(* IEC 61131-3 sources: Explicit_MPC_on_PLC/Quad-Tank/MATLAB_Files/plcsrc, 1 file *)

(* ---- sim_mixed.st ---- *)
(*
 *
 * File: sim_mixed.st
 *
 * IEC 61131-3 Structured Text (ST) code generated for subsystem "sim_mixed/Explicit Controller"
 *
 * Model name                      : sim_mixed
 * Model version                   : 1.162
 * Model creator                   : andrewralea
 * Model last modified by          : andrewralea
 * Model last modified on          : Fri May 21 18:47:45 2021
 * Model sample time               : 0s
 * Subsystem name                  : sim_mixed/Explicit Controller
 * Subsystem sample time           : 0.5s
 * Simulink PLC Coder version      : 3.3 (R2020b) 29-Jul-2020
 * ST code generated on            : Fri May 21 23:25:07 2021
 *
 * Target IDE selection            : Beckhoff TwinCAT 3
 * Test Bench included             : No
 *
 *)
FUNCTION_BLOCK Explicit
VAR_INPUT
    ssMethodType: SINT;
    MeasuredTankOutputs: ARRAY [0..1] OF LREAL;
    ref: ARRAY [0..1] OF LREAL;
END_VAR
VAR_OUTPUT
    mv: ARRAY [0..1] OF LREAL;
END_VAR
VAR
    last_x_PreviousInput: ARRAY [0..5] OF LREAL;
    last_mv_DSTATE: ARRAY [0..1] OF LREAL;
    Explicit_b_M: ARRAY [0..11] OF LREAL := 1.23046367255072E-5,1.0600898470460902E-6,2.3336033090402565E-6,
        8.7638681898692419E-6,0.39038774660580289,5.7642544662640772E-8,2.7337306073553671E-6,1.2817201955703276E-5,
        8.74919612830075E-6,2.5558076546081948E-6,-1.9842244313224275E-7,0.39038772758565754;
    Explicit_b_Cm: ARRAY [0..11] OF LREAL := 0.15299877600979192,0.0,0.0,0.15299877600979192,0.0,0.0,0.0,0.0,1.0,
        0.0,0.0,1.0;
    Explicit_b_thmin: ARRAY [0..9] OF LREAL := -12.5,-17.5,-3.260954352640991,-0.9466686383552787,-1.25,-1.25,-12.5,
        -17.5,-44.314868949193837,-76.652836957418671;
    Explicit_b_thmax: ARRAY [0..9] OF LREAL := 30.0,25.0,39.239045647359006,41.553331361644723,1.25,1.25,25.0,20.0,
        150.328,150.328;
    b_i1: ARRAY [0..124] OF INT := 1,31,57,83,108,132,157,182,208,234,258,283,308,333,355,381,402,422,442,463,481,
        502,521,544,564,587,608,627,648,668,687,708,723,742,763,779,799,817,837,852,872,892,907,926,948,968,985,
        1011,1032,1049,1072,1093,1112,1126,1146,1165,1185,1205,1222,1243,1265,1287,1306,1326,1346,1365,1390,1411,
        1427,1446,1466,1485,1504,1524,1544,1560,1579,1597,1616,1632,1653,1672,1691,1709,1731,1751,1771,1787,1807,
        1825,1845,1861,1886,1904,1922,1941,1961,1982,1998,2015,2036,2057,2075,2096,2114,2134,2153,2174,2194,2216,
        2235,2254,2272,2293,2313,2330,2350,2370,2390,2410,2429,2450,2469,2487,2507;
    b_i2: ARRAY [0..124] OF INT := 30,56,82,107,131,156,181,207,233,257,282,307,332,354,380,401,421,441,462,480,501,
        520,543,563,586,607,626,647,667,686,707,722,741,762,778,798,816,836,851,871,891,906,925,947,967,984,1010,
        1031,1048,1071,1092,1111,1125,1145,1164,1184,1204,1221,1242,1264,1286,1305,1325,1345,1364,1389,1410,1426,
        1445,1465,1484,1503,1523,1543,1559,1578,1596,1615,1631,1652,1671,1690,1708,1730,1750,1770,1786,1806,1824,
        1844,1860,1885,1903,1921,1940,1960,1981,1997,2014,2035,2056,2074,2095,2113,2133,2152,2173,2193,2215,2234,
        2253,2271,2292,2312,2329,2349,2369,2389,2409,2428,2449,2468,2486,2506,2526;
    Explicit_b_L: ARRAY [0..11] OF LREAL := 1.19928863023028E-5,2.1952511223334454E-6,2.1569802942442451E-6,
        7.5728062260383986E-6,0.39038774660580267,5.7642544623488507E-8,3.2749111187589827E-6,1.2730433289085341E-5,
        8.0869972913321024E-6,2.2084581488572959E-6,-1.9842244312551109E-7,0.39038772758565737;
    Explicit_b_Bu: ARRAY [0..11] OF LREAL := 0.010205131094390857,0.00040302205517911383,0.0,0.0054488837150258882,
        0.0,0.0,0.00022154024327610144,0.010236745349900997,0.0056320000157246437,0.0,0.0,0.0;
    Explicit_b_A: ARRAY [0..35] OF LREAL := 0.96059819818356329,0.0,0.0,0.0,0.0,0.0,0.0,0.96659623833897423,0.0,0.0,
        0.0,0.0,0.074166176359097585,0.0,0.92431317949013092,0.0,0.0,0.0,0.0,0.1335679905776915,0.0,
        0.86409403496045134,0.0,0.0,0.0,0.0,0.0,0.0,1.0,0.0,0.0,0.0,0.0,0.0,0.0,1.0;
    Explicit_c_K: ARRAY [0..2525] OF LREAL := 85.828012190346456,83.122636404418486,64.080512591089587,
        62.020995879684413,58.758889676769776,56.867312090766596,6.1162428161412166,8.53615478597103,
        4.5664808584950682,6.3691533823982,4.1872534117759654,5.8399035361094738,30.0,25.0,39.239045647359006,
        41.553331361644723,1.25,1.25,25.0,20.0,150.328,150.328,12.5,17.5,3.260954352640991,0.9466686383552787,1.25,
        1.25,12.5,17.5,-85.828012190346442,83.160013557517672,0.39842731610608123,62.06462880871775,
        0.41050111399720146,56.91260957310422,8.4951416229813166,6.3221365550079094,5.7913950841796,30.0,25.0,
        39.239045647359006,41.553331361644723,1.25,1.25,20.0,150.328,150.328,12.5,17.5,3.260954352640991,
        0.9466686383552787,1.25,1.25,12.5,17.5,-83.122636404418486,85.864225454146336,64.121415141998071,
        0.38892275664372283,58.800482042349721,0.400834317759825,6.0763592904683081,4.52235846378462,
        4.1427133961342912,30.0,25.0,39.239045647359006,41.553331361644723,1.25,1.25,25.0,150.328,150.328,12.5,17.5,
        3.260954352640991,0.9466686383552787,1.25,1.25,12.5,17.5,-64.080512591089587,8.505599391495803,
        5.8036863919186326,-77.527008024685543,118.15715787051693,83.1493054364041,62.0524437250436,
        56.9000995036549,6.33408222099711,30.0,25.0,39.239045647359006,41.553331361644723,1.25,1.25,25.0,20.0,
        150.328,12.5,17.5,3.260954352640991,0.9466686383552787,1.25,1.25,17.5,-62.020995879684421,6.085443991111319,
        4.1528211444790628,-75.0536194743548,85.854610754335354,114.60675801046474,64.110937969245654,
        58.789954915559505,30.0,25.0,39.239045647359006,41.553331361644723,1.25,1.25,25.0,20.0,150.328,12.5,17.5,
        3.260954352640991,0.9466686383552787,1.25,1.25,12.5,-58.758889676769776,106.51779109033414,
        83.142049521683674,77.527008024685614,62.043935540441744,56.891257027927281,8.5137096448380447,
        6.3433957805279579,5.813284165486909,30.0,25.0,39.239045647359006,41.553331361644723,1.25,1.25,25.0,20.0,
        150.328,12.5,17.5,3.260954352640991,0.9466686383552787,1.25,1.25,17.5,-56.8673120907666,85.84776398721317,
        103.24892161906958,64.103194722139946,75.053619474354818,58.78208141394331,6.0931186576995735,
        4.5408406057656192,4.161356421857743,30.0,25.0,39.239045647359006,41.553331361644723,1.25,1.25,25.0,20.0,
        150.328,12.5,17.5,3.260954352640991,0.9466686383552787,1.25,1.25,12.5,-6.1162428161412148,
        83.116440481385681,62.014599085134925,56.860964676950751,8.53871469911331,0.028392574262163343,
        6.3721662785907309,0.029252972606836448,5.8430399803330584,30.0,25.0,39.239045647359006,41.553331361644723,
        1.25,1.25,25.0,20.0,150.328,12.5,17.5,3.260954352640991,0.9466686383552787,1.25,1.25,17.5,
        44.314868949193837,-8.53615478597103,85.820515372368362,64.072997847575692,58.751584273947309,
        6.1200693722462738,4.5707757582069863,0.039939840627104373,4.1916111645367051,0.041163080575065084,30.0,
        25.0,39.239045647359006,41.553331361644723,1.25,1.25,25.0,20.0,150.328,12.5,17.5,3.260954352640991,
        0.9466686383552787,1.25,1.25,12.5,76.652836957418671,-4.5664808584950682,-5.524699847834043,
        83.11695127091906,62.015234820715769,56.861634602583806,8.420069969679389,8.5379442187057482,
        5.8421419917176536,30.0,25.0,39.239045647359006,41.553331361644723,1.25,1.25,20.0,150.328,12.5,17.5,
        3.260954352640991,0.9466686383552787,1.25,1.25,12.5,17.5,-6.3691533823982,85.821037326316272,
        58.752296293187449,-7.7075191643753813,64.073586813938277,6.1190978799236042,11.769369550983704,
        4.5697137015683689,4.1905427066538907,30.0,25.0,39.239045647359006,41.553331361644723,1.25,1.25,25.0,
        150.328,12.5,17.5,3.260954352640991,0.9466686383552787,1.25,1.25,12.5,17.5,-4.1872534117759654,
        83.118307397217492,62.016623545698224,56.863007536175935,7.5906298878580278,8.5374517693042264,
        5.5246998478340474,6.3707077752714794,5.8415336572382541,30.0,25.0,39.239045647359006,41.553331361644723,
        1.25,1.25,20.0,150.328,12.5,17.5,3.260954352640991,0.9466686383552787,1.25,1.25,12.5,17.5,
        -5.8399035361094747,85.822512499078186,64.075138367645479,58.75372340844936,6.1183701458345565,
        10.602993535201676,4.5688969602600853,7.7075191643753822,4.1897144273516966,30.0,25.0,39.239045647359006,
        41.553331361644723,1.25,1.25,25.0,150.328,12.5,17.5,3.260954352640991,0.9466686383552787,1.25,1.25,12.5,
        17.5,-85.864225454146322,-83.160013557517686,0.44629698661502609,0.44356800965144572,0.45744577207009696,
        0.45640388165452567,30.0,25.0,39.239045647359006,41.553331361644723,1.25,1.25,150.328,150.328,12.5,17.5,
        3.260954352640991,0.9466686383552787,1.25,1.25,12.5,17.5,-0.398427316106117,-118.15715787051693,
        -0.37406353461084024,83.159322276278772,62.063996287931914,56.912013263967516,8.4950256940452444,
        6.3220198554896259,5.7912802018971812,30.0,25.0,39.239045647359006,41.553331361644723,1.25,1.25,25.0,20.0,
        150.328,150.328,12.5,17.5,3.260954352640991,0.9466686383552787,1.25,1.25,17.5,-85.8546972344799,
        114.6331530507331,0.42416405806333568,12.5,-118.17578392102031,-62.063996287931936,0.4242260045196693,30.0,
        25.0,39.239045647359006,41.553331361644723,1.25,1.25,25.0,150.328,12.5,17.5,3.260954352640991,
        0.9466686383552787,1.25,1.25,-106.51779109033414,-0.41050111399722317,83.159485968072531,
        0.37406353461083286,5.7913051165041507,30.0,25.0,39.239045647359006,41.553331361644723,1.25,1.25,150.328,
        150.328,12.5,17.5,3.260954352640991,0.9466686383552787,1.25,1.25,17.5,-85.847763987213185,75.09263865743236,
        12.5,-118.17085773789718,-56.91201326396753,30.0,25.0,39.239045647359006,41.553331361644723,1.25,1.25,25.0,
        20.0,150.328,12.5,17.5,3.260954352640991,0.9466686383552787,1.25,1.25,-85.820515372368362,
        -8.4951416229813166,12.5,-118.15424814904154,0.4416142007094101,-0.014455303353979251,30.0,25.0,
        39.239045647359006,41.553331361644723,1.25,1.25,20.0,150.328,12.5,17.5,3.260954352640991,0.9466686383552787,
        1.25,1.25,76.652836957418671,-85.821037326316258,-6.3221365550079085,0.39462833151258975,11.743492163705721,
        -0.020734861096918376,30.0,25.0,39.239045647359006,1.25,1.25,150.328,12.5,17.5,3.260954352640991,
        0.9466686383552787,1.25,1.25,12.5,-85.8225124990782,-5.7913950841796,0.395566095525043,0.40769403601124449,
        10.57062075206243,7.6648400160986254,30.0,25.0,39.239045647359006,41.553331361644723,1.25,1.25,150.328,12.5,
        17.5,3.260954352640991,0.9466686383552787,1.25,1.25,12.5,17.5,-83.1493575575283,-64.120717438993182,
        -114.62360062013384,118.1846753798998,0.41885284236598441,30.0,25.0,39.239045647359006,41.553331361644723,
        1.25,1.25,20.0,150.328,12.5,17.5,3.260954352640991,0.9466686383552787,1.25,1.25,-114.60941055213036,
        -0.38892275664366538,85.863418000357726,64.120717438993168,58.799849575245759,0.43609812832468658,
        6.0762590176834195,4.5222612688740718,4.1426203395211836,30.0,25.0,39.239045647359006,41.553331361644723,
        1.25,1.25,25.0,150.328,12.5,17.5,3.260954352640991,0.9466686383552787,1.25,1.25,-83.142049521683688,
        -58.800482042349707,106.54814350107794,77.565803690576558,0.4188608700639273,30.0,25.0,39.239045647359006,
        41.553331361644723,1.25,1.25,25.0,150.328,12.5,17.5,3.260954352640991,0.9466686383552787,1.25,1.25,17.5,
        -103.24892161906961,-0.40083431775979822,58.799926098422773,6.0762686203119909,4.5222701309312336,
        4.1426286413254676,30.0,25.0,39.239045647359006,41.553331361644723,1.25,1.25,25.0,20.0,150.328,150.328,12.5,
        17.5,3.260954352640991,0.9466686383552787,1.25,1.25,12.5,-83.116440481385666,-6.076359290468309,
        0.38503032707136814,-0.01947372407836211,-0.017687831808316137,30.0,25.0,39.239045647359006,
        41.553331361644723,1.25,1.25,25.0,150.328,12.5,17.5,3.260954352640991,0.9466686383552787,1.25,1.25,17.5,
        44.314868949193837,-83.117007264204418,-4.52235846378462,0.38602131564609687,8.3918353890059159,
        -0.017493533221530456,30.0,25.0,39.239045647359006,41.553331361644723,1.25,1.25,150.328,12.5,17.5,
        3.260954352640991,0.9466686383552787,1.25,1.25,17.5,-83.1183073972175,-4.1427133961342912,
        0.38679247515387888,0.39865998103592931,7.55674387574281,5.4820594007599839,30.0,25.0,39.239045647359006,
        41.553331361644723,1.25,1.25,150.328,12.5,17.5,3.260954352640991,0.9466686383552787,1.25,1.25,12.5,17.5,
        -64.111012657460421,-62.05249072734096,-77.555645848818614,-75.081475575886287,118.17571595289762,
        114.62356476522335,30.0,25.0,39.239045647359006,41.553331361644723,1.25,1.25,25.0,20.0,12.5,17.5,
        3.260954352640991,0.9466686383552787,1.25,1.25,-64.103194722139961,-56.900143592917374,-77.548207597133882,
        118.17085773789714,75.081423676406,30.0,25.0,39.239045647359006,41.553331361644723,1.25,1.25,25.0,20.0,12.5,
        17.5,3.260954352640991,0.9466686383552787,1.25,1.25,-64.072997847575721,-0.00038946835147730041,
        -77.519066370906955,-8.5055900532206987,118.1515689116242,-0.00082231448690014367,30.0,25.0,
        39.239045647359006,41.553331361644723,1.25,1.25,25.0,20.0,12.5,17.5,3.260954352640991,0.9466686383552787,
        1.25,1.25,76.652836957418671,-77.51962271516804,-6.3340822209971117,118.15191973090961,11.750255328683597,
        -0.0063432264244943359,30.0,25.0,39.239045647359006,1.25,1.25,12.5,3.260954352640991,0.9466686383552787,
        1.25,1.25,-62.043935540441744,-58.790022508827825,-75.073834709949978,114.61897100925754,77.555554626286366,
        30.0,25.0,39.239045647359006,41.553331361644723,1.25,1.25,25.0,20.0,12.5,17.5,3.260954352640991,
        0.9466686383552787,1.25,1.25,-62.014599085134925,-0.0070706326789994178,-75.047283265141758,
        -6.0854329422821021,114.60272685911939,-0.0086568972280961238,30.0,25.0,39.239045647359006,
        41.553331361644723,1.25,1.25,25.0,20.0,12.5,17.5,3.260954352640991,0.9466686383552787,1.25,1.25,
        44.314868949193837,-62.015286283395191,-75.047891103343,-4.5323625462609973,114.603090854087,
        8.3983970252048046,-0.0074926324264197172,30.0,25.0,41.553331361644723,1.25,1.25,17.5,3.260954352640991,
        0.9466686383552787,1.25,1.25,-62.016623545698216,7.5645109612818882,5.4917443184814969,-75.049221181750653,
        -4.1528107607208362,114.60393228403262,30.0,25.0,39.239045647359006,41.553331361644723,1.25,1.25,20.0,12.5,
        17.5,3.260954352640991,0.9466686383552787,1.25,1.25,12.5,-58.782081413943317,-56.891257027927274,
        77.548207597133867,75.073834709949978,30.0,25.0,39.239045647359006,41.553331361644723,1.25,1.25,25.0,20.0,
        12.5,17.5,3.260954352640991,0.9466686383552787,1.25,1.25,-58.7515842739473,-8.5137096448380465,
        77.519066370907012,0.010004976673610552,0.01060860807900669,30.0,25.0,39.239045647359006,41.553331361644723,
        1.25,1.25,25.0,20.0,12.5,17.5,3.260954352640991,0.9466686383552787,1.25,1.25,76.652836957418671,
        -58.752296293187442,-6.3433957805279588,77.519622715168069,11.755417270134494,0.0051808031401439766,30.0,
        25.0,39.239045647359006,1.25,1.25,12.5,3.260954352640991,0.9466686383552787,1.25,1.25,-58.753723408449368,
        -5.8132841654869081,106.51277089775623,77.5211858423469,10.585362190891489,7.6842594239932183,30.0,25.0,
        39.239045647359006,41.553331361644723,1.25,1.25,25.0,12.5,17.5,3.260954352640991,0.9466686383552787,1.25,
        1.25,17.5,-56.860964676950758,-6.0931186576995744,75.047283265141758,0.0004819952794122263,
        0.0018653631060791922,30.0,25.0,39.239045647359006,41.553331361644723,1.25,1.25,25.0,20.0,12.5,17.5,
        3.260954352640991,0.9466686383552787,1.25,1.25,44.314868949193837,-56.861683329367956,-4.5408406057656192,
        75.047891103343034,8.4039168003417171,0.00086263338459051614,30.0,25.0,41.553331361644723,1.25,1.25,17.5,
        3.260954352640991,0.9466686383552787,1.25,1.25,-56.863007536175942,-4.1613564218577421,75.049221181750667,
        7.5710632281136787,5.4999590543921695,30.0,25.0,39.239045647359006,41.553331361644723,1.25,1.25,20.0,12.5,
        17.5,3.260954352640991,0.9466686383552787,1.25,1.25,12.5,-6.1200693722462729,-8.53871469911331,
        0.033308379514583306,0.043833998920251686,0.034073770963663527,0.045123106671733478,30.0,25.0,
        39.239045647359006,41.553331361644723,1.25,1.25,25.0,20.0,12.5,17.5,3.260954352640991,0.9466686383552787,
        1.25,1.25,44.314868949193837,76.652836957418671,-8.4202608646752974,-0.028392574262167184,
        83.115761676948409,0.03179317101742711,5.8429818276867413,30.0,25.0,39.239045647359006,41.553331361644723,
        1.25,1.25,150.328,12.5,17.5,3.260954352640991,0.9466686383552787,1.25,1.25,17.5,44.314868949193837,
        -6.1191038992749363,-6.3721662785907309,11.771265259713571,0.032197136802679695,0.0329836210389647,
        0.041726222624840562,30.0,25.0,39.239045647359006,1.25,1.25,12.5,3.260954352640991,0.9466686383552787,1.25,
        1.25,44.314868949193837,-7.5906298878580269,-0.029252972606838269,-8.4200699696793873,-0.031793171017425036,
        83.115705542269154,62.013916295543666,56.860316251743967,8.5386424280548709,5.8429772141207312,30.0,25.0,
        39.239045647359006,41.553331361644723,1.25,1.25,20.0,150.328,12.5,17.5,3.260954352640991,0.9466686383552787,
        1.25,1.25,12.5,17.5,44.314868949193837,-6.1183701458345565,-5.8430399803330584,10.604988621801292,
        0.031259206362317861,7.7101954083892581,0.0320659337330362,30.0,25.0,39.239045647359006,41.553331361644723,
        1.25,1.25,25.0,12.5,17.5,3.260954352640991,0.9466686383552787,1.25,1.25,17.5,44.314868949193837,
        -8.5379496848197061,-4.5707757582069872,8.4229686692129437,0.042844600630423051,0.031233264023239459,
        0.0441245220372481,30.0,25.0,41.553331361644723,1.25,1.25,17.5,3.260954352640991,0.9466686383552787,1.25,
        1.25,76.652836957418671,-11.76964194978159,-0.039939840627101146,85.81966393244727,64.0722512761259,
        58.750902412901056,6.1200130855938886,4.5707274317413553,4.1915675018658884,0.044784444842926388,30.0,25.0,
        39.239045647359006,1.25,1.25,150.328,12.5,17.5,3.260954352640991,0.9466686383552787,1.25,1.25,12.5,
        76.652836957418671,-8.5374517693042282,-4.1916111645367051,7.5938505626709718,5.5287967204295976,
        0.042073371583645526,0.043340776816804351,30.0,25.0,39.239045647359006,41.553331361644723,1.25,1.25,20.0,
        12.5,17.5,3.260954352640991,0.9466686383552787,1.25,1.25,12.5,76.652836957418671,-10.602993535201678,
        -0.041163080575063606,58.750981868299043,6.1200199184728907,0.03747611419719786,30.0,25.0,
        39.239045647359006,41.553331361644723,1.25,1.25,25.0,12.5,17.5,3.260954352640991,0.9466686383552787,1.25,
        1.25,76.652836957418671,-4.5697188630749395,-6.3712960830276284,8.4222683561715836,11.770769743636622,
        0.030205806756567293,0.040700404868083094,30.0,25.0,1.25,1.25,3.260954352640991,0.9466686383552787,1.25,
        1.25,-4.5688969602600862,-5.5269808091791131,-5.8421419917176527,8.4215544623245489,10.604372229290151,
        7.7093889571683532,30.0,25.0,39.239045647359006,41.553331361644723,1.25,1.25,12.5,17.5,3.260954352640991,
        0.9466686383552787,1.25,1.25,12.5,17.5,-6.3707077752714785,-4.1905473601194307,7.593021267767619,
        11.77045485602477,5.52776745213207,0.039879617824932635,30.0,25.0,39.239045647359006,41.553331361644723,
        1.25,1.25,12.5,17.5,3.260954352640991,0.9466686383552787,1.25,1.25,12.5,-4.1897144273516975,
        -5.8415336572382524,7.5924009228672258,10.603989796750705,5.5269808091791148,7.7088729521925243,30.0,25.0,
        39.239045647359006,41.553331361644723,1.25,1.25,12.5,17.5,3.260954352640991,0.9466686383552787,1.25,1.25,
        12.5,17.5,-0.44634767231186967,-118.18206484525585,-114.63269219140271,-0.002932140532956061,
        0.49446522872235754,30.0,25.0,39.239045647359006,41.553331361644723,1.25,1.25,25.0,150.328,150.328,12.5,
        17.5,3.260954352640991,0.9466686383552787,1.25,1.25,-85.863418000357726,-114.63315305073311,
        -0.44356800965144572,0.44634767231188421,0.49440252833552661,30.0,25.0,39.239045647359006,
        41.553331361644723,1.25,1.25,17.5,3.260954352640991,0.9466686383552787,1.25,1.25,12.5,-106.54814350107794,
        -0.45744577207011383,-118.18270354170637,-83.159322276278786,0.44362468763113161,30.0,25.0,
        39.239045647359006,41.553331361644723,1.25,1.25,25.0,150.328,150.328,12.5,17.5,3.260954352640991,
        0.9466686383552787,1.25,1.25,17.5,-85.854610754335368,114.63050198966798,12.5,-0.4242192328574797,
        -118.17571595289762,-0.68401755435542955,-0.0009446396613658611,30.0,25.0,39.239045647359006,
        41.553331361644723,1.25,1.25,25.0,20.0,150.328,12.5,17.5,3.260954352640991,0.9466686383552787,1.25,1.25,
        -106.51277089775624,-0.40769403601121151,-118.15302843537035,-0.44350123965052496,-5.7912802018971812,
        10.570524291867653,7.6647227436564362,30.0,25.0,39.239045647359006,41.553331361644723,1.25,1.25,25.0,
        150.328,12.5,17.5,3.260954352640991,0.9466686383552787,1.25,1.25,17.5,-85.81966393244727,
        -11.743492163705717,0.01470368365977508,0.39351182868930534,-0.01351795809839609,30.0,25.0,
        39.239045647359006,1.25,1.25,150.328,12.5,17.5,3.260954352640991,0.9466686383552787,1.25,1.25,12.5,
        76.652836957418671,-85.820945816693865,-7.6648400160986263,0.394628129370387,0.4067764251094641,
        11.743217822719652,30.0,25.0,39.239045647359006,41.553331361644723,1.25,1.25,150.328,12.5,17.5,
        3.260954352640991,0.9466686383552787,1.25,1.25,12.5,17.5,-83.1493054364041,-77.5658036905766,
        -0.41879942848729695,118.18270354170636,0.429688452146867,30.0,25.0,39.239045647359006,41.553331361644723,
        1.25,1.25,25.0,150.328,12.5,17.5,3.260954352640991,0.9466686383552787,1.25,1.25,17.5,-0.41886087006396983,
        -58.799849575245752,-114.61897100925758,77.564863200154221,30.0,25.0,39.239045647359006,41.553331361644723,
        1.25,1.25,25.0,20.0,150.328,12.5,17.5,3.260954352640991,0.9466686383552787,1.25,1.25,-114.60675801046473,
        -0.00097133111195961744,85.863332283572987,64.120643632089468,58.799782885627366,6.0762470854561723,
        4.5222494737506054,4.1426089522719654,30.0,25.0,39.239045647359006,41.553331361644723,1.25,1.25,25.0,20.0,
        150.328,150.328,12.5,17.5,3.260954352640991,0.9466686383552787,1.25,1.25,12.5,-0.38503032707140167,
        -0.017735509254940576,-114.60272685911937,-6.0762470854561732,-0.019529134072728146,30.0,25.0,
        39.239045647359006,41.553331361644723,1.25,1.25,25.0,20.0,150.328,12.5,17.5,3.260954352640991,
        0.9466686383552787,1.25,1.25,44.314868949193837,-0.38602131564614095,-114.60309085408703,
        -4.5222494737506045,8.391750925351861,-0.017545002408333659,30.0,25.0,41.553331361644723,1.25,1.25,150.328,
        17.5,3.260954352640991,0.9466686383552787,1.25,1.25,-114.60658526808871,-0.38679247515393256,
        -4.1426203395211836,0.43379366916949563,7.5566517708082808,5.4819530873798339,30.0,25.0,39.239045647359006,
        41.553331361644723,1.25,1.25,150.328,12.5,17.5,3.260954352640991,0.9466686383552787,1.25,1.25,
        -114.60393228403267,-0.00096624459998579521,-0.033098274961671253,7.55664099352456,5.4819404256920183,30.0,
        25.0,39.239045647359006,41.553331361644723,1.25,1.25,20.0,150.328,12.5,17.5,3.260954352640991,
        0.9466686383552787,1.25,1.25,12.5,-83.115761676948424,-8.3918353890059141,0.0194737240783594,
        -0.012398005368195967,30.0,25.0,39.239045647359006,41.553331361644723,1.25,1.25,150.328,12.5,17.5,
        3.260954352640991,0.9466686383552787,1.25,1.25,17.5,44.314868949193837,-83.1158775962047,
        -114.60500434458611,-7.5566517708082817,0.017735509254940669,0.43194320846841294,-0.023118977973232171,25.0,
        39.239045647359006,41.553331361644723,1.25,1.25,150.328,12.5,17.5,3.260954352640991,0.9466686383552787,1.25,
        1.25,44.314868949193837,-83.11695127091906,-5.4820594007599839,0.38602116679095089,0.39787613417225604,
        8.3916432470157343,30.0,25.0,39.239045647359006,41.553331361644723,1.25,1.25,150.328,12.5,17.5,
        3.260954352640991,0.9466686383552787,1.25,1.25,12.5,17.5,-77.521185842346924,-0.37195926026359716,
        -5.803677090646552,118.15302843537032,10.578959214695042,7.6758005279589154,30.0,25.0,39.239045647359006,
        41.553331361644723,1.25,1.25,25.0,12.5,17.5,3.260954352640991,0.9466686383552787,1.25,1.25,17.5,
        -77.518169208191026,-11.750255328683602,0.00082231448689868152,118.1508991703279,0.0008731014305541501,30.0,
        25.0,39.239045647359006,1.25,1.25,3.260954352640991,0.9466686383552787,1.25,1.25,12.5,76.652836957418671,
        -64.073586813938277,-77.519526121135655,-7.6758005279589119,118.15184831703415,11.749981442806606,30.0,25.0,
        39.239045647359006,41.553331361644723,1.25,1.25,25.0,12.5,17.5,3.260954352640991,0.9466686383552787,1.25,
        1.25,17.5,-62.01407694508385,-7.56451096128189,0.0070706326789994178,114.60500434458612,0.36170035909111187,
        -0.01183364944556279,25.0,39.239045647359006,41.553331361644723,1.25,1.25,12.5,17.5,3.260954352640991,
        0.9466686383552787,1.25,1.25,44.314868949193837,-62.015234820715762,-75.0478352471966,-5.4917325994290085,
        114.6030525611145,8.39820515126693,30.0,25.0,39.239045647359006,41.553331361644723,1.25,1.25,20.0,12.5,17.5,
        3.260954352640991,0.9466686383552787,1.25,1.25,12.5,-58.750902412901056,-11.755417270134494,
        -0.010004976673607866,77.518169208190983,0.012396379096950183,30.0,25.0,39.239045647359006,1.25,1.25,
        3.260954352640991,0.9466686383552787,1.25,1.25,12.5,76.652836957418671,-10.585362190891495,
        -0.01060860807900669,77.518274070116234,-0.46940252178175107,-11.755143770144398,106.51012568504407,30.0,
        25.0,39.239045647359006,41.553331361644723,1.25,1.25,25.0,12.5,17.5,3.260954352640991,0.9466686383552787,
        1.25,1.25,17.5,76.652836957418671,-58.752222969626445,-7.6842594239932129,106.51134625768024,
        77.519526121135613,11.755143770144398,30.0,25.0,39.239045647359006,41.553331361644723,1.25,1.25,25.0,12.5,
        17.5,3.260954352640991,0.9466686383552787,1.25,1.25,17.5,-56.860468976817742,-7.5710632281136787,
        -0.0018653631060791924,75.0467199903292,-0.002304359115311651,30.0,25.0,39.239045647359006,
        41.553331361644723,1.25,1.25,20.0,12.5,17.5,3.260954352640991,0.9466686383552787,1.25,1.25,
        44.314868949193837,-56.861634602583806,-5.4999590543921677,75.0478352471966,8.4037251597977,30.0,25.0,
        39.239045647359006,41.553331361644723,1.25,1.25,20.0,12.5,17.5,3.260954352640991,0.9466686383552787,1.25,
        1.25,12.5,-7.5938505626709727,-8.5386594834923439,-0.034073770963664769,-8.4227778770978858,
        0.043838081888991604,0.045127298509467346,30.0,25.0,39.239045647359006,41.553331361644723,1.25,1.25,20.0,
        12.5,17.5,3.260954352640991,0.9466686383552787,1.25,1.25,12.5,44.314868949193837,76.652836957418671,
        -6.1200199184728907,-10.604988621801295,-0.045123106671733464,0.033313252740456621,0.041237554015286768,
        0.034078572021591425,30.0,39.239045647359006,41.553331361644723,1.25,1.25,25.0,12.5,17.5,3.260954352640991,
        0.9466686383552787,1.25,1.25,44.314868949193837,76.652836957418671,-0.031259206362318236,
        -8.4215544623245453,-0.029630789771451348,-5.8429772141207321,7.7101231200214224,30.0,25.0,
        39.239045647359006,41.553331361644723,1.25,1.25,12.5,17.5,3.260954352640991,0.9466686383552787,1.25,1.25,
        12.5,17.5,44.314868949193837,-7.5930212677676163,-6.3721156394759433,-0.032983621038964073,
        11.771228317467887,0.030609387563068639,0.041729840131366033,25.0,39.239045647359006,1.25,1.25,12.5,
        3.260954352640991,0.9466686383552787,1.25,1.25,44.314868949193837,-6.1190978799236042,-7.71019540838926,
        11.770992953268273,0.032197753901730748,0.032984231966322344,30.0,25.0,39.239045647359006,
        41.553331361644723,1.25,1.25,25.0,12.5,17.5,3.260954352640991,0.9466686383552787,1.25,1.25,17.5,
        44.314868949193837,-7.5924009228672258,-0.032065933733037143,-5.8429921672978837,10.604940845072546,
        0.02963078977144552,7.7101402281230822,25.0,39.239045647359006,41.553331361644723,1.25,1.25,12.5,17.5,
        3.260954352640991,0.9466686383552787,1.25,1.25,44.314868949193837,-8.5379442187057482,-5.5287967204295967,
        8.4227778770978876,0.042844970869026749,0.044124904981453182,30.0,25.0,39.239045647359006,
        41.553331361644723,1.25,1.25,20.0,12.5,17.5,3.260954352640991,0.9466686383552787,1.25,1.25,12.5,
        76.652836957418671,-10.604377024927771,-4.5707333389510429,-0.044124522037249814,8.42292953358605,
        0.040266686663842088,0.031237784200925479,30.0,41.553331361644723,1.25,1.25,17.5,3.260954352640991,
        0.9466686383552787,1.25,1.25,76.652836957418671,-11.769369550983704,-0.00016426179431715824,
        85.819572220872473,64.07217074193909,58.750828893770574,6.1200071481566889,4.570722363900976,
        4.1915629441287612,30.0,25.0,39.239045647359006,41.553331361644723,1.25,1.25,25.0,150.328,12.5,17.5,
        3.260954352640991,0.9466686383552787,1.25,1.25,12.5,17.5,76.652836957418671,-5.5277674521320668,
        -6.3712911253249436,8.4220775324286361,11.770765990925339,0.040700817731536956,30.0,25.0,39.239045647359006,
        41.553331361644723,1.25,1.25,12.5,17.5,3.260954352640991,0.9466686383552787,1.25,1.25,12.5,
        -4.569713701568368,-7.7093944030003776,8.4222636116464233,11.770497400517035,0.030206389050708594,30.0,25.0,
        39.239045647359006,41.553331361644723,1.25,1.25,12.5,17.5,3.260954352640991,0.9466686383552787,1.25,1.25,
        17.5,-7.70887295219252,-4.1905427066538907,7.59301540205904,11.770182495369303,5.5277611045797483,30.0,25.0,
        39.239045647359006,41.553331361644723,1.25,1.25,12.5,17.5,3.260954352640991,0.9466686383552787,1.25,1.25,
        12.5,17.5,-85.863332283572987,-114.63050198966802,-0.49440252833559767,0.44635490076680528,30.0,25.0,
        39.239045647359006,41.553331361644723,1.25,1.25,20.0,150.328,150.328,12.5,17.5,3.260954352640991,
        0.9466686383552787,1.25,1.25,12.5,-118.15156891162422,-0.00098058513524279045,-8.4950256940452444,
        -0.014758817879689093,-0.014461312360842374,30.0,25.0,39.239045647359006,41.553331361644723,1.25,1.25,25.0,
        20.0,150.328,12.5,17.5,3.260954352640991,0.9466686383552787,1.25,1.25,76.652836957418671,
        -118.15191973090963,-0.44264422484231769,-6.3220198554896267,11.743416534177809,-0.020795705173902376,30.0,
        25.0,39.239045647359006,1.25,1.25,150.328,12.5,3.260954352640991,0.9466686383552787,1.25,1.25,
        -0.39351182868926454,0.014752997394703711,-118.15089917032793,-11.743416534177813,9.7548511906835519E-5,
        -0.013578719429673154,30.0,25.0,39.239045647359006,1.25,1.25,3.260954352640991,0.9466686383552787,1.25,1.25,
        12.5,76.652836957418671,-106.51134625768027,-0.40677642510946205,-7.6647485126274715,-118.15184831703417,
        -0.069818470214603592,11.74314218041998,30.0,25.0,39.239045647359006,41.553331361644723,1.25,1.25,25.0,
        150.328,12.5,17.5,3.260954352640991,0.9466686383552787,1.25,1.25,17.5,-85.819572220872473,
        -11.743217822719652,0.015304801598363425,0.39351151324681566,0.40568104262717841,30.0,25.0,
        39.239045647359006,41.553331361644723,1.25,1.25,150.328,12.5,17.5,3.260954352640991,0.9466686383552787,1.25,
        1.25,12.5,17.5,76.652836957418671,-118.15452758849368,-0.39462812937039843,-7.6647328602357874,
        0.44264413175858619,11.743148813560541,30.0,25.0,39.239045647359006,41.553331361644723,1.25,1.25,150.328,
        12.5,17.5,3.260954352640991,0.9466686383552787,1.25,1.25,-77.564953604651592,-0.42968845214694085,
        -0.41884602854483993,-114.62356476522336,-0.000929749021845083,118.18199739509683,30.0,25.0,
        39.239045647359006,41.553331361644723,1.25,1.25,25.0,20.0,150.328,12.5,17.5,3.260954352640991,
        0.9466686383552787,1.25,1.25,-114.60570567060375,-0.386021166790991,-5.4819530873798357,0.43297278618731544,
        8.39156757255133,30.0,25.0,39.239045647359006,41.553331361644723,1.25,1.25,150.328,12.5,17.5,
        3.260954352640991,0.9466686383552787,1.25,1.25,-0.00096214311185142476,20.0,12.5,-114.60489159987256,
        -8.3915675725513328,0.00010087232721741922,30.0,25.0,39.239045647359006,41.553331361644723,1.25,1.25,
        150.328,12.5,17.5,3.260954352640991,0.9466686383552787,1.25,1.25,44.314868949193837,-114.60305256111451,
        -0.00096442945721852611,-0.049759590977661979,8.39155877484419,30.0,25.0,39.239045647359006,
        41.553331361644723,1.25,1.25,20.0,150.328,12.5,17.5,3.260954352640991,0.9466686383552787,1.25,1.25,12.5,
        -83.115705542269168,-8.3916432470157325,0.0001006508275222847,0.38502778786240521,0.39687344589249135,30.0,
        25.0,39.239045647359006,41.553331361644723,1.25,1.25,150.328,12.5,17.5,3.260954352640991,0.9466686383552787,
        1.25,1.25,12.5,17.5,44.314868949193837,-10.578959214695042,0.00039451180860772874,118.15097923815829,
        -0.70363179395700481,-11.749981442806607,30.0,25.0,39.239045647359006,41.553331361644723,1.25,1.25,25.0,
        12.5,17.5,3.260954352640991,0.9466686383552787,1.25,1.25,17.5,76.652836957418671,-0.36170035909112136,
        -7.5645009189634447,0.00707627176763845,114.60235116779576,-0.6836039993018449,-0.0008054098834180505,
        -8.3982051512669322,30.0,25.0,39.239045647359006,41.553331361644723,1.25,1.25,20.0,12.5,17.5,
        3.260954352640991,0.9466686383552787,1.25,1.25,12.5,44.314868949193837,-62.013916295543666,
        -8.3982133423179413,0.011833649445564786,114.60489159987254,0.36169963089352436,30.0,25.0,
        39.239045647359006,41.553331361644723,1.25,1.25,12.5,17.5,3.260954352640991,0.9466686383552787,1.25,1.25,
        12.5,44.314868949193837,-56.860316251743967,-8.4037251597977018,0.0023043591153104723,75.046547210187924,
        30.0,25.0,39.239045647359006,41.553331361644723,1.25,1.25,20.0,12.5,17.5,3.260954352640991,
        0.9466686383552787,1.25,1.25,12.5,44.314868949193837,-7.5938023247904125,-10.604940845072548,
        -0.034078572021590869,-0.045126507890494459,0.03176800656216968,0.041240681639767594,39.239045647359006,
        41.553331361644723,1.25,1.25,12.5,17.5,3.260954352640991,0.9466686383552787,1.25,1.25,44.314868949193837,
        76.652836957418671,-6.1200071481566889,-11.770992953268275,-0.041237554015278816,0.033314253447269578,
        0.034079552664745452,30.0,25.0,39.239045647359006,41.553331361644723,1.25,1.25,25.0,12.5,17.5,
        3.260954352640991,0.9466686383552787,1.25,1.25,17.5,44.314868949193837,76.652836957418671,
        -6.3720998478778679,12.5,-8.4222636116464233,-0.032197753901727778,-7.7101285249689635,11.770948537206152,
        30.0,25.0,39.239045647359006,41.553331361644723,1.25,1.25,12.5,17.5,3.260954352640991,0.9466686383552787,
        1.25,1.25,17.5,44.314868949193837,-7.5930154020590379,-7.7101402281230875,-0.032984231966323295,
        11.770956002817599,0.030610017337793428,25.0,39.239045647359006,41.553331361644723,1.25,1.25,12.5,17.5,
        3.260954352640991,0.9466686383552787,1.25,1.25,44.314868949193837,-4.570722363900976,-11.770493646915464,
        -0.050184311204822224,-0.00010672665139996041,8.422728557974823,30.0,25.0,39.239045647359006,
        41.553331361644723,1.25,1.25,12.5,17.5,3.260954352640991,0.9466686383552787,1.25,1.25,12.5,17.5,
        76.652836957418671,-11.770182495369301,-0.00017323226355056993,-0.0334894035237961,7.593789840265794,
        5.528731223950869,30.0,25.0,39.239045647359006,41.553331361644723,1.25,1.25,12.5,17.5,3.260954352640991,
        0.9466686383552787,1.25,1.25,12.5,17.5,76.652836957418671,-5.5277611045797475,-7.7093889571683558,
        -0.030206389050703015,-0.040700817731524709,8.4220727871303609,11.770493646915462,30.0,25.0,
        39.239045647359006,41.553331361644723,1.25,1.25,12.5,17.5,3.260954352640991,0.9466686383552787,1.25,1.25,
        12.5,17.5,-118.18467537989979,-114.63007650534455,-0.0029377381217029126,-0.0011013946382212041,
        0.49039849886577358,30.0,25.0,39.239045647359006,41.553331361644723,1.25,1.25,20.0,150.328,150.328,12.5,
        17.5,3.260954352640991,0.9466686383552787,1.25,1.25,-118.15097923815836,6.3888721868823271E-5,
        -0.0153570751143045,30.0,25.0,39.239045647359006,1.25,1.25,25.0,20.0,150.328,150.328,12.5,17.5,
        3.260954352640991,0.9466686383552787,1.25,1.25,76.652836957418671,-118.15350694827737,6.7292882587897872E-5,
        -0.0016098236165544761,-11.74314218041998,6.7316800382371969E-5,30.0,25.0,39.239045647359006,
        41.553331361644723,1.25,1.25,25.0,150.328,12.5,17.5,3.260954352640991,0.9466686383552787,1.25,1.25,17.5,
        76.652836957418671,-106.5101256850441,-0.0017851219951556655,-11.743158642519889,0.368955677450731,30.0,
        25.0,39.239045647359006,41.553331361644723,1.25,1.25,150.328,12.5,17.5,3.260954352640991,0.9466686383552787,
        1.25,1.25,17.5,76.652836957418671,-7.5937898402657913,-11.7709560028176,-0.00018077542171376562,
        -0.00014996056668787019,0.031769047906501834,25.0,39.239045647359006,41.553331361644723,1.25,1.25,12.5,17.5,
        3.260954352640991,0.9466686383552787,1.25,1.25,44.314868949193837,76.652836957418671,-8.4229193569742868,
        -0.00021926174033258425,-11.770944808710672,-0.00010902148921661218,30.0,25.0,39.239045647359006,
        41.553331361644723,1.25,1.25,12.5,17.5,3.260954352640991,0.9466686383552787,1.25,1.25,12.5,17.5,
        44.314868949193837,76.652836957418671,-118.1819973950968,-114.63004102821941,-0.0010889190560573953,
        -0.0011014109134511317,30.0,25.0,39.239045647359006,41.553331361644723,1.25,1.25,25.0,20.0,150.328,150.328,
        12.5,17.5,3.260954352640991,0.9466686383552787,1.25,1.25;
    Explicit_g_H: ARRAY [0..25259] OF LREAL := -0.077476528795167823,-0.0036970316053708055,-0.086721354914861964,
        -0.0037551531516151274,-0.088333425061435933,-0.0036263143516392839,0.077476528795167823,
        0.0036970316053708055,0.086721354914861964,0.0037551531516151274,0.088333425061435933,0.0036263143516392839,
        1.0,0.0,0.0,0.0,0.0,0.0,0.0,0.0,0.0,0.0,-1.0,-0.0,-0.0,-0.0,-0.0,-0.0,-0.0,-0.0,0.077476528795167809,
        -0.0037336016594598032,-0.096558209785564425,-0.0037971247337723361,-0.096261840305030433,
        -0.0036696470680512121,0.0037336016594598032,0.0037971247337723361,0.0036696470680512121,1.0,0.0,0.0,0.0,
        0.0,0.0,0.0,0.0,0.0,-1.0,-0.0,-0.0,-0.0,-0.0,-0.0,-0.0,-0.0,0.0036970316053708055,-0.0774751990947586,
        -0.086719240202544429,-0.0033360406615825823,-0.08833126085023621,-0.0029980663592998539,0.0774751990947586,
        0.086719240202544429,0.0883312608502362,1.0,0.0,0.0,0.0,0.0,0.0,0.0,0.0,0.0,-1.0,-0.0,-0.0,-0.0,-0.0,-0.0,
        -0.0,-0.0,0.086721354914861964,0.0037377448931881934,0.0036747051937017308,0.081735628272827751,
        -0.05352855586820774,-0.003738667688927728,-0.0038030215471528527,-0.0036758118677038785,
        0.0038030215471528527,1.0,0.0,0.0,0.0,0.0,0.0,0.0,0.0,0.0,-1.0,-0.0,-0.0,-0.0,-0.0,-0.0,-0.0,
        0.0037551531516151274,0.077474910522772944,0.088330866369964178,0.0040622390547605577,-0.077474853387268755,
        -0.0032595505975352855,-0.086718768354052969,-0.088330785510104329,1.0,0.0,0.0,0.0,0.0,0.0,0.0,0.0,0.0,-1.0,
        -0.0,-0.0,-0.0,-0.0,-0.0,-0.0,0.088333425061435933,-0.064270763159980787,-0.003730227048632441,
        -0.081735628272827862,-0.0037933258252242827,-0.0036658026975738616,0.003730227048632441,
        0.0037933258252242827,0.0036658026975738616,1.0,0.0,0.0,0.0,0.0,0.0,0.0,0.0,0.0,-1.0,-0.0,-0.0,-0.0,-0.0,
        -0.0,-0.0,0.0036263143516392839,-0.07747514736147483,-0.0035996316889970238,-0.086719240415959062,
        -0.0040622390547605594,-0.088331268656470549,0.07747514736147483,0.086719240415959062,0.088331268656470549,
        1.0,0.0,0.0,0.0,0.0,0.0,0.0,0.0,0.0,-1.0,-0.0,-0.0,-0.0,-0.0,-0.0,-0.0,-0.077476528795167809,
        -0.0037336016594598032,-0.0037971247337723361,-0.0036696470680512121,0.0037336016594598032,
        0.096558209785564425,0.0037971247337723361,0.096261840305030419,0.0036696470680512121,1.0,0.0,0.0,0.0,0.0,
        0.0,0.0,0.0,0.0,-1.0,-0.0,-0.0,-0.0,-0.0,-0.0,-0.0,-0.0,-0.0036970316053708055,-0.0774751990947586,
        -0.086719240202544429,-0.08833126085023621,0.0774751990947586,0.086719240202544429,0.0033360406615825823,
        0.0883312608502362,0.0029980663592998539,1.0,0.0,0.0,0.0,0.0,0.0,0.0,0.0,0.0,-1.0,-0.0,-0.0,-0.0,-0.0,-0.0,
        -0.0,-0.0,-0.086721354914861964,-0.081735628272827779,-0.003738667688927728,-0.0038030215471528527,
        -0.0036758118677038785,0.05352855586820774,0.003738667688927728,0.0036758118677038785,1.0,0.0,0.0,0.0,0.0,
        0.0,0.0,0.0,-1.0,-0.0,-0.0,-0.0,-0.0,-0.0,-0.0,-0.0,-0.0037551531516151274,-0.077474910522772944,
        -0.088330866369964192,-0.0040622390547605577,-0.086718768354052969,0.077474853387268755,
        0.0032595505975352855,0.086718768354052969,0.088330785510104315,1.0,0.0,0.0,0.0,0.0,0.0,0.0,0.0,-1.0,-0.0,
        -0.0,-0.0,-0.0,-0.0,-0.0,-0.0,-0.088333425061435933,-0.003730227048632441,-0.0037933258252242827,
        -0.0036658026975738616,0.064270763159980787,0.003730227048632441,0.081735628272827862,0.0037933258252242827,
        0.0036658026975738616,1.0,0.0,0.0,0.0,0.0,0.0,0.0,0.0,-1.0,-0.0,-0.0,-0.0,-0.0,-0.0,-0.0,-0.0,
        -0.0036263143516392839,-0.07747514736147483,-0.086719240415959062,-0.088331268656470549,0.07747514736147483,
        0.0035996316889970238,0.086719240415959062,0.0040622390547605594,0.088331268656470549,1.0,0.0,0.0,0.0,0.0,
        0.0,0.0,0.0,-1.0,-0.0,-0.0,-0.0,-0.0,-0.0,-0.0,-0.0,0.077475199094758584,0.0037336016594598036,
        -0.096555446100995979,-0.0033851653375543203,-0.096259405810541626,-0.003048048206429072,1.0,0.0,0.0,0.0,
        0.0,0.0,0.0,0.0,-1.0,-0.0,-0.0,-0.0,-0.0,-0.0,-0.0,-0.0,0.0965582097855644,0.053528555868207726,
        0.097144200416782928,-0.0037434082923276293,-0.0038084364001372724,-0.003681379431249545,
        0.0037434082923276293,0.0038084364001372724,0.003681379431249545,1.0,0.0,0.0,0.0,0.0,0.0,0.0,0.0,0.0,0.0,
        -1.0,-0.0,-0.0,-0.0,-0.0,-0.0,-0.0,0.07747491052277293,-0.0032828819692694222,-0.0020476052876290248,-0.0,
        0.053528511294535119,0.0038084364001372728,-0.00206233763359849,1.0,0.0,0.0,0.0,0.0,0.0,0.0,0.0,-1.0,-0.0,
        -0.0,-0.0,-0.0,-0.0,0.064270763159980773,0.096261840305030391,-0.003741367013872285,-0.097144200416783025,
        0.0036789408701099892,1.0,0.0,0.0,0.0,0.0,0.0,0.0,0.0,-1.0,-0.0,-0.0,-0.0,-0.0,-0.0,-0.0,
        0.077475147361474844,-0.0041002780928197317,-0.0,0.053528477903539248,0.0036813794312495437,1.0,0.0,0.0,0.0,
        0.0,0.0,0.0,0.0,0.0,-1.0,-0.0,-0.0,-0.0,-0.0,-0.0,0.077475199094758584,-0.0037336016594598036,-0.0,
        0.053525792212392634,-0.095362049810915089,0.0030604564304645169,1.0,0.0,0.0,0.0,0.0,0.0,0.0,0.0,-1.0,-0.0,
        -0.0,-0.0,-0.0,-0.0,-0.0,0.07747491052277293,-0.0037971247337723361,-0.096554979303422925,
        0.0032828819692694222,0.0020476052876290253,1.0,0.0,0.0,0.0,0.0,0.0,-1.0,-0.0,-0.0,-0.0,-0.0,-0.0,-0.0,
        0.077475147361474844,-0.0036696470680512121,-0.0965555005652539,-0.0962594506372809,0.0036284930825631052,
        0.0041002780928197317,1.0,0.0,0.0,0.0,0.0,0.0,0.0,-1.0,-0.0,-0.0,-0.0,-0.0,-0.0,-0.0,-0.0,
        0.0037377448931881943,0.0867186204896591,0.0032853953061778079,-0.053525720906035079,-0.095360309634866941,
        1.0,0.0,0.0,0.0,0.0,0.0,0.0,0.0,-1.0,-0.0,-0.0,-0.0,-0.0,-0.0,0.0032595408520208523,0.0033360406615825819,
        -0.077474779701193708,-0.086718620489659087,-0.088330631297803677,-0.0019964228655007152,
        0.077474779701193708,0.086718620489659087,0.088330631297803677,1.0,0.0,0.0,0.0,0.0,0.0,0.0,0.0,-1.0,-0.0,
        -0.0,-0.0,-0.0,-0.0,0.0037302270486324414,0.088331260850236182,-0.064270277646497315,-0.081733734629335822,
        -0.0033808752939656975,1.0,0.0,0.0,0.0,0.0,0.0,0.0,0.0,-1.0,-0.0,-0.0,-0.0,-0.0,-0.0,-0.0,
        0.0035996316889970238,0.0029980663592998548,-0.0883306802521518,0.077474806162417684,0.086718668191616846,
        0.088330680252151766,1.0,0.0,0.0,0.0,0.0,0.0,0.0,0.0,0.0,0.0,-1.0,-0.0,-0.0,-0.0,-0.0,-0.0,-0.0,
        0.0037336016594598028,-0.077475199094758612,-0.0033851653375543203,0.09655544610099602,0.096259405810541571,
        1.0,0.0,0.0,0.0,0.0,0.0,0.0,0.0,-1.0,-0.0,-0.0,-0.0,-0.0,-0.0,-0.0,-0.0,0.0037377448931881943,
        -0.086719240202544429,-0.0033909861531741582,0.053525792212392627,0.0953608011034519,1.0,0.0,0.0,0.0,0.0,
        0.0,0.0,-1.0,-0.0,-0.0,-0.0,-0.0,-0.0,-0.0,0.0037302270486324414,-0.088331260850236182,
        -0.0033808752939656975,-0.0030438513190736054,0.064270277646497315,0.08173373462933585,1.0,0.0,0.0,0.0,0.0,
        0.0,0.0,-1.0,-0.0,-0.0,-0.0,-0.0,-0.0,-0.0,-0.0,0.086718848216881667,0.0038019574628289773,
        0.081733362969809764,0.0041044771204881876,-0.053528496548426494,-0.0032859751799926063,1.0,0.0,0.0,0.0,0.0,
        0.0,0.0,0.0,-1.0,-0.0,-0.0,-0.0,-0.0,-0.0,0.086719240415959048,0.0036747051937017308,0.081733710919780447,
        -0.053528477903539262,-0.004105420208706986,1.0,0.0,0.0,0.0,0.0,0.0,0.0,0.0,-1.0,-0.0,-0.0,-0.0,-0.0,-0.0,
        0.086719240202544443,0.0030541120213779097,0.081733734629335753,-0.0037386676889277271,
        -0.053528602848912449,0.0033922419380553385,1.0,0.0,0.0,0.0,0.0,0.0,0.0,0.0,-1.0,-0.0,-0.0,-0.0,-0.0,-0.0,
        -0.0,0.081733362969809764,-0.0038030215471528536,-0.053528511294535126,0.0032859634458799053,
        0.0020558076887912374,1.0,0.0,0.0,0.0,0.0,-1.0,-0.0,-0.0,-0.0,-0.0,0.0037933258252242823,
        0.088330866369964178,0.0040966303107997674,-0.0032806030586776964,-0.081733288636505308,1.0,0.0,0.0,0.0,0.0,
        0.0,0.0,0.0,-1.0,-0.0,-0.0,-0.0,-0.0,-0.0,0.0037971247337723357,0.096258993277645352,0.0041002780928197291,
        -0.077474853387268755,-0.0032828934231975719,0.096554881960142766,1.0,0.0,0.0,0.0,0.0,0.0,0.0,0.0,-1.0,-0.0,
        -0.0,-0.0,-0.0,-0.0,-0.0,0.0038019574628289751,0.0041044771204881867,-0.086718768354052969,
        -0.0032853953061778097,0.05352568587932538,0.095360481095178293,1.0,0.0,0.0,0.0,0.0,-0.0,-0.0,-0.0,-0.0,
        -0.0,0.0037933258252242823,0.0642701047402686,0.081733362969809792,0.0040966303107997674,
        -0.088330785510104287,-0.0032806030586776951,1.0,0.0,0.0,0.0,0.0,0.0,0.0,-1.0,-0.0,-0.0,-0.0,-0.0,-0.0,-0.0,
        0.088331268656470577,0.0036658026975738608,-0.0817337109197805,-0.00409663031079977,1.0,0.0,0.0,0.0,0.0,0.0,
        0.0,0.0,-1.0,-0.0,-0.0,-0.0,-0.0,-0.0,0.08833126085023621,-0.003730227048632441,-0.081733734629335864,
        0.0033808752939656983,0.003043851319073605,1.0,0.0,0.0,0.0,0.0,0.0,0.0,0.0,-1.0,-0.0,-0.0,-0.0,-0.0,-0.0,
        -0.0,0.088330866369964192,-0.0037933258252242827,-0.081733362969809792,0.0032805917192938643,
        0.0020436855192036149,1.0,0.0,0.0,0.0,0.0,-1.0,-0.0,-0.0,-0.0,-0.0,0.088331268656470577,
        -0.0036658026975738608,-0.0642701751144813,-0.0817337109197805,0.0036256899023540735,0.00409663031079977,
        1.0,0.0,0.0,0.0,0.0,0.0,0.0,-1.0,-0.0,-0.0,-0.0,-0.0,-0.0,-0.0,0.0036696470680512121,-0.077475147361474844,
        -0.0041002780928197325,0.096555500565253888,0.096259450637280822,1.0,0.0,0.0,0.0,0.0,0.0,0.0,0.0,-1.0,-0.0,
        -0.0,-0.0,-0.0,-0.0,-0.0,0.00367470519370173,-0.086719240415959062,-0.00410447712048819,
        0.053525667262608191,0.095360820958319881,1.0,0.0,0.0,0.0,0.0,-0.0,-0.0,-0.0,-0.0,-0.0,
        0.0036658026975738612,-0.088331268656470549,-0.0040966303107997691,0.0642701751144813,0.081733710919780544,
        1.0,0.0,0.0,0.0,0.0,0.0,0.0,-1.0,-0.0,-0.0,-0.0,-0.0,-0.0,-0.0,-0.077475199094758584,-0.0037336016594598036,
        0.096555446100995979,0.0033851653375543203,0.096259405810541585,0.0030480482064290729,1.0,0.0,0.0,0.0,0.0,
        0.0,0.0,0.0,-1.0,-0.0,-0.0,-0.0,-0.0,-0.0,-0.0,-0.0,-0.053525745363213646,-0.0965582097855644,
        -0.0037424848355660516,0.0953635804275615,0.0036802719765434704,1.0,0.0,0.0,0.0,0.0,0.0,0.0,-1.0,-0.0,-0.0,
        -0.0,-0.0,-0.0,-0.0,-0.0,-0.07747491052277293,-0.0037971247337723361,0.0032828819692694222,
        0.096554979303422925,0.09625899327764538,0.0020476052876290253,1.0,0.0,0.0,0.0,0.0,-1.0,-0.0,-0.0,-0.0,-0.0,
        -0.0,-0.064270763159980773,-0.096261840305030377,-0.053528555868207733,-0.0953635804275615,
        -0.0037434082923276293,-0.0038084364001372724,-0.003681379431249545,0.0037434082923276293,
        0.003681379431249545,1.0,0.0,0.0,0.0,0.0,0.0,0.0,0.0,-1.0,-0.0,-0.0,-0.0,-0.0,-0.0,-0.0,-0.0,-0.0,
        -0.077475147361474844,-0.0036696470680512121,0.0036284930825631052,0.0965555005652539,0.0041002780928197317,
        0.096259450637280863,1.0,0.0,0.0,0.0,0.0,0.0,0.0,-1.0,-0.0,-0.0,-0.0,-0.0,-0.0,-0.0,-0.0,
        -0.0037377448931881943,-0.086719240202544429,0.053525792212392627,0.0033909861531741582,0.0953608011034519,
        0.0030541120213779067,1.0,0.0,0.0,0.0,0.0,-0.0,-0.0,-0.0,-0.0,-0.0,-0.0,-0.0032595408520208523,
        -0.0033360406615825823,-0.077474779701193708,-0.086718620489659087,-0.088330631297803677,
        0.077474779701193708,0.086718620489659087,0.088330631297803677,0.0019964228655007152,1.0,0.0,0.0,0.0,0.0,
        0.0,-1.0,-0.0,-0.0,-0.0,-0.0,-0.0,-0.0,-0.0,-0.0037302270486324414,-0.088331260850236182,
        0.064270277646497315,0.08173373462933585,0.0033808752939656975,0.0030438513190736054,1.0,0.0,0.0,0.0,0.0,
        0.0,0.0,-1.0,-0.0,-0.0,-0.0,-0.0,-0.0,-0.0,-0.0,-0.0035996316889970238,-0.0029980663592998548,
        -0.0883306802521518,0.077474806162417684,0.0040161961339407514,1.0,0.0,0.0,0.0,0.0,0.0,0.0,-1.0,-0.0,-0.0,
        -0.0,-0.0,-0.0,-0.0,-0.086718848216881667,-0.0038019574628289773,0.053525700631027615,0.00328538361939746,
        0.095360537347830912,0.0020543895893986456,1.0,0.0,0.0,0.0,-0.0,-0.0,-0.0,-0.0,-0.086719240415959048,
        -0.081733710919780475,-0.0036758118677038781,0.053528477903539269,0.0036323443884875278,
        0.004105420208706986,1.0,0.0,0.0,0.0,0.0,0.0,-1.0,-0.0,-0.0,-0.0,-0.0,-0.0,-0.0,-0.0,-0.0037933258252242823,
        -0.088330866369964178,0.0642701047402686,0.0032805917192938643,0.081733362969809834,0.002043685519203618,
        1.0,0.0,0.0,0.0,0.0,0.0,-1.0,-0.0,-0.0,-0.0,-0.0,-0.0,-0.0,-0.088331268656470577,-0.0036658026975738608,
        0.0642701751144813,0.0036256899023540735,0.081733710919780531,0.00409663031079977,1.0,0.0,0.0,0.0,0.0,0.0,
        -1.0,-0.0,-0.0,-0.0,-0.0,-0.0,-0.0,-0.0,0.096554668429779264,0.053528546349668679,0.0032890369305916766,
        2.246257328490169E-5,-0.0020636698815925556,1.0,0.0,0.0,0.0,0.0,0.0,0.0,0.0,0.0,-1.0,-0.0,-0.0,-0.0,-0.0,
        -0.0,0.077474779701193708,0.0032828819692694209,0.00338516533755432,-0.096554668429779222,
        -0.00204893865289483,1.0,0.0,0.0,0.0,0.0,0.0,-0.0,-0.0,-0.0,-0.0,-0.0,-0.0,0.0642702776464973,
        0.09625940581054164,0.053528602848912407,0.0037434082923276288,-0.0033985247108398306,1.0,0.0,0.0,0.0,0.0,
        0.0,0.0,0.0,0.0,-1.0,-0.0,-0.0,-0.0,-0.0,-0.0,-0.0,0.077474853387268741,-0.0032828934231975719,-0.0,
        0.0020609185794669728,0.053528496548426514,3.744179842189145E-5,4.5922831299071462E-6,1.0,0.0,0.0,0.0,0.0,
        0.0,0.0,0.0,0.0,-1.0,-0.0,-0.0,-0.0,-0.0,-0.0,0.064270175114481284,0.0962594506372809,0.053528477903539248,
        0.095362069702500829,-0.0036813794312495437,0.0036361307619490525,0.0041103880254833337,1.0,0.0,0.0,0.0,0.0,
        0.0,0.0,0.0,-1.0,-0.0,-0.0,-0.0,-0.0,-0.0,-0.0,0.077474779701193708,-0.0032828819692694209,
        -0.00338516533755432,-0.096554668429779222,0.00204893865289483,1.0,0.0,0.0,0.0,0.0,0.0,-1.0,-0.0,-0.0,-0.0,
        -0.0,-0.0,-0.0,-0.0,0.077474853387268741,-0.0041002780928197308,-0.096554881960142849,-0.096258906749754139,
        0.0032828934231975719,1.0,0.0,0.0,0.0,0.0,0.0,0.0,-1.0,-0.0,-0.0,-0.0,-0.0,-0.0,-0.0,-0.0,
        0.0037386676889277271,0.081733734629335822,0.095360801103452145,-0.053528602848912435,
        -0.0033922419380553364,1.0,0.0,0.0,0.0,0.0,0.0,0.0,0.0,-1.0,-0.0,-0.0,-0.0,-0.0,-0.0,-0.0,
        0.0033808752939656983,0.088330631297803663,0.0032806030586776951,-0.081733090816521414,1.0,0.0,0.0,0.0,0.0,
        0.0,0.0,0.0,0.0,-1.0,-0.0,-0.0,-0.0,-0.0,-0.0,0.0032595505975352851,4.4466772864598856E-6,
        -0.077474722496114493,-0.086718540525974191,-0.088330550333579838,0.077474722496114493,0.086718540525974191,
        0.088330550333579824,1.0,0.0,0.0,0.0,0.0,0.0,0.0,0.0,0.0,0.0,-1.0,-0.0,-0.0,-0.0,-0.0,-0.0,-0.0,
        0.0033851653375543207,0.09625871958337659,0.0032828934231975706,-0.077474722496114493,0.096554570952769647,
        1.0,0.0,0.0,0.0,0.0,0.0,0.0,0.0,0.0,-1.0,-0.0,-0.0,-0.0,-0.0,-0.0,-0.0,0.0033909861531741603,
        0.0032853953061778083,-0.086718540525974178,0.053525720906035079,0.095360309634866927,1.0,0.0,0.0,0.0,0.0,
        0.0,-0.0,-0.0,-0.0,-0.0,-0.0,0.0032805917192938643,0.0033808752939656983,-0.088330631297803663,
        -0.0020450187866071388,0.064270077055509661,0.0817331652386774,1.0,0.0,0.0,0.0,0.0,0.0,0.0,-1.0,-0.0,-0.0,
        -0.0,-0.0,-0.0,0.0032806030586776946,4.5551341567806142E-6,-0.00070573613781555692,0.064270045132796841,
        0.081733090816521484,1.0,0.0,0.0,0.0,0.0,0.0,0.0,0.0,-1.0,-0.0,-0.0,-0.0,-0.0,-0.0,-0.0,
        0.0037424848355660512,-0.053525792212392669,-0.096555446100995992,0.09536204981091484,1.0,0.0,0.0,0.0,0.0,
        0.0,0.0,-1.0,-0.0,-0.0,-0.0,-0.0,-0.0,-0.0,-0.0,0.0037413670138722855,0.0032877566122254086,
        -0.064270077055509675,-0.09625871958337652,-0.0020606458502567715,0.097139764931133091,0.0,0.0,0.0,0.0,0.0,
        0.0,-1.0,-0.0,-0.0,-0.0,-0.0,-0.0,-0.0,0.0037386676889277271,-0.081733734629335836,-0.0033922419380553364,
        -0.0030554087647135957,0.053528602848912435,1.0,0.0,0.0,0.0,0.0,0.0,0.0,-1.0,-0.0,-0.0,-0.0,-0.0,-0.0,-0.0,
        -0.0,0.081733710919780447,0.095360820958320186,-0.0036758118677038781,-0.053528477903539262,
        0.0036323443884875278,0.004105420208706986,1.0,0.0,0.0,0.0,0.0,0.0,0.0,-1.0,-0.0,-0.0,-0.0,-0.0,-0.0,-0.0,
        0.081733165238677352,-0.003285963445879904,-0.00339224193805534,-0.053528546349668707,0.0020571402226554035,
        1.0,0.0,0.0,0.0,0.0,-0.0,-0.0,-0.0,-0.0,-0.0,-0.0,0.086718768354052955,0.081733288636505308,
        -0.0041054202087069886,-0.05352849654842648,0.0032859751799926037,1.0,0.0,0.0,0.0,0.0,0.0,0.0,-1.0,-0.0,
        -0.0,-0.0,-0.0,-0.0,-0.0,0.0038060814101328554,-0.0642701047402686,-0.096258993277645352,
        -0.00328775661222541,-0.0020593133828706875,0.097140154750072039,0.0,0.0,0.0,0.0,0.0,-1.0,-0.0,-0.0,-0.0,
        -0.0,-0.0,-0.0,0.0038030215471528527,0.004105420208706986,-0.081733288636505336,-0.0032859751799926059,
        0.0535284965484265,1.0,0.0,0.0,0.0,0.0,0.0,0.0,-1.0,-0.0,-0.0,-0.0,-0.0,-0.0,-0.0,0.088330631297803663,
        -0.0032805917192938639,-0.0033808752939656979,-0.081733165238677324,0.0020450187866071436,1.0,0.0,0.0,0.0,
        0.0,-0.0,-0.0,-0.0,-0.0,-0.0,-0.0,-0.0036256899023540726,-0.003043851319073605,-0.081733207269128971,
        0.00070573613781555681,-0.0032806030586776946,-0.064270045132796827,1.0,0.0,0.0,0.0,0.0,0.0,0.0,-1.0,-0.0,
        -0.0,-0.0,-0.0,-0.0,-0.0,-0.0,0.088330785510104329,-0.0040966303107997639,-0.064270072853593943,
        -0.081733288636505252,0.0032806030586776968,1.0,0.0,0.0,0.0,0.0,0.0,0.0,-1.0,-0.0,-0.0,-0.0,-0.0,-0.0,-0.0,
        0.0036789408701099883,-0.064270175114481312,-0.096259450637280849,-0.00410827263902433,0.09714081282206144,
        1.0,0.0,0.0,0.0,0.0,0.0,0.0,-1.0,-0.0,-0.0,-0.0,-0.0,-0.0,-0.0,0.0036758118677038777,-0.081733710919780544,
        -0.0041054202087069868,0.053528477903539234,1.0,0.0,0.0,0.0,0.0,0.0,0.0,-1.0,-0.0,-0.0,-0.0,-0.0,-0.0,-0.0,
        -0.0642702776464973,-0.0037413670138722855,-0.096259405810541585,-0.053528602848912407,
        0.0033985247108398306,0.0030617540729862567,1.0,0.0,0.0,0.0,0.0,0.0,0.0,-1.0,-0.0,-0.0,-0.0,-0.0,-0.0,-0.0,
        -0.0,-0.0,-0.07747480616241767,-0.0036284930825631048,-0.003048048206429072,0.096554733505586993,
        0.0040635927394609929,0.0962587757779151,1.0,0.0,0.0,0.0,0.0,0.0,-1.0,-0.0,-0.0,-0.0,-0.0,-0.0,-0.0,-0.0,
        -0.0965555005652539,-0.053528477903539248,-0.097140812822061412,-0.0036813794312495437,
        0.0041103880254833337,1.0,0.0,0.0,0.0,0.0,0.0,-1.0,-0.0,-0.0,-0.0,-0.0,-0.0,-0.0,-0.0,-0.0,
        -0.064270104740268577,-0.0038060814101328558,-0.09625899327764538,0.0032877566122254103,
        0.097140154750072039,0.00205931338287069,0.0,0.0,0.0,0.0,-1.0,-0.0,-0.0,-0.0,-0.0,-0.0,
        -0.077474853387268741,-0.0041002780928197308,0.0032828934231975719,0.096554881960142849,
        0.096258906749754111,1.0,0.0,0.0,0.0,0.0,0.0,0.0,-1.0,-0.0,-0.0,-0.0,-0.0,-0.0,-0.0,-0.0,
        -0.064270175114481284,-0.096259450637280863,-0.0036789408701099887,0.0036345377179377619,
        0.097140812822061551,0.0041082726390243261,0.0,0.0,0.0,0.0,0.0,-1.0,-0.0,-0.0,-0.0,-0.0,-0.0,-0.0,
        -0.0037386676889277271,-0.081733734629335836,0.053528602848912435,0.0033922419380553364,
        0.0030554087647135957,1.0,0.0,0.0,0.0,0.0,0.0,0.0,-1.0,-0.0,-0.0,-0.0,-0.0,-0.0,-0.0,-0.0,
        -0.0036316281145198134,-0.08671866819161686,-0.0030541120213779089,0.053525725625599235,
        0.0040689244198050265,0.09536039894190243,1.0,0.0,0.0,0.0,-0.0,-0.0,-0.0,-0.0,-0.0,-0.0,
        -0.0032595505975352851,-1.760341479960766E-5,-0.077474722496114493,-0.086718540525974191,
        -0.088330550333579838,0.077474722496114493,0.086718540525974191,0.088330550333579824,1.0,0.0,0.0,0.0,0.0,
        0.0,0.0,0.0,-1.0,-0.0,-0.0,-0.0,-0.0,-0.0,-0.0,-0.0,-0.0,-0.081733362969809778,-0.0038030215471528519,
        0.053528511294535126,0.0032859634458799083,0.0020558076887912538,1.0,0.0,0.0,0.0,0.0,0.0,-1.0,-0.0,-0.0,
        -0.0,-0.0,-0.0,-0.0,-0.086718768354052955,-0.0041044771204881876,0.053525685879325394,0.0032853953061778105,
        0.095360481095178265,1.0,0.0,0.0,0.0,0.0,0.0,-1.0,-0.0,-0.0,-0.0,-0.0,-0.0,-0.0,-0.0040966303107997674,
        -0.0883307855101043,0.064270072853593943,0.0032806030586776964,0.0817332886365053,1.0,0.0,0.0,0.0,0.0,0.0,
        -1.0,-0.0,-0.0,-0.0,-0.0,-0.0,-0.0,-0.0,0.077474722496114479,0.0032828934231975714,0.0020489386528948252,
        -0.096554570952769689,1.0,0.0,0.0,0.0,0.0,0.0,0.0,0.0,0.0,-1.0,-0.0,-0.0,-0.0,-0.0,-0.0,-0.0,
        0.053528602848912407,0.00021174728611677174,-0.0037434082923276288,0.0033985247108398306,
        0.0030617540729862567,1.0,0.0,0.0,0.0,0.0,0.0,0.0,0.0,0.0,-1.0,-0.0,-0.0,-0.0,-0.0,-0.0,-0.0,
        0.053528511294535105,0.095361785907785684,-0.0038084364001372728,0.0032890369305916753,0.00206233763359849,
        1.0,0.0,0.0,0.0,0.0,0.0,-1.0,-0.0,-0.0,-0.0,-0.0,0.096554668429779236,-0.0033972680454078283,
        0.053528546349668686,-0.0032890369305916753,-2.24625732849017E-5,0.0020636698815925587,1.0,0.0,0.0,0.0,0.0,
        -0.0,-0.0,-0.0,-0.0,-0.0,-0.0,0.064270072853593929,0.096258906749754153,-0.0041082726390243279,
        0.053528496548426514,-3.744179842189147E-5,0.0032890488730985008,1.0,0.0,0.0,0.0,0.0,0.0,0.0,0.0,-1.0,-0.0,
        -0.0,-0.0,-0.0,-0.0,-0.0,0.077474722496114479,-0.0032828934231975714,-0.0040635927394609929,
        -0.096554570952769689,-0.096258632930764434,1.0,0.0,0.0,0.0,0.0,0.0,0.0,-1.0,-0.0,-0.0,-0.0,-0.0,-0.0,-0.0,
        -0.0,-0.0,0.05352568587932538,0.096554881960142822,-0.0041094442537653805,-0.095361729623989588,
        0.00328846857351035,1.0,0.0,0.0,0.0,0.0,0.0,0.0,-1.0,-0.0,-0.0,-0.0,-0.0,-0.0,0.081733165238677366,
        0.0033922419380553381,0.095360365986835671,0.0032859751799926059,0.00021167614407259223,
        -0.053528531588205183,1.0,0.0,0.0,0.0,0.0,0.0,0.0,0.0,0.0,-1.0,-0.0,-0.0,-0.0,-0.0,-0.0,
        0.0032859634458799053,0.0033922419380553377,-0.08173316523867738,-0.0020571402226554139,
        0.053528546349668693,1.0,0.0,0.0,0.0,0.0,0.0,0.0,-1.0,-0.0,-0.0,-0.0,-0.0,-0.0,4.5967813251915519E-6,0.0,
        -0.0,0.0032890369305916766,-0.053528546349668714,-0.00042383855226207613,1.0,0.0,0.0,0.0,0.0,0.0,0.0,-1.0,
        -0.0,-0.0,-0.0,-0.0,-0.0,-0.0,0.0032859751799926059,4.5821970609936686E-6,-0.00074189152974182631,
        0.053528531588205169,1.0,0.0,0.0,0.0,0.0,0.0,0.0,0.0,-1.0,-0.0,-0.0,-0.0,-0.0,-0.0,-0.0,
        0.0037434082923276288,-0.053528602848912442,-0.00042383659715075443,-0.003398524710839831,
        -0.0030617540729862567,1.0,0.0,0.0,0.0,0.0,0.0,0.0,-1.0,-0.0,-0.0,-0.0,-0.0,-0.0,-0.0,-0.0,-0.0,
        -0.0036323443884875265,-0.0030554087647135957,-0.053528536300004093,0.000741891529741826,
        -0.0032859751799926042,1.0,0.0,0.0,0.0,0.0,0.0,0.0,-1.0,-0.0,-0.0,-0.0,-0.0,-0.0,-0.0,-0.0,
        0.00205931338287068,-0.064270072853593971,-0.096258906749754083,-0.0032877684548394651,3.74417984218915E-5,
        4.5922831299071115E-6,-0.053528496548426528,1.0,0.0,0.0,0.0,0.0,0.0,0.0,-1.0,-0.0,-0.0,-0.0,-0.0,-0.0,-0.0,
        -0.0,0.0038084364001372728,-0.053528511294535154,-0.097140154750072011,-0.0032890369305916744,
        -0.0020623376335984836,1.0,0.0,0.0,0.0,0.0,0.0,-1.0,-0.0,-0.0,-0.0,-0.0,-0.0,-0.0,-0.0,
        0.0036813794312495446,-0.053528477903539283,-0.097140812822061384,-0.0041103880254833337,1.0,0.0,0.0,0.0,
        0.0,0.0,0.0,-1.0,-0.0,-0.0,-0.0,-0.0,-0.0,-0.0,-0.0,-0.064270080950603922,-0.0036345377179377619,
        -0.096258775777915084,-0.0030589105208496891,0.09713984949811369,0.0040735945200531861,0.0,0.0,0.0,0.0,-1.0,
        -0.0,-0.0,-0.0,-0.0,-0.0,-0.0,-0.0,-0.077474722496114479,-0.0032828934231975714,-0.0040635927394609929,
        0.096554570952769689,0.096258632930764421,1.0,0.0,0.0,0.0,0.0,0.0,0.0,-1.0,-0.0,-0.0,-0.0,-0.0,-0.0,-0.0,
        -0.0,-0.0,-0.0038084364001372728,-0.0,-0.05352568587932538,-0.096554881960142822,-0.0041094442537653805,
        0.00328846857351035,1.0,0.0,0.0,0.0,0.0,0.0,-1.0,-0.0,-0.0,-0.0,-0.0,-0.0,-0.0,-0.0,-0.064270072853593929,
        -0.0041082726390243279,-0.096258906749754125,0.0032877684548394646,0.0971400347070677,0.0,0.0,0.0,0.0,0.0,
        -1.0,-0.0,-0.0,-0.0,-0.0,-0.0,-0.0,-0.0867185405259742,-0.0032859751799926059,-0.00074189152974182642,
        -4.5821970609936661E-6,0.053528531588205183,1.0,0.0,0.0,0.0,0.0,0.0,-1.0,-0.0,-0.0,-0.0,-0.0,-0.0,-0.0,-0.0,
        -0.0,-0.0032806030586776951,-1.7792453231023226E-5,-0.00070573613781555692,0.064270045132796827,
        0.081733090816521414,1.0,0.0,0.0,0.0,0.0,0.0,-1.0,-0.0,-0.0,-0.0,-0.0,-0.0,-0.0,-0.0,-0.0,
        -0.081733288636505322,-0.0041054202087069877,-0.095360481095178154,-0.0020558076887912404,
        0.05352849654842648,0.0032859751799926063,1.0,0.0,0.0,0.0,0.0,0.0,-1.0,-0.0,-0.0,-0.0,-0.0,-0.0,-0.0,-0.0,
        0.053525720906035051,0.0032884685735103504,0.00063548544762325539,4.5936164882535738E-6,
        -0.095361558052087569,1.0,0.0,0.0,0.0,0.0,0.0,0.0,0.0,0.0,-1.0,-0.0,-0.0,-0.0,-0.0,-0.0,
        0.053528536300004093,-1.3526542371728022E-5,0.0040762541459071506,1.0,0.0,0.0,0.0,0.0,0.0,0.0,0.0,0.0,-1.0,
        -0.0,-0.0,-0.0,-0.0,-0.0,-0.0,0.053525720906035038,-1.786284616987506E-5,0.0004238386986740823,
        -0.0032890488730985008,-1.786801097252406E-5,1.0,0.0,0.0,0.0,0.0,0.0,0.0,0.0,-1.0,-0.0,-0.0,-0.0,-0.0,-0.0,
        -0.0,-0.0,0.064270045132796813,0.00042356774118783937,-0.0032877684548394642,-0.097139644735603992,1.0,0.0,
        0.0,0.0,0.0,0.0,0.0,-1.0,-0.0,-0.0,-0.0,-0.0,-0.0,-0.0,-0.0,-0.064270045132796827,-0.0032877684548394655,
        -1.7856294754925308E-5,-0.0004235677411878392,0.097139644735603867,0.0,0.0,0.0,0.0,0.0,-1.0,-0.0,-0.0,-0.0,
        -0.0,-0.0,-0.0,-0.0,-0.053525720906035051,-0.00063548544762325539,-0.0032890488730985016,
        -4.5967813251915774E-6,1.0,0.0,0.0,0.0,0.0,0.0,-1.0,-0.0,-0.0,-0.0,-0.0,-0.0,-0.0,-0.0,-0.0,-0.0,
        0.053528531588205142,0.0032890488730985016,0.00021174823744038085,4.5967813251915774E-6,1.0,0.0,0.0,0.0,0.0,
        0.0,0.0,0.0,0.0,0.0,-1.0,-0.0,-0.0,-0.0,-0.0,-0.0,-0.0066911055783920089,-0.07890051805766235,
        -0.0068363474510417148,-0.088265396281155942,-0.0066161395077661729,-0.089903879918856469,
        0.0066911055783920089,0.07890051805766235,0.0068363474510417148,0.088265396281155942,0.0066161395077661712,
        0.089903879918856455,0.0,1.0,0.0,0.0,0.0,0.0,0.0,0.0,0.0,0.0,-0.0,-1.0,-0.0,-0.0,-0.0,-0.0,-0.0,-0.0,
        0.006691105578392008,-0.078900559120748739,-0.006163079957235881,-0.088264669807283563,
        -0.0055621477032858748,-0.089903034703890675,0.078900559120748739,0.088264669807283563,0.089903034703890661,
        0.0,1.0,0.0,0.0,0.0,0.0,0.0,0.0,0.0,-0.0,-1.0,-0.0,-0.0,-0.0,-0.0,-0.0,-0.0,0.07890051805766235,
        -0.0067284644196904985,-0.006877704736632846,-0.098249906447994834,-0.0066579212217880539,
        -0.097975501728056191,0.0067284644196904985,0.006877704736632846,0.0066579212217880513,0.0,1.0,0.0,0.0,0.0,
        0.0,0.0,0.0,0.0,-0.0,-1.0,-0.0,-0.0,-0.0,-0.0,-0.0,-0.0,0.0068363474510417157,0.078900439184654059,
        0.0899028560363271,0.0073567864102199376,-0.0058246010853626861,-0.078900422955217944,-0.088264467351155715,
        -0.0899028234772885,0.088264467351155715,0.0,1.0,0.0,0.0,0.0,0.0,0.0,0.0,0.0,-0.0,-1.0,-0.0,-0.0,-0.0,-0.0,
        -0.0,0.088265396281155942,0.0067342482080704246,0.0066644827548763986,0.0832050411250591,
        -0.0067354608622506237,-0.054584413035237804,-0.0068855488483819168,-0.0066658657231402118,0.0,1.0,0.0,0.0,
        0.0,0.0,0.0,0.0,0.0,-0.0,-1.0,-0.0,-0.0,-0.0,-0.0,-0.0,0.006616139507766172,-0.0064653841410221794,
        -0.078900403556479828,-0.0073567864102199419,-0.088264630109820233,-0.089903014806282017,
        0.078900403556479828,0.088264630109820233,0.089903014806282,0.0,1.0,0.0,0.0,0.0,0.0,0.0,0.0,0.0,-0.0,-1.0,
        -0.0,-0.0,-0.0,-0.0,-0.0,0.089903879918856469,-0.0067270634377785653,-0.065500982446408618,
        -0.0068762774998331775,-0.083205041125059123,-0.006656512283104341,0.0067270634377785653,
        0.0068762774998331775,0.0066565122831043393,0.0,1.0,0.0,0.0,0.0,0.0,0.0,0.0,0.0,-0.0,-1.0,-0.0,-0.0,-0.0,
        -0.0,-0.0,-0.006691105578392008,-0.078900559120748739,-0.088264669807283563,-0.089903034703890675,
        0.078900559120748739,0.006163079957235881,0.088264669807283563,0.0055621477032858687,0.089903034703890661,
        0.0,1.0,0.0,0.0,0.0,0.0,0.0,0.0,0.0,-0.0,-1.0,-0.0,-0.0,-0.0,-0.0,-0.0,-0.0,-0.07890051805766235,
        -0.0067284644196904985,-0.006877704736632846,-0.0066579212217880539,0.0067284644196904985,
        0.006877704736632846,0.098249906447994834,0.0066579212217880513,0.097975501728056164,0.0,1.0,0.0,0.0,0.0,
        0.0,0.0,0.0,0.0,-0.0,-1.0,-0.0,-0.0,-0.0,-0.0,-0.0,-0.0,-0.0068363474510417157,-0.0073567864102199428,
        -0.078900422955217944,-0.088264467351155715,-0.0899028234772885,0.0058246010853626852,0.078900422955217944,
        0.089902823477288479,0.0,1.0,0.0,0.0,0.0,0.0,0.0,0.0,-0.0,-1.0,-0.0,-0.0,-0.0,-0.0,-0.0,-0.0,
        -0.088265396281155942,-0.0067342482080704246,-0.0066644827548764012,-0.083205041125059123,
        -0.0068855488483819168,0.0067354608622506237,0.054584413035237783,0.0068855488483819168,0.00666586572314021,
        0.0,1.0,0.0,0.0,0.0,0.0,0.0,0.0,-0.0,-1.0,-0.0,-0.0,-0.0,-0.0,-0.0,-0.0,-0.0066161395077661712,
        -0.078900403556479828,-0.088264630109820233,-0.089903014806282017,0.0064653841410221794,
        0.078900403556479828,0.0073567864102199454,0.088264630109820233,0.089903014806282,0.0,1.0,0.0,0.0,0.0,0.0,
        0.0,0.0,-0.0,-1.0,-0.0,-0.0,-0.0,-0.0,-0.0,-0.0,-0.089903879918856455,-0.0067270634377785653,
        -0.0068762774998331775,-0.006656512283104341,0.0067270634377785653,0.065500982446408618,
        0.0068762774998331775,0.083205041125059165,0.0066565122831043393,0.0,1.0,0.0,0.0,0.0,0.0,0.0,0.0,-0.0,-1.0,
        -0.0,-0.0,-0.0,-0.0,-0.0,-0.0,0.0067284644196904976,0.078900559120748739,-0.0062082033463722475,
        -0.098248210795103,-0.0056064437356273134,-0.097973967439853871,0.0,1.0,0.0,0.0,0.0,0.0,0.0,0.0,-0.0,-1.0,
        -0.0,-0.0,-0.0,-0.0,-0.0,-0.0,0.0061630799572358827,0.0058246010853626835,0.0073727576513090464,
        -0.078900469896698883,-0.08826440165511483,-0.089902739686908359,0.078900469896698883,0.08826440165511483,
        0.089902739686908345,0.0,1.0,0.0,0.0,0.0,0.0,0.0,0.0,0.0,0.0,-0.0,-1.0,-0.0,-0.0,-0.0,-0.0,-0.0,
        0.0067342482080704228,-0.054582503993362751,-0.0971529032726468,-0.0,0.0058552526337344261,
        0.08826440165511483,-0.09715259031372557,0.0,1.0,0.0,0.0,0.0,0.0,0.0,0.0,-0.0,-1.0,-0.0,-0.0,-0.0,-0.0,
        0.0064653841410221785,0.005562147703285873,-0.078900477182149778,-0.0073727576513090464,
        0.089902794278946513,0.0,1.0,0.0,0.0,0.0,0.0,0.0,0.0,-0.0,-1.0,-0.0,-0.0,-0.0,-0.0,-0.0,
        0.0067270634377785653,-0.083204667535680926,-0.0,0.005850041999444641,0.089902739686908359,0.0,1.0,0.0,0.0,
        0.0,0.0,0.0,0.0,0.0,-0.0,-1.0,-0.0,-0.0,-0.0,-0.0,0.0067284644196904976,-0.078900559120748739,-0.0,
        0.00585124190111772,-0.00382410479030098,0.097973566528557168,0.0,1.0,0.0,0.0,0.0,0.0,0.0,0.0,-0.0,-1.0,
        -0.0,-0.0,-0.0,-0.0,-0.0,0.0067342482080704228,-0.088264669807283549,-0.0062154506546600041,
        0.054582503993362751,0.09715290327264671,0.0,1.0,0.0,0.0,0.0,0.0,-0.0,-1.0,-0.0,-0.0,-0.0,-0.0,-0.0,
        0.0067270634377785653,-0.089903034703890661,-0.00620691946854217,-0.0056052081304373879,0.0655016932872773,
        0.083204667535680968,0.0,1.0,0.0,0.0,0.0,0.0,0.0,-0.0,-1.0,-0.0,-0.0,-0.0,-0.0,-0.0,-0.0,
        0.078900439184654059,0.0068889490139224735,0.054585368753362618,-0.00585919104027798,-0.00383471710458173,
        0.0,1.0,0.0,0.0,0.0,0.0,0.0,0.0,-0.0,-1.0,-0.0,-0.0,-0.0,-0.0,0.054581513793381407,0.098249906447994875,
        -0.0067385738200007195,-0.0068889490139224727,-0.0066692894645364867,-0.09715507100044829,
        0.0067385738200007195,0.0068889490139224727,0.0066692894645364849,0.0,1.0,0.0,0.0,0.0,0.0,0.0,0.0,-0.0,-1.0,
        -0.0,-0.0,-0.0,-0.0,0.078900403556479842,0.006657921221788053,-0.0064971260842139906,-0.0073966778428481593,
        -0.0982483356597771,0.0,1.0,0.0,0.0,0.0,0.0,0.0,0.0,-0.0,-1.0,-0.0,-0.0,-0.0,-0.0,-0.0,0.065500982446408632,
        0.097975501728056191,-0.0066682627334341913,0.0067376264600041268,0.0068879216085573286,
        0.0066682627334341887,0.0,1.0,0.0,0.0,0.0,0.0,0.0,0.0,0.0,0.0,-0.0,-1.0,-0.0,-0.0,-0.0,-0.0,-0.0,
        0.078900559120748726,-0.0067284644196904993,-0.098248210795103041,0.0062082033463722467,
        0.0056064437356273065,0.0,1.0,0.0,0.0,0.0,0.0,0.0,0.0,-0.0,-1.0,-0.0,-0.0,-0.0,-0.0,-0.0,-0.0,
        0.078900439184654059,-0.0068777047366328451,-0.098247986163974121,0.0058512419011177222,
        0.0038218069458475176,0.0,1.0,0.0,0.0,0.0,0.0,0.0,-0.0,-1.0,-0.0,-0.0,-0.0,-0.0,-0.0,0.078900403556479842,
        -0.0066579212217880513,-0.0982483356597771,-0.0979740721734243,0.0064971260842139915,0.0073966778428481645,
        0.0,1.0,0.0,0.0,0.0,0.0,0.0,-0.0,-1.0,-0.0,-0.0,-0.0,-0.0,-0.0,-0.0,0.0068841868972328336,
        0.0882644978684177,0.0074028962019264018,0.083204517782092591,-0.0058560823614811283,-0.054585373826226039,
        0.0,1.0,0.0,0.0,0.0,0.0,0.0,0.0,-0.0,-1.0,-0.0,-0.0,-0.0,-0.0,0.0068762774998331784,0.0899028560363271,
        0.0073952142518775446,-0.0058500419994446436,-0.083204493772720892,0.0,1.0,0.0,0.0,0.0,0.0,0.0,0.0,-0.0,
        -1.0,-0.0,-0.0,-0.0,-0.0,0.0068777047366328468,0.097973756761605024,0.007396677842848161,
        -0.078900422955217944,-0.0058512700152415888,0.0982479399525699,0.0,1.0,0.0,0.0,0.0,0.0,0.0,0.0,-0.0,-1.0,
        -0.0,-0.0,-0.0,-0.0,-0.0,0.0074028962019264,-0.088264467351155729,-0.0058552526337344243,
        0.054582474317580759,0.0971527128705612,0.0,1.0,0.0,0.0,0.0,-0.0,-0.0,-0.0,-0.0,-0.0,0.0882646301098202,
        0.0066644827548764012,0.083204572117854689,-0.054585132435202473,-0.0074041913329832305,0.0,1.0,0.0,0.0,0.0,
        0.0,0.0,0.0,-0.0,-1.0,-0.0,-0.0,-0.0,-0.0,0.088264669807283549,0.0056135514717663929,0.083204667535680885,
        -0.0067354608622506246,-0.054585403472766414,0.0062169798578465005,0.0,1.0,0.0,0.0,0.0,0.0,0.0,0.0,-0.0,
        -1.0,-0.0,-0.0,-0.0,-0.0,-0.0,0.088264497868417668,0.083204517782092577,-0.0068855488483819159,
        -0.054585368753362618,0.0058560540134461594,0.0038299476112679106,0.0,1.0,0.0,0.0,0.0,-1.0,-0.0,-0.0,-0.0,
        -0.0,0.0882646301098202,0.0065019558665754219,0.0074028962019264052,0.083204572117854689,
        -0.0066658657231402083,-0.054585132435202473,0.0,1.0,0.0,0.0,0.0,0.0,0.0,-0.0,-1.0,-0.0,-0.0,-0.0,-0.0,-0.0,
        0.006656512283104341,0.089903014806281989,-0.0073952142518775464,-0.083204572117854772,0.0,1.0,0.0,0.0,0.0,
        0.0,0.0,0.0,-0.0,-1.0,-0.0,-0.0,-0.0,-0.0,0.006657921221788053,-0.078900403556479842,-0.0073966778428481671,
        0.098248335659777,0.097974072173424229,0.0,1.0,0.0,0.0,0.0,0.0,0.0,0.0,-0.0,-1.0,-0.0,-0.0,-0.0,-0.0,-0.0,
        0.0066644827548763995,-0.088264630109820233,-0.0074028962019264044,0.054582232982383738,
        0.097152952807911461,0.0,1.0,0.0,0.0,0.0,-0.0,-0.0,-0.0,-0.0,-0.0,0.006656512283104341,
        -0.089903014806281975,-0.0064957925478311522,-0.0073952142518775464,0.065501447211985434,
        0.083204572117854814,0.0,1.0,0.0,0.0,0.0,0.0,0.0,-0.0,-1.0,-0.0,-0.0,-0.0,-0.0,-0.0,0.089903034703890661,
        -0.0067270634377785661,-0.083204667535680926,0.0062069194685421677,0.0056052081304373783,0.0,1.0,0.0,0.0,
        0.0,0.0,0.0,0.0,-0.0,-1.0,-0.0,-0.0,-0.0,-0.0,-0.0,0.0899028560363271,-0.0068762774998331775,
        -0.083204517782092619,0.0058500139029652532,0.00382071618166485,0.0,1.0,0.0,0.0,0.0,-1.0,-0.0,-0.0,-0.0,
        -0.0,0.089903014806282,-0.0066565122831043393,-0.08320457211785473,0.0064957925478311539,
        0.0073952142518775542,0.0,1.0,0.0,0.0,0.0,0.0,0.0,-0.0,-1.0,-0.0,-0.0,-0.0,-0.0,-0.0,-0.0067284644196904976,
        -0.078900559120748739,0.0062082033463722475,0.098248210795103,0.0056064437356273073,0.0979739674398539,0.0,
        1.0,0.0,0.0,0.0,0.0,0.0,0.0,-0.0,-1.0,-0.0,-0.0,-0.0,-0.0,-0.0,-0.0,-0.00582457412621729,
        -0.0061630799572358827,-0.078900486165718819,0.0037822955399082294,0.089902772322115618,0.0,1.0,0.0,0.0,0.0,
        0.0,0.0,-0.0,-1.0,-0.0,-0.0,-0.0,-0.0,-0.0,-0.0,-0.0067342482080704228,-0.088264669807283549,
        0.054582503993362751,0.0062154506546600041,0.0056135514717663947,0.09715290327264671,0.0,1.0,0.0,0.0,0.0,
        -0.0,-0.0,-0.0,-0.0,-0.0,-0.0,-0.0064653841410221794,-0.00556214770328587,-0.0058246010853626852,
        -0.003782295539908232,-0.078900469896698883,-0.08826440165511483,-0.089902739686908359,0.078900469896698883,
        0.089902739686908345,0.0,1.0,0.0,0.0,0.0,0.0,0.0,0.0,-0.0,-1.0,-0.0,-0.0,-0.0,-0.0,-0.0,-0.0,-0.0,
        -0.0067270634377785653,-0.089903034703890661,0.0655016932872773,0.00620691946854217,0.083204667535680968,
        0.0056052081304373818,0.0,1.0,0.0,0.0,0.0,0.0,0.0,-0.0,-1.0,-0.0,-0.0,-0.0,-0.0,-0.0,-0.0,
        -0.078900439184654059,-0.0068777047366328451,0.0058512419011177222,0.098247986163974121,
        0.0038218069458475176,0.097973756761605024,0.0,1.0,0.0,0.0,0.0,-1.0,-0.0,-0.0,-0.0,-0.0,-0.0,
        -0.054581513793381407,-0.098249906447994889,-0.0067385738200007195,-0.0068889490139224727,
        -0.0066692894645364867,0.0067385738200007195,0.0068889490139224727,0.0066692894645364849,
        0.097155071000448165,0.0,1.0,0.0,0.0,0.0,0.0,-0.0,-1.0,-0.0,-0.0,-0.0,-0.0,-0.0,-0.0,-0.078900403556479842,
        -0.0066579212217880513,0.0064971260842139915,0.0073966778428481645,0.0982483356597771,0.09797407217342427,
        0.0,1.0,0.0,0.0,0.0,0.0,0.0,-0.0,-1.0,-0.0,-0.0,-0.0,-0.0,-0.0,-0.0,-0.065500982446408645,
        -0.097975501728056164,-0.0066682627334341913,0.0067376264600041268,0.09879842016046593,0.0,1.0,0.0,0.0,0.0,
        0.0,0.0,-0.0,-1.0,-0.0,-0.0,-0.0,-0.0,-0.0,-0.0068841868972328336,-0.0882644978684177,0.0058552243280781671,
        0.05458246924988279,0.0038284953491074382,0.097152743979504255,0.0,1.0,0.0,0.0,-0.0,-0.0,-0.0,-0.0,
        -0.0068762774998331784,-0.0073952142518775524,-0.089902823477288479,0.0058500419994446436,
        0.065501624272337883,0.083204493772720947,0.0,1.0,0.0,0.0,0.0,0.0,-0.0,-1.0,-0.0,-0.0,-0.0,-0.0,-0.0,-0.0,
        -0.0882646301098202,-0.0066644827548763995,0.0065019558665754219,0.054582232982383766,0.00740289620192641,
        0.097152952807911613,0.0,1.0,0.0,0.0,0.0,0.0,-0.0,-1.0,-0.0,-0.0,-0.0,-0.0,-0.0,-0.00665651228310434,
        -0.089903014806281975,0.0064957925478311539,0.065501447211985434,0.0073952142518775516,0.083204572117854814,
        0.0,1.0,0.0,0.0,0.0,0.0,-0.0,-1.0,-0.0,-0.0,-0.0,-0.0,-0.0,-0.0,0.0062205881626396691,0.0058583892699475767,
        0.0545826542019275,0.00064936905438700327,-0.097153733897863068,0.0,1.0,0.0,0.0,0.0,0.0,0.0,0.0,0.0,-0.0,
        -1.0,-0.0,-0.0,-0.0,-0.0,0.0067385738200007187,0.054582503993362758,0.098248210795102958,
        -0.0062205881626396682,-0.097154047019902,0.0,1.0,0.0,0.0,0.0,0.0,-1.0,-0.0,-0.0,-0.0,-0.0,-0.0,
        0.00649712608421399,0.0056064437356273152,0.0058512700152415879,0.078900469896698869,-0.098247727444134764,
        0.0,1.0,0.0,0.0,0.0,0.0,0.0,0.0,0.0,-0.0,-1.0,-0.0,-0.0,-0.0,-0.0,-0.0,0.0067354608622506229,
        -0.054585403472766435,-0.0,0.0971526215369334,0.0058560823614811248,0.00075791516333985364,
        0.00021633324934580575,0.0,1.0,0.0,0.0,0.0,0.0,0.0,0.0,0.0,-0.0,-1.0,-0.0,-0.0,-0.0,-0.0,
        0.0064957925478311513,0.00560520813043739,0.005850041999444641,0.0038230136475926814,-0.089902739686908345,
        0.06550176750368647,0.083204481168909758,0.0,1.0,0.0,0.0,0.0,0.0,0.0,0.0,-0.0,-1.0,-0.0,-0.0,-0.0,-0.0,-0.0,
        0.0067385738200007187,-0.054582503993362758,-0.098248210795102958,-0.0062205881626396682,
        0.097154047019901879,0.0,1.0,0.0,0.0,0.0,0.0,-0.0,-1.0,-0.0,-0.0,-0.0,-0.0,-0.0,-0.0,0.0067354608622506229,
        -0.0832046675356809,-0.0062169798578465057,-0.0056150615503170534,0.054585403472766435,0.0,1.0,0.0,0.0,0.0,
        0.0,0.0,-0.0,-1.0,-0.0,-0.0,-0.0,-0.0,-0.0,-0.0,0.078900422955217944,0.0073966778428481593,
        0.0038218069458475436,-0.00585127001524159,-0.098247939952569877,0.0,1.0,0.0,0.0,0.0,0.0,0.0,0.0,-0.0,-1.0,
        -0.0,-0.0,-0.0,-0.0,-0.0,0.098248335659777086,0.0066692894645364875,0.054585132435202452,
        -0.0074087967816751574,0.0,1.0,0.0,0.0,0.0,0.0,0.0,0.0,0.0,-0.0,-1.0,-0.0,-0.0,-0.0,-0.0,
        0.05458441303523779,0.00021639566193494715,-0.0067397872086759729,-0.0068903117801117717,
        -0.0066706732583767542,0.0067397872086759729,0.0068903117801117717,0.0066706732583767516,0.0,1.0,0.0,0.0,
        0.0,0.0,0.0,0.0,0.0,0.0,-0.0,-1.0,-0.0,-0.0,-0.0,-0.0,-0.0,0.098248210795102986,0.0056185970201033395,
        0.054585403472766407,-0.0067397872086759738,0.0062221182641002178,0.0,1.0,0.0,0.0,0.0,0.0,0.0,0.0,0.0,-0.0,
        -1.0,-0.0,-0.0,-0.0,-0.0,-0.0,0.098247986163974135,0.05458536875336259,-0.0068903117801117708,
        0.0058591910402779777,0.0038347171045817014,0.0,1.0,0.0,0.0,0.0,0.0,-1.0,-0.0,-0.0,-0.0,-0.0,
        0.054582232982383745,0.098248335659777086,-0.0066692894645364858,-0.097154096608237525,
        0.0065056592751906736,0.0074075008698108805,0.0,1.0,0.0,0.0,0.0,0.0,0.0,-0.0,-1.0,-0.0,-0.0,-0.0,-0.0,
        0.054585132435202445,0.00021640385253652057,-5.329679441843836E-5,0.0065066659943081714,
        0.0074087967816751626,0.0,1.0,0.0,0.0,0.0,0.0,0.0,0.0,-0.0,-1.0,-0.0,-0.0,-0.0,-0.0,-0.0,
        0.078900486165718833,-0.0058512419011177213,-0.0062082033463722484,0.0038241047903009593,0.0,1.0,0.0,0.0,
        0.0,0.0,0.0,-0.0,-1.0,-0.0,-0.0,-0.0,-0.0,-0.0,-0.0,0.0789004771821498,0.054582609835987422,
        -0.0065056592751906745,-0.0056185970201033386,-0.0971537969830813,0.0074323718720727475,1.0,0.0,0.0,0.0,0.0,
        0.0,-0.0,-1.0,-0.0,-0.0,-0.0,-0.0,-0.0,0.078900422955217944,-0.0073966778428481653,-0.098247939952569877,
        -0.097973713942593882,0.00585127001524159,0.0,1.0,0.0,0.0,0.0,0.0,0.0,-0.0,-1.0,-0.0,-0.0,-0.0,-0.0,-0.0,
        -0.0,0.0073952142518775446,0.0038207161816648759,-0.089902823477288479,-0.0058500419994446436,
        0.065501624272337883,0.083204493772720947,0.0,1.0,0.0,0.0,0.0,0.0,0.0,-0.0,-1.0,-0.0,-0.0,-0.0,-0.0,-0.0,
        0.0074075008698108787,-0.054582474317580752,-0.098247939952569918,-0.0058583892699475776,
        0.097153856531895927,0.0,1.0,0.0,0.0,0.0,-0.0,-0.0,-0.0,-0.0,-0.0,-0.0,0.0068855488483819186,
        0.0074041913329832331,-0.083204493772720961,-0.0058560823614811292,0.054585373826226,0.0,1.0,0.0,0.0,0.0,
        0.0,0.0,-0.0,-1.0,-0.0,-0.0,-0.0,-0.0,-0.0,0.088264449906324149,-0.0065019558665754228,
        -0.0056135514717663938,-0.054582609835987457,-0.097152653365209174,0.007427051555939564,1.0,0.0,0.0,0.0,0.0,
        -0.0,-1.0,-0.0,-0.0,-0.0,-0.0,-0.0,0.088264467351155715,0.083204493772720933,-0.0074041913329832339,
        -0.054585373826225983,0.0058560823614811275,0.0,1.0,0.0,0.0,0.0,0.0,0.0,-0.0,-1.0,-0.0,-0.0,-0.0,-0.0,-0.0,
        0.0066692894645364867,-0.05458223298238378,-0.098248335659777045,-0.0074075008698108779,0.0971540966082374,
        0.0,1.0,0.0,0.0,0.0,-0.0,-0.0,-0.0,-0.0,-0.0,-0.0,-0.065501447211985447,-0.097974072173424229,
        -0.0074064803715496981,5.3296794418438353E-5,-0.054585132435202473,-0.00650666599430817,0.0,1.0,0.0,0.0,0.0,
        0.0,0.0,-0.0,-1.0,-0.0,-0.0,-0.0,-0.0,-0.0,-0.0,0.0066658657231402109,-0.08320457211785473,
        -0.006502961965049194,-0.0074041913329832313,0.054585132435202459,0.0,1.0,0.0,0.0,0.0,0.0,0.0,-0.0,-1.0,
        -0.0,-0.0,-0.0,-0.0,-0.0,0.089902794278946527,-0.0064957925478311565,-0.0056052081304373792,
        -0.083204510522891642,0.0074181462343939717,0.0,1.0,0.0,0.0,0.0,0.0,0.0,-0.0,-1.0,-0.0,-0.0,-0.0,-0.0,-0.0,
        0.0899028234772885,-0.0073952142518775542,-0.083204493772720933,0.005850041999444641,0.0,1.0,0.0,0.0,0.0,
        0.0,0.0,-0.0,-1.0,-0.0,-0.0,-0.0,-0.0,-0.0,-0.0064971260842139923,-0.0789004771821498,
        -0.0056064437356273065,-0.0058512700152415879,0.098247727444134764,0.097973523596097969,0.0,1.0,0.0,0.0,0.0,
        0.0,0.0,-0.0,-1.0,-0.0,-0.0,-0.0,-0.0,-0.0,-0.0,-0.0,-0.0067376264600041268,-0.065501693287277313,
        -0.097973967439853843,0.00621951472423367,0.0987964165818141,0.00561756258799417,0.0,0.0,0.0,0.0,0.0,0.0,
        -0.0,-1.0,-0.0,-0.0,-0.0,-0.0,-0.0,-0.0,-0.0062069194685421721,-0.00585004199944464,-0.0074181462343939717,
        -0.089902739686908345,0.083204481168909758,0.0,1.0,0.0,0.0,0.0,0.0,-0.0,-1.0,-0.0,-0.0,-0.0,-0.0,-0.0,-0.0,
        -0.0,-0.0065019558665754219,-0.088264449906324149,-0.0056135514717663947,0.054582609835987464,
        0.007427051555939564,0.0971526533652088,1.0,0.0,0.0,0.0,-0.0,-0.0,-0.0,-0.0,-0.0,-0.0,
        -0.0067354608622506229,-0.0832046675356809,0.054585403472766435,0.0062169798578465057,0.0056150615503170473,
        0.0,1.0,0.0,0.0,0.0,0.0,0.0,-0.0,-1.0,-0.0,-0.0,-0.0,-0.0,-0.0,-0.0,-0.0064957925478311531,
        -0.0056052081304373844,-0.089902794278946527,0.065501738694921013,0.0074181462343939769,
        0.083204510522891614,1.0,0.0,0.0,0.0,0.0,-0.0,-1.0,-0.0,-0.0,-0.0,-0.0,-0.0,-0.078900422955217944,
        -0.0073966778428481653,0.00585127001524159,0.098247939952569877,0.097973713942593854,0.0,1.0,0.0,0.0,0.0,
        0.0,0.0,-0.0,-1.0,-0.0,-0.0,-0.0,-0.0,-0.0,-0.0,-0.0655016264921725,-0.0068879216085573295,
        -0.097973756761605,0.0058576452378786862,0.098796169093499323,0.0038323462521122906,0.0,0.0,0.0,0.0,-1.0,
        -0.0,-0.0,-0.0,-0.0,-0.0,-0.054584413035237804,-0.00043304398331863418,-0.0067397872086759729,
        -0.0068903117801117717,-0.0066706732583767542,0.0067397872086759729,0.0068903117801117717,
        0.0066706732583767516,0.0,1.0,0.0,0.0,0.0,0.0,0.0,0.0,-0.0,-1.0,-0.0,-0.0,-0.0,-0.0,-0.0,-0.0,-0.0,
        -0.0074028962019264061,-0.0882644673511557,0.0058552526337344226,0.054582474317580787,0.0971527128705616,
        0.0,1.0,0.0,0.0,0.0,0.0,-0.0,-1.0,-0.0,-0.0,-0.0,-0.0,-0.0,-0.0068855488483819186,-0.0832045177820926,
        0.0058560540134461551,0.054585368753362624,0.0038299476112678842,0.0,1.0,0.0,0.0,0.0,0.0,-0.0,-1.0,-0.0,
        -0.0,-0.0,-0.0,-0.0,-0.083204572117854717,-0.0066658657231402092,0.0065029619650491949,0.054585132435202473,
        0.0074041913329832339,0.0,1.0,0.0,0.0,0.0,0.0,-0.0,-1.0,-0.0,-0.0,-0.0,-0.0,-0.0,-0.0,0.0067397872086759738,
        0.054585403472766428,0.097154047019901976,-0.00622211826410022,0.0,1.0,0.0,0.0,0.0,0.0,0.0,0.0,0.0,-0.0,
        -1.0,-0.0,-0.0,-0.0,-0.0,-0.0,0.0058512700152415871,8.4912584490156191E-6,-0.078900469896698883,
        0.098247727444134722,0.097973523596097942,0.0,1.0,0.0,0.0,0.0,0.0,0.0,0.0,0.0,-0.0,-1.0,-0.0,-0.0,-0.0,-0.0,
        -0.0,0.0058552526337344261,0.0038307934422769628,-0.088264401655114816,0.054582654201927511,
        0.097152590313725321,0.0,1.0,0.0,0.0,0.0,0.0,-0.0,-0.0,-0.0,-0.0,-0.0,0.0062205881626396691,
        -0.098247773768529445,0.0058583892699475767,-0.054582654201927455,-0.0006493690543870037,
        0.097153733897862971,0.0,1.0,0.0,0.0,0.0,-0.0,-0.0,-0.0,-0.0,-0.0,-0.0,0.0065029619650491931,
        0.0056150615503170508,-0.083204510522891614,0.0058560823614811248,-0.0007579151633398544,
        0.054585553741930588,0.0,1.0,0.0,0.0,0.0,0.0,0.0,0.0,-0.0,-1.0,-0.0,-0.0,-0.0,-0.0,-0.0,
        0.0067397872086759738,-0.054585403472766421,-0.098796416581814067,-0.00622211826410022,
        -0.0056201079854152026,0.0,1.0,0.0,0.0,0.0,0.0,0.0,-0.0,-1.0,-0.0,-0.0,-0.0,-0.0,-0.0,-0.0,-0.0,
        0.0058560540134461559,0.0062169798578465049,-0.083204505229654863,-0.0038322457367332527,
        0.054585548665854335,0.0,1.0,0.0,0.0,0.0,0.0,0.0,-0.0,-1.0,-0.0,-0.0,-0.0,-0.0,0.0074075008698108735,
        0.098247939952569946,0.0038332639910602486,0.054585373826226004,8.5121171839220313E-6,
        -0.0058592195178481313,0.0,1.0,0.0,0.0,0.0,0.0,0.0,0.0,0.0,-0.0,-1.0,-0.0,-0.0,-0.0,-0.0,
        0.054582474317580738,0.098247939952569946,-0.0074075008698108787,-0.097153856531896066,
        0.0058583892699475785,0.0,1.0,0.0,0.0,0.0,0.0,0.0,-0.0,-1.0,-0.0,-0.0,-0.0,-0.0,0.00021640790207670476,0.0,
        -0.0,0.0545826542019275,-0.0058583892699475776,-3.2428797170406639E-5,0.0,1.0,0.0,0.0,0.0,0.0,0.0,-0.0,-1.0,
        -0.0,-0.0,-0.0,-0.0,-0.0,0.054585373826226,0.00021640630568683743,-6.72496723541531E-5,
        0.0058592195178481278,0.0,1.0,0.0,0.0,0.0,0.0,0.0,0.0,-0.0,-1.0,-0.0,-0.0,-0.0,-0.0,-0.0,
        0.078900469896698883,-0.0058512700152415888,-3.2372276985735869E-5,-0.098247727444134778,
        -0.097973523596097969,0.0,1.0,0.0,0.0,0.0,0.0,0.0,-0.0,-1.0,-0.0,-0.0,-0.0,-0.0,-0.0,-0.0,-0.0,
        -0.065501624272337855,-0.097973713942593868,-0.0058576736506951114,6.7249672354153031E-5,
        -0.054585373826226018,0.0,1.0,0.0,0.0,0.0,0.0,0.0,-0.0,-1.0,-0.0,-0.0,-0.0,-0.0,-0.0,-0.0,
        0.097152653365208869,-0.0065029619650491975,-0.0056150615503170413,-0.054585509362638229,
        0.00075791516333985494,0.00021633324934580478,-0.0058560823614811292,0.0,1.0,0.0,0.0,0.0,0.0,0.0,-0.0,-1.0,
        -0.0,-0.0,-0.0,-0.0,-0.0,-0.0,0.08826440165511483,-0.0058552526337344321,-0.0074270515559395579,
        -0.054582654201927469,-0.097152590313725487,0.0,1.0,0.0,0.0,0.0,0.0,-0.0,-1.0,-0.0,-0.0,-0.0,-0.0,-0.0,-0.0,
        0.089902739686908345,-0.0058500419994446445,-0.0074181462343939674,-0.083204481168909716,0.0,1.0,0.0,0.0,
        0.0,0.0,0.0,-0.0,-1.0,-0.0,-0.0,-0.0,-0.0,-0.0,-0.0,-0.0065048246753232923,-0.065501738694921,
        -0.00561756258799417,-0.097973614654771057,0.0074312205013612881,0.09879597673186849,0.0,0.0,0.0,0.0,-0.0,
        -1.0,-0.0,-0.0,-0.0,-0.0,-0.0,-0.0,-0.0067397872086759738,-0.054585403472766421,-0.098796416581814067,
        0.00622211826410022,0.0056201079854151974,0.0,1.0,0.0,0.0,0.0,0.0,0.0,-0.0,-1.0,-0.0,-0.0,-0.0,-0.0,-0.0,
        -0.0,-0.0,-0.08826440165511483,-0.0,-0.0058560540134461559,-0.0062169798578465049,-0.083204505229654863,
        0.054585548665854335,0.0,1.0,0.0,0.0,0.0,0.0,-0.0,-1.0,-0.0,-0.0,-0.0,-0.0,-0.0,-0.0,-0.006502961965049194,
        -0.0832045105228916,-0.0056150615503170447,0.054585509362638292,0.0074286186340326637,1.0,0.0,0.0,0.0,0.0,
        -0.0,-1.0,-0.0,-0.0,-0.0,-0.0,-0.0,-0.0068903117801117708,-0.054585373826226004,-6.7249672354153072E-5,
        -0.00021640630568683708,0.0058592195178481295,0.0,1.0,0.0,0.0,0.0,0.0,-0.0,-1.0,-0.0,-0.0,-0.0,-0.0,-0.0,
        -0.0,-0.0,-0.054585132435202459,-0.00043305825939417666,-5.3296794418438367E-5,0.00650666599430817,
        0.0074087967816751574,0.0,1.0,0.0,0.0,0.0,0.0,-0.0,-1.0,-0.0,-0.0,-0.0,-0.0,-0.0,-0.0,-0.0,
        -0.0074041913329832383,-0.083204493772720947,-0.0038299476112678916,-0.097152712870561236,
        0.0058560823614811275,0.054585373826226039,0.0,1.0,0.0,0.0,0.0,0.0,-0.0,-1.0,-0.0,-0.0,-0.0,-0.0,-0.0,-0.0,
        0.0058591910402779777,0.054585548665854307,4.0951614938672555E-5,0.00021640777473473565,
        -0.0038370155782307246,0.0,1.0,0.0,0.0,0.0,0.0,0.0,0.0,0.0,-0.0,-1.0,-0.0,-0.0,-0.0,-0.0,
        0.0058576736506951105,-0.00043283783956480509,0.098795860873172964,0.0,1.0,0.0,0.0,0.0,0.0,0.0,0.0,0.0,-0.0,
        -1.0,-0.0,-0.0,-0.0,-0.0,-0.0,0.0058591910402779768,-0.00043306541148648795,3.2435689974901612E-5,
        -0.054585553741930574,-0.00043306561930008404,0.0,1.0,0.0,0.0,0.0,0.0,0.0,0.0,-0.0,-1.0,-0.0,-0.0,-0.0,-0.0,
        -0.0,-0.0,0.00650666599430817,2.4730212471709076E-5,-0.054585509362638229,-0.0074339398709295035,0.0,1.0,
        0.0,0.0,0.0,0.0,0.0,-0.0,-1.0,-0.0,-0.0,-0.0,-0.0,-0.0,-0.0,-0.0065066659943081705,-0.054585509362638236,
        -0.00043306472267690317,-2.4730212471709049E-5,0.0074339398709295087,1.0,0.0,0.0,0.0,0.0,-0.0,-1.0,-0.0,
        -0.0,-0.0,-0.0,-0.0,-0.0,-0.0058591910402779777,-4.0951614938672562E-5,-0.054585553741930623,
        -0.00021640790207670509,0.0,1.0,0.0,0.0,0.0,0.0,-0.0,-1.0,-0.0,-0.0,-0.0,-0.0,-0.0,-0.0,-0.0,-0.0,
        0.0058592195178481252,0.054585553741930623,8.520008505711021E-6,0.00021640790207670536,0.0,1.0,0.0,0.0,0.0,
        0.0,0.0,0.0,0.0,0.0,-0.0,-1.0,-0.0,-0.0,-0.0,-0.0,-0.013355084776427602,-0.00070241106942519444,
        -0.015696854540883667,-0.00073180354810950109,-0.016360890164250554,-0.0007121884817449227,
        0.013355084776427602,0.00070241106942519444,0.015696854540883667,0.00073180354810950109,
        0.016360890164250557,0.0007121884817449227,0.0,0.0,1.0,0.0,0.0,0.0,0.0,0.0,0.0,0.0,-0.0,-0.0,-1.0,-0.0,-0.0,
        -0.0,-0.0,-0.0,0.0133550847764276,-0.000708712280935733,-0.01913681977138957,-0.00073903425520361,
        -0.01967530511425436,-0.00071965353685171413,0.000708712280935733,0.00073903425520361,
        0.00071965353685171413,0.0,0.0,1.0,0.0,0.0,0.0,0.0,0.0,0.0,-0.0,-0.0,-1.0,-0.0,-0.0,-0.0,-0.0,-0.0,
        0.00070241106942519433,-0.013354886628180915,-0.015696489327294644,-0.0006949277575493321,
        -0.016360498733859103,-0.00063267402481259887,0.013354886628180915,0.015696489327294644,
        0.016360498733859103,0.0,0.0,1.0,0.0,0.0,0.0,0.0,0.0,0.0,-0.0,-0.0,-1.0,-0.0,-0.0,-0.0,-0.0,-0.0,
        0.015696854540883667,0.00070977892002071043,0.00072094437214855291,0.013815309769759592,
        -0.0078504940691150014,-0.00070998479812853861,-0.00074050995988770771,-0.00072119125834864851,
        0.00074050995988770771,0.0,0.0,1.0,0.0,0.0,0.0,0.0,0.0,0.0,-0.0,-0.0,-1.0,-0.0,-0.0,-0.0,-0.0,
        0.00073180354810950109,0.01335484741688741,0.016360436265260729,0.00077719632837294642,-0.01335483887448634,
        -0.00058545773453366626,-0.015696416044310806,-0.01636042241173408,0.0,0.0,1.0,0.0,0.0,0.0,0.0,0.0,0.0,-0.0,
        -0.0,-1.0,-0.0,-0.0,-0.0,-0.0,0.016360890164250554,-0.010053984761327208,-0.00070855886012245229,
        -0.013815309769759605,-0.00073887229766321256,-0.00071950068311493829,0.00070855886012245229,
        0.00073887229766321256,0.00071950068311493829,0.0,0.0,1.0,0.0,0.0,0.0,0.0,0.0,0.0,-0.0,-0.0,-1.0,-0.0,-0.0,
        -0.0,-0.0,0.00071218848174492281,-0.013354881724508197,-0.00066290338327761684,-0.015696496781502488,
        -0.00077719632837294685,-0.016360509090127547,0.013354881724508197,0.015696496781502488,0.01636050909012755,
        0.0,0.0,1.0,0.0,0.0,0.0,0.0,0.0,0.0,-0.0,-0.0,-1.0,-0.0,-0.0,-0.0,-0.0,-0.0133550847764276,
        -0.000708712280935733,-0.00073903425520361,-0.00071965353685171413,0.000708712280935733,0.01913681977138957,
        0.00073903425520361,0.01967530511425436,0.00071965353685171413,0.0,0.0,1.0,0.0,0.0,0.0,0.0,0.0,0.0,-0.0,
        -0.0,-1.0,-0.0,-0.0,-0.0,-0.0,-0.0,-0.00070241106942519433,-0.013354886628180915,-0.015696489327294644,
        -0.016360498733859103,0.013354886628180915,0.015696489327294644,0.0006949277575493321,0.016360498733859103,
        0.00063267402481259887,0.0,0.0,1.0,0.0,0.0,0.0,0.0,0.0,0.0,-0.0,-0.0,-1.0,-0.0,-0.0,-0.0,-0.0,-0.0,
        -0.015696854540883667,-0.013815309769759589,-0.00070998479812853861,-0.00074050995988770771,
        -0.00072119125834864851,0.0078504940691150014,0.00070998479812853861,0.00072119125834864851,0.0,0.0,1.0,0.0,
        0.0,0.0,0.0,0.0,-0.0,-0.0,-1.0,-0.0,-0.0,-0.0,-0.0,-0.0,-0.00073180354810950109,-0.01335484741688741,
        -0.016360436265260729,-0.00077719632837294642,-0.015696416044310806,0.01335483887448634,
        0.00058545773453366626,0.015696416044310806,0.01636042241173408,0.0,0.0,1.0,0.0,0.0,0.0,0.0,0.0,-0.0,-0.0,
        -1.0,-0.0,-0.0,-0.0,-0.0,-0.0,-0.016360890164250557,-0.00070855886012245229,-0.00073887229766321256,
        -0.00071950068311493829,0.010053984761327205,0.00070855886012245229,0.0138153097697596,
        0.00073887229766321256,0.00071950068311493829,0.0,0.0,1.0,0.0,0.0,0.0,0.0,0.0,-0.0,-0.0,-1.0,-0.0,-0.0,-0.0,
        -0.0,-0.0,-0.00071218848174492281,-0.013354881724508197,-0.015696496781502488,-0.016360509090127547,
        0.013354881724508197,0.00066290338327761684,0.015696496781502488,0.00077719632837294685,0.01636050909012755,
        0.0,0.0,1.0,0.0,0.0,0.0,0.0,0.0,-0.0,-0.0,-1.0,-0.0,-0.0,-0.0,-0.0,-0.0,0.013354886628180915,
        0.00070871228093573313,-0.019136254043089853,-0.00070338839082327153,-0.019674776790317681,
        -0.00064128274259411312,0.0,0.0,1.0,0.0,0.0,0.0,0.0,0.0,-0.0,-0.0,-1.0,-0.0,-0.0,-0.0,-0.0,-0.0,
        0.01913681977138957,0.0078504940691149928,0.01805005232413056,-0.00071067908889347979,
        -0.00074130273940990277,-0.00072200639376403209,0.00071067908889347979,0.00074130273940990277,
        0.00072200639376403209,0.0,0.0,1.0,0.0,0.0,0.0,0.0,0.0,0.0,0.0,-0.0,-0.0,-1.0,-0.0,-0.0,-0.0,-0.0,
        0.013354847416887408,-0.00058947514464916862,-0.00045700543323026527,-0.0,0.0078505513076336155,
        0.00074130273940990277,-0.00045995981458201189,0.0,0.0,1.0,0.0,0.0,0.0,0.0,0.0,-0.0,-0.0,-1.0,-0.0,-0.0,
        -0.0,0.010053984761327205,0.019675305114254353,-0.00071029983670461842,-0.018050052324130553,
        0.00072155339410677672,0.0,0.0,1.0,0.0,0.0,0.0,0.0,0.0,-0.0,-0.0,-1.0,-0.0,-0.0,-0.0,-0.0,
        0.013354881724508197,-0.00078374994311405,-0.0,0.007850534412593509,0.00072200639376403209,0.0,0.0,1.0,0.0,
        0.0,0.0,0.0,0.0,0.0,-0.0,-0.0,-1.0,-0.0,-0.0,-0.0,0.013354886628180915,-0.00070871228093573313,-0.0,
        0.00784983585460256,-0.021264396690767656,0.00064374146358048734,0.0,0.0,1.0,0.0,0.0,0.0,0.0,0.0,-0.0,-0.0,
        -1.0,-0.0,-0.0,-0.0,-0.0,0.013354847416887408,-0.00073903425520361,-0.019136171450666897,
        0.00058947514464916862,0.00045700543323026538,0.0,0.0,1.0,0.0,0.0,0.0,-0.0,-0.0,-1.0,-0.0,-0.0,-0.0,-0.0,
        0.013354881724508197,-0.00071965353685171413,-0.01913627908650652,-0.019674802040209542,
        0.00066787723649602772,0.00078374994311405,0.0,0.0,1.0,0.0,0.0,0.0,0.0,-0.0,-0.0,-1.0,-0.0,-0.0,-0.0,-0.0,
        -0.0,0.00070977892002071054,0.015696387656065527,0.00059013581334217821,-0.0078498418577679328,
        -0.021266481483774708,0.0,0.0,1.0,0.0,0.0,0.0,0.0,0.0,-0.0,-0.0,-1.0,-0.0,-0.0,-0.0,0.00058545213764139327,
        0.00069492775754933231,-0.013354826750081004,-0.015696387656065527,-0.016360391103343891,
        -0.0004481686028084641,0.013354826750081004,0.015696387656065527,0.016360391103343894,0.0,0.0,1.0,0.0,0.0,
        0.0,0.0,0.0,-0.0,-0.0,-1.0,-0.0,-0.0,-0.0,0.00070855886012245251,0.0163604987338591,-0.010053959431077385,
        -0.013815029502340643,-0.00070322802658466608,0.0,0.0,1.0,0.0,0.0,0.0,0.0,0.0,-0.0,-0.0,-1.0,-0.0,-0.0,-0.0,
        -0.0,0.00066290338327761684,0.00063267402481259919,-0.016360399418003064,0.013354829801521528,
        0.0156963952424949,0.016360399418003064,0.0,0.0,1.0,0.0,0.0,0.0,0.0,0.0,0.0,0.0,-0.0,-0.0,-1.0,-0.0,-0.0,
        -0.0,-0.0,0.00070871228093573281,-0.013354886628180915,-0.00070338839082327207,0.019136254043089867,
        0.019674776790317688,0.0,0.0,1.0,0.0,0.0,0.0,0.0,0.0,-0.0,-0.0,-1.0,-0.0,-0.0,-0.0,-0.0,-0.0,
        0.00070977892002071054,-0.015696489327294644,-0.00070486724956031889,0.0078498358546025652,
        0.021266597087506126,0.0,0.0,1.0,0.0,0.0,0.0,0.0,-0.0,-0.0,-1.0,-0.0,-0.0,-0.0,-0.0,0.00070855886012245251,
        -0.016360498733859103,-0.00070322802658466608,-0.00064115033886434007,0.010053959431077382,
        0.013815029502340643,0.0,0.0,1.0,0.0,0.0,0.0,0.0,-0.0,-0.0,-1.0,-0.0,-0.0,-0.0,-0.0,-0.0,
        0.015696429274739486,0.0007402725668637,0.013814978346247547,0.00078483961287594765,-0.0078505504957846264,
        -0.00059026517985183739,0.0,0.0,1.0,0.0,0.0,0.0,0.0,0.0,-0.0,-0.0,-1.0,-0.0,-0.0,-0.0,0.015696496781502492,
        0.00072094437214855291,0.013815028737181446,-0.0078505344125935073,-0.00078505003013483422,0.0,0.0,1.0,0.0,
        0.0,0.0,0.0,0.0,-0.0,-0.0,-1.0,-0.0,-0.0,-0.0,0.015696489327294647,0.00064281278721221359,
        0.013815029502340637,-0.0007099847981285385,-0.00785055587835492,0.00070514735512079252,0.0,0.0,1.0,0.0,0.0,
        0.0,0.0,0.0,-0.0,-0.0,-1.0,-0.0,-0.0,-0.0,-0.0,0.013814978346247547,-0.000740509959887708,
        -0.0078505513076336172,0.0005902592207076454,0.00045900348534280938,0.0,0.0,1.0,0.0,0.0,-0.0,-1.0,-0.0,-0.0,
        -0.0,0.00073887229766321256,0.016360436265260729,0.00078356528008410354,-0.00058935731463155463,
        -0.013814967279330388,0.0,0.0,1.0,0.0,0.0,0.0,0.0,0.0,-0.0,-0.0,-1.0,-0.0,-0.0,-0.0,0.00073903425520360994,
        0.019674701485866784,0.00078374994311404967,-0.01335483887448634,-0.00058948103625439357,
        0.019136152968431349,0.0,0.0,1.0,0.0,0.0,0.0,0.0,0.0,-0.0,-0.0,-1.0,-0.0,-0.0,-0.0,-0.0,
        0.0007402725668636999,0.00078483961287594722,-0.015696416044310803,-0.00059013581334217832,
        0.0078498304624371844,0.021266532224969138,0.0,0.0,0.0,0.0,0.0,-0.0,-1.0,-0.0,-0.0,-0.0,
        0.00073887229766321256,0.01005394241171902,0.01381497834624754,0.00078356528008410354,-0.016360422411734073,
        -0.00058935731463155463,0.0,0.0,1.0,0.0,0.0,0.0,0.0,-0.0,-0.0,-1.0,-0.0,-0.0,-0.0,-0.0,0.016360509090127547,
        0.00071950068311493818,-0.013815028737181451,-0.00078356528008410376,0.0,0.0,1.0,0.0,0.0,0.0,0.0,0.0,-0.0,
        -0.0,-1.0,-0.0,-0.0,-0.0,0.0163604987338591,-0.0007085588601224524,-0.013815029502340658,
        0.00070322802658466575,0.00064115033886434007,0.0,0.0,1.0,0.0,0.0,0.0,0.0,0.0,-0.0,-0.0,-1.0,-0.0,-0.0,-0.0,
        -0.0,0.016360436265260726,-0.00073887229766321266,-0.013814978346247555,0.00058935142225332476,
        0.00045695607481956147,0.0,0.0,1.0,0.0,0.0,-0.0,-1.0,-0.0,-0.0,-0.0,0.016360509090127547,
        -0.00071950068311493818,-0.010053942472644632,-0.013815028737181451,0.00066772991164514863,
        0.00078356528008410376,0.0,0.0,1.0,0.0,0.0,0.0,0.0,-0.0,-0.0,-1.0,-0.0,-0.0,-0.0,-0.0,
        0.00071965353685171413,-0.013354881724508197,-0.00078374994311405011,0.01913627908650653,
        0.019674802040209546,0.0,0.0,1.0,0.0,0.0,0.0,0.0,0.0,-0.0,-0.0,-1.0,-0.0,-0.0,-0.0,-0.0,
        0.00072094437214855281,-0.015696496781502488,-0.00078483961287594754,0.0078498143875897573,
        0.021266622548422189,0.0,0.0,0.0,0.0,0.0,-0.0,-1.0,-0.0,-0.0,-0.0,0.00071950068311493818,
        -0.016360509090127547,-0.00078356528008410376,0.010053942472644628,0.013815028737181455,0.0,0.0,1.0,0.0,0.0,
        0.0,0.0,-0.0,-0.0,-1.0,-0.0,-0.0,-0.0,-0.0,-0.013354886628180915,-0.00070871228093573313,
        0.019136254043089853,0.00070338839082327153,0.019674776790317681,0.00064128274259411333,0.0,0.0,1.0,0.0,0.0,
        0.0,0.0,0.0,-0.0,-0.0,-1.0,-0.0,-0.0,-0.0,-0.0,-0.0,-0.0078497740839998265,-0.01913681977138957,
        -0.00071047308705639756,0.021264803951796803,0.00072175936181417908,0.0,0.0,1.0,0.0,0.0,0.0,0.0,-0.0,-0.0,
        -1.0,-0.0,-0.0,-0.0,-0.0,-0.0,-0.013354847416887408,-0.00073903425520361,0.00058947514464916862,
        0.019136171450666897,0.019674701485866791,0.00045700543323026538,0.0,0.0,1.0,0.0,0.0,-0.0,-1.0,-0.0,-0.0,
        -0.0,-0.0,-0.010053984761327205,-0.019675305114254357,-0.0078504940691149945,-0.021264803951796817,
        -0.00071067908889347979,-0.00074130273940990277,-0.00072200639376403209,0.00071067908889347979,
        0.00072200639376403209,0.0,0.0,1.0,0.0,0.0,0.0,0.0,0.0,-0.0,-0.0,-1.0,-0.0,-0.0,-0.0,-0.0,-0.0,-0.0,
        -0.013354881724508197,-0.00071965353685171413,0.00066787723649602772,0.01913627908650652,
        0.00078374994311405,0.019674802040209542,0.0,0.0,1.0,0.0,0.0,0.0,0.0,-0.0,-0.0,-1.0,-0.0,-0.0,-0.0,-0.0,
        -0.0,-0.00070977892002071054,-0.015696489327294644,0.0078498358546025652,0.00070486724956031889,
        0.021266597087506126,0.00064281278721221337,0.0,0.0,0.0,0.0,0.0,-0.0,-1.0,-0.0,-0.0,-0.0,-0.0,
        -0.00058545213764139327,-0.00069492775754933231,-0.013354826750081004,-0.015696387656065527,
        -0.016360391103343891,0.013354826750081004,0.015696387656065527,0.016360391103343894,0.0004481686028084641,
        0.0,0.0,1.0,0.0,0.0,0.0,-0.0,-0.0,-1.0,-0.0,-0.0,-0.0,-0.0,-0.0,-0.00070855886012245251,
        -0.016360498733859103,0.010053959431077382,0.013815029502340643,0.00070322802658466608,
        0.00064115033886434007,0.0,0.0,1.0,0.0,0.0,0.0,0.0,-0.0,-0.0,-1.0,-0.0,-0.0,-0.0,-0.0,-0.0,
        -0.00066290338327761684,-0.00063267402481259919,-0.016360399418003064,0.013354829801521528,
        0.00082020698923774085,0.0,0.0,1.0,0.0,0.0,0.0,0.0,-0.0,-0.0,-1.0,-0.0,-0.0,-0.0,-0.0,-0.015696429274739486,
        -0.0007402725668637,0.0078498312759191675,0.0005901298647647122,0.021266544761989165,0.00045868723263609631,
        0.0,0.0,0.0,0.0,-1.0,-0.0,-0.0,-0.0,-0.015696496781502492,-0.013815028737181443,-0.00072119125834864851,
        0.0078505344125935142,0.00066885432718430675,0.00078505003013483422,0.0,0.0,1.0,0.0,0.0,0.0,-0.0,-0.0,-1.0,
        -0.0,-0.0,-0.0,-0.0,-0.0,-0.00073887229766321256,-0.016360436265260733,0.01005394241171902,
        0.00058935142225332476,0.013814978346247547,0.00045695607481956217,0.0,0.0,1.0,0.0,0.0,0.0,-0.0,-0.0,-1.0,
        -0.0,-0.0,-0.0,-0.0,-0.01636050909012755,-0.00071950068311493818,0.010053942472644628,
        0.00066772991164514863,0.01381502873718145,0.00078356528008410376,0.0,0.0,1.0,0.0,0.0,0.0,-0.0,-0.0,-1.0,
        -0.0,-0.0,-0.0,-0.0,-0.0,0.019136104037587275,0.0078505627081109745,0.00059070966910656456,
        4.6667541046249082E-6,-0.00046016924547736962,0.0,0.0,1.0,0.0,0.0,0.0,0.0,0.0,0.0,-0.0,-0.0,-1.0,-0.0,-0.0,
        -0.0,0.013354826750081004,0.000589475144649169,0.00070338839082327109,-0.019136104037587275,
        -0.00045721508909140403,0.0,0.0,1.0,0.0,0.0,0.0,-0.0,-1.0,-0.0,-0.0,-0.0,-0.0,0.01005395943107738,
        0.019674776790317691,0.0078505558783549187,0.00071067908889347968,-0.00070606688480528491,0.0,0.0,1.0,0.0,
        0.0,0.0,0.0,0.0,0.0,-0.0,-0.0,-1.0,-0.0,-0.0,-0.0,-0.0,0.01335483887448634,-0.00058948103625439325,-0.0,
        0.00045964338544026849,0.0078505504957846264,7.1576985742576626E-6,1.0242094517058181E-6,0.0,0.0,1.0,0.0,
        0.0,0.0,0.0,0.0,0.0,-0.0,-0.0,-1.0,-0.0,-0.0,-0.0,0.010053942472644626,0.019674802040209546,
        0.007850534412593509,0.021264422151952962,-0.00072200639376403209,0.00066940907433716364,
        0.00078577738649557045,0.0,0.0,1.0,0.0,0.0,0.0,0.0,0.0,-0.0,-0.0,-1.0,-0.0,-0.0,-0.0,-0.0,
        0.013354826750081004,-0.000589475144649169,-0.00070338839082327109,-0.019136104037587275,
        0.00045721508909140403,0.0,0.0,1.0,0.0,0.0,0.0,-0.0,-0.0,-1.0,-0.0,-0.0,-0.0,-0.0,-0.0,0.01335483887448634,
        -0.00078374994311405,-0.019136152968431349,-0.019674684401114268,0.00058948103625439325,0.0,0.0,1.0,0.0,0.0,
        0.0,0.0,-0.0,-0.0,-1.0,-0.0,-0.0,-0.0,-0.0,-0.0,0.00070998479812853861,0.013815029502340646,
        0.021266597087506119,-0.007850555878354917,-0.000705147355120792,0.0,0.0,1.0,0.0,0.0,0.0,0.0,0.0,-0.0,-0.0,
        -1.0,-0.0,-0.0,-0.0,-0.0,0.0007032280265846663,0.016360391103343884,0.000589357314631555,
        -0.013814936811065831,0.0,0.0,1.0,0.0,0.0,0.0,0.0,0.0,0.0,-0.0,-0.0,-1.0,-0.0,-0.0,-0.0,
        0.00058545773453366594,9.9821594966206443E-7,-0.013354818196216901,-0.015696374407663447,
        -0.016360377230620737,0.013354818196216901,0.015696374407663447,0.016360377230620737,0.0,0.0,1.0,0.0,0.0,
        0.0,0.0,0.0,0.0,0.0,-0.0,-0.0,-1.0,-0.0,-0.0,-0.0,-0.0,0.00070338839082327185,0.019674637958108528,
        0.00058948103625439336,-0.013354818196216903,0.019136085528464446,0.0,0.0,1.0,0.0,0.0,0.0,0.0,0.0,0.0,-0.0,
        -0.0,-1.0,-0.0,-0.0,-0.0,-0.0,0.0007048672495603191,0.00059013581334217821,-0.015696374407663444,
        0.00784984185776794,0.021266481483774712,0.0,0.0,0.0,0.0,0.0,0.0,-0.0,-1.0,-0.0,-0.0,-0.0,
        0.00058935142225332465,0.0007032280265846663,-0.016360391103343887,-0.0004571656718651675,
        0.010053943283910695,0.013814947892318402,0.0,0.0,1.0,0.0,0.0,0.0,0.0,-0.0,-0.0,-1.0,-0.0,-0.0,-0.0,
        0.00058935731463155485,1.0183040766464289E-6,-0.00013071479116047661,0.010053939720042822,
        0.013814936811065836,0.0,0.0,1.0,0.0,0.0,0.0,0.0,0.0,-0.0,-0.0,-1.0,-0.0,-0.0,-0.0,-0.0,
        0.00071047308705639756,-0.0078498358546025635,-0.019136254043089867,0.021264396690767625,0.0,0.0,1.0,0.0,
        0.0,0.0,0.0,-0.0,-0.0,-1.0,-0.0,-0.0,-0.0,-0.0,-0.0,0.00071029983670461863,0.00059047175686875969,
        -0.010053943283910698,-0.019674637958108521,-0.00045960759224737192,0.01804924706676608,0.0,1.0,0.0,0.0,0.0,
        0.0,-0.0,-0.0,-1.0,-0.0,-0.0,-0.0,-0.0,0.00070998479812853861,-0.013815029502340641,-0.000705147355120792,
        -0.00064310201354924451,0.007850555878354917,0.0,0.0,1.0,0.0,0.0,0.0,0.0,-0.0,-0.0,-1.0,-0.0,-0.0,-0.0,-0.0,
        -0.0,0.013815028737181446,0.021266622548422178,-0.00072119125834864851,-0.0078505344125935073,
        0.00066885432718430675,0.00078505003013483422,0.0,0.0,1.0,0.0,0.0,0.0,0.0,-0.0,-0.0,-1.0,-0.0,-0.0,-0.0,
        -0.0,0.013814947892318402,-0.0005902592207076454,-0.00070514735512079263,-0.0078505627081109815,
        0.00045921295820314543,0.0,0.0,1.0,0.0,0.0,-1.0,-0.0,-0.0,-0.0,-0.0,-0.0,0.015696416044310803,
        0.01381496727933039,-0.00078505003013483454,-0.0078505504957846247,0.00059026517985183728,0.0,0.0,1.0,0.0,
        0.0,0.0,0.0,-0.0,-0.0,-1.0,-0.0,-0.0,-0.0,-0.0,0.0007408652531395556,-0.010053942411719023,
        -0.019674701485866784,-0.00059047175686875969,-0.00045939812049741193,0.018049321508312247,0.0,1.0,0.0,0.0,
        0.0,-0.0,-0.0,-1.0,-0.0,-0.0,-0.0,-0.0,0.00074050995988770782,0.00078505003013483476,-0.013814967279330386,
        -0.00059026517985183717,0.007850550495784623,0.0,0.0,1.0,0.0,0.0,0.0,0.0,-0.0,-0.0,-1.0,-0.0,-0.0,-0.0,-0.0,
        0.016360391103343887,-0.00058935142225332465,-0.000703228026584666,-0.013814947892318404,
        0.00045716567186516885,0.0,0.0,1.0,0.0,0.0,-1.0,-0.0,-0.0,-0.0,-0.0,-0.0,-0.00066772991164514874,
        -0.00064115033886434018,-0.01381495313599773,0.00013071479116047655,-0.00058935731463155463,
        -0.010053939720042825,0.0,0.0,1.0,0.0,0.0,0.0,0.0,-0.0,-0.0,-1.0,-0.0,-0.0,-0.0,-0.0,-0.0,
        0.016360422411734077,-0.00078356528008410322,-0.010053938852608935,-0.013814967279330383,
        0.00058935731463155474,0.0,0.0,1.0,0.0,0.0,0.0,0.0,-0.0,-0.0,-1.0,-0.0,-0.0,-0.0,-0.0,
        0.00072155339410677672,-0.010053942472644626,-0.019674802040209542,-0.00078538438365502385,
        0.018049442230007151,0.0,0.0,1.0,0.0,0.0,0.0,0.0,-0.0,-0.0,-1.0,-0.0,-0.0,-0.0,-0.0,0.0007211912583486484,
        -0.01381502873718145,-0.00078505003013483443,0.0078505344125935073,0.0,0.0,1.0,0.0,0.0,0.0,0.0,-0.0,-0.0,
        -1.0,-0.0,-0.0,-0.0,-0.0,-0.010053959431077376,-0.00071029983670461863,-0.019674776790317688,
        -0.0078505558783549187,0.00070606688480528491,0.00064403085718071711,0.0,0.0,1.0,0.0,0.0,0.0,0.0,-0.0,-0.0,
        -1.0,-0.0,-0.0,-0.0,-0.0,-0.0,-0.0,-0.013354829801521528,-0.00066787723649602794,-0.00064128274259411312,
        0.019136117134310814,0.00082836908801823649,0.019674650101301497,0.0,1.0,0.0,0.0,0.0,0.0,-0.0,-0.0,-1.0,
        -0.0,-0.0,-0.0,-0.0,-0.0,-0.019136279086506527,-0.0078505344125935073,-0.018049442230007113,
        -0.00072200639376403209,0.00078577738649557045,0.0,0.0,1.0,0.0,0.0,0.0,-0.0,-0.0,-1.0,-0.0,-0.0,-0.0,-0.0,
        -0.0,-0.0,-0.010053942411719021,-0.0007408652531395556,-0.019674701485866787,0.00059047175686876,
        0.018049321508312247,0.00045939812049741166,0.0,1.0,0.0,0.0,-0.0,-1.0,-0.0,-0.0,-0.0,-0.0,
        -0.01335483887448634,-0.00078374994311405,0.00058948103625439325,0.019136152968431349,0.019674684401114268,
        0.0,0.0,1.0,0.0,0.0,0.0,0.0,-0.0,-0.0,-1.0,-0.0,-0.0,-0.0,-0.0,-0.0,-0.010053942472644626,
        -0.019674802040209546,-0.00072155339410677683,0.00066911306678242447,0.018049442230007123,
        0.00078538438365502352,0.0,1.0,0.0,0.0,0.0,-0.0,-0.0,-1.0,-0.0,-0.0,-0.0,-0.0,-0.00070998479812853861,
        -0.013815029502340641,0.007850555878354917,0.000705147355120792,0.00064310201354924451,0.0,0.0,1.0,0.0,0.0,
        0.0,0.0,-0.0,-0.0,-1.0,-0.0,-0.0,-0.0,-0.0,-0.0,-0.00066869452258176915,-0.015696395242494905,
        -0.00064281278721221348,0.0078498388863461367,0.00082974490333613884,0.021266503270189141,0.0,0.0,0.0,0.0,
        -0.0,-1.0,-0.0,-0.0,-0.0,-0.0,-0.00058545773453366594,-3.5950544673529394E-6,-0.013354818196216901,
        -0.015696374407663447,-0.016360377230620737,0.013354818196216901,0.015696374407663447,0.016360377230620737,
        0.0,0.0,1.0,0.0,0.0,0.0,0.0,0.0,-0.0,-0.0,-1.0,-0.0,-0.0,-0.0,-0.0,-0.0,-0.0,-0.013814978346247541,
        -0.00074050995988770782,0.0078505513076336225,0.00059025922070764572,0.00045900348534281133,0.0,0.0,1.0,0.0,
        0.0,0.0,-0.0,-0.0,-1.0,-0.0,-0.0,-0.0,-0.0,-0.015696416044310803,-0.00078483961287594765,
        0.0078498304624371948,0.00059013581334217821,0.021266532224969107,0.0,0.0,1.0,0.0,0.0,0.0,-0.0,-0.0,-1.0,
        -0.0,-0.0,-0.0,-0.0,-0.00078356528008410354,-0.016360422411734073,0.010053938852608933,
        0.00058935731463155463,0.013814967279330381,0.0,0.0,1.0,0.0,0.0,0.0,-0.0,-0.0,-1.0,-0.0,-0.0,-0.0,-0.0,-0.0,
        0.013354818196216903,0.00058948103625439347,0.0004572150890914036,-0.01913608552846445,0.0,0.0,1.0,0.0,0.0,
        0.0,0.0,0.0,0.0,-0.0,-0.0,-1.0,-0.0,-0.0,-0.0,-0.0,0.007850555878354917,4.72166684662135E-5,
        -0.00071067908889347968,0.00070606688480528491,0.00064403085718071711,0.0,0.0,1.0,0.0,0.0,0.0,0.0,0.0,0.0,
        -0.0,-0.0,-1.0,-0.0,-0.0,-0.0,-0.0,0.0078505513076336155,0.021264344306911508,-0.00074130273940990277,
        0.00059070966910656445,0.00045995981458200994,0.0,0.0,1.0,0.0,0.0,0.0,-0.0,-1.0,-0.0,-0.0,-0.0,
        0.019136104037587285,-0.00070578661505656148,0.0078505627081109728,-0.00059070966910656456,
        -4.6667541046249082E-6,0.00046016924547737027,0.0,0.0,1.0,0.0,0.0,-1.0,-0.0,-0.0,-0.0,-0.0,-0.0,
        0.010053938852608935,0.019674684401114268,-0.00078538438365502331,0.0078505504957846282,
        -7.1576985742576693E-6,0.00059071565881779026,0.0,0.0,1.0,0.0,0.0,0.0,0.0,0.0,-0.0,-0.0,-1.0,-0.0,-0.0,-0.0,
        -0.0,0.013354818196216903,-0.00058948103625439347,-0.00082836908801823736,-0.01913608552846445,
        -0.019674620847241392,0.0,0.0,1.0,0.0,0.0,0.0,0.0,-0.0,-0.0,-1.0,-0.0,-0.0,-0.0,-0.0,-0.0,-0.0,
        0.0078498304624371861,0.019136152968431349,-0.00078556684097776574,-0.021264331757721504,
        0.00059058621231803418,0.0,0.0,1.0,0.0,0.0,0.0,0.0,-0.0,-0.0,-1.0,-0.0,-0.0,-0.0,0.013814947892318409,
        0.0007051473551207923,0.0212664940442422,0.0005902651798518375,4.7206293852370952E-5,-0.007850561894963819,
        0.0,0.0,1.0,0.0,0.0,0.0,0.0,0.0,0.0,-0.0,-0.0,-1.0,-0.0,-0.0,-0.0,0.00059025922070764572,
        0.00070514735512079241,-0.013814947892318418,-0.00045921295820314608,0.0078505627081109711,0.0,0.0,1.0,0.0,
        0.0,0.0,0.0,-0.0,-0.0,-1.0,-0.0,-0.0,-0.0,1.0250173309722677E-6,0.0,-0.0,0.00059070966910656467,
        -0.0078505627081109745,-7.8752164488168983E-5,0.0,0.0,1.0,0.0,0.0,0.0,0.0,-0.0,-0.0,-1.0,-0.0,-0.0,-0.0,
        -0.0,0.00059026517985183772,1.0228783844071197E-6,-0.00012539822612430226,0.0078505618949638225,0.0,0.0,1.0,
        0.0,0.0,0.0,0.0,0.0,-0.0,-0.0,-1.0,-0.0,-0.0,-0.0,-0.0,0.00071067908889347979,-0.0078505558783549152,
        -7.8751758300344045E-5,-0.00070606688480528469,-0.00064403085718071711,0.0,0.0,1.0,0.0,0.0,0.0,0.0,-0.0,
        -0.0,-1.0,-0.0,-0.0,-0.0,-0.0,-0.0,-0.0,-0.00066885432718430643,-0.000643102013549245,-0.0078505589212312,
        0.00012539822612430221,-0.00059026517985183706,0.0,0.0,1.0,0.0,0.0,0.0,0.0,-0.0,-0.0,-1.0,-0.0,-0.0,-0.0,
        -0.0,-0.0,0.00045939812049741,-0.010053938852608933,-0.019674684401114268,-0.00059047772800183325,
        7.1576985742576753E-6,1.0242094517058098E-6,-0.00785055049578463,0.0,0.0,1.0,0.0,0.0,0.0,0.0,-0.0,-0.0,-1.0,
        -0.0,-0.0,-0.0,-0.0,-0.0,0.00074130273940990277,-0.00785055130763362,-0.018049321508312233,
        -0.00059070966910656445,-0.00045995981458201091,0.0,0.0,1.0,0.0,0.0,0.0,-0.0,-0.0,-1.0,-0.0,-0.0,-0.0,-0.0,
        -0.0,0.00072200639376403209,-0.007850534412593509,-0.018049442230007113,-0.00078577738649557056,0.0,0.0,1.0,
        0.0,0.0,0.0,0.0,-0.0,-0.0,-1.0,-0.0,-0.0,-0.0,-0.0,-0.0,-0.010053941700689279,-0.00066911306678242458,
        -0.019674650101301497,-0.00064350274257291972,0.018049261985986123,0.00083041340795978814,1.0,0.0,0.0,0.0,
        -0.0,-0.0,-1.0,-0.0,-0.0,-0.0,-0.0,-0.0,-0.013354818196216903,-0.00058948103625439347,
        -0.00082836908801823736,0.01913608552846445,0.019674620847241395,0.0,0.0,1.0,0.0,0.0,0.0,0.0,-0.0,-0.0,-1.0,
        -0.0,-0.0,-0.0,-0.0,-0.0,-0.0,-0.00074130273940990277,-0.0,-0.0078498304624371861,-0.019136152968431349,
        -0.00078556684097776574,0.00059058621231803418,0.0,0.0,1.0,0.0,0.0,0.0,-0.0,-0.0,-1.0,-0.0,-0.0,-0.0,-0.0,
        -0.0,-0.010053938852608928,-0.00078538438365502374,-0.019674684401114275,0.00059047772800183335,
        0.018049300450950378,0.0,1.0,0.0,0.0,0.0,-0.0,-0.0,-1.0,-0.0,-0.0,-0.0,-0.0,-0.015696374407663447,
        -0.0005902651798518375,-0.00012539822612430229,-1.0228783844071214E-6,0.007850561894963819,0.0,0.0,1.0,0.0,
        0.0,0.0,-0.0,-0.0,-1.0,-0.0,-0.0,-0.0,-0.0,-0.0,-0.0,-0.000589357314631555,-3.6300677219671527E-6,
        -0.00013071479116047663,0.01005393972004282,0.013814936811065819,0.0,0.0,1.0,0.0,0.0,0.0,-0.0,-0.0,-1.0,
        -0.0,-0.0,-0.0,-0.0,-0.0,-0.0,-0.013814967279330381,-0.00078505003013483476,-0.021266532224969107,
        -0.00045900348534281117,0.0078505504957846247,0.00059026517985183739,0.0,0.0,1.0,0.0,0.0,0.0,-0.0,-0.0,-1.0,
        -0.0,-0.0,-0.0,-0.0,-0.0,0.0078498418577679363,0.00059058621231803429,0.00012594643379194981,
        1.0243116170212105E-6,-0.021264280982048623,0.0,0.0,1.0,0.0,0.0,0.0,0.0,0.0,0.0,-0.0,-0.0,-1.0,-0.0,-0.0,
        -0.0,0.007850558921231196,-2.8452679316136533E-6,0.0008309073466565292,0.0,0.0,1.0,0.0,0.0,0.0,0.0,0.0,0.0,
        -0.0,-0.0,-1.0,-0.0,-0.0,-0.0,-0.0,0.0078498418577679328,-3.6410799041126835E-6,7.8752197135979057E-5,
        -0.00059071565881779048,-3.6422315821786528E-6,0.0,0.0,1.0,0.0,0.0,0.0,0.0,0.0,-0.0,-0.0,-1.0,-0.0,-0.0,
        -0.0,-0.0,-0.0,0.01005393972004282,8.6574413715050772E-5,-0.00059047772800183325,-0.018049225981178776,0.0,
        0.0,1.0,0.0,0.0,0.0,0.0,-0.0,-0.0,-1.0,-0.0,-0.0,-0.0,-0.0,-0.0,-0.01005393972004282,
        -0.00059047772800183325,-3.6400546269338619E-6,-8.6574413715050745E-5,0.018049225981178765,0.0,1.0,0.0,0.0,
        0.0,-0.0,-0.0,-1.0,-0.0,-0.0,-0.0,-0.0,-0.0,-0.0078498418577679363,-0.00012594643379194981,
        -0.00059071565881779048,-1.0250173309722696E-6,0.0,0.0,1.0,0.0,0.0,0.0,-0.0,-0.0,-1.0,-0.0,-0.0,-0.0,-0.0,
        -0.0,-0.0,-0.0,0.00785056189496382,0.00059071565881779048,4.721686715653703E-5,1.0250173309722696E-6,0.0,
        0.0,1.0,0.0,0.0,0.0,0.0,0.0,0.0,0.0,-0.0,-0.0,-1.0,-0.0,-0.0,-0.0,-0.002139599215214946,
        -0.023117048152407872,-0.0022397649528431126,-0.027072995129471072,-0.0021836277363616002,
        -0.028166145144496873,0.002139599215214946,0.023117048152407872,0.0022397649528431126,0.027072995129471072,
        0.0021836277363616007,0.028166145144496869,0.0,0.0,0.0,1.0,0.0,0.0,0.0,0.0,0.0,0.0,-0.0,-0.0,-0.0,-1.0,-0.0,
        -0.0,-0.0,-0.0,0.0021395992152149455,-0.023117145095115522,-0.0021497242199081533,-0.027072819798329567,
        -0.0019633569630565072,-0.02816590468451018,0.023117145095115522,0.027072819798329567,0.028165904684510173,
        0.0,0.0,0.0,1.0,0.0,0.0,0.0,0.0,0.0,-0.0,-0.0,-0.0,-1.0,-0.0,-0.0,-0.0,-0.0,0.023117048152407872,
        -0.0021505378228925251,-0.0022518711100377505,-0.032822477959688887,-0.00219585787232726,
        -0.0336642766045134,0.0021505378228925251,0.0022518711100377505,0.0021958578723272597,0.0,0.0,0.0,1.0,0.0,
        0.0,0.0,0.0,0.0,-0.0,-0.0,-0.0,-1.0,-0.0,-0.0,-0.0,-0.0,0.0022397649528431126,0.023117136629619534,
        0.028165879272568334,0.002368167038278622,-0.0017636731113387088,-0.023117134816530223,
        -0.027072790466377776,-0.028165871707620763,0.027072790466377776,0.0,0.0,0.0,1.0,0.0,0.0,0.0,0.0,0.0,-0.0,
        -0.0,-0.0,-1.0,-0.0,-0.0,-0.0,0.027072995129471072,0.0021528281310241241,0.0021984476162807444,
        0.023967033731365443,-0.0021532798422932995,-0.013757776970334581,-0.0022549381705200254,
        -0.002198962690806161,0.0,0.0,0.0,1.0,0.0,0.0,0.0,0.0,0.0,-0.0,-0.0,-0.0,-1.0,-0.0,-0.0,-0.0,
        0.0021836277363616002,-0.0020059903769841761,-0.023117107076915992,-0.0023681670382786246,
        -0.027072827080784432,-0.028165923858112191,0.023117107076915992,0.027072827080784432,0.028165923858112184,
        0.0,0.0,0.0,1.0,0.0,0.0,0.0,0.0,0.0,-0.0,-0.0,-0.0,-1.0,-0.0,-0.0,-0.0,0.028166145144496876,
        -0.0021508629271109274,-0.017539733206627071,-0.0022522704855525342,-0.023967033731365443,
        -0.0021962714305260589,0.0021508629271109274,0.0022522704855525342,0.0021962714305260593,0.0,0.0,0.0,1.0,
        0.0,0.0,0.0,0.0,0.0,-0.0,-0.0,-0.0,-1.0,-0.0,-0.0,-0.0,-0.0021395992152149455,-0.023117145095115522,
        -0.027072819798329567,-0.02816590468451018,0.023117145095115522,0.0021497242199081533,0.027072819798329567,
        0.0019633569630565077,0.028165904684510173,0.0,0.0,0.0,1.0,0.0,0.0,0.0,0.0,0.0,-0.0,-0.0,-0.0,-1.0,-0.0,
        -0.0,-0.0,-0.0,-0.023117048152407872,-0.0021505378228925251,-0.0022518711100377505,-0.00219585787232726,
        0.0021505378228925251,0.0022518711100377505,0.032822477959688887,0.0021958578723272597,0.033664276604513384,
        0.0,0.0,0.0,1.0,0.0,0.0,0.0,0.0,0.0,-0.0,-0.0,-0.0,-1.0,-0.0,-0.0,-0.0,-0.0,-0.0022397649528431126,
        -0.0023681670382786225,-0.023117134816530223,-0.027072790466377776,-0.028165871707620763,
        0.0017636731113387079,0.023117134816530223,0.028165871707620756,0.0,0.0,0.0,1.0,0.0,0.0,0.0,0.0,-0.0,-0.0,
        -0.0,-1.0,-0.0,-0.0,-0.0,-0.0,-0.027072995129471072,-0.0021528281310241241,-0.0021984476162807444,
        -0.023967033731365456,-0.0022549381705200254,0.0021532798422932995,0.013757776970334581,
        0.0022549381705200254,0.0021989626908061606,0.0,0.0,0.0,1.0,0.0,0.0,0.0,0.0,-0.0,-0.0,-0.0,-1.0,-0.0,-0.0,
        -0.0,-0.0,-0.0021836277363616007,-0.023117107076915992,-0.027072827080784432,-0.028165923858112191,
        0.0020059903769841761,0.023117107076915992,0.0023681670382786238,0.027072827080784432,0.028165923858112184,
        0.0,0.0,0.0,1.0,0.0,0.0,0.0,0.0,-0.0,-0.0,-0.0,-1.0,-0.0,-0.0,-0.0,-0.0,-0.028166145144496869,
        -0.0021508629271109274,-0.0022522704855525342,-0.0021962714305260589,0.0021508629271109274,
        0.017539733206627078,0.0022522704855525342,0.023967033731365467,0.0021962714305260593,0.0,0.0,0.0,1.0,0.0,
        0.0,0.0,0.0,-0.0,-0.0,-0.0,-1.0,-0.0,-0.0,-0.0,-0.0,0.0021505378228925246,0.023117145095115525,
        -0.0021629274560676956,-0.032821849572960068,-0.0019763195483343526,-0.033663644953626663,0.0,0.0,0.0,1.0,
        0.0,0.0,0.0,0.0,-0.0,-0.0,-0.0,-1.0,-0.0,-0.0,-0.0,-0.0,0.0021497242199081537,0.0017636731113387075,
        0.0025248548165844459,-0.023117153652107741,-0.027072767990336359,-0.028165839066171924,
        0.023117153652107741,0.027072767990336359,0.028165839066171917,0.0,0.0,0.0,1.0,0.0,0.0,0.0,0.0,0.0,0.0,-0.0,
        -0.0,-0.0,-1.0,-0.0,-0.0,-0.0,0.0021528281310241237,-0.013756932403821471,-0.03615897334115932,-0.0,
        0.0017730752489912573,0.027072767990336356,-0.036158836489428262,0.0,0.0,0.0,1.0,0.0,0.0,0.0,0.0,-0.0,-0.0,
        -0.0,-1.0,-0.0,-0.0,0.0020059903769841761,0.0019633569630565068,-0.023117148094275803,
        -0.0025248548165844454,0.028165850749951267,0.0,0.0,0.0,1.0,0.0,0.0,0.0,0.0,-0.0,-0.0,-0.0,-1.0,-0.0,-0.0,
        -0.0,0.0021508629271109274,-0.023967031267238804,-0.0,0.0017716448391260384,0.028165839066171927,0.0,0.0,
        0.0,1.0,0.0,0.0,0.0,0.0,0.0,-0.0,-0.0,-0.0,-1.0,-0.0,-0.0,0.0021505378228925246,-0.023117145095115525,-0.0,
        0.0017714658173675476,-0.0014235573934133095,0.033663511042732373,0.0,0.0,0.0,1.0,0.0,0.0,0.0,0.0,-0.0,-0.0,
        -0.0,-1.0,-0.0,-0.0,-0.0,0.0021528281310241237,-0.027072819798329564,-0.0021657727568646559,
        0.013756932403821471,0.036158973341159265,0.0,0.0,0.0,0.0,0.0,0.0,-0.0,-0.0,-0.0,-1.0,-0.0,-0.0,-0.0,
        0.0021508629271109274,-0.028165904684510176,-0.0021634485653239869,-0.0019768379174131762,
        0.017540054199611115,0.023967031267238814,0.0,0.0,0.0,1.0,0.0,0.0,0.0,-0.0,-0.0,-0.0,-1.0,-0.0,-0.0,-0.0,
        -0.0,0.023117136629619537,0.0022556280308783936,0.013758173064519321,-0.0017741542886565819,
        -0.0014273157197953927,0.0,0.0,0.0,1.0,0.0,0.0,0.0,0.0,-0.0,-0.0,-0.0,-1.0,-0.0,-0.0,0.013756545225322915,
        0.032822477959688887,-0.0021539160439461116,-0.002255628030878394,-0.0021996560033501643,
        -0.036155994182829158,0.0021539160439461116,0.002255628030878394,0.0021996560033501647,0.0,0.0,0.0,1.0,0.0,
        0.0,0.0,0.0,-0.0,-0.0,-0.0,-1.0,-0.0,-0.0,0.023117107076915996,0.0021958578723272597,-0.0020152870120824654,
        -0.0023798449910123255,-0.032821938754042893,0.0,0.0,0.0,1.0,0.0,0.0,0.0,0.0,-0.0,-0.0,-0.0,-1.0,-0.0,-0.0,
        -0.0,0.017539733206627082,0.0336642766045134,-0.00219941213896084,0.00215368729603372,0.0022553827543743792,
        0.00219941213896084,0.0,0.0,0.0,1.0,0.0,0.0,0.0,0.0,0.0,0.0,-0.0,-0.0,-0.0,-1.0,-0.0,-0.0,-0.0,
        0.023117145095115518,-0.0021505378228925251,-0.032821849572960082,0.0021629274560676964,
        0.0019763195483343534,0.0,0.0,0.0,1.0,0.0,0.0,0.0,0.0,-0.0,-0.0,-0.0,-1.0,-0.0,-0.0,-0.0,-0.0,
        0.023117136629619537,-0.00225187111003775,-0.032821807333186945,0.0017714658173675487,0.0014229487589399608,
        0.0,0.0,0.0,1.0,0.0,0.0,0.0,-0.0,-0.0,-0.0,-1.0,-0.0,-0.0,-0.0,0.023117107076915996,-0.0021958578723272597,
        -0.032821938754042893,-0.033663737674327086,0.0020152870120824654,0.0023798449910123263,0.0,0.0,0.0,1.0,0.0,
        0.0,0.0,-0.0,-0.0,-0.0,-1.0,-0.0,-0.0,-0.0,-0.0,0.0022544308843389775,0.027072797014430487,
        0.0023823041653880553,0.023967015852373385,-0.0017733843081747245,-0.013758177150392206,0.0,0.0,0.0,1.0,0.0,
        0.0,0.0,0.0,-0.0,-0.0,-0.0,-1.0,-0.0,-0.0,0.0022522704855525342,0.028165879272568337,0.0023802034757232954,
        -0.0017716448391260397,-0.023967012140249259,0.0,0.0,0.0,1.0,0.0,0.0,0.0,0.0,-0.0,-0.0,-0.0,-1.0,-0.0,-0.0,
        0.0022518711100377505,0.03366360485977575,0.0023798449910123263,-0.023117134816530216,
        -0.0017714855698833817,0.032821793825602318,0.0,0.0,0.0,1.0,0.0,0.0,0.0,0.0,-0.0,-0.0,-0.0,-1.0,-0.0,-0.0,
        -0.0,0.0023823041653880553,-0.027072790466377783,-0.0017730752489912573,0.01375694528625826,
        0.036158931786919049,0.0,0.0,0.0,0.0,0.0,-0.0,-0.0,-1.0,-0.0,-0.0,0.027072827080784432,
        0.0021984476162807444,0.023967007687598831,-0.013758082261467377,-0.0023827866608640042,0.0,0.0,0.0,1.0,0.0,
        0.0,0.0,0.0,-0.0,-0.0,-0.0,-1.0,-0.0,-0.0,0.027072819798329564,0.0019791101348432538,0.0239670312672388,
        -0.0021532798422932995,-0.013758164253474777,0.0021663421034936255,0.0,0.0,0.0,1.0,0.0,0.0,0.0,0.0,-0.0,
        -0.0,-0.0,-1.0,-0.0,-0.0,-0.0,0.02707279701443048,0.023967015852373378,-0.0022549381705200249,
        -0.013758173064519324,0.0017733644650094233,0.001426115796022355,0.0,0.0,1.0,0.0,0.0,-0.0,-0.0,-1.0,-0.0,
        -0.0,0.027072827080784432,0.0020172069825707454,0.0023823041653880544,0.023967007687598831,
        -0.00219896269080616,-0.013758082261467377,0.0,0.0,0.0,1.0,0.0,0.0,0.0,-0.0,-0.0,-0.0,-1.0,-0.0,-0.0,-0.0,
        0.0021962714305260589,0.028165923858112184,-0.0023802034757232967,-0.023967007687598837,0.0,0.0,0.0,1.0,0.0,
        0.0,0.0,0.0,-0.0,-0.0,-0.0,-1.0,-0.0,-0.0,0.0021958578723272597,-0.023117107076915992,
        -0.0023798449910123281,0.032821938754042886,0.033663737674327066,0.0,0.0,0.0,1.0,0.0,0.0,0.0,0.0,-0.0,-0.0,
        -0.0,-1.0,-0.0,-0.0,-0.0,0.002198447616280744,-0.027072827080784435,-0.0023823041653880561,
        0.013756850421972387,0.036159076531973151,0.0,0.0,0.0,0.0,0.0,-0.0,-0.0,-1.0,-0.0,-0.0,
        0.0021962714305260589,-0.028165923858112181,-0.0020155176559669297,-0.0023802034757232967,
        0.017539980122310408,0.023967007687598862,0.0,0.0,0.0,1.0,0.0,0.0,0.0,-0.0,-0.0,-0.0,-1.0,-0.0,-0.0,-0.0,
        0.02816590468451018,-0.0021508629271109274,-0.023967031267238807,0.0021634485653239869,
        0.0019768379174131758,0.0,0.0,0.0,1.0,0.0,0.0,0.0,0.0,-0.0,-0.0,-0.0,-1.0,-0.0,-0.0,-0.0,
        0.028165879272568337,-0.0022522704855525342,-0.023967015852373392,0.0017716250685312594,
        0.0014234593859236441,0.0,0.0,1.0,0.0,0.0,-0.0,-0.0,-1.0,-0.0,-0.0,0.028165923858112191,
        -0.0021962714305260589,-0.023967007687598817,0.0020155176559669297,0.0023802034757232963,0.0,0.0,0.0,1.0,
        0.0,0.0,0.0,-0.0,-0.0,-0.0,-1.0,-0.0,-0.0,-0.0,-0.0021505378228925246,-0.023117145095115525,
        0.0021629274560676956,0.032821849572960068,0.001976319548334353,0.033663644953626656,0.0,0.0,0.0,1.0,0.0,
        0.0,0.0,0.0,-0.0,-0.0,-0.0,-1.0,-0.0,-0.0,-0.0,-0.0,-0.0017636536977724872,-0.0021497242199081537,
        -0.023117155475339022,0.0014113188375514472,0.028165846654428471,0.0,0.0,0.0,1.0,0.0,0.0,0.0,-0.0,-0.0,-0.0,
        -1.0,-0.0,-0.0,-0.0,-0.0,-0.0021528281310241237,-0.027072819798329564,0.013756932403821471,
        0.0021657727568646559,0.0019791101348432556,0.036158973341159265,0.0,0.0,0.0,0.0,0.0,-0.0,-0.0,-1.0,-0.0,
        -0.0,-0.0,-0.0020059903769841757,-0.0019633569630565077,-0.0017636731113387079,-0.0014113188375514463,
        -0.023117153652107741,-0.027072767990336359,-0.028165839066171924,0.023117153652107741,0.028165839066171917,
        0.0,0.0,0.0,1.0,0.0,0.0,0.0,0.0,-0.0,-0.0,-0.0,-1.0,-0.0,-0.0,-0.0,-0.0,-0.0,-0.0021508629271109274,
        -0.028165904684510176,0.017540054199611115,0.0021634485653239869,0.023967031267238814,0.0019768379174131762,
        0.0,0.0,0.0,1.0,0.0,0.0,0.0,-0.0,-0.0,-0.0,-1.0,-0.0,-0.0,-0.0,-0.0,-0.023117136629619537,
        -0.00225187111003775,0.0017714658173675487,0.032821807333186945,0.0014229487589399608,0.033663604859775743,
        0.0,0.0,1.0,0.0,0.0,-0.0,-0.0,-1.0,-0.0,-0.0,-0.0,-0.013756545225322915,-0.032822477959688887,
        -0.0021539160439461116,-0.002255628030878394,-0.0021996560033501643,0.0021539160439461116,
        0.002255628030878394,0.0021996560033501647,0.036155994182829096,0.0,0.0,0.0,0.0,0.0,0.0,-0.0,-0.0,-0.0,-1.0,
        -0.0,-0.0,-0.0,-0.0,-0.023117107076915996,-0.0021958578723272597,0.0020152870120824654,
        0.0023798449910123263,0.032821938754042893,0.033663737674327072,0.0,0.0,0.0,1.0,0.0,0.0,0.0,-0.0,-0.0,-0.0,
        -1.0,-0.0,-0.0,-0.0,-0.0,-0.017539733206627085,-0.033664276604513384,-0.00219941213896084,
        0.00215368729603372,0.03112680478206669,0.0,0.0,0.0,1.0,0.0,0.0,0.0,-0.0,-0.0,-0.0,-1.0,-0.0,-0.0,-0.0,
        -0.0022544308843389775,-0.027072797014430487,0.0017730554216371041,0.013756941202814331,
        0.0014255752842010033,0.0361589433554084,0.0,0.0,0.0,0.0,-0.0,-1.0,-0.0,-0.0,-0.0022522704855525342,
        -0.0023802034757232954,-0.028165871707620752,0.00177164483912604,0.017540060210790732,0.023967012140249284,
        0.0,0.0,0.0,1.0,0.0,0.0,-0.0,-0.0,-0.0,-1.0,-0.0,-0.0,-0.0,-0.0,-0.027072827080784432,
        -0.0021984476162807448,0.0020172069825707454,0.013756850421972387,0.0023823041653880557,
        0.036159076531973207,0.0,0.0,0.0,1.0,0.0,0.0,-0.0,-0.0,-0.0,-1.0,-0.0,-0.0,-0.0,-0.0021962714305260593,
        -0.028165923858112181,0.0020155176559669297,0.017539980122310408,0.0023802034757232963,0.023967007687598862,
        0.0,0.0,0.0,1.0,0.0,0.0,-0.0,-0.0,-0.0,-1.0,-0.0,-0.0,-0.0,-0.0,0.0021670637484648039,0.0017738649457463914,
        0.013757007748269136,0.00021693526799154337,-0.036155235792572543,0.0,0.0,0.0,1.0,0.0,0.0,0.0,0.0,0.0,-0.0,
        -0.0,-0.0,-1.0,-0.0,-0.0,0.002153916043946112,0.013756932403821469,0.032821849572960068,
        -0.002167063748464803,-0.036155372747005976,0.0,0.0,0.0,1.0,0.0,0.0,-0.0,-0.0,-1.0,-0.0,-0.0,-0.0,
        0.002015287012082465,0.0019763195483343526,0.0017714855698833811,0.023117153652107737,-0.032821701216996041,
        0.0,0.0,0.0,1.0,0.0,0.0,0.0,0.0,0.0,-0.0,-0.0,-0.0,-1.0,-0.0,-0.0,-0.0,0.002153279842293299,
        -0.013758164253474777,-0.0,0.036158848104067796,0.0017733843081747236,0.00021831715113692992,
        8.0516212332184942E-5,0.0,0.0,0.0,1.0,0.0,0.0,0.0,0.0,0.0,-0.0,-0.0,-0.0,-1.0,-0.0,-0.0,
        0.0020155176559669297,0.0019768379174131766,0.0017716448391260384,0.0014240679527817289,
        -0.02816583906617192,0.017540113132327881,0.023967016586099663,0.0,0.0,0.0,1.0,0.0,0.0,0.0,0.0,-0.0,-0.0,
        -0.0,-1.0,-0.0,-0.0,-0.0,0.002153916043946112,-0.013756932403821469,-0.032821849572960068,
        -0.002167063748464803,0.036155372747005914,0.0,0.0,0.0,0.0,0.0,0.0,-0.0,-0.0,-0.0,-1.0,-0.0,-0.0,-0.0,-0.0,
        0.002153279842293299,-0.023967031267238814,-0.0021663421034936268,-0.0019796723009276795,
        0.013758164253474772,0.0,0.0,0.0,1.0,0.0,0.0,0.0,-0.0,-0.0,-0.0,-1.0,-0.0,-0.0,-0.0,-0.0,
        0.023117134816530216,0.0023798449910123268,0.0014229487589399567,-0.001771485569883382,
        -0.032821793825602304,0.0,0.0,0.0,1.0,0.0,0.0,0.0,0.0,-0.0,-0.0,-0.0,-1.0,-0.0,-0.0,-0.0,
        0.032821938754042893,0.0021996560033501643,0.013758082261467375,-0.00238394443966586,0.0,0.0,0.0,1.0,0.0,
        0.0,0.0,0.0,0.0,-0.0,-0.0,-0.0,-1.0,-0.0,-0.0,0.013757776970334586,8.0531054257304872E-5,
        -0.0021543679790237634,-0.0022561355647809592,-0.002200171328627197,0.0021543679790237634,
        0.0022561355647809592,0.002200171328627197,0.0,0.0,0.0,1.0,0.0,0.0,0.0,0.0,0.0,0.0,-0.0,-0.0,-0.0,-1.0,-0.0,
        -0.0,-0.0,0.032821849572960062,0.0019803784157214573,0.013758164253474772,-0.0021543679790237639,
        0.0021676333667632283,0.0,0.0,0.0,1.0,0.0,0.0,0.0,0.0,0.0,-0.0,-0.0,-0.0,-1.0,-0.0,-0.0,-0.0,
        0.032821807333186952,0.013758173064519319,-0.0022561355647809588,0.0017741542886565826,
        0.0014273157197953908,0.0,0.0,1.0,0.0,0.0,0.0,-0.0,-0.0,-1.0,-0.0,-0.0,0.013756850421972394,
        0.032821938754042893,-0.0021996560033501647,-0.036155475949002973,0.0020181389031338108,
        0.0023834617064148775,0.0,0.0,0.0,1.0,0.0,0.0,0.0,-0.0,-0.0,-0.0,-1.0,-0.0,-0.0,0.013758082261467373,
        8.05337557427544E-5,-1.7578747218645929E-5,0.0020185138829726234,0.0023839444396658582,0.0,0.0,0.0,1.0,0.0,
        0.0,0.0,0.0,-0.0,-0.0,-0.0,-1.0,-0.0,-0.0,-0.0,0.023117155475339025,-0.0017714658173675481,
        -0.0021629274560676964,0.0014235573934133154,0.0,0.0,0.0,1.0,0.0,0.0,0.0,-0.0,-0.0,-0.0,-1.0,-0.0,-0.0,-0.0,
        -0.0,0.023117148094275806,0.013756987718843332,-0.0020181389031338121,-0.0019803784157214573,
        -0.036155266228744543,0.0025428266645309921,0.0,0.0,1.0,0.0,0.0,0.0,-0.0,-0.0,-0.0,-1.0,-0.0,-0.0,-0.0,
        0.023117134816530216,-0.0023798449910123259,-0.032821793825602304,-0.033663591643505526,
        0.0017714855698833828,0.0,0.0,0.0,1.0,0.0,0.0,0.0,-0.0,-0.0,-0.0,-1.0,-0.0,-0.0,-0.0,-0.0,
        0.0023802034757232954,0.0014234593859236444,-0.028165871707620752,-0.0017716448391260397,
        0.017540060210790732,0.023967012140249284,0.0,0.0,0.0,1.0,0.0,0.0,0.0,-0.0,-0.0,-0.0,-1.0,-0.0,-0.0,-0.0,
        0.0023834617064148788,-0.01375694528625827,-0.032821793825602311,-0.0017738649457463916,0.03615533112817032,
        0.0,0.0,0.0,0.0,0.0,-0.0,-1.0,-0.0,-0.0,-0.0,-0.0,0.0022549381705200249,0.0023827866608640046,
        -0.02396701214024928,-0.0017733843081747234,0.0137581771503922,0.0,0.0,0.0,1.0,0.0,0.0,0.0,-0.0,-0.0,-0.0,
        -1.0,-0.0,-0.0,-0.0,0.027072776376697909,-0.0020172069825707458,-0.0019791101348432543,
        -0.013756987718843334,-0.036158866905630971,0.0025414906519322343,0.0,0.0,1.0,0.0,0.0,-0.0,-0.0,-0.0,-1.0,
        -0.0,-0.0,-0.0,0.027072790466377776,0.023967012140249266,-0.0023827866608640033,-0.013758177150392204,
        0.0017733843081747238,0.0,0.0,0.0,1.0,0.0,0.0,0.0,-0.0,-0.0,-0.0,-1.0,-0.0,-0.0,-0.0,0.0021996560033501638,
        -0.013756850421972376,-0.032821938754042906,-0.0023834617064148788,0.036155475949002897,0.0,0.0,0.0,0.0,0.0,
        -0.0,-1.0,-0.0,-0.0,-0.0,-0.0,-0.0175399801223104,-0.033663737674327059,-0.0023832147743805109,
        1.7578747218645923E-5,-0.013758082261467368,-0.002018513882972623,0.0,0.0,0.0,1.0,0.0,0.0,0.0,-0.0,-0.0,
        -0.0,-1.0,-0.0,-0.0,-0.0,-0.0,0.00219896269080616,-0.023967007687598848,-0.0020175817725937989,
        -0.0023827866608640037,0.013758082261467373,0.0,0.0,0.0,1.0,0.0,0.0,0.0,-0.0,-0.0,-0.0,-1.0,-0.0,-0.0,-0.0,
        0.02816585074995127,-0.0020155176559669297,-0.0019768379174131762,-0.023967016242290962,
        0.0025390630631617036,0.0,0.0,0.0,1.0,0.0,0.0,0.0,-0.0,-0.0,-0.0,-1.0,-0.0,-0.0,-0.0,0.028165871707620759,
        -0.0023802034757232963,-0.023967012140249263,0.0017716448391260375,0.0,0.0,0.0,1.0,0.0,0.0,0.0,-0.0,-0.0,
        -0.0,-1.0,-0.0,-0.0,-0.0,-0.002015287012082465,-0.023117148094275806,-0.0019763195483343526,
        -0.0017714855698833811,0.032821701216996041,0.0336634977860711,0.0,0.0,0.0,1.0,0.0,0.0,0.0,-0.0,-0.0,-0.0,
        -1.0,-0.0,-0.0,-0.0,-0.0,-0.0,-0.0021536872960337197,-0.017540054199611122,-0.033663644953626642,
        0.0021668136920060164,0.03112619259567026,0.0019801394547201774,0.0,0.0,1.0,0.0,0.0,0.0,-0.0,-0.0,-0.0,-1.0,
        -0.0,-0.0,-0.0,-0.0,-0.0021634485653239878,-0.0017716448391260386,-0.0025390630631616988,
        -0.02816583906617192,0.023967016586099663,0.0,0.0,0.0,1.0,0.0,0.0,-0.0,-0.0,-0.0,-1.0,-0.0,-0.0,-0.0,-0.0,
        -0.0,-0.0020172069825707454,-0.027072776376697909,-0.0019791101348432543,0.013756987718843336,
        0.0025414906519322382,0.036158866905630881,0.0,0.0,0.0,0.0,-0.0,-0.0,-1.0,-0.0,-0.0,-0.0,
        -0.002153279842293299,-0.023967031267238814,0.013758164253474772,0.0021663421034936268,0.00197967230092768,
        0.0,0.0,0.0,1.0,0.0,0.0,0.0,-0.0,-0.0,-0.0,-1.0,-0.0,-0.0,-0.0,-0.0,-0.0020155176559669297,
        -0.0019768379174131771,-0.02816585074995127,0.017540096325751132,0.0025390630631616997,0.023967016242290966,
        0.0,0.0,1.0,0.0,0.0,-0.0,-0.0,-0.0,-1.0,-0.0,-0.0,-0.0,-0.023117134816530216,-0.0023798449910123259,
        0.0017714855698833828,0.032821793825602304,0.033663591643505512,0.0,0.0,0.0,1.0,0.0,0.0,0.0,-0.0,-0.0,-0.0,
        -1.0,-0.0,-0.0,-0.0,-0.0,-0.017540057790927686,-0.0022553827543743796,-0.033663604859775743,
        0.0017736671849664688,0.031126147710011594,0.00142656920316686,0.0,1.0,0.0,0.0,-0.0,-0.0,-1.0,-0.0,-0.0,
        -0.0,-0.013757776970334586,-0.00013643209586666446,-0.0021543679790237634,-0.0022561355647809592,
        -0.002200171328627197,0.0021543679790237634,0.0022561355647809592,0.002200171328627197,0.0,0.0,0.0,1.0,0.0,
        0.0,0.0,0.0,-0.0,-0.0,-0.0,-1.0,-0.0,-0.0,-0.0,-0.0,-0.0,-0.0023823041653880544,-0.027072790466377773,
        0.0017730752489912573,0.013756945286258279,0.036158931786919229,0.0,0.0,0.0,1.0,0.0,0.0,-0.0,-0.0,-0.0,-1.0,
        -0.0,-0.0,-0.0,-0.0022549381705200249,-0.0239670158523734,0.0017733644650094235,0.013758173064519321,
        0.0014261157960223586,0.0,0.0,0.0,1.0,0.0,0.0,-0.0,-0.0,-0.0,-1.0,-0.0,-0.0,-0.0,-0.023967007687598844,
        -0.00219896269080616,0.0020175817725937989,0.013758082261467377,0.0023827866608640033,0.0,0.0,0.0,1.0,0.0,
        0.0,-0.0,-0.0,-0.0,-1.0,-0.0,-0.0,-0.0,-0.0,0.0021543679790237634,0.013758164253474772,0.03615537274700599,
        -0.0021676333667632296,0.0,0.0,0.0,1.0,0.0,0.0,0.0,0.0,0.0,-0.0,-0.0,-0.0,-1.0,-0.0,-0.0,-0.0,
        0.001771485569883382,3.1609473085406838E-6,-0.023117153652107744,0.032821701216996027,0.033663497786071091,
        0.0,0.0,0.0,1.0,0.0,0.0,0.0,0.0,0.0,-0.0,-0.0,-0.0,-1.0,-0.0,-0.0,-0.0,0.0017730752489912571,
        0.0014261840281970283,-0.027072767990336359,0.013757007748269138,0.036158836489428171,0.0,0.0,0.0,0.0,0.0,
        0.0,-0.0,-0.0,-1.0,-0.0,-0.0,0.0021670637484648039,-0.032821714763063607,0.0017738649457463914,
        -0.013757007748269151,-0.00021693526799154326,0.036155235792572536,0.0,0.0,0.0,0.0,0.0,-0.0,-1.0,-0.0,-0.0,
        -0.0,-0.0,0.0020175817725937989,0.0019796723009276795,-0.023967016242290948,0.001773384308174724,
        -0.00021831715113693025,0.013758239625790694,0.0,0.0,0.0,1.0,0.0,0.0,0.0,0.0,-0.0,-0.0,-0.0,-1.0,-0.0,-0.0,
        -0.0,0.0021543679790237634,-0.013758164253474772,-0.031126192595670284,-0.0021676333667632296,
        -0.0019809408498811915,0.0,0.0,0.0,1.0,0.0,0.0,0.0,-0.0,-0.0,-0.0,-1.0,-0.0,-0.0,-0.0,-0.0,-0.0,
        0.0017733644650094228,0.0021663421034936259,-0.02396702031125434,-0.0014267245515185119,
        0.013758235536900225,0.0,0.0,0.0,1.0,0.0,0.0,0.0,-0.0,-0.0,-0.0,-1.0,-0.0,-0.0,0.0023834617064148775,
        0.032821793825602311,0.0014267749509501136,0.013758177150392209,3.1682855172904752E-6,
        -0.0017741741644841874,0.0,0.0,0.0,1.0,0.0,0.0,0.0,0.0,0.0,-0.0,-0.0,-0.0,-1.0,-0.0,-0.0,
        0.013756945286258268,0.032821793825602311,-0.002383461706414877,-0.036155331128170466,0.0017738649457463927,
        0.0,0.0,0.0,1.0,0.0,0.0,0.0,-0.0,-0.0,-0.0,-1.0,-0.0,-0.0,8.0535028485727747E-5,0.0,-0.0,
        0.013757007748269136,-0.0017738649457463922,-1.1094817584871507E-5,0.0,0.0,0.0,1.0,0.0,0.0,0.0,-0.0,-0.0,
        -0.0,-1.0,-0.0,-0.0,-0.0,0.013758177150392211,8.05345450981963E-5,-2.1639071390723852E-5,
        0.0017741741644841872,0.0,0.0,0.0,1.0,0.0,0.0,0.0,0.0,-0.0,-0.0,-0.0,-1.0,-0.0,-0.0,-0.0,
        0.023117153652107741,-0.0017714855698833822,-1.107593583908204E-5,-0.032821701216996048,
        -0.033663497786071112,0.0,0.0,0.0,1.0,0.0,0.0,0.0,-0.0,-0.0,-0.0,-1.0,-0.0,-0.0,-0.0,-0.0,-0.0,
        -0.017540060210790728,-0.033663591643505519,-0.001773687040351414,2.1639071390723859E-5,
        -0.013758177150392211,0.0,0.0,0.0,1.0,0.0,0.0,0.0,-0.0,-0.0,-0.0,-1.0,-0.0,-0.0,-0.0,-0.0,
        0.036158866905630936,-0.0020175817725937989,-0.0019796723009276795,-0.013758219590295969,
        0.00021831715113693025,8.0516212332184712E-5,-0.0017733843081747243,0.0,0.0,0.0,1.0,0.0,0.0,0.0,-0.0,-0.0,
        -0.0,-1.0,-0.0,-0.0,-0.0,-0.0,0.027072767990336359,-0.0017730752489912582,-0.0025414906519322356,
        -0.013757007748269127,-0.036158836489428296,0.0,0.0,0.0,1.0,0.0,0.0,-0.0,-0.0,-0.0,-1.0,-0.0,-0.0,-0.0,-0.0,
        0.02816583906617192,-0.0017716448391260386,-0.0025390630631616979,-0.023967016586099656,0.0,0.0,0.0,1.0,0.0,
        0.0,0.0,-0.0,-0.0,-0.0,-1.0,-0.0,-0.0,-0.0,-0.0,-0.002017933713019439,-0.017540096325751129,
        -0.0019801394547201766,-0.033663529390784139,0.0025425544502436937,0.031126075963179154,0.0,1.0,0.0,0.0,
        -0.0,-0.0,-0.0,-1.0,-0.0,-0.0,-0.0,-0.0,-0.0021543679790237634,-0.013758164253474772,-0.031126192595670284,
        0.0021676333667632296,0.0019809408498811919,0.0,0.0,0.0,1.0,0.0,0.0,0.0,-0.0,-0.0,-0.0,-1.0,-0.0,-0.0,-0.0,
        -0.0,-0.0,-0.027072767990336356,-0.0,-0.0017733644650094228,-0.0021663421034936259,-0.02396702031125434,
        0.013758235536900225,0.0,0.0,0.0,1.0,0.0,0.0,-0.0,-0.0,-0.0,-1.0,-0.0,-0.0,-0.0,-0.0,-0.0020175817725937989,
        -0.023967016242290959,-0.00197967230092768,0.013758219590295984,0.0025420742486267352,0.0,0.0,1.0,0.0,0.0,
        -0.0,-0.0,-0.0,-1.0,-0.0,-0.0,-0.0,-0.0022561355647809592,-0.013758177150392209,-2.1639071390723856E-5,
        -8.0534545098196153E-5,0.0017741741644841874,0.0,0.0,0.0,1.0,0.0,0.0,-0.0,-0.0,-0.0,-1.0,-0.0,-0.0,-0.0,
        -0.0,-0.0,-0.013758082261467375,-0.00013643680450863756,-1.7578747218645926E-5,0.0020185138829726234,
        0.0023839444396658587,0.0,0.0,0.0,1.0,0.0,0.0,-0.0,-0.0,-0.0,-1.0,-0.0,-0.0,-0.0,-0.0,-0.0,
        -0.0023827866608640033,-0.023967012140249294,-0.001426115796022355,-0.036158931786919105,
        0.0017733843081747249,0.013758177150392206,0.0,0.0,0.0,1.0,0.0,0.0,-0.0,-0.0,-0.0,-1.0,-0.0,-0.0,-0.0,-0.0,
        0.0017741542886565815,0.013758235536900216,1.4266538049601484E-5,8.0534981096103676E-5,
        -0.0014279245624933968,0.0,0.0,0.0,1.0,0.0,0.0,0.0,0.0,0.0,-0.0,-0.0,-0.0,-1.0,-0.0,-0.0,
        0.0017736870403514127,-0.00014872217635028418,0.031126045000755019,0.0,0.0,0.0,0.0,0.0,0.0,0.0,0.0,0.0,-0.0,
        -0.0,-0.0,-1.0,-0.0,-0.0,-0.0,0.0017741542886565813,-0.00013643903899346717,1.1097382704726312E-5,
        -0.01375823962579072,-0.00013643911633017095,0.0,0.0,0.0,1.0,0.0,0.0,0.0,0.0,-0.0,-0.0,-0.0,-1.0,-0.0,-0.0,
        -0.0,-0.0,0.0020185138829726234,8.7167521048673558E-6,-0.013758219590295984,-0.0025434105399164903,0.0,0.0,
        0.0,1.0,0.0,0.0,0.0,-0.0,-0.0,-0.0,-1.0,-0.0,-0.0,-0.0,-0.0,-0.0020185138829726234,-0.013758219590295977,
        -0.00013643880956405708,-8.7167521048673558E-6,0.0025434105399164829,0.0,0.0,1.0,0.0,0.0,-0.0,-0.0,-0.0,
        -1.0,-0.0,-0.0,-0.0,-0.0,-0.0017741542886565815,-1.4266538049601484E-5,-0.013758239625790697,
        -8.0535028485727734E-5,0.0,0.0,0.0,1.0,0.0,0.0,-0.0,-0.0,-0.0,-1.0,-0.0,-0.0,-0.0,-0.0,-0.0,-0.0,
        0.0017741741644841864,0.013758239625790697,3.1706750128877981E-6,8.0535028485727883E-5,0.0,0.0,0.0,1.0,0.0,
        0.0,0.0,0.0,0.0,0.0,-0.0,-0.0,-0.0,-1.0,-0.0,-0.0,-0.555673663731469,-0.026771909379554294,
        -0.62490021645747618,-0.027265477962947069,-0.63800507768378811,-0.026352061912650541,0.555673663731469,
        0.026771909379554294,0.62490021645747618,0.027265477962947066,0.63800507768378822,0.026352061912650541,0.0,
        0.0,0.0,0.0,1.0,0.0,0.0,0.0,0.0,0.0,-0.0,-0.0,-0.0,-0.0,-1.0,-0.0,-0.0,-0.0,0.555673663731469,
        -0.027034185307057625,-0.70226225634217321,-0.027566488177000262,-0.7025340602672151,-0.026662833272981429,
        0.027034185307057625,0.027566488177000258,0.026662833272981429,0.0,0.0,0.0,0.0,1.0,0.0,0.0,0.0,0.0,-0.0,
        -0.0,-0.0,-0.0,-1.0,-0.0,-0.0,-0.0,0.026771909379554291,-0.55566424910285672,-0.62488504774223075,
        -0.024399835479656965,-0.63798948327222038,-0.021960985394712317,0.55566424910285672,0.62488504774223075,
        0.63798948327222038,0.0,0.0,0.0,0.0,1.0,0.0,0.0,0.0,0.0,-0.0,-0.0,-0.0,-0.0,-1.0,-0.0,-0.0,-0.0,
        0.62490021645747618,0.02706527731251647,0.026700746627905073,0.58505858013174894,-0.37854052611351124,
        -0.027072082181883242,-0.027610578309122807,-0.026708907388227909,0.027610578309122804,0.0,0.0,0.0,0.0,1.0,
        0.0,0.0,0.0,0.0,-0.0,-0.0,-0.0,-0.0,-1.0,-0.0,-0.0,0.027265477962947069,0.55566222109490582,
        0.63798667601923609,0.029437135799321903,-0.55566181651356428,-0.023469887537635181,-0.62488169574462793,
        -0.63798609648432814,0.0,0.0,0.0,0.0,1.0,0.0,0.0,0.0,0.0,-0.0,-0.0,-0.0,-0.0,-1.0,-0.0,-0.0,
        0.63800507768378822,-0.45692709004827581,-0.027011667529779945,-0.58505858013174894,-0.027541181508898387,
        -0.026637267215644224,0.027011667529779945,0.027541181508898383,0.026637267215644224,0.0,0.0,0.0,0.0,1.0,
        0.0,0.0,0.0,0.0,-0.0,-0.0,-0.0,-0.0,-1.0,-0.0,-0.0,0.026352061912650541,-0.55566389422834717,
        -0.02598312883534095,-0.62488507878410182,-0.02943713579932191,-0.637989575133729,0.55566389422834717,
        0.62488507878410182,0.63798957513372911,0.0,0.0,0.0,0.0,1.0,0.0,0.0,0.0,0.0,-0.0,-0.0,-0.0,-0.0,-1.0,-0.0,
        -0.0,-0.555673663731469,-0.027034185307057625,-0.027566488177000262,-0.026662833272981429,
        0.027034185307057625,0.70226225634217321,0.027566488177000258,0.7025340602672151,0.026662833272981429,0.0,
        0.0,0.0,0.0,1.0,0.0,0.0,0.0,0.0,-0.0,-0.0,-0.0,-0.0,-1.0,-0.0,-0.0,-0.0,-0.026771909379554291,
        -0.55566424910285672,-0.62488504774223075,-0.63798948327222038,0.55566424910285672,0.62488504774223075,
        0.024399835479656955,0.63798948327222038,0.021960985394712317,0.0,0.0,0.0,0.0,1.0,0.0,0.0,0.0,0.0,-0.0,-0.0,
        -0.0,-0.0,-1.0,-0.0,-0.0,-0.0,-0.62490021645747618,-0.58505858013174883,-0.027072082181883242,
        -0.027610578309122807,-0.026708907388227909,0.37854052611351124,0.027072082181883242,0.026708907388227909,
        0.0,0.0,0.0,0.0,1.0,0.0,0.0,0.0,-0.0,-0.0,-0.0,-0.0,-1.0,-0.0,-0.0,-0.0,-0.027265477962947069,
        -0.55566222109490582,-0.63798667601923609,-0.029437135799321879,-0.62488169574462793,0.55566181651356428,
        0.023469887537635192,0.62488169574462793,0.63798609648432814,0.0,0.0,0.0,0.0,1.0,0.0,0.0,0.0,-0.0,-0.0,-0.0,
        -0.0,-1.0,-0.0,-0.0,-0.0,-0.63800507768378822,-0.027011667529779945,-0.027541181508898387,
        -0.026637267215644224,0.45692709004827581,0.027011667529779945,0.58505858013174894,0.027541181508898383,
        0.026637267215644224,0.0,0.0,0.0,0.0,1.0,0.0,0.0,0.0,-0.0,-0.0,-0.0,-0.0,-1.0,-0.0,-0.0,-0.0,
        -0.026352061912650541,-0.55566389422834717,-0.62488507878410182,-0.637989575133729,0.55566389422834717,
        0.02598312883534095,0.62488507878410182,0.0294371357993219,0.63798957513372911,0.0,0.0,0.0,0.0,1.0,0.0,0.0,
        0.0,-0.0,-0.0,-0.0,-0.0,-1.0,-0.0,-0.0,-0.0,0.55566424910285672,0.027034185307057621,-0.70224208707170055,
        -0.024752136540096732,-0.70251617195999394,-0.022319435462106595,0.0,0.0,0.0,0.0,1.0,0.0,0.0,0.0,-0.0,-0.0,
        -0.0,-0.0,-1.0,-0.0,-0.0,-0.0,0.70226225634217332,0.3785405261135113,0.70163518723474272,
        -0.027105602758215112,-0.027648865450003536,-0.026748274296612785,0.027105602758215112,0.027648865450003533,
        0.026748274296612785,0.0,0.0,0.0,0.0,1.0,0.0,0.0,0.0,0.0,0.0,-0.0,-0.0,-0.0,-0.0,-1.0,-0.0,-0.0,
        0.55566222109490582,-0.023637206391576536,-0.015100165961297108,-0.0,0.378540460951947,0.02764886545000354,
        -0.015207454024849647,0.0,0.0,0.0,0.0,1.0,0.0,0.0,0.0,-0.0,-0.0,-0.0,-0.0,-1.0,-0.0,0.45692709004827575,
        0.702534060267215,-0.027090859530371859,-0.70163518723474272,0.026730661933064313,0.0,0.0,0.0,0.0,1.0,0.0,
        0.0,0.0,-0.0,-0.0,-0.0,-0.0,-1.0,-0.0,-0.0,0.55566389422834728,-0.029709944333287521,-0.0,
        0.37854017792555505,0.026748274296612796,0.0,0.0,0.0,0.0,1.0,0.0,0.0,0.0,0.0,-0.0,-0.0,-0.0,-0.0,-1.0,-0.0,
        0.55566424910285672,-0.027034185307057621,-0.0,0.37851997948504351,-0.70317323754735273,0.02240967789339866,
        0.0,0.0,0.0,0.0,1.0,0.0,0.0,0.0,-0.0,-0.0,-0.0,-0.0,-1.0,-0.0,-0.0,0.55566222109490582,
        -0.027566488177000255,-0.70223873149897853,0.023637206391576546,0.015100165961297143,0.0,0.0,0.0,1.0,0.0,
        0.0,-0.0,-0.0,-0.0,-0.0,-1.0,-0.0,-0.0,0.55566389422834728,-0.026662833272981429,-0.70224253943268344,
        -0.70251656286365771,0.026190122699982339,0.029709944333287511,0.0,0.0,0.0,0.0,1.0,0.0,0.0,-0.0,-0.0,-0.0,
        -0.0,-1.0,-0.0,-0.0,-0.0,0.02706527731251647,0.6248806237808493,0.023656120772106486,-0.378519539943052,
        -0.70317018870025627,0.0,0.0,0.0,0.0,1.0,0.0,0.0,0.0,-0.0,-0.0,-0.0,-0.0,-1.0,-0.0,0.02346980199155271,
        0.024399835479656976,-0.55566129015943833,-0.6248806237808493,-0.63798497169620461,-0.01473301981127613,
        0.55566129015943833,0.6248806237808493,0.63798497169620461,0.0,0.0,0.0,0.0,1.0,0.0,0.0,0.0,-0.0,-0.0,-0.0,
        -0.0,-1.0,-0.0,0.027011667529779945,0.63798948327222027,-0.456923837504278,-0.58504518410006956,
        -0.024723646828030479,0.0,0.0,0.0,0.0,1.0,0.0,0.0,0.0,-0.0,-0.0,-0.0,-0.0,-1.0,-0.0,-0.0,
        0.02598312883534095,0.021960985394712324,-0.63798532239475636,0.55566147407010114,0.62488096344828059,
        0.63798532239475636,0.0,0.0,0.0,0.0,1.0,0.0,0.0,0.0,0.0,0.0,-0.0,-0.0,-0.0,-0.0,-1.0,-0.0,-0.0,
        0.027034185307057618,-0.55566424910285683,-0.024752136540096732,0.70224208707170055,0.70251617195999394,0.0,
        0.0,0.0,0.0,1.0,0.0,0.0,0.0,-0.0,-0.0,-0.0,-0.0,-1.0,-0.0,-0.0,-0.0,0.02706527731251647,
        -0.62488504774223075,-0.024795740829694754,0.37851997948504357,0.7031738370963756,0.0,0.0,0.0,0.0,1.0,0.0,
        0.0,-0.0,-0.0,-0.0,-0.0,-1.0,-0.0,-0.0,0.027011667529779945,-0.63798948327222038,-0.024723646828030479,
        -0.02229166073122648,0.456923837504278,0.58504518410006945,0.0,0.0,0.0,0.0,1.0,0.0,0.0,-0.0,-0.0,-0.0,-0.0,
        -1.0,-0.0,-0.0,-0.0,0.6248822663250807,0.0276027315782233,0.58504257002809312,0.02974148887250478,
        -0.37854036201549385,-0.023660396850780661,0.0,0.0,0.0,0.0,1.0,0.0,0.0,0.0,-0.0,-0.0,-0.0,-0.0,-1.0,-0.0,
        0.62488507878410182,0.026700746627905073,0.58504502721143925,-0.37854017792555522,-0.029748443430697026,0.0,
        0.0,0.0,0.0,1.0,0.0,0.0,0.0,-0.0,-0.0,-0.0,-0.0,-1.0,-0.0,0.62488504774223086,0.022364818883998015,
        0.58504518410006956,-0.027072082181883231,-0.37854107343057747,0.024805000972806229,0.0,0.0,0.0,0.0,1.0,0.0,
        0.0,0.0,-0.0,-0.0,-0.0,-0.0,-1.0,-0.0,-0.0,0.58504257002809312,-0.027610578309122814,-0.37854046095194716,
        0.023660296965944735,0.015161281241640749,0.0,0.0,0.0,1.0,0.0,-0.0,-0.0,-0.0,-1.0,-0.0,0.027541181508898383,
        0.637986676019236,0.029685529684818829,-0.023621944154890266,-0.58504204394174086,0.0,0.0,0.0,0.0,1.0,0.0,
        0.0,0.0,-0.0,-0.0,-0.0,-0.0,-1.0,-0.0,0.027566488177000262,0.70251319697861081,0.029709944333287532,
        -0.55566181651356417,-0.023637304191565071,0.70223802681964376,0.0,0.0,0.0,0.0,1.0,0.0,0.0,0.0,-0.0,-0.0,
        -0.0,-0.0,-1.0,-0.0,-0.0,0.027602731578223291,0.02974148887250478,-0.62488169574462793,
        -0.023656120772106482,0.37851926782050033,0.70317150299940423,0.0,0.0,0.0,1.0,0.0,-0.0,-0.0,-0.0,-1.0,-0.0,
        0.027541181508898383,0.4569226479042604,0.58504257002809312,0.029685529684818829,-0.637986096484328,
        -0.023621944154890266,0.0,0.0,0.0,0.0,1.0,0.0,0.0,-0.0,-0.0,-0.0,-0.0,-1.0,-0.0,-0.0,0.637989575133729,
        0.026637267215644217,-0.58504502721143936,-0.029685529684818846,0.0,0.0,0.0,0.0,1.0,0.0,0.0,0.0,-0.0,-0.0,
        -0.0,-0.0,-1.0,-0.0,0.63798948327222038,-0.027011667529779945,-0.58504518410006945,0.024723646828030466,
        0.02229166073122648,0.0,0.0,0.0,0.0,1.0,0.0,0.0,0.0,-0.0,-0.0,-0.0,-0.0,-1.0,-0.0,-0.0,0.637986676019236,
        -0.02754118150889838,-0.58504257002809312,0.023621847095687702,0.015074517622588319,0.0,0.0,0.0,1.0,0.0,
        -0.0,-0.0,-0.0,-1.0,-0.0,0.637989575133729,-0.026637267215644217,-0.45692310525642205,-0.58504502721143936,
        0.026171339658097509,0.029685529684818822,0.0,0.0,0.0,0.0,1.0,0.0,0.0,-0.0,-0.0,-0.0,-0.0,-1.0,-0.0,-0.0,
        0.026662833272981426,-0.55566389422834728,-0.029709944333287525,0.70224253943268344,0.70251656286365771,0.0,
        0.0,0.0,0.0,1.0,0.0,0.0,0.0,-0.0,-0.0,-0.0,-0.0,-1.0,-0.0,-0.0,0.026700746627905069,-0.62488507878410182,
        -0.02974148887250477,0.37851908394641454,0.703174067452467,0.0,0.0,0.0,1.0,0.0,-0.0,-0.0,-0.0,-1.0,-0.0,
        0.026637267215644227,-0.637989575133729,-0.029685529684818811,0.456923105256422,0.58504502721143925,0.0,0.0,
        0.0,0.0,1.0,0.0,0.0,-0.0,-0.0,-0.0,-0.0,-1.0,-0.0,-0.0,-0.55566424910285672,-0.027034185307057621,
        0.70224208707170055,0.024752136540096722,0.70251617195999394,0.022319435462106609,0.0,0.0,0.0,0.0,1.0,0.0,
        0.0,0.0,-0.0,-0.0,-0.0,-0.0,-1.0,-0.0,-0.0,-0.0,-0.37851943317454484,-0.70226225634217332,
        -0.027098793108292794,0.70318478827029374,0.02674010789169564,0.0,0.0,0.0,0.0,1.0,0.0,0.0,-0.0,-0.0,-0.0,
        -0.0,-1.0,-0.0,-0.0,-0.0,-0.55566222109490582,-0.027566488177000255,0.023637206391576546,
        0.70223873149897853,0.70251319697861081,0.015100165961297143,0.0,0.0,0.0,1.0,0.0,-0.0,-0.0,-0.0,-1.0,-0.0,
        -0.0,-0.45692709004827575,-0.7025340602672151,-0.37854052611351124,-0.70318478827029385,
        -0.027105602758215112,-0.027648865450003536,-0.026748274296612785,0.027105602758215112,0.026748274296612785,
        0.0,0.0,0.0,0.0,1.0,0.0,0.0,0.0,-0.0,-0.0,-0.0,-0.0,-1.0,-0.0,-0.0,-0.0,-0.0,-0.55566389422834728,
        -0.026662833272981429,0.026190122699982339,0.70224253943268344,0.029709944333287511,0.70251656286365771,0.0,
        0.0,0.0,0.0,1.0,0.0,0.0,-0.0,-0.0,-0.0,-0.0,-1.0,-0.0,-0.0,-0.0,-0.02706527731251647,-0.62488504774223075,
        0.37851997948504357,0.024795740829694744,0.7031738370963756,0.022364818883998022,0.0,0.0,0.0,1.0,0.0,-0.0,
        -0.0,-0.0,-1.0,-0.0,-0.0,-0.02346980199155272,-0.024399835479656965,-0.55566129015943833,
        -0.6248806237808493,-0.63798497169620461,0.55566129015943833,0.6248806237808493,0.63798497169620461,
        0.014733019811276159,0.0,0.0,0.0,1.0,0.0,0.0,-0.0,-0.0,-0.0,-0.0,-1.0,-0.0,-0.0,-0.0,-0.027011667529779945,
        -0.63798948327222038,0.456923837504278,0.58504518410006945,0.024723646828030469,0.02229166073122648,0.0,0.0,
        0.0,0.0,1.0,0.0,0.0,-0.0,-0.0,-0.0,-0.0,-1.0,-0.0,-0.0,-0.0,-0.02598312883534095,-0.021960985394712324,
        -0.63798532239475636,0.55566147407010114,0.029307880059563592,0.0,0.0,0.0,0.0,1.0,0.0,0.0,-0.0,-0.0,-0.0,
        -0.0,-1.0,-0.0,-0.0,-0.6248822663250807,-0.027602731578223294,0.37851936679972537,0.023656021236335204,
        0.703171917764931,0.01515082442675411,0.0,0.0,1.0,0.0,-0.0,-0.0,-1.0,-0.0,-0.62488507878410182,
        -0.58504502721143936,-0.026708907388227905,0.37854017792555511,0.026218970645527549,0.029748443430697016,
        0.0,0.0,0.0,0.0,1.0,0.0,-0.0,-0.0,-0.0,-0.0,-1.0,-0.0,-0.0,-0.0,-0.02754118150889838,-0.63798667601923609,
        0.4569226479042604,0.023621847095687692,0.585042570028093,0.015074517622588279,0.0,0.0,0.0,0.0,1.0,0.0,-0.0,
        -0.0,-0.0,-0.0,-1.0,-0.0,-0.0,-0.63798957513372911,-0.026637267215644217,0.456923105256422,
        0.026171339658097509,0.58504502721143925,0.029685529684818822,0.0,0.0,0.0,0.0,1.0,0.0,-0.0,-0.0,-0.0,-0.0,
        -1.0,-0.0,-0.0,-0.0,0.702236447861886,0.37854073327939103,0.023682030674840704,0.00016424244292451563,
        -0.015216927320390218,0.0,0.0,0.0,0.0,1.0,0.0,0.0,0.0,0.0,-0.0,-0.0,-0.0,-0.0,-1.0,-0.0,0.55566129015943833,
        0.023637206391576532,0.024752136540096732,-0.702236447861886,-0.015109647396991065,0.0,0.0,0.0,0.0,1.0,0.0,
        -0.0,-0.0,-0.0,-1.0,-0.0,-0.0,0.45692383750427795,0.70251617195999394,0.37854107343057741,
        0.027105602758215115,-0.024849423695496659,0.0,0.0,0.0,0.0,1.0,0.0,0.0,0.0,0.0,-0.0,-0.0,-0.0,-0.0,-1.0,
        -0.0,-0.0,0.55566181651356428,-0.023637304191565081,-0.0,0.015196990314225767,0.37854036201549374,
        0.00027130052193601533,3.3862997711630647E-5,0.0,0.0,0.0,0.0,1.0,0.0,0.0,0.0,0.0,-0.0,-0.0,-0.0,-0.0,-1.0,
        -0.0,0.45692310525642194,0.70251656286365771,0.37854017792555505,0.70317346814293025,-0.026748274296612796,
        0.026245744732980112,0.029783569798323813,0.0,0.0,0.0,0.0,1.0,0.0,0.0,0.0,-0.0,-0.0,-0.0,-0.0,-1.0,-0.0,
        -0.0,0.55566129015943833,-0.023637206391576536,-0.024752136540096725,-0.702236447861886,
        0.015109647396991065,0.0,0.0,0.0,1.0,0.0,0.0,-0.0,-0.0,-0.0,-0.0,-1.0,-0.0,-0.0,-0.0,0.55566181651356428,
        -0.029709944333287493,-0.70223802681964376,-0.7025125679269647,0.023637304191565092,0.0,0.0,0.0,0.0,1.0,0.0,
        0.0,-0.0,-0.0,-0.0,-0.0,-1.0,-0.0,-0.0,-0.0,0.027072082181883235,0.58504518410006945,0.70317383709637549,
        -0.37854107343057752,-0.024805000972806222,0.0,0.0,0.0,0.0,1.0,0.0,0.0,0.0,-0.0,-0.0,-0.0,-0.0,-1.0,-0.0,
        -0.0,0.024723646828030497,0.63798497169620449,0.023621944154890263,-0.5850406398453023,0.0,0.0,0.0,0.0,1.0,
        0.0,0.0,0.0,0.0,-0.0,-0.0,-0.0,-0.0,-1.0,-0.0,0.023469887537635181,3.2815184442066549E-5,
        -0.55566088508118927,-0.62488005247477207,-0.63798439140804353,0.55566088508118927,0.62488005247477207,
        0.63798439140804353,0.0,0.0,0.0,0.0,1.0,0.0,0.0,0.0,0.0,0.0,-0.0,-0.0,-0.0,-0.0,-1.0,-0.0,-0.0,
        0.024752136540096736,0.70251116957088389,0.023637304191565078,-0.55566088508118927,0.7022357422084774,0.0,
        0.0,0.0,0.0,1.0,0.0,0.0,0.0,0.0,-0.0,-0.0,-0.0,-0.0,-1.0,-0.0,-0.0,0.024795740829694764,
        0.023656120772106475,-0.624880052474772,0.37851953994305221,0.70317018870025627,0.0,0.0,0.0,1.0,0.0,0.0,
        -0.0,-0.0,-0.0,-1.0,-0.0,0.023621847095687688,0.024723646828030497,-0.63798497169620461,
        -0.015083998191321592,0.45692247149286119,0.58504116656491612,0.0,0.0,0.0,0.0,1.0,0.0,0.0,-0.0,-0.0,-0.0,
        -0.0,-1.0,-0.0,0.023621944154890259,3.3598535051162514E-5,-0.0050973150136454475,0.45692225021991206,
        0.58504063984530219,0.0,0.0,0.0,0.0,1.0,0.0,0.0,0.0,-0.0,-0.0,-0.0,-0.0,-1.0,-0.0,-0.0,0.027098793108292798,
        -0.37851997948504373,-0.70224208707170055,0.70317323754735284,0.0,0.0,0.0,0.0,1.0,0.0,0.0,-0.0,-0.0,-0.0,
        -0.0,-1.0,-0.0,-0.0,-0.0,0.027090859530371859,0.023672783354342114,-0.4569224714928613,-0.70251116957088389,
        -0.015195086849570095,0.70160323232532973,0.0,0.0,0.0,1.0,0.0,0.0,-0.0,-0.0,-0.0,-0.0,-1.0,-0.0,-0.0,
        0.027072082181883235,-0.58504518410006934,-0.024805000972806222,-0.022374380992921029,0.37854107343057752,
        0.0,0.0,0.0,0.0,1.0,0.0,0.0,-0.0,-0.0,-0.0,-0.0,-1.0,-0.0,-0.0,-0.0,0.58504502721143925,0.70317406745246691,
        -0.026708907388227905,-0.37854017792555522,0.026218970645527549,0.029748443430697016,0.0,0.0,0.0,0.0,1.0,
        0.0,0.0,-0.0,-0.0,-0.0,-0.0,-1.0,-0.0,-0.0,0.585041166564916,-0.023660296965944742,-0.024805000972806225,
        -0.37854073327939119,0.015170756558948674,0.0,0.0,0.0,1.0,0.0,-0.0,-0.0,-1.0,-0.0,-0.0,-0.0,
        0.62488169574462793,0.58504204394174075,-0.029748443430697009,-0.37854036201549396,0.023660396850780658,0.0,
        0.0,0.0,0.0,1.0,0.0,0.0,-0.0,-0.0,-0.0,-0.0,-1.0,-0.0,-0.0,0.027631856629547157,-0.4569226479042604,
        -0.70251319697861081,-0.023672783354342117,-0.015185611969090922,0.70160605506782658,0.0,0.0,0.0,1.0,0.0,
        -0.0,-0.0,-0.0,-0.0,-1.0,-0.0,-0.0,0.027610578309122811,0.02974844343069703,-0.58504204394174075,
        -0.023660396850780651,0.37854036201549374,0.0,0.0,0.0,0.0,1.0,0.0,0.0,-0.0,-0.0,-0.0,-0.0,-1.0,-0.0,-0.0,
        0.63798497169620449,-0.0236218470956877,-0.024723646828030469,-0.58504116656491612,0.015083998191321633,0.0,
        0.0,0.0,1.0,0.0,-0.0,-0.0,-1.0,-0.0,-0.0,-0.0,-0.026171339658097509,-0.022291660731226463,
        -0.58504146009743707,0.0050973150136454448,-0.023621944154890263,-0.45692225021991223,0.0,0.0,0.0,0.0,1.0,
        0.0,0.0,-0.0,-0.0,-0.0,-0.0,-1.0,-0.0,-0.0,-0.0,0.637986096484328,-0.029685529684818798,
        -0.45692242688405121,-0.58504204394174086,0.02362194415489029,0.0,0.0,0.0,0.0,1.0,0.0,0.0,-0.0,-0.0,-0.0,
        -0.0,-1.0,-0.0,-0.0,0.026730661933064309,-0.45692310525642194,-0.70251656286365771,-0.029768291394636794,
        0.70161080096520145,0.0,0.0,0.0,0.0,1.0,0.0,0.0,-0.0,-0.0,-0.0,-0.0,-1.0,-0.0,-0.0,0.026708907388227905,
        -0.58504502721143925,-0.029748443430697019,0.378540177925555,0.0,0.0,0.0,0.0,1.0,0.0,0.0,-0.0,-0.0,-0.0,
        -0.0,-1.0,-0.0,-0.0,-0.4569238375042779,-0.027090859530371863,-0.70251617195999394,-0.37854107343057747,
        0.024849423695496649,0.022419246501157553,0.0,0.0,0.0,0.0,1.0,0.0,0.0,-0.0,-0.0,-0.0,-0.0,-1.0,-0.0,-0.0,
        -0.0,-0.0,-0.55566147407010114,-0.026190122699982339,-0.0223194354621066,0.70223692196481524,
        0.029647784654081327,0.70251158235928435,0.0,0.0,0.0,1.0,0.0,0.0,-0.0,-0.0,-0.0,-0.0,-1.0,-0.0,-0.0,-0.0,
        -0.70224253943268344,-0.378540177925555,-0.70161080096520145,-0.026748274296612796,0.029783569798323813,0.0,
        0.0,0.0,0.0,1.0,0.0,-0.0,-0.0,-0.0,-0.0,-1.0,-0.0,-0.0,-0.0,-0.0,-0.45692264790426035,-0.027631856629547154,
        -0.70251319697861092,0.023672783354342128,0.70160605506782658,0.015185611969090976,0.0,0.0,1.0,0.0,-0.0,
        -0.0,-0.0,-1.0,-0.0,-0.0,-0.55566181651356428,-0.029709944333287493,0.023637304191565092,
        0.70223802681964376,0.7025125679269647,0.0,0.0,0.0,0.0,1.0,0.0,0.0,-0.0,-0.0,-0.0,-0.0,-1.0,-0.0,-0.0,-0.0,
        -0.45692310525642188,-0.70251656286365771,-0.026730661933064316,0.026234238763943405,0.70161080096520145,
        0.029768291394636756,0.0,0.0,0.0,1.0,0.0,-0.0,-0.0,-0.0,-0.0,-1.0,-0.0,-0.0,-0.027072082181883235,
        -0.58504518410006934,0.37854107343057752,0.024805000972806211,0.022374380992921029,0.0,0.0,0.0,0.0,1.0,0.0,
        0.0,-0.0,-0.0,-0.0,-0.0,-1.0,-0.0,-0.0,-0.0,-0.026213688698745,-0.62488096344828059,-0.022364818883998026,
        0.3785195589565879,0.029687807671632122,0.70317085483536168,0.0,0.0,1.0,0.0,-0.0,-0.0,-0.0,-1.0,-0.0,-0.0,
        -0.023469887537635188,-0.00012845955535528616,-0.55566088508118927,-0.62488005247477207,
        -0.63798439140804353,0.55566088508118927,0.62488005247477207,0.63798439140804353,0.0,0.0,0.0,0.0,1.0,0.0,
        0.0,0.0,-0.0,-0.0,-0.0,-0.0,-1.0,-0.0,-0.0,-0.0,-0.0,-0.585042570028093,-0.027610578309122811,
        0.37854046095194716,0.023660296965944742,0.015161281241640751,0.0,0.0,0.0,0.0,1.0,0.0,-0.0,-0.0,-0.0,-0.0,
        -1.0,-0.0,-0.0,-0.62488169574462793,-0.029741488872504766,0.3785192678205006,0.023656120772106493,
        0.70317150299940423,0.0,0.0,0.0,0.0,1.0,0.0,-0.0,-0.0,-0.0,-0.0,-1.0,-0.0,-0.0,-0.029685529684818805,
        -0.637986096484328,0.45692242688405116,0.02362194415489028,0.58504204394174075,0.0,0.0,0.0,0.0,1.0,0.0,-0.0,
        -0.0,-0.0,-0.0,-1.0,-0.0,-0.0,-0.0,0.55566088508118927,0.023637304191565081,0.015109647396991093,
        -0.7022357422084774,0.0,0.0,0.0,0.0,1.0,0.0,0.0,0.0,0.0,-0.0,-0.0,-0.0,-0.0,-1.0,-0.0,-0.0,
        0.37854107343057741,0.0015613656062954475,-0.027105602758215108,0.02484942369549667,0.02241924650115756,0.0,
        0.0,0.0,0.0,1.0,0.0,0.0,0.0,0.0,-0.0,-0.0,-0.0,-0.0,-1.0,-0.0,-0.0,0.37854046095194693,0.70317131702755065,
        -0.027648865450003536,0.023682030674840704,0.015207454024849647,0.0,0.0,0.0,1.0,0.0,0.0,-0.0,-0.0,-0.0,-1.0,
        -0.0,0.702236447861886,-0.024840157186683216,0.37854073327939092,-0.023682030674840707,
        -0.0001642424429245156,0.015216927320390209,0.0,0.0,0.0,1.0,0.0,-0.0,-0.0,-1.0,-0.0,-0.0,-0.0,
        0.45692242688405105,0.7025125679269647,-0.02976829139463676,0.37854036201549374,-0.00027130052193601533,
        0.023682132033406258,0.0,0.0,0.0,0.0,1.0,0.0,0.0,0.0,-0.0,-0.0,-0.0,-0.0,-1.0,-0.0,-0.0,0.55566088508118927,
        -0.023637304191565085,-0.029647784654081352,-0.7022357422084774,-0.70251053960656562,0.0,0.0,0.0,0.0,1.0,
        0.0,0.0,-0.0,-0.0,-0.0,-0.0,-1.0,-0.0,-0.0,-0.0,-0.0,0.37851926782050049,0.70223802681964376,
        -0.029776610295742294,-0.70317090201170729,0.023677852874347757,0.0,0.0,0.0,0.0,1.0,0.0,0.0,-0.0,-0.0,-0.0,
        -0.0,-1.0,-0.0,0.58504116656491612,0.024805000972806236,0.70317060420331423,0.023660396850780658,
        0.0015608627398630522,-0.3785406342380947,0.0,0.0,0.0,0.0,1.0,0.0,0.0,0.0,0.0,-0.0,-0.0,-0.0,-0.0,-1.0,-0.0,
        0.023660296965944735,0.024805000972806239,-0.58504116656491578,-0.015170756558948695,0.37854073327939125,
        0.0,0.0,0.0,0.0,1.0,0.0,0.0,-0.0,-0.0,-0.0,-0.0,-1.0,-0.0,3.3895386058154954E-5,0.0,-0.0,
        0.023682030674840707,-0.37854073327939108,-0.0030612231608958297,0.0,0.0,0.0,0.0,1.0,0.0,0.0,-0.0,-0.0,-0.0,
        -0.0,-1.0,-0.0,-0.0,0.023660396850780651,3.37922497221569E-5,-0.0053104157804372727,0.37854063423809481,0.0,
        0.0,0.0,0.0,1.0,0.0,0.0,0.0,-0.0,-0.0,-0.0,-0.0,-1.0,-0.0,-0.0,0.027105602758215112,-0.37854107343057758,
        -0.0030612088654606811,-0.024849423695496673,-0.02241924650115756,0.0,0.0,0.0,0.0,1.0,0.0,0.0,-0.0,-0.0,
        -0.0,-0.0,-1.0,-0.0,-0.0,-0.0,-0.0,-0.026218970645527546,-0.022374380992921033,-0.37854065319208563,
        0.00531041578043727,-0.023660396850780661,0.0,0.0,0.0,0.0,1.0,0.0,0.0,-0.0,-0.0,-0.0,-0.0,-1.0,-0.0,-0.0,
        -0.0,0.015185611969090872,-0.45692242688405116,-0.7025125679269647,-0.023672883991351843,
        0.00027130052193601566,3.3862997711630437E-5,-0.3785403620154939,0.0,0.0,0.0,0.0,1.0,0.0,0.0,-0.0,-0.0,-0.0,
        -0.0,-1.0,-0.0,-0.0,-0.0,0.027648865450003536,-0.378540460951947,-0.70160605506782647,-0.0236820306748407,
        -0.015207454024849618,0.0,0.0,0.0,0.0,1.0,0.0,-0.0,-0.0,-0.0,-0.0,-1.0,-0.0,-0.0,-0.0,0.026748274296612789,
        -0.37854017792555505,-0.70161080096520156,-0.029783569798323847,0.0,0.0,0.0,0.0,1.0,0.0,0.0,-0.0,-0.0,-0.0,
        -0.0,-1.0,-0.0,-0.0,-0.0,-0.45692249061308471,-0.026234238763943405,-0.70251158235928435,
        -0.022398709579893369,0.70160383989347,0.029720779304182428,0.0,0.0,1.0,0.0,-0.0,-0.0,-0.0,-0.0,-1.0,-0.0,
        -0.0,-0.0,-0.55566088508118927,-0.023637304191565085,-0.029647784654081352,0.7022357422084774,
        0.70251053960656573,0.0,0.0,0.0,0.0,1.0,0.0,0.0,-0.0,-0.0,-0.0,-0.0,-1.0,-0.0,-0.0,-0.0,-0.0,
        -0.027648865450003536,-0.0,-0.37851926782050049,-0.70223802681964376,-0.029776610295742294,
        0.023677852874347757,0.0,0.0,0.0,0.0,1.0,0.0,-0.0,-0.0,-0.0,-0.0,-1.0,-0.0,-0.0,-0.0,-0.45692242688405105,
        -0.02976829139463676,-0.7025125679269647,0.023672883991351864,0.70160519311325342,0.0,0.0,0.0,1.0,0.0,-0.0,
        -0.0,-0.0,-0.0,-1.0,-0.0,-0.0,-0.62488005247477207,-0.023660396850780661,-0.0053104157804372719,
        -3.3792249722156905E-5,0.3785406342380947,0.0,0.0,0.0,0.0,1.0,0.0,-0.0,-0.0,-0.0,-0.0,-1.0,-0.0,-0.0,-0.0,
        -0.0,-0.023621944154890277,-0.00012982492179038625,-0.0050973150136454466,0.45692225021991212,
        0.5850406398453023,0.0,0.0,0.0,0.0,1.0,0.0,-0.0,-0.0,-0.0,-0.0,-1.0,-0.0,-0.0,-0.0,-0.0,
        -0.58504204394174064,-0.029748443430697026,-0.70317150299940412,-0.015161281241640776,0.37854036201549396,
        0.023660396850780654,0.0,0.0,0.0,0.0,1.0,0.0,-0.0,-0.0,-0.0,-0.0,-1.0,-0.0,-0.0,-0.0,0.378519539943052,
        0.023677852874347757,0.0046218484590718626,3.3872049431451388E-5,-0.70316958685172248,0.0,0.0,0.0,0.0,1.0,
        0.0,0.0,0.0,0.0,-0.0,-0.0,-0.0,-0.0,-1.0,-0.0,0.37854065319208546,-9.9046128627942282E-5,
        0.029739987791949973,0.0,0.0,0.0,1.0,0.0,0.0,0.0,0.0,0.0,-0.0,-0.0,-0.0,-0.0,-1.0,-0.0,-0.0,
        0.37851953994305204,-0.00013032533543202578,0.0030612242404972137,-0.023682132033406265,
        -0.00013036341924922685,0.0,0.0,0.0,0.0,1.0,0.0,0.0,0.0,-0.0,-0.0,-0.0,-0.0,-1.0,-0.0,-0.0,-0.0,
        0.45692225021991212,0.0030912635403395824,-0.02367288399135186,-0.70160236926968877,0.0,0.0,0.0,0.0,1.0,0.0,
        0.0,-0.0,-0.0,-0.0,-0.0,-1.0,-0.0,-0.0,-0.0,-0.45692225021991212,-0.02367288399135186,
        -0.00013027879750649216,-0.003091263540339582,0.70160236926968877,0.0,0.0,0.0,1.0,0.0,-0.0,-0.0,-0.0,-0.0,
        -1.0,-0.0,-0.0,-0.0,-0.378519539943052,-0.0046218484590718626,-0.023682132033406265,-3.389538605815513E-5,
        0.0,0.0,0.0,0.0,1.0,0.0,-0.0,-0.0,-0.0,-0.0,-1.0,-0.0,-0.0,-0.0,-0.0,-0.0,0.37854063423809459,
        0.023682132033406265,0.001561372566461268,3.389538605815513E-5,0.0,0.0,0.0,0.0,1.0,0.0,0.0,0.0,0.0,0.0,-0.0,
        -0.0,-0.0,-0.0,-1.0,-0.0,-0.047678521358187322,-0.55787204405389446,-0.048825402242851326,
        -0.62654723292970194,-0.047286920841764508,-0.63943141348019983,0.047678521358187322,0.55787204405389446,
        0.048825402242851333,0.62654723292970194,0.047286920841764508,0.63943141348019983,0.0,0.0,0.0,0.0,0.0,1.0,
        0.0,0.0,0.0,0.0,-0.0,-0.0,-0.0,-0.0,-0.0,-1.0,-0.0,-0.0,0.047678521358187315,-0.557872509055183,
        -0.044288901125137163,-0.62654217515979649,-0.040021361425923357,-0.63942545184526778,0.557872509055183,
        0.62654217515979649,0.63942545184526778,0.0,0.0,0.0,0.0,0.0,1.0,0.0,0.0,0.0,-0.0,-0.0,-0.0,-0.0,-0.0,-1.0,
        -0.0,-0.0,0.55787204405389446,-0.047942655141777091,-0.049117799127055072,-0.702875228655225,
        -0.0475823178492932,-0.70295568967385469,0.047942655141777091,0.049117799127055078,0.04758231784929319,0.0,
        0.0,0.0,0.0,0.0,1.0,0.0,0.0,0.0,-0.0,-0.0,-0.0,-0.0,-0.0,-1.0,-0.0,-0.0,0.048825402242851333,
        0.55787171658183987,0.63942424475811355,0.052452304750527382,-0.041298149353625656,-0.557871608027596,
        -0.62654080641868248,-0.63942401877909183,0.62654080641868248,0.0,0.0,0.0,0.0,0.0,1.0,0.0,0.0,0.0,-0.0,-0.0,
        -0.0,-0.0,-0.0,-1.0,-0.0,0.626547232929702,0.047984758880296075,0.04763006590676714,0.58732864799299578,
        -0.047993536136706469,-0.38140732638781982,-0.049174830154444668,-0.047640075741515714,0.0,0.0,0.0,0.0,0.0,
        1.0,0.0,0.0,0.0,-0.0,-0.0,-0.0,-0.0,-0.0,-1.0,-0.0,0.047286920841764508,-0.045941301434432633,
        -0.55787142569916037,-0.052452304750527444,-0.62654193427993921,-0.639425363845251,0.55787142569916037,
        0.62654193427993921,0.639425363845251,0.0,0.0,0.0,0.0,0.0,1.0,0.0,0.0,0.0,-0.0,-0.0,-0.0,-0.0,-0.0,-1.0,
        -0.0,0.63943141348019983,-0.047934264404490834,-0.45972838564453733,-0.0491093915715111,
        -0.58732864799299578,-0.04757405784581345,0.047934264404490834,0.0491093915715111,0.04757405784581345,0.0,
        0.0,0.0,0.0,0.0,1.0,0.0,0.0,0.0,-0.0,-0.0,-0.0,-0.0,-0.0,-1.0,-0.0,-0.047678521358187315,-0.557872509055183,
        -0.62654217515979649,-0.63942545184526778,0.557872509055183,0.044288901125137184,0.62654217515979649,
        0.04002136142592335,0.63942545184526778,0.0,0.0,0.0,0.0,0.0,1.0,0.0,0.0,0.0,-0.0,-0.0,-0.0,-0.0,-0.0,-1.0,
        -0.0,-0.0,-0.55787204405389446,-0.047942655141777091,-0.049117799127055072,-0.0475823178492932,
        0.047942655141777091,0.049117799127055078,0.702875228655225,0.04758231784929319,0.70295568967385469,0.0,0.0,
        0.0,0.0,0.0,1.0,0.0,0.0,0.0,-0.0,-0.0,-0.0,-0.0,-0.0,-1.0,-0.0,-0.0,-0.048825402242851333,
        -0.05245230475052743,-0.557871608027596,-0.62654080641868248,-0.63942401877909183,0.041298149353625628,
        0.557871608027596,0.63942401877909183,0.0,0.0,0.0,0.0,0.0,1.0,0.0,0.0,-0.0,-0.0,-0.0,-0.0,-0.0,-1.0,-0.0,
        -0.0,-0.626547232929702,-0.047984758880296075,-0.047630065906767147,-0.58732864799299578,
        -0.049174830154444668,0.047993536136706469,0.38140732638781982,0.049174830154444675,0.047640075741515707,
        0.0,0.0,0.0,0.0,0.0,1.0,0.0,0.0,-0.0,-0.0,-0.0,-0.0,-0.0,-1.0,-0.0,-0.0,-0.047286920841764508,
        -0.55787142569916037,-0.62654193427993921,-0.639425363845251,0.045941301434432633,0.55787142569916037,
        0.052452304750527472,0.62654193427993921,0.639425363845251,0.0,0.0,0.0,0.0,0.0,1.0,0.0,0.0,-0.0,-0.0,-0.0,
        -0.0,-0.0,-1.0,-0.0,-0.0,-0.63943141348019983,-0.047934264404490834,-0.0491093915715111,
        -0.04757405784581345,0.047934264404490834,0.45972838564453733,0.0491093915715111,0.58732864799299578,
        0.04757405784581345,0.0,0.0,0.0,0.0,0.0,1.0,0.0,0.0,-0.0,-0.0,-0.0,-0.0,-0.0,-1.0,-0.0,-0.0,
        0.047942655141777091,0.557872509055183,-0.044607913288060984,-0.70286297549379462,-0.040334527208629158,
        -0.70294446596883164,0.0,0.0,0.0,0.0,0.0,1.0,0.0,0.0,-0.0,-0.0,-0.0,-0.0,-0.0,-1.0,-0.0,-0.0,
        0.04428890112513717,0.041298149353625621,0.052879406986409215,-0.557871950150472,-0.62654033525020214,
        -0.6394234093758725,0.557871950150472,0.62654033525020214,0.6394234093758725,0.0,0.0,0.0,0.0,0.0,1.0,0.0,
        0.0,0.0,0.0,-0.0,-0.0,-0.0,-0.0,-0.0,-1.0,-0.0,0.047984758880296068,-0.38139322558672084,
        -0.70313339581753054,-0.0,0.041515729018567704,0.62654033525020214,-0.70313108620605158,0.0,0.0,0.0,0.0,0.0,
        1.0,0.0,0.0,-0.0,-0.0,-0.0,-0.0,-0.0,-1.0,0.045941301434432633,0.040021361425923357,-0.55787198584888142,
        -0.0528794069864092,0.63942378652894072,0.0,0.0,0.0,0.0,0.0,1.0,0.0,0.0,-0.0,-0.0,-0.0,-0.0,-0.0,-1.0,-0.0,
        0.047934264404490841,-0.587326232489261,-0.0,0.041479097778282452,0.6394234093758725,0.0,0.0,0.0,0.0,0.0,
        1.0,0.0,0.0,0.0,-0.0,-0.0,-0.0,-0.0,-0.0,-1.0,0.047942655141777091,-0.557872509055183,-0.0,
        0.041486488318378048,-0.027677161979573293,0.70294159791647837,0.0,0.0,0.0,0.0,0.0,1.0,0.0,0.0,-0.0,-0.0,
        -0.0,-0.0,-0.0,-1.0,-0.0,0.047984758880296068,-0.62654217515979649,-0.044660621016635559,
        0.38139322558672084,0.70313339581753065,0.0,0.0,0.0,0.0,1.0,0.0,-0.0,-0.0,-0.0,-0.0,-0.0,-1.0,-0.0,
        0.047934264404490841,-0.63942545184526778,-0.0446006835917423,-0.040327604063683457,0.45973364369000819,
        0.587326232489261,0.0,0.0,0.0,0.0,0.0,1.0,0.0,-0.0,-0.0,-0.0,-0.0,-0.0,-1.0,-0.0,-0.0,0.55787171658183987,
        0.049198241144151271,0.38141432182325924,-0.041543427917705961,-0.027753531302003462,0.0,0.0,0.0,0.0,0.0,
        1.0,0.0,0.0,-0.0,-0.0,-0.0,-0.0,-0.0,-1.0,0.381386025829566,0.702875228655225,-0.048014979218259819,
        -0.049198241144151264,-0.047663646280299156,-0.70314122138856006,0.048014979218259819,0.049198241144151271,
        0.047663646280299156,0.0,0.0,0.0,0.0,0.0,1.0,0.0,0.0,-0.0,-0.0,-0.0,-0.0,-0.0,-1.0,0.55787142569916048,
        0.04758231784929319,-0.046165728248822986,-0.052734339992385214,-0.70286396678410767,0.0,0.0,0.0,0.0,0.0,
        1.0,0.0,0.0,-0.0,-0.0,-0.0,-0.0,-0.0,-1.0,-0.0,0.45972838564453744,0.70295568967385458,-0.04765651814247162,
        0.048008393947647693,0.049191105586226781,0.047656518142471613,0.0,0.0,0.0,0.0,0.0,1.0,0.0,0.0,0.0,0.0,-0.0,
        -0.0,-0.0,-0.0,-0.0,-1.0,-0.0,0.557872509055183,-0.0479426551417771,-0.70286297549379462,
        0.044607913288061025,0.040334527208629151,0.0,0.0,0.0,0.0,0.0,1.0,0.0,0.0,-0.0,-0.0,-0.0,-0.0,-0.0,-1.0,
        -0.0,-0.0,0.55787171658183987,-0.049117799127055085,-0.70286143698134129,0.041486488318378041,
        0.027661054311066195,0.0,0.0,0.0,0.0,0.0,1.0,0.0,-0.0,-0.0,-0.0,-0.0,-0.0,-1.0,-0.0,0.55787142569916048,
        -0.04758231784929319,-0.70286396678410767,-0.70294533564091966,0.046165728248822986,0.052734339992385255,
        0.0,0.0,0.0,0.0,0.0,1.0,0.0,-0.0,-0.0,-0.0,-0.0,-0.0,-1.0,-0.0,-0.0,0.049164972356125373,
        0.62654101707515264,0.052779600708881172,0.58732523320298258,-0.041521734602731605,-0.38141436310945664,0.0,
        0.0,0.0,0.0,0.0,1.0,0.0,0.0,-0.0,-0.0,-0.0,-0.0,-0.0,-1.0,0.049109391571511091,0.63942424475811355,
        0.052725613098002319,-0.041479097778282452,-0.58732507052489791,0.0,0.0,0.0,0.0,0.0,1.0,0.0,0.0,-0.0,-0.0,
        -0.0,-0.0,-0.0,-1.0,0.049117799127055078,0.70294302173702006,0.052734339992385228,-0.557871608027596,
        -0.041486711482857687,0.70286111061272671,0.0,0.0,0.0,0.0,0.0,1.0,0.0,0.0,-0.0,-0.0,-0.0,-0.0,-0.0,-1.0,
        -0.0,0.052779600708881172,-0.62654080641868259,-0.041515729018567711,0.381393060579516,0.70313207851881332,
        0.0,0.0,0.0,0.0,1.0,-0.0,-0.0,-0.0,-0.0,-1.0,0.62654193427993921,0.047630065906767147,0.58732556690019289,
        -0.38141260703668056,-0.052788975072809517,0.0,0.0,0.0,0.0,0.0,1.0,0.0,0.0,-0.0,-0.0,-0.0,-0.0,-0.0,-1.0,
        0.62654217515979649,0.040386220026432475,0.587326232489261,-0.047993536136706476,-0.38141452789755637,
        0.044671688889686353,0.0,0.0,0.0,0.0,0.0,1.0,0.0,0.0,-0.0,-0.0,-0.0,-0.0,-0.0,-1.0,-0.0,0.62654101707515253,
        0.58732523320298247,-0.049174830154444668,-0.38141432182325907,0.041521509739207062,0.027720209169872088,
        0.0,0.0,0.0,0.0,1.0,-0.0,-0.0,-0.0,-0.0,-1.0,0.62654193427993921,0.04620090230449761,0.0527796007088812,
        0.58732556690019289,-0.0476400757415157,-0.38141260703668056,0.0,0.0,0.0,0.0,0.0,1.0,0.0,-0.0,-0.0,-0.0,
        -0.0,-0.0,-1.0,-0.0,0.047574057845813457,0.639425363845251,-0.052725613098002347,-0.58732556690019289,0.0,
        0.0,0.0,0.0,0.0,1.0,0.0,0.0,-0.0,-0.0,-0.0,-0.0,-0.0,-1.0,0.04758231784929319,-0.55787142569916037,
        -0.052734339992385269,0.70286396678410767,0.70294533564091966,0.0,0.0,0.0,0.0,0.0,1.0,0.0,0.0,-0.0,-0.0,
        -0.0,-0.0,-0.0,-1.0,-0.0,0.04763006590676714,-0.62654193427993921,-0.052779600708881193,0.38139130491870232,
        0.703133933677141,0.0,0.0,0.0,0.0,1.0,-0.0,-0.0,-0.0,-0.0,-1.0,0.047574057845813457,-0.639425363845251,
        -0.04615757913241255,-0.052725613098002347,0.45973190050489804,0.58732556690019289,0.0,0.0,0.0,0.0,0.0,1.0,
        0.0,-0.0,-0.0,-0.0,-0.0,-0.0,-1.0,-0.0,0.63942545184526778,-0.047934264404490834,-0.587326232489261,
        0.044600683591742338,0.04032760406368343,0.0,0.0,0.0,0.0,0.0,1.0,0.0,0.0,-0.0,-0.0,-0.0,-0.0,-0.0,-1.0,-0.0,
        0.63942424475811355,-0.0491093915715111,-0.58732523320298258,0.041478874690674995,0.027655051949837254,0.0,
        0.0,0.0,0.0,1.0,-0.0,-0.0,-0.0,-0.0,-1.0,0.639425363845251,-0.047574057845813443,-0.58732556690019289,
        0.04615757913241255,0.052725613098002382,0.0,0.0,0.0,0.0,0.0,1.0,0.0,-0.0,-0.0,-0.0,-0.0,-0.0,-1.0,-0.0,
        -0.047942655141777091,-0.557872509055183,0.044607913288061012,0.70286297549379462,0.040334527208629144,
        0.70294446596883164,0.0,0.0,0.0,0.0,0.0,1.0,0.0,0.0,-0.0,-0.0,-0.0,-0.0,-0.0,-1.0,-0.0,-0.0,
        -0.041297934356687133,-0.0442889011251372,-0.55787205898156167,0.027381569976781938,0.63942363589545237,0.0,
        0.0,0.0,0.0,0.0,1.0,0.0,-0.0,-0.0,-0.0,-0.0,-0.0,-1.0,-0.0,-0.0,-0.047984758880296068,-0.62654217515979649,
        0.38139322558672084,0.044660621016635579,0.040386220026432489,0.70313339581753065,0.0,0.0,0.0,0.0,1.0,-0.0,
        -0.0,-0.0,-0.0,-1.0,-0.0,-0.045941301434432633,-0.04002136142592335,-0.041298149353625628,
        -0.027381569976781941,-0.557871950150472,-0.62654033525020214,-0.6394234093758725,0.557871950150472,
        0.6394234093758725,0.0,0.0,0.0,0.0,0.0,1.0,0.0,0.0,-0.0,-0.0,-0.0,-0.0,-0.0,-1.0,-0.0,-0.0,-0.0,
        -0.047934264404490841,-0.63942545184526778,0.45973364369000819,0.044600683591742324,0.587326232489261,
        0.040327604063683443,0.0,0.0,0.0,0.0,0.0,1.0,0.0,-0.0,-0.0,-0.0,-0.0,-0.0,-1.0,-0.0,-0.0,
        -0.55787171658183987,-0.049117799127055085,0.041486488318378041,0.70286143698134129,0.027661054311066195,
        0.70294302173702006,0.0,0.0,0.0,0.0,1.0,-0.0,-0.0,-0.0,-0.0,-1.0,-0.0,-0.381386025829566,
        -0.70287522865522511,-0.048014979218259819,-0.049198241144151264,-0.047663646280299156,0.048014979218259819,
        0.049198241144151271,0.047663646280299156,0.70314122138856006,0.0,0.0,0.0,0.0,1.0,0.0,-0.0,-0.0,-0.0,-0.0,
        -0.0,-1.0,-0.0,-0.0,-0.55787142569916048,-0.04758231784929319,0.046165728248822986,0.052734339992385255,
        0.70286396678410767,0.70294533564091966,0.0,0.0,0.0,0.0,0.0,1.0,0.0,-0.0,-0.0,-0.0,-0.0,-0.0,-1.0,-0.0,-0.0,
        -0.45972838564453744,-0.70295568967385458,-0.04765651814247162,0.048008393947647693,0.70268597089371387,0.0,
        0.0,0.0,0.0,0.0,1.0,0.0,-0.0,-0.0,-0.0,-0.0,-0.0,-1.0,-0.0,-0.049164972356125373,-0.62654101707515264,
        0.041515504461835731,0.38139301933175634,0.027709698583410016,0.70313230364575241,0.0,0.0,0.0,1.0,-0.0,-0.0,
        -0.0,-1.0,-0.049109391571511105,-0.052725613098002361,-0.63942401877909172,0.041479097778282459,
        0.45973321032477427,0.58732507052489791,0.0,0.0,0.0,0.0,0.0,1.0,-0.0,-0.0,-0.0,-0.0,-0.0,-1.0,-0.0,-0.0,
        -0.62654193427993921,-0.047630065906767147,0.04620090230449761,0.38139130491870232,0.052779600708881227,
        0.703133933677141,0.0,0.0,0.0,0.0,0.0,1.0,-0.0,-0.0,-0.0,-0.0,-0.0,-1.0,-0.0,-0.047574057845813457,
        -0.639425363845251,0.046157579132412557,0.45973190050489804,0.052725613098002388,0.58732556690019289,0.0,
        0.0,0.0,0.0,0.0,1.0,-0.0,-0.0,-0.0,-0.0,-0.0,-1.0,-0.0,-0.0,0.044696511233766632,0.041537644408465073,
        0.38139435220779871,0.0046455551781967915,-0.70313098732427648,0.0,0.0,0.0,0.0,0.0,1.0,0.0,0.0,0.0,-0.0,
        -0.0,-0.0,-0.0,-0.0,-1.0,0.048014979218259812,0.38139322558672073,0.70286297549379451,-0.04469651123376666,
        -0.70313329820348291,0.0,0.0,0.0,0.0,0.0,1.0,-0.0,-0.0,-0.0,-0.0,-1.0,-0.0,0.046165728248822986,
        0.040334527208629165,0.041486711482857673,0.55787195015047186,-0.70285954634074388,0.0,0.0,0.0,0.0,0.0,1.0,
        0.0,0.0,0.0,-0.0,-0.0,-0.0,-0.0,-0.0,-1.0,-0.0,0.047993536136706476,-0.38141452789755642,-0.0,
        0.70313131216765046,0.0415217346027316,0.0053499825507371153,0.0015656878741349531,0.0,0.0,0.0,0.0,0.0,1.0,
        0.0,0.0,0.0,-0.0,-0.0,-0.0,-0.0,-0.0,-1.0,0.04615757913241255,0.040327604063683457,0.041479097778282452,
        0.027671157031094271,-0.6394234093758725,0.45973424542066693,0.58732499879699229,0.0,0.0,0.0,0.0,0.0,1.0,
        0.0,0.0,-0.0,-0.0,-0.0,-0.0,-0.0,-1.0,-0.0,0.048014979218259812,-0.38139322558672073,-0.70286297549379451,
        -0.04469651123376666,0.70313329820348291,0.0,0.0,0.0,0.0,1.0,0.0,-0.0,-0.0,-0.0,-0.0,-0.0,-1.0,-0.0,-0.0,
        0.047993536136706476,-0.587326232489261,-0.044671688889686333,-0.040397149349959804,0.38141452789755642,0.0,
        0.0,0.0,0.0,0.0,1.0,0.0,-0.0,-0.0,-0.0,-0.0,-0.0,-1.0,-0.0,-0.0,0.557871608027596,0.052734339992385235,
        0.027661054311066337,-0.041486711482857694,-0.70286111061272671,0.0,0.0,0.0,0.0,0.0,1.0,0.0,0.0,-0.0,-0.0,
        -0.0,-0.0,-0.0,-1.0,-0.0,0.70286396678410779,0.047663646280299149,0.38141260703668067,-0.052821149416567043,
        0.0,0.0,0.0,0.0,0.0,1.0,0.0,0.0,0.0,-0.0,-0.0,-0.0,-0.0,-0.0,-1.0,0.38140732638781988,0.0015661221639725058,
        -0.048023761687426413,-0.049208104725552843,-0.047673661972528605,0.048023761687426413,0.049208104725552849,
        0.0476736619725286,0.0,0.0,0.0,0.0,0.0,1.0,0.0,0.0,0.0,0.0,-0.0,-0.0,-0.0,-0.0,-0.0,-1.0,-0.0,
        0.70286297549379451,0.04042146861842183,0.38141452789755653,-0.048023761687426413,0.044707585477670696,0.0,
        0.0,0.0,0.0,0.0,1.0,0.0,0.0,0.0,-0.0,-0.0,-0.0,-0.0,-0.0,-1.0,-0.0,0.70286143698134129,0.38141432182325918,
        -0.049208104725552843,0.041543427917705954,0.027753531302003361,0.0,0.0,0.0,0.0,1.0,0.0,-0.0,-0.0,-0.0,-0.0,
        -1.0,0.38139130491870249,0.70286396678410779,-0.047663646280299149,-0.70313383642924188,
        0.046226776721425993,0.052811769511494744,0.0,0.0,0.0,0.0,0.0,1.0,0.0,-0.0,-0.0,-0.0,-0.0,-0.0,-1.0,
        0.38141260703668073,0.0015661807001885121,-0.0003808990881292652,0.046234063364270737,0.052821149416567105,
        0.0,0.0,0.0,0.0,0.0,1.0,0.0,0.0,-0.0,-0.0,-0.0,-0.0,-0.0,-1.0,-0.0,0.55787205898156167,
        -0.041486488318378034,-0.044607913288061032,0.02767716197957313,0.0,0.0,0.0,0.0,0.0,1.0,0.0,-0.0,-0.0,-0.0,
        -0.0,-0.0,-1.0,-0.0,-0.0,0.55787198584888142,0.38139402411953655,-0.046226776721426013,-0.04042146861842183,
        -0.70313145912642394,0.053301939043787668,0.0,0.0,0.0,0.0,1.0,0.0,-0.0,-0.0,-0.0,-0.0,-0.0,-1.0,-0.0,
        0.557871608027596,-0.052734339992385269,-0.70286111061272671,-0.70294271779415229,0.041486711482857687,0.0,
        0.0,0.0,0.0,0.0,1.0,0.0,-0.0,-0.0,-0.0,-0.0,-0.0,-1.0,-0.0,-0.0,0.052725613098002319,0.027655051949837452,
        -0.63942401877909172,-0.041479097778282452,0.45973321032477427,0.58732507052489791,0.0,0.0,0.0,0.0,0.0,1.0,
        0.0,-0.0,-0.0,-0.0,-0.0,-0.0,-1.0,-0.0,0.052811769511494709,-0.381393060579516,-0.70286111061272671,
        -0.041537644408465066,0.70313198021515855,0.0,0.0,0.0,0.0,1.0,-0.0,-0.0,-0.0,-1.0,-0.0,-0.0,
        0.049174830154444661,0.052788975072809545,-0.58732507052489813,-0.041521734602731612,0.38141436310945631,
        0.0,0.0,0.0,0.0,0.0,1.0,0.0,-0.0,-0.0,-0.0,-0.0,-0.0,-1.0,-0.0,0.6265406645097189,-0.046200902304497617,
        -0.040386220026432475,-0.38139402411953627,-0.70313155774868141,0.053264773578912634,0.0,0.0,0.0,0.0,1.0,
        -0.0,-0.0,-0.0,-0.0,-0.0,-1.0,-0.0,0.62654080641868248,0.58732507052489791,-0.052788975072809559,
        -0.38141436310945637,0.0415217346027316,0.0,0.0,0.0,0.0,0.0,1.0,0.0,-0.0,-0.0,-0.0,-0.0,-0.0,-1.0,-0.0,
        0.047663646280299156,-0.38139130491870238,-0.70286396678410779,-0.052811769511494681,0.70313383642924188,
        0.0,0.0,0.0,0.0,1.0,-0.0,-0.0,-0.0,-1.0,-0.0,-0.0,-0.45973190050489809,-0.70294533564091954,
        -0.052804674695198853,0.00038089908812926509,-0.38141260703668056,-0.046234063364270724,0.0,0.0,0.0,0.0,0.0,
        1.0,0.0,-0.0,-0.0,-0.0,-0.0,-0.0,-1.0,-0.0,-0.0,0.047640075741515714,-0.58732556690019289,
        -0.046208184541143907,-0.0527889750728095,0.38141260703668045,0.0,0.0,0.0,0.0,0.0,1.0,0.0,-0.0,-0.0,-0.0,
        -0.0,-0.0,-1.0,-0.0,0.63942378652894072,-0.046157579132412543,-0.040327604063683443,-0.587325187651558,
        0.053202204406742878,0.0,0.0,0.0,0.0,0.0,1.0,0.0,-0.0,-0.0,-0.0,-0.0,-0.0,-1.0,-0.0,0.63942401877909172,
        -0.052725613098002388,-0.5873250705248978,0.041479097778282417,0.0,0.0,0.0,0.0,0.0,1.0,0.0,-0.0,-0.0,-0.0,
        -0.0,-0.0,-1.0,-0.0,-0.046165728248822993,-0.55787198584888142,-0.040334527208629144,-0.041486711482857666,
        0.70285954634074388,0.70294129315678422,0.0,0.0,0.0,0.0,0.0,1.0,0.0,-0.0,-0.0,-0.0,-0.0,-0.0,-1.0,-0.0,-0.0,
        -0.0,-0.048008393947647693,-0.45973364369000813,-0.70294446596883153,0.04468906953870326,0.7026717750678485,
        0.040414301735567953,0.0,0.0,0.0,0.0,1.0,0.0,-0.0,-0.0,-0.0,-0.0,-0.0,-1.0,-0.0,-0.0,-0.044600683591742331,
        -0.041479097778282431,-0.053202204406742781,-0.6394234093758725,0.58732499879699229,0.0,0.0,0.0,0.0,0.0,1.0,
        -0.0,-0.0,-0.0,-0.0,-0.0,-1.0,-0.0,-0.0,-0.0,-0.04620090230449761,-0.62654066450971879,
        -0.040386220026432489,0.38139402411953638,0.053264773578912634,0.70313155774868152,0.0,0.0,0.0,1.0,-0.0,
        -0.0,-0.0,-0.0,-1.0,-0.0,-0.047993536136706476,-0.587326232489261,0.38141452789755642,0.044671688889686353,
        0.040397149349959791,0.0,0.0,0.0,0.0,0.0,1.0,0.0,-0.0,-0.0,-0.0,-0.0,-0.0,-1.0,-0.0,-0.0,
        -0.046157579132412557,-0.040327604063683437,-0.63942378652894072,0.4597340245185435,0.0532022044067428,
        0.58732518765155828,0.0,0.0,0.0,0.0,1.0,-0.0,-0.0,-0.0,-0.0,-0.0,-1.0,-0.0,-0.557871608027596,
        -0.052734339992385269,0.041486711482857687,0.70286111061272671,0.70294271779415229,0.0,0.0,0.0,0.0,0.0,1.0,
        0.0,-0.0,-0.0,-0.0,-0.0,-0.0,-1.0,-0.0,-0.0,-0.45973321958975349,-0.049191105586226788,-0.70294302173702006,
        0.041532433509010709,0.70267008402296527,0.027736669979992645,0.0,0.0,0.0,1.0,-0.0,-0.0,-0.0,-0.0,-1.0,-0.0,
        -0.38140732638781988,-0.0030799473449444718,-0.048023761687426413,-0.049208104725552843,
        -0.047673661972528605,0.048023761687426413,0.049208104725552849,0.0476736619725286,0.0,0.0,0.0,0.0,0.0,1.0,
        0.0,0.0,-0.0,-0.0,-0.0,-0.0,-0.0,-1.0,-0.0,-0.0,-0.0,-0.052779600708881207,-0.62654080641868259,
        0.0415157290185677,0.38139306057951583,0.70313207851881332,0.0,0.0,0.0,0.0,0.0,1.0,-0.0,-0.0,-0.0,-0.0,-0.0,
        -1.0,-0.0,-0.049174830154444675,-0.58732523320298258,0.041521509739207041,0.381414321823259,
        0.027720209169872008,0.0,0.0,0.0,0.0,0.0,1.0,-0.0,-0.0,-0.0,-0.0,-0.0,-1.0,-0.0,-0.58732556690019289,
        -0.047640075741515707,0.046208184541143907,0.38141260703668056,0.052788975072809566,0.0,0.0,0.0,0.0,0.0,1.0,
        -0.0,-0.0,-0.0,-0.0,-0.0,-1.0,-0.0,-0.0,0.048023761687426413,0.38141452789755642,0.70313329820348291,
        -0.044707585477670654,0.0,0.0,0.0,0.0,0.0,1.0,0.0,0.0,0.0,-0.0,-0.0,-0.0,-0.0,-0.0,-1.0,-0.0,
        0.0414867114828577,6.14559350203706E-5,-0.55787195015047186,0.70285954634074388,0.70294129315678422,0.0,0.0,
        0.0,0.0,0.0,1.0,0.0,0.0,0.0,-0.0,-0.0,-0.0,-0.0,-0.0,-1.0,-0.0,0.041515729018567704,0.027725808084743217,
        -0.62654033525020214,0.38139435220779894,0.70313108620605158,0.0,0.0,0.0,0.0,1.0,0.0,-0.0,-0.0,-0.0,-0.0,
        -1.0,0.044696511233766639,-0.70285987351907608,0.04153764440846508,-0.3813943522077986,
        -0.0046455551781967924,0.70313098732427659,0.0,0.0,0.0,0.0,1.0,-0.0,-0.0,-0.0,-1.0,-0.0,-0.0,
        0.046208184541143921,0.040397149349959804,-0.58732518765155828,0.041521734602731619,-0.0053499825507371188,
        0.38141565496819624,0.0,0.0,0.0,0.0,0.0,1.0,0.0,0.0,-0.0,-0.0,-0.0,-0.0,-0.0,-1.0,-0.0,0.048023761687426413,
        -0.38141452789755642,-0.7026717750678485,-0.044707585477670654,-0.040432404230908,0.0,0.0,0.0,0.0,0.0,1.0,
        0.0,-0.0,-0.0,-0.0,-0.0,-0.0,-1.0,-0.0,-0.0,-0.0,0.041521509739207062,0.044671688889686333,
        -0.58732516183395489,-0.027736318903840668,0.3814156136550157,0.0,0.0,0.0,0.0,0.0,1.0,0.0,-0.0,-0.0,-0.0,
        -0.0,-0.0,-1.0,0.052811769511494695,0.70286111061272671,0.027743014678389594,0.38141436310945653,
        6.1605929268691053E-5,-0.04154365368638769,0.0,0.0,0.0,0.0,0.0,1.0,0.0,0.0,0.0,-0.0,-0.0,-0.0,-0.0,-0.0,
        -1.0,0.38139306057951616,0.70286111061272671,-0.052811769511494744,-0.70313198021515855,0.04153764440846508,
        0.0,0.0,0.0,0.0,0.0,1.0,0.0,-0.0,-0.0,-0.0,-0.0,-0.0,-1.0,0.0015662095088587794,0.0,-0.0,
        0.38139435220779888,-0.041537644408465059,-0.00023256610403676135,0.0,0.0,0.0,0.0,0.0,1.0,0.0,-0.0,-0.0,
        -0.0,-0.0,-0.0,-1.0,-0.0,0.38141436310945653,0.0015661981899676553,-0.0004794577441265344,
        0.041543653686387648,0.0,0.0,0.0,0.0,0.0,1.0,0.0,0.0,-0.0,-0.0,-0.0,-0.0,-0.0,-1.0,-0.0,0.55787195015047186,
        -0.041486711482857659,-0.00023216176133703439,-0.70285954634074388,-0.70294129315678422,0.0,0.0,0.0,0.0,0.0,
        1.0,0.0,-0.0,-0.0,-0.0,-0.0,-0.0,-1.0,-0.0,-0.0,-0.0,-0.45973321032477421,-0.70294271779415229,
        -0.041532658817056131,0.0004794577441265338,-0.38141436310945637,0.0,0.0,0.0,0.0,0.0,1.0,0.0,-0.0,-0.0,-0.0,
        -0.0,-0.0,-1.0,-0.0,-0.0,0.70313155774868141,-0.046208184541143935,-0.040397149349959777,
        -0.38141532678103607,0.0053499825507371248,0.0015656878741349477,-0.041521734602731612,0.0,0.0,0.0,0.0,0.0,
        1.0,0.0,-0.0,-0.0,-0.0,-0.0,-0.0,-1.0,-0.0,-0.0,0.62654033525020214,-0.041515729018567704,
        -0.053264773578912579,-0.38139435220779877,-0.70313108620605158,0.0,0.0,0.0,0.0,0.0,1.0,-0.0,-0.0,-0.0,-0.0,
        -0.0,-1.0,-0.0,-0.0,0.63942340937587239,-0.041479097778282424,-0.053202204406742795,-0.58732499879699218,
        0.0,0.0,0.0,0.0,0.0,1.0,0.0,-0.0,-0.0,-0.0,-0.0,-0.0,-1.0,-0.0,-0.0,-0.046220967236855211,
        -0.45973402451854339,-0.04041430173556794,-0.7029419471796341,0.05329394831239747,0.70266869475347082,0.0,
        0.0,0.0,1.0,-0.0,-0.0,-0.0,-0.0,-0.0,-1.0,-0.0,-0.0,-0.048023761687426413,-0.38141452789755642,
        -0.7026717750678485,0.044707585477670675,0.040432404230907985,0.0,0.0,0.0,0.0,0.0,1.0,0.0,-0.0,-0.0,-0.0,
        -0.0,-0.0,-1.0,-0.0,-0.0,-0.0,-0.62654033525020214,-0.0,-0.041521509739207055,-0.04467168888968636,
        -0.58732516183395489,0.3814156136550157,0.0,0.0,0.0,0.0,0.0,1.0,-0.0,-0.0,-0.0,-0.0,-0.0,-1.0,-0.0,-0.0,
        -0.046208184541143914,-0.58732518765155806,-0.040397149349959791,0.38141532678103618,0.053276115903559441,
        0.0,0.0,0.0,0.0,1.0,-0.0,-0.0,-0.0,-0.0,-0.0,-1.0,-0.0,-0.049208104725552843,-0.38141436310945653,
        -0.00047945774412653418,-0.0015661981899676573,0.041543653686387676,0.0,0.0,0.0,0.0,0.0,1.0,-0.0,-0.0,-0.0,
        -0.0,-0.0,-1.0,-0.0,-0.0,-0.0,-0.38141260703668067,-0.0030800493725469838,-0.00038089908812926525,
        0.046234063364270724,0.052821149416567063,0.0,0.0,0.0,0.0,0.0,1.0,-0.0,-0.0,-0.0,-0.0,-0.0,-1.0,-0.0,-0.0,
        -0.0,-0.052788975072809573,-0.5873250705248978,-0.027720209169872036,-0.70313207851881321,
        0.041521734602731585,0.38141436310945664,0.0,0.0,0.0,0.0,0.0,1.0,-0.0,-0.0,-0.0,-0.0,-0.0,-1.0,-0.0,-0.0,
        0.041543427917705968,0.38141561365501536,0.00029424831666778297,0.0015662085872463908,-0.027769643467705708,
        0.0,0.0,0.0,0.0,0.0,1.0,0.0,0.0,0.0,-0.0,-0.0,-0.0,-0.0,-0.0,-1.0,0.041532658817056138,
        -0.0031055287133001592,0.70266788285587956,0.0,0.0,0.0,0.0,1.0,0.0,0.0,0.0,0.0,-0.0,-0.0,-0.0,-0.0,-0.0,
        -1.0,-0.0,0.041543427917705961,-0.0030801002245625041,0.00023261598934981646,-0.381415654968196,
        -0.0030801017285724173,0.0,0.0,0.0,0.0,0.0,1.0,0.0,0.0,-0.0,-0.0,-0.0,-0.0,-0.0,-1.0,-0.0,-0.0,
        0.046234063364270724,0.00017791507742684638,-0.38141532678103585,-0.053313287899267439,0.0,0.0,0.0,0.0,0.0,
        1.0,0.0,-0.0,-0.0,-0.0,-0.0,-0.0,-1.0,-0.0,-0.0,-0.04623406336427073,-0.38141532678103612,
        -0.003080095298344224,-0.00017791507742684627,0.053313287899267488,0.0,0.0,0.0,0.0,1.0,-0.0,-0.0,-0.0,-0.0,
        -0.0,-1.0,-0.0,-0.0,-0.041543427917705961,-0.00029424831666778313,-0.38141565496819613,
        -0.0015662095088587807,0.0,0.0,0.0,0.0,0.0,1.0,-0.0,-0.0,-0.0,-0.0,-0.0,-1.0,-0.0,-0.0,-0.0,-0.0,
        0.041543653686387669,0.38141565496819613,6.1661881147355389E-5,0.0015662095088587807,0.0,0.0,0.0,0.0,0.0,
        1.0,0.0,0.0,0.0,0.0,-0.0,-0.0,-0.0,-0.0,-0.0,-1.0,0.555673663731469,0.026771909379554294,
        0.62490021645747618,0.027265477962947069,0.63800507768378811,0.026352061912650541,-0.555673663731469,
        -0.026771909379554294,-0.62490021645747618,-0.027265477962947066,-0.63800507768378822,-0.026352061912650541,
        0.0,0.0,0.0,0.0,0.0,0.0,1.0,0.0,0.0,0.0,-0.0,-0.0,-0.0,-0.0,-0.0,-0.0,-1.0,-0.0,-0.555673663731469,
        0.027034185307057625,0.70226225634217321,0.027566488177000262,0.7025340602672151,0.026662833272981429,
        -0.027034185307057625,-0.027566488177000258,-0.026662833272981429,0.0,0.0,0.0,0.0,0.0,0.0,0.0,0.0,0.0,-0.0,
        -0.0,-0.0,-0.0,-0.0,-0.0,-1.0,-0.0,-0.026771909379554291,0.55566424910285672,0.62488504774223075,
        0.024399835479656965,0.63798948327222038,0.021960985394712317,-0.55566424910285672,-0.62488504774223075,
        -0.63798948327222038,0.0,0.0,0.0,0.0,0.0,0.0,1.0,0.0,0.0,-0.0,-0.0,-0.0,-0.0,-0.0,-0.0,-1.0,-0.0,
        -0.62490021645747618,-0.02706527731251647,-0.026700746627905073,-0.58505858013174894,0.37854052611351124,
        0.027072082181883242,0.027610578309122807,0.026708907388227909,-0.027610578309122804,0.0,0.0,0.0,0.0,0.0,
        0.0,1.0,0.0,0.0,-0.0,-0.0,-0.0,-0.0,-0.0,-0.0,-0.0,-0.027265477962947069,-0.55566222109490582,
        -0.63798667601923609,-0.029437135799321903,0.55566181651356428,0.023469887537635181,0.62488169574462793,
        0.63798609648432814,0.0,0.0,0.0,0.0,0.0,0.0,1.0,0.0,0.0,-0.0,-0.0,-0.0,-0.0,-0.0,-0.0,-1.0,
        -0.63800507768378822,0.45692709004827581,0.027011667529779945,0.58505858013174894,0.027541181508898387,
        0.026637267215644224,-0.027011667529779945,-0.027541181508898383,-0.026637267215644224,0.0,0.0,0.0,0.0,0.0,
        0.0,1.0,0.0,0.0,-0.0,-0.0,-0.0,-0.0,-0.0,-0.0,-0.0,-0.026352061912650541,0.55566389422834717,
        0.02598312883534095,0.62488507878410182,0.02943713579932191,0.637989575133729,-0.55566389422834717,
        -0.62488507878410182,-0.63798957513372911,0.0,0.0,0.0,0.0,0.0,0.0,1.0,0.0,0.0,-0.0,-0.0,-0.0,-0.0,-0.0,-0.0,
        -1.0,0.555673663731469,0.027034185307057625,0.027566488177000262,0.026662833272981429,-0.027034185307057625,
        -0.70226225634217321,-0.027566488177000258,-0.7025340602672151,-0.026662833272981429,0.0,0.0,0.0,0.0,0.0,
        0.0,1.0,0.0,0.0,-0.0,-0.0,-0.0,-0.0,-0.0,-0.0,-0.0,-0.0,0.026771909379554291,0.55566424910285672,
        0.62488504774223075,0.63798948327222038,-0.55566424910285672,-0.62488504774223075,-0.024399835479656955,
        -0.63798948327222038,-0.021960985394712317,0.0,0.0,0.0,0.0,0.0,0.0,1.0,0.0,0.0,-0.0,-0.0,-0.0,-0.0,-0.0,
        -0.0,-1.0,-0.0,0.62490021645747618,0.58505858013174883,0.027072082181883242,0.027610578309122807,
        0.026708907388227909,-0.37854052611351124,-0.027072082181883242,-0.026708907388227909,0.0,0.0,0.0,0.0,0.0,
        0.0,0.0,0.0,-0.0,-0.0,-0.0,-0.0,-0.0,-0.0,-1.0,-0.0,0.027265477962947069,0.55566222109490582,
        0.63798667601923609,0.029437135799321879,0.62488169574462793,-0.55566181651356428,-0.023469887537635192,
        -0.62488169574462793,-0.63798609648432814,0.0,0.0,0.0,0.0,0.0,0.0,1.0,0.0,-0.0,-0.0,-0.0,-0.0,-0.0,-0.0,
        -1.0,-0.0,0.63800507768378822,0.027011667529779945,0.027541181508898387,0.026637267215644224,
        -0.45692709004827581,-0.027011667529779945,-0.58505858013174894,-0.027541181508898383,-0.026637267215644224,
        0.0,0.0,0.0,0.0,0.0,0.0,0.0,0.0,-0.0,-0.0,-0.0,-0.0,-0.0,-0.0,-1.0,-0.0,0.026352061912650541,
        0.55566389422834717,0.62488507878410182,0.637989575133729,-0.55566389422834717,-0.02598312883534095,
        -0.62488507878410182,-0.0294371357993219,-0.63798957513372911,0.0,0.0,0.0,0.0,0.0,0.0,1.0,0.0,-0.0,-0.0,
        -0.0,-0.0,-0.0,-0.0,-1.0,-0.0,-0.55566424910285672,-0.027034185307057621,0.70224208707170055,
        0.024752136540096732,0.70251617195999394,0.022319435462106595,0.0,0.0,0.0,0.0,0.0,0.0,0.0,0.0,-0.0,-0.0,
        -0.0,-0.0,-0.0,-0.0,-1.0,-0.0,-0.70226225634217332,-0.3785405261135113,-0.70163518723474272,
        0.027105602758215112,0.027648865450003536,0.026748274296612785,-0.027105602758215112,-0.027648865450003533,
        -0.026748274296612785,0.0,0.0,0.0,0.0,0.0,0.0,1.0,0.0,0.0,0.0,-0.0,-0.0,-0.0,-0.0,-0.0,-0.0,-0.0,
        -0.55566222109490582,0.023637206391576536,0.015100165961297108,-1.0,-0.378540460951947,-0.02764886545000354,
        0.015207454024849647,0.0,0.0,0.0,0.0,0.0,0.0,1.0,0.0,-0.0,-0.0,-0.0,-0.0,-0.0,-0.0,-0.45692709004827575,
        -0.702534060267215,0.027090859530371859,0.70163518723474272,-0.026730661933064313,0.0,0.0,0.0,0.0,0.0,0.0,
        0.0,0.0,-0.0,-0.0,-0.0,-0.0,-0.0,-0.0,-0.0,-0.55566389422834728,0.029709944333287521,-1.0,
        -0.37854017792555505,-0.026748274296612796,0.0,0.0,0.0,0.0,0.0,0.0,1.0,0.0,0.0,-0.0,-0.0,-0.0,-0.0,-0.0,
        -0.0,-0.55566424910285672,0.027034185307057621,-1.0,-0.37851997948504351,0.70317323754735273,
        -0.02240967789339866,0.0,0.0,0.0,0.0,0.0,0.0,0.0,0.0,-0.0,-0.0,-0.0,-0.0,-0.0,-0.0,-0.0,
        -0.55566222109490582,0.027566488177000255,0.70223873149897853,-0.023637206391576546,-0.015100165961297143,
        0.0,0.0,0.0,0.0,0.0,0.0,-0.0,-0.0,-0.0,-0.0,-0.0,-0.0,-1.0,-0.55566389422834728,0.026662833272981429,
        0.70224253943268344,0.70251656286365771,-0.026190122699982339,-0.029709944333287511,0.0,0.0,0.0,0.0,0.0,0.0,
        0.0,-0.0,-0.0,-0.0,-0.0,-0.0,-0.0,-1.0,-0.0,-0.02706527731251647,-0.6248806237808493,-0.023656120772106486,
        0.378519539943052,0.70317018870025627,0.0,0.0,0.0,0.0,0.0,0.0,0.0,0.0,-0.0,-0.0,-0.0,-0.0,-0.0,-0.0,
        -0.02346980199155271,-0.024399835479656976,0.55566129015943833,0.6248806237808493,0.63798497169620461,
        0.01473301981127613,-0.55566129015943833,-0.6248806237808493,-0.63798497169620461,0.0,0.0,0.0,0.0,0.0,0.0,
        1.0,0.0,-0.0,-0.0,-0.0,-0.0,-0.0,-0.0,-0.027011667529779945,-0.63798948327222027,0.456923837504278,
        0.58504518410006956,0.024723646828030479,0.0,0.0,0.0,0.0,0.0,0.0,1.0,0.0,-0.0,-0.0,-0.0,-0.0,-0.0,-0.0,-0.0,
        -0.02598312883534095,-0.021960985394712324,0.63798532239475636,-0.55566147407010114,-0.62488096344828059,
        -0.63798532239475636,0.0,0.0,0.0,0.0,0.0,0.0,1.0,0.0,0.0,0.0,-0.0,-0.0,-0.0,-0.0,-0.0,-0.0,-1.0,
        -0.027034185307057618,0.55566424910285683,0.024752136540096732,-0.70224208707170055,-0.70251617195999394,
        0.0,0.0,0.0,0.0,0.0,0.0,1.0,0.0,-0.0,-0.0,-0.0,-0.0,-0.0,-0.0,-0.0,-0.0,-0.02706527731251647,
        0.62488504774223075,0.024795740829694754,-0.37851997948504357,-0.7031738370963756,0.0,0.0,0.0,0.0,0.0,0.0,
        0.0,-0.0,-0.0,-0.0,-0.0,-0.0,-0.0,-0.0,-0.027011667529779945,0.63798948327222038,0.024723646828030479,
        0.02229166073122648,-0.456923837504278,-0.58504518410006945,0.0,0.0,0.0,0.0,0.0,0.0,0.0,-0.0,-0.0,-0.0,-0.0,
        -0.0,-0.0,-1.0,-0.0,-0.6248822663250807,-0.0276027315782233,-0.58504257002809312,-0.02974148887250478,
        0.37854036201549385,0.023660396850780661,0.0,0.0,0.0,0.0,0.0,0.0,1.0,0.0,-0.0,-0.0,-0.0,-0.0,-0.0,-0.0,
        -0.62488507878410182,-0.026700746627905073,-0.58504502721143925,0.37854017792555522,0.029748443430697026,
        0.0,0.0,0.0,0.0,0.0,0.0,1.0,0.0,-0.0,-0.0,-0.0,-0.0,-0.0,-0.0,-0.62488504774223086,-0.022364818883998015,
        -0.58504518410006956,0.027072082181883231,0.37854107343057747,-0.024805000972806229,0.0,0.0,0.0,0.0,0.0,0.0,
        1.0,0.0,-0.0,-0.0,-0.0,-0.0,-0.0,-0.0,-0.0,-0.58504257002809312,0.027610578309122814,0.37854046095194716,
        -0.023660296965944735,-0.015161281241640749,0.0,0.0,0.0,0.0,0.0,-0.0,-0.0,-0.0,-0.0,-0.0,
        -0.027541181508898383,-0.637986676019236,-0.029685529684818829,0.023621944154890266,0.58504204394174086,0.0,
        0.0,0.0,0.0,0.0,0.0,1.0,0.0,-0.0,-0.0,-0.0,-0.0,-0.0,-0.0,-0.027566488177000262,-0.70251319697861081,
        -0.029709944333287532,0.55566181651356417,0.023637304191565071,-0.70223802681964376,0.0,0.0,0.0,0.0,0.0,0.0,
        1.0,0.0,-0.0,-0.0,-0.0,-0.0,-0.0,-0.0,-0.0,-0.027602731578223291,-0.02974148887250478,0.62488169574462793,
        0.023656120772106482,-0.37851926782050033,-0.70317150299940423,0.0,0.0,0.0,0.0,0.0,-0.0,-0.0,-0.0,-0.0,-0.0,
        -0.027541181508898383,-0.4569226479042604,-0.58504257002809312,-0.029685529684818829,0.637986096484328,
        0.023621944154890266,0.0,0.0,0.0,0.0,0.0,0.0,0.0,-0.0,-0.0,-0.0,-0.0,-0.0,-0.0,-1.0,-0.637989575133729,
        -0.026637267215644217,0.58504502721143936,0.029685529684818846,0.0,0.0,0.0,0.0,0.0,0.0,1.0,0.0,-0.0,-0.0,
        -0.0,-0.0,-0.0,-0.0,-0.63798948327222038,0.027011667529779945,0.58504518410006945,-0.024723646828030466,
        -0.02229166073122648,0.0,0.0,0.0,0.0,0.0,0.0,1.0,0.0,-0.0,-0.0,-0.0,-0.0,-0.0,-0.0,-0.0,-0.637986676019236,
        0.02754118150889838,0.58504257002809312,-0.023621847095687702,-0.015074517622588319,0.0,0.0,0.0,0.0,0.0,
        -0.0,-0.0,-0.0,-0.0,-0.0,-0.637989575133729,0.026637267215644217,0.45692310525642205,0.58504502721143936,
        -0.026171339658097509,-0.029685529684818822,0.0,0.0,0.0,0.0,0.0,0.0,1.0,-0.0,-0.0,-0.0,-0.0,-0.0,-0.0,-0.0,
        -0.026662833272981426,0.55566389422834728,0.029709944333287525,-0.70224253943268344,-0.70251656286365771,
        0.0,0.0,0.0,0.0,0.0,0.0,1.0,0.0,-0.0,-0.0,-0.0,-0.0,-0.0,-0.0,-0.0,-0.026700746627905069,
        0.62488507878410182,0.02974148887250477,-0.37851908394641454,-0.703174067452467,0.0,0.0,0.0,0.0,0.0,-0.0,
        -0.0,-0.0,-0.0,-0.0,-0.026637267215644227,0.637989575133729,0.029685529684818811,-0.456923105256422,
        -0.58504502721143925,0.0,0.0,0.0,0.0,0.0,0.0,0.0,-0.0,-0.0,-0.0,-0.0,-0.0,-0.0,-1.0,0.55566424910285672,
        0.027034185307057621,-0.70224208707170055,-0.024752136540096722,-0.70251617195999394,-0.022319435462106609,
        0.0,0.0,0.0,0.0,0.0,0.0,1.0,0.0,-0.0,-0.0,-0.0,-0.0,-0.0,-0.0,-0.0,-0.0,0.37851943317454484,
        0.70226225634217332,0.027098793108292794,-0.70318478827029374,-0.02674010789169564,0.0,0.0,0.0,0.0,0.0,0.0,
        0.0,-0.0,-0.0,-0.0,-0.0,-0.0,-0.0,-0.0,-0.0,0.55566222109490582,0.027566488177000255,-0.023637206391576546,
        -0.70223873149897853,-0.70251319697861081,-0.015100165961297143,0.0,0.0,0.0,0.0,0.0,-0.0,-0.0,-0.0,-0.0,
        -0.0,-0.0,0.45692709004827575,0.7025340602672151,0.37854052611351124,0.70318478827029385,
        0.027105602758215112,0.027648865450003536,0.026748274296612785,-0.027105602758215112,-0.026748274296612785,
        0.0,0.0,0.0,0.0,0.0,0.0,0.0,0.0,-0.0,-0.0,-0.0,-0.0,-0.0,-0.0,-1.0,-0.0,-0.0,0.55566389422834728,
        0.026662833272981429,-0.026190122699982339,-0.70224253943268344,-0.029709944333287511,-0.70251656286365771,
        0.0,0.0,0.0,0.0,0.0,0.0,1.0,-0.0,-0.0,-0.0,-0.0,-0.0,-0.0,-0.0,-0.0,0.02706527731251647,0.62488504774223075,
        -0.37851997948504357,-0.024795740829694744,-0.7031738370963756,-0.022364818883998022,0.0,0.0,0.0,0.0,0.0,
        -0.0,-0.0,-0.0,-0.0,-0.0,-0.0,0.02346980199155272,0.024399835479656965,0.55566129015943833,
        0.6248806237808493,0.63798497169620461,-0.55566129015943833,-0.6248806237808493,-0.63798497169620461,
        -0.014733019811276159,0.0,0.0,0.0,0.0,0.0,0.0,-0.0,-0.0,-0.0,-0.0,-0.0,-0.0,-1.0,-0.0,0.027011667529779945,
        0.63798948327222038,-0.456923837504278,-0.58504518410006945,-0.024723646828030469,-0.02229166073122648,0.0,
        0.0,0.0,0.0,0.0,0.0,0.0,-0.0,-0.0,-0.0,-0.0,-0.0,-0.0,-1.0,-0.0,0.02598312883534095,0.021960985394712324,
        0.63798532239475636,-0.55566147407010114,-0.029307880059563592,0.0,0.0,0.0,0.0,0.0,0.0,1.0,-0.0,-0.0,-0.0,
        -0.0,-0.0,-0.0,-0.0,0.6248822663250807,0.027602731578223294,-0.37851936679972537,-0.023656021236335204,
        -0.703171917764931,-0.01515082442675411,0.0,0.0,0.0,0.0,-0.0,-0.0,-0.0,-0.0,0.62488507878410182,
        0.58504502721143936,0.026708907388227905,-0.37854017792555511,-0.026218970645527549,-0.029748443430697016,
        0.0,0.0,0.0,0.0,0.0,0.0,-0.0,-0.0,-0.0,-0.0,-0.0,-0.0,-1.0,-0.0,0.02754118150889838,0.63798667601923609,
        -0.4569226479042604,-0.023621847095687692,-0.585042570028093,-0.015074517622588279,0.0,0.0,0.0,0.0,0.0,0.0,
        -0.0,-0.0,-0.0,-0.0,-0.0,-0.0,-1.0,0.63798957513372911,0.026637267215644217,-0.456923105256422,
        -0.026171339658097509,-0.58504502721143925,-0.029685529684818822,0.0,0.0,0.0,0.0,0.0,0.0,-0.0,-0.0,-0.0,
        -0.0,-0.0,-0.0,-1.0,-0.0,-0.702236447861886,-0.37854073327939103,-0.023682030674840704,
        -0.00016424244292451563,0.015216927320390218,0.0,0.0,0.0,0.0,0.0,0.0,1.0,0.0,0.0,-0.0,-0.0,-0.0,-0.0,-0.0,
        -0.0,-0.55566129015943833,-0.023637206391576532,-0.024752136540096732,0.702236447861886,
        0.015109647396991065,0.0,0.0,0.0,0.0,0.0,0.0,-0.0,-0.0,-0.0,-0.0,-0.0,-1.0,-0.45692383750427795,
        -0.70251617195999394,-0.37854107343057741,-0.027105602758215115,0.024849423695496659,0.0,0.0,0.0,0.0,0.0,
        0.0,1.0,0.0,0.0,-0.0,-0.0,-0.0,-0.0,-0.0,-0.0,-0.0,-0.55566181651356428,0.023637304191565081,-1.0,
        -0.015196990314225767,-0.37854036201549374,-0.00027130052193601533,-3.3862997711630647E-5,0.0,0.0,0.0,0.0,
        0.0,0.0,1.0,0.0,0.0,-0.0,-0.0,-0.0,-0.0,-0.0,-0.0,-0.45692310525642194,-0.70251656286365771,
        -0.37854017792555505,-0.70317346814293025,0.026748274296612796,-0.026245744732980112,-0.029783569798323813,
        0.0,0.0,0.0,0.0,0.0,0.0,1.0,0.0,-0.0,-0.0,-0.0,-0.0,-0.0,-0.0,-0.0,-0.55566129015943833,
        0.023637206391576536,0.024752136540096725,0.702236447861886,-0.015109647396991065,0.0,0.0,0.0,0.0,0.0,0.0,
        -0.0,-0.0,-0.0,-0.0,-0.0,-0.0,-1.0,-0.0,-0.55566181651356428,0.029709944333287493,0.70223802681964376,
        0.7025125679269647,-0.023637304191565092,0.0,0.0,0.0,0.0,0.0,0.0,0.0,-0.0,-0.0,-0.0,-0.0,-0.0,-0.0,-1.0,
        -0.0,-0.027072082181883235,-0.58504518410006945,-0.70317383709637549,0.37854107343057752,
        0.024805000972806222,0.0,0.0,0.0,0.0,0.0,0.0,1.0,0.0,-0.0,-0.0,-0.0,-0.0,-0.0,-0.0,-0.0,
        -0.024723646828030497,-0.63798497169620449,-0.023621944154890263,0.5850406398453023,0.0,0.0,0.0,0.0,0.0,0.0,
        1.0,0.0,0.0,-0.0,-0.0,-0.0,-0.0,-0.0,-0.0,-0.023469887537635181,-3.2815184442066549E-5,0.55566088508118927,
        0.62488005247477207,0.63798439140804353,-0.55566088508118927,-0.62488005247477207,-0.63798439140804353,0.0,
        0.0,0.0,0.0,0.0,0.0,1.0,0.0,0.0,0.0,-0.0,-0.0,-0.0,-0.0,-0.0,-0.0,-1.0,-0.024752136540096736,
        -0.70251116957088389,-0.023637304191565078,0.55566088508118927,-0.7022357422084774,0.0,0.0,0.0,0.0,0.0,0.0,
        1.0,0.0,0.0,-0.0,-0.0,-0.0,-0.0,-0.0,-0.0,-0.0,-0.024795740829694764,-0.023656120772106475,
        0.624880052474772,-0.37851953994305221,-0.70317018870025627,0.0,0.0,0.0,0.0,0.0,0.0,-0.0,-0.0,-0.0,-0.0,
        -0.0,-0.023621847095687688,-0.024723646828030497,0.63798497169620461,0.015083998191321592,
        -0.45692247149286119,-0.58504116656491612,0.0,0.0,0.0,0.0,0.0,0.0,0.0,-0.0,-0.0,-0.0,-0.0,-0.0,-0.0,
        -0.023621944154890259,-3.3598535051162514E-5,0.0050973150136454475,-0.45692225021991206,
        -0.58504063984530219,0.0,0.0,0.0,0.0,0.0,0.0,0.0,0.0,-0.0,-0.0,-0.0,-0.0,-0.0,-0.0,-1.0,
        -0.027098793108292798,0.37851997948504373,0.70224208707170055,-0.70317323754735284,0.0,0.0,0.0,0.0,0.0,0.0,
        0.0,-0.0,-0.0,-0.0,-0.0,-0.0,-0.0,-0.0,-0.0,-0.027090859530371859,-0.023672783354342114,0.4569224714928613,
        0.70251116957088389,0.015195086849570095,-0.70160323232532973,0.0,0.0,0.0,0.0,0.0,0.0,-0.0,-0.0,-0.0,-0.0,
        -0.0,-0.0,-0.0,-0.027072082181883235,0.58504518410006934,0.024805000972806222,0.022374380992921029,
        -0.37854107343057752,0.0,0.0,0.0,0.0,0.0,0.0,0.0,-0.0,-0.0,-0.0,-0.0,-0.0,-0.0,-1.0,-0.0,
        -0.58504502721143925,-0.70317406745246691,0.026708907388227905,0.37854017792555522,-0.026218970645527549,
        -0.029748443430697016,0.0,0.0,0.0,0.0,0.0,0.0,1.0,-0.0,-0.0,-0.0,-0.0,-0.0,-0.0,-0.0,-0.585041166564916,
        0.023660296965944742,0.024805000972806225,0.37854073327939119,-0.015170756558948674,0.0,0.0,0.0,0.0,0.0,
        -0.0,-0.0,-0.0,-0.0,-1.0,-0.0,-0.62488169574462793,-0.58504204394174075,0.029748443430697009,
        0.37854036201549396,-0.023660396850780658,0.0,0.0,0.0,0.0,0.0,0.0,1.0,-0.0,-0.0,-0.0,-0.0,-0.0,-0.0,-0.0,
        -0.027631856629547157,0.4569226479042604,0.70251319697861081,0.023672783354342117,0.015185611969090922,
        -0.70160605506782658,0.0,0.0,0.0,0.0,0.0,-0.0,-0.0,-0.0,-0.0,-0.0,-0.0,-0.0,-0.027610578309122811,
        -0.02974844343069703,0.58504204394174075,0.023660396850780651,-0.37854036201549374,0.0,0.0,0.0,0.0,0.0,0.0,
        0.0,-0.0,-0.0,-0.0,-0.0,-0.0,-0.0,-1.0,-0.63798497169620449,0.0236218470956877,0.024723646828030469,
        0.58504116656491612,-0.015083998191321633,0.0,0.0,0.0,0.0,0.0,-0.0,-0.0,-0.0,-0.0,-1.0,-0.0,
        0.026171339658097509,0.022291660731226463,0.58504146009743707,-0.0050973150136454448,0.023621944154890263,
        0.45692225021991223,0.0,0.0,0.0,0.0,0.0,0.0,1.0,-0.0,-0.0,-0.0,-0.0,-0.0,-0.0,-0.0,-0.0,-0.637986096484328,
        0.029685529684818798,0.45692242688405121,0.58504204394174086,-0.02362194415489029,0.0,0.0,0.0,0.0,0.0,0.0,
        1.0,-0.0,-0.0,-0.0,-0.0,-0.0,-0.0,-0.0,-0.026730661933064309,0.45692310525642194,0.70251656286365771,
        0.029768291394636794,-0.70161080096520145,0.0,0.0,0.0,0.0,0.0,0.0,0.0,-0.0,-0.0,-0.0,-0.0,-0.0,-0.0,-0.0,
        -0.026708907388227905,0.58504502721143925,0.029748443430697019,-0.378540177925555,0.0,0.0,0.0,0.0,0.0,0.0,
        0.0,-0.0,-0.0,-0.0,-0.0,-0.0,-0.0,-1.0,0.4569238375042779,0.027090859530371863,0.70251617195999394,
        0.37854107343057747,-0.024849423695496649,-0.022419246501157553,0.0,0.0,0.0,0.0,0.0,0.0,0.0,-0.0,-0.0,-0.0,
        -0.0,-0.0,-0.0,-1.0,-0.0,-0.0,0.55566147407010114,0.026190122699982339,0.0223194354621066,
        -0.70223692196481524,-0.029647784654081327,-0.70251158235928435,0.0,0.0,0.0,0.0,0.0,1.0,-0.0,-0.0,-0.0,-0.0,
        -0.0,-0.0,-0.0,-0.0,0.70224253943268344,0.378540177925555,0.70161080096520145,0.026748274296612796,
        -0.029783569798323813,0.0,0.0,0.0,0.0,0.0,0.0,-0.0,-0.0,-0.0,-0.0,-0.0,-0.0,-1.0,-0.0,-0.0,
        0.45692264790426035,0.027631856629547154,0.70251319697861092,-0.023672783354342128,-0.70160605506782658,
        -0.015185611969090976,0.0,0.0,0.0,0.0,-0.0,-0.0,-0.0,-0.0,-0.0,-0.0,0.55566181651356428,
        0.029709944333287493,-0.023637304191565092,-0.70223802681964376,-0.7025125679269647,0.0,0.0,0.0,0.0,0.0,0.0,
        1.0,-0.0,-0.0,-0.0,-0.0,-0.0,-0.0,-0.0,-0.0,0.45692310525642188,0.70251656286365771,0.026730661933064316,
        -0.026234238763943405,-0.70161080096520145,-0.029768291394636756,0.0,0.0,0.0,0.0,0.0,-0.0,-0.0,-0.0,-0.0,
        -0.0,-0.0,-0.0,0.027072082181883235,0.58504518410006934,-0.37854107343057752,-0.024805000972806211,
        -0.022374380992921029,0.0,0.0,0.0,0.0,0.0,0.0,0.0,-0.0,-0.0,-0.0,-0.0,-0.0,-0.0,-1.0,-0.0,0.026213688698745,
        0.62488096344828059,0.022364818883998026,-0.3785195589565879,-0.029687807671632122,-0.70317085483536168,0.0,
        0.0,0.0,0.0,-0.0,-0.0,-0.0,-0.0,-0.0,-0.0,0.023469887537635188,0.00012845955535528616,0.55566088508118927,
        0.62488005247477207,0.63798439140804353,-0.55566088508118927,-0.62488005247477207,-0.63798439140804353,0.0,
        0.0,0.0,0.0,0.0,0.0,1.0,0.0,-0.0,-0.0,-0.0,-0.0,-0.0,-0.0,-1.0,-0.0,-0.0,0.585042570028093,
        0.027610578309122811,-0.37854046095194716,-0.023660296965944742,-0.015161281241640751,0.0,0.0,0.0,0.0,0.0,
        0.0,-0.0,-0.0,-0.0,-0.0,-0.0,-0.0,-1.0,0.62488169574462793,0.029741488872504766,-0.3785192678205006,
        -0.023656120772106493,-0.70317150299940423,0.0,0.0,0.0,0.0,0.0,0.0,-0.0,-0.0,-0.0,-0.0,-0.0,-0.0,-0.0,
        0.029685529684818805,0.637986096484328,-0.45692242688405116,-0.02362194415489028,-0.58504204394174075,0.0,
        0.0,0.0,0.0,0.0,0.0,-0.0,-0.0,-0.0,-0.0,-0.0,-0.0,-1.0,-0.0,-0.55566088508118927,-0.023637304191565081,
        -0.015109647396991093,0.7022357422084774,0.0,0.0,0.0,0.0,0.0,0.0,0.0,0.0,0.0,-0.0,-0.0,-0.0,-0.0,-0.0,-0.0,
        -1.0,-0.37854107343057741,-0.0015613656062954475,0.027105602758215108,-0.02484942369549667,
        -0.02241924650115756,0.0,0.0,0.0,0.0,0.0,0.0,1.0,0.0,0.0,-0.0,-0.0,-0.0,-0.0,-0.0,-0.0,-0.0,
        -0.37854046095194693,-0.70317131702755065,0.027648865450003536,-0.023682030674840704,-0.015207454024849647,
        0.0,0.0,0.0,0.0,0.0,0.0,-0.0,-0.0,-0.0,-0.0,-0.0,-0.702236447861886,0.024840157186683216,
        -0.37854073327939092,0.023682030674840707,0.0001642424429245156,-0.015216927320390209,0.0,0.0,0.0,0.0,0.0,
        -0.0,-0.0,-0.0,-0.0,-1.0,-0.0,-0.45692242688405105,-0.7025125679269647,0.02976829139463676,
        -0.37854036201549374,0.00027130052193601533,-0.023682132033406258,0.0,0.0,0.0,0.0,0.0,0.0,1.0,0.0,-0.0,-0.0,
        -0.0,-0.0,-0.0,-0.0,-0.0,-0.55566088508118927,0.023637304191565085,0.029647784654081352,0.7022357422084774,
        0.70251053960656562,0.0,0.0,0.0,0.0,0.0,0.0,0.0,-0.0,-0.0,-0.0,-0.0,-0.0,-0.0,-1.0,-0.0,-0.0,
        -0.37851926782050049,-0.70223802681964376,0.029776610295742294,0.70317090201170729,-0.023677852874347757,
        0.0,0.0,0.0,0.0,0.0,0.0,0.0,-0.0,-0.0,-0.0,-0.0,-0.0,-0.0,-0.58504116656491612,-0.024805000972806236,
        -0.70317060420331423,-0.023660396850780658,-0.0015608627398630522,0.3785406342380947,0.0,0.0,0.0,0.0,0.0,
        0.0,1.0,0.0,0.0,-0.0,-0.0,-0.0,-0.0,-0.0,-0.0,-0.023660296965944735,-0.024805000972806239,
        0.58504116656491578,0.015170756558948695,-0.37854073327939125,0.0,0.0,0.0,0.0,0.0,0.0,0.0,-0.0,-0.0,-0.0,
        -0.0,-0.0,-0.0,-3.3895386058154954E-5,0.0,-1.0,-0.023682030674840707,0.37854073327939108,
        0.0030612231608958297,0.0,0.0,0.0,0.0,0.0,0.0,0.0,-0.0,-0.0,-0.0,-0.0,-0.0,-0.0,-0.0,-0.023660396850780651,
        -3.37922497221569E-5,0.0053104157804372727,-0.37854063423809481,0.0,0.0,0.0,0.0,0.0,0.0,0.0,0.0,-0.0,-0.0,
        -0.0,-0.0,-0.0,-0.0,-1.0,-0.027105602758215112,0.37854107343057758,0.0030612088654606811,
        0.024849423695496673,0.02241924650115756,0.0,0.0,0.0,0.0,0.0,0.0,0.0,-0.0,-0.0,-0.0,-0.0,-0.0,-0.0,-1.0,
        -0.0,-0.0,0.026218970645527546,0.022374380992921033,0.37854065319208563,-0.00531041578043727,
        0.023660396850780661,0.0,0.0,0.0,0.0,0.0,0.0,1.0,-0.0,-0.0,-0.0,-0.0,-0.0,-0.0,-0.0,-0.0,
        -0.015185611969090872,0.45692242688405116,0.7025125679269647,0.023672883991351843,-0.00027130052193601566,
        -3.3862997711630437E-5,0.3785403620154939,0.0,0.0,0.0,0.0,0.0,0.0,0.0,-0.0,-0.0,-0.0,-0.0,-0.0,-0.0,-1.0,
        -0.0,-0.027648865450003536,0.378540460951947,0.70160605506782647,0.0236820306748407,0.015207454024849618,
        0.0,0.0,0.0,0.0,0.0,0.0,-0.0,-0.0,-0.0,-0.0,-0.0,-0.0,-1.0,-0.0,-0.026748274296612789,0.37854017792555505,
        0.70161080096520156,0.029783569798323847,0.0,0.0,0.0,0.0,0.0,0.0,0.0,-0.0,-0.0,-0.0,-0.0,-0.0,-0.0,-1.0,
        -0.0,0.45692249061308471,0.026234238763943405,0.70251158235928435,0.022398709579893369,-0.70160383989347,
        -0.029720779304182428,0.0,0.0,0.0,0.0,-0.0,-0.0,-0.0,-0.0,-0.0,-0.0,-0.0,-0.0,0.55566088508118927,
        0.023637304191565085,0.029647784654081352,-0.7022357422084774,-0.70251053960656573,0.0,0.0,0.0,0.0,0.0,0.0,
        1.0,-0.0,-0.0,-0.0,-0.0,-0.0,-0.0,-0.0,-0.0,-0.0,0.027648865450003536,-1.0,0.37851926782050049,
        0.70223802681964376,0.029776610295742294,-0.023677852874347757,0.0,0.0,0.0,0.0,0.0,0.0,-0.0,-0.0,-0.0,-0.0,
        -0.0,-0.0,-0.0,-0.0,0.45692242688405105,0.02976829139463676,0.7025125679269647,-0.023672883991351864,
        -0.70160519311325342,0.0,0.0,0.0,0.0,0.0,-0.0,-0.0,-0.0,-0.0,-0.0,-0.0,-0.0,0.62488005247477207,
        0.023660396850780661,0.0053104157804372719,3.3792249722156905E-5,-0.3785406342380947,0.0,0.0,0.0,0.0,0.0,
        0.0,-0.0,-0.0,-0.0,-0.0,-0.0,-0.0,-1.0,-0.0,-0.0,0.023621944154890277,0.00012982492179038625,
        0.0050973150136454466,-0.45692225021991212,-0.5850406398453023,0.0,0.0,0.0,0.0,0.0,0.0,-0.0,-0.0,-0.0,-0.0,
        -0.0,-0.0,-1.0,-0.0,-0.0,0.58504204394174064,0.029748443430697026,0.70317150299940412,0.015161281241640776,
        -0.37854036201549396,-0.023660396850780654,0.0,0.0,0.0,0.0,0.0,0.0,-0.0,-0.0,-0.0,-0.0,-0.0,-0.0,-1.0,-0.0,
        -0.378519539943052,-0.023677852874347757,-0.0046218484590718626,-3.3872049431451388E-5,0.70316958685172248,
        0.0,0.0,0.0,0.0,0.0,0.0,0.0,0.0,0.0,-0.0,-0.0,-0.0,-0.0,-0.0,-0.0,-0.37854065319208546,
        9.9046128627942282E-5,-0.029739987791949973,0.0,0.0,0.0,0.0,0.0,1.0,0.0,0.0,0.0,-0.0,-0.0,-0.0,-0.0,-0.0,
        -0.0,-0.0,-0.37851953994305204,0.00013032533543202578,-0.0030612242404972137,0.023682132033406265,
        0.00013036341924922685,0.0,0.0,0.0,0.0,0.0,0.0,1.0,0.0,-0.0,-0.0,-0.0,-0.0,-0.0,-0.0,-0.0,-0.0,
        -0.45692225021991212,-0.0030912635403395824,0.02367288399135186,0.70160236926968877,0.0,0.0,0.0,0.0,0.0,0.0,
        0.0,-0.0,-0.0,-0.0,-0.0,-0.0,-0.0,-0.0,-0.0,0.45692225021991212,0.02367288399135186,0.00013027879750649216,
        0.003091263540339582,-0.70160236926968877,0.0,0.0,0.0,0.0,0.0,-0.0,-0.0,-0.0,-0.0,-0.0,-0.0,-0.0,-0.0,
        0.378519539943052,0.0046218484590718626,0.023682132033406265,3.389538605815513E-5,0.0,0.0,0.0,0.0,0.0,0.0,
        -0.0,-0.0,-0.0,-0.0,-0.0,-0.0,-1.0,-0.0,-0.0,-0.0,-0.37854063423809459,-0.023682132033406265,
        -0.001561372566461268,-3.389538605815513E-5,0.0,0.0,0.0,0.0,0.0,0.0,1.0,0.0,0.0,0.0,-0.0,-0.0,-0.0,-0.0,
        -0.0,-0.0,0.047678521358187322,0.55787204405389446,0.048825402242851326,0.62654723292970194,
        0.047286920841764508,0.63943141348019983,-0.047678521358187322,-0.55787204405389446,-0.048825402242851333,
        -0.62654723292970194,-0.047286920841764508,-0.63943141348019983,0.0,0.0,0.0,0.0,0.0,0.0,0.0,1.0,0.0,0.0,
        -0.0,-0.0,-0.0,-0.0,-0.0,-0.0,-0.0,-1.0,-0.047678521358187315,0.557872509055183,0.044288901125137163,
        0.62654217515979649,0.040021361425923357,0.63942545184526778,-0.557872509055183,-0.62654217515979649,
        -0.63942545184526778,0.0,0.0,0.0,0.0,0.0,0.0,1.0,0.0,0.0,-0.0,-0.0,-0.0,-0.0,-0.0,-0.0,-0.0,-1.0,
        -0.55787204405389446,0.047942655141777091,0.049117799127055072,0.702875228655225,0.0475823178492932,
        0.70295568967385469,-0.047942655141777091,-0.049117799127055078,-0.04758231784929319,0.0,0.0,0.0,0.0,0.0,
        0.0,0.0,0.0,0.0,-0.0,-0.0,-0.0,-0.0,-0.0,-0.0,-0.0,-1.0,-0.048825402242851333,-0.55787171658183987,
        -0.63942424475811355,-0.052452304750527382,0.041298149353625656,0.557871608027596,0.62654080641868248,
        0.63942401877909183,-0.62654080641868248,0.0,0.0,0.0,0.0,0.0,0.0,0.0,1.0,0.0,-0.0,-0.0,-0.0,-0.0,-0.0,-0.0,
        -1.0,-0.626547232929702,-0.047984758880296075,-0.04763006590676714,-0.58732864799299578,
        0.047993536136706469,0.38140732638781982,0.049174830154444668,0.047640075741515714,0.0,0.0,0.0,0.0,0.0,0.0,
        0.0,1.0,0.0,-0.0,-0.0,-0.0,-0.0,-0.0,-0.0,-0.0,-0.047286920841764508,0.045941301434432633,
        0.55787142569916037,0.052452304750527444,0.62654193427993921,0.639425363845251,-0.55787142569916037,
        -0.62654193427993921,-0.639425363845251,0.0,0.0,0.0,0.0,0.0,0.0,0.0,1.0,0.0,-0.0,-0.0,-0.0,-0.0,-0.0,-0.0,
        -1.0,-0.63943141348019983,0.047934264404490834,0.45972838564453733,0.0491093915715111,0.58732864799299578,
        0.04757405784581345,-0.047934264404490834,-0.0491093915715111,-0.04757405784581345,0.0,0.0,0.0,0.0,0.0,0.0,
        0.0,1.0,0.0,-0.0,-0.0,-0.0,-0.0,-0.0,-0.0,-0.0,0.047678521358187315,0.557872509055183,0.62654217515979649,
        0.63942545184526778,-0.557872509055183,-0.044288901125137184,-0.62654217515979649,-0.04002136142592335,
        -0.63942545184526778,0.0,0.0,0.0,0.0,0.0,0.0,0.0,1.0,0.0,-0.0,-0.0,-0.0,-0.0,-0.0,-0.0,-1.0,-0.0,
        0.55787204405389446,0.047942655141777091,0.049117799127055072,0.0475823178492932,-0.047942655141777091,
        -0.049117799127055078,-0.702875228655225,-0.04758231784929319,-0.70295568967385469,0.0,0.0,0.0,0.0,0.0,0.0,
        0.0,1.0,0.0,-0.0,-0.0,-0.0,-0.0,-0.0,-0.0,-0.0,-0.0,0.048825402242851333,0.05245230475052743,
        0.557871608027596,0.62654080641868248,0.63942401877909183,-0.041298149353625628,-0.557871608027596,
        -0.63942401877909183,0.0,0.0,0.0,0.0,0.0,0.0,1.0,0.0,-0.0,-0.0,-0.0,-0.0,-0.0,-0.0,-0.0,-1.0,
        0.626547232929702,0.047984758880296075,0.047630065906767147,0.58732864799299578,0.049174830154444668,
        -0.047993536136706469,-0.38140732638781982,-0.049174830154444675,-0.047640075741515707,0.0,0.0,0.0,0.0,0.0,
        0.0,0.0,0.0,-0.0,-0.0,-0.0,-0.0,-0.0,-0.0,-0.0,-1.0,0.047286920841764508,0.55787142569916037,
        0.62654193427993921,0.639425363845251,-0.045941301434432633,-0.55787142569916037,-0.052452304750527472,
        -0.62654193427993921,-0.639425363845251,0.0,0.0,0.0,0.0,0.0,0.0,1.0,0.0,-0.0,-0.0,-0.0,-0.0,-0.0,-0.0,-0.0,
        -1.0,0.63943141348019983,0.047934264404490834,0.0491093915715111,0.04757405784581345,-0.047934264404490834,
        -0.45972838564453733,-0.0491093915715111,-0.58732864799299578,-0.04757405784581345,0.0,0.0,0.0,0.0,0.0,0.0,
        0.0,0.0,-0.0,-0.0,-0.0,-0.0,-0.0,-0.0,-0.0,-1.0,-0.047942655141777091,-0.557872509055183,
        0.044607913288060984,0.70286297549379462,0.040334527208629158,0.70294446596883164,0.0,0.0,0.0,0.0,0.0,0.0,
        0.0,0.0,-0.0,-0.0,-0.0,-0.0,-0.0,-0.0,-0.0,-1.0,-0.04428890112513717,-0.041298149353625621,
        -0.052879406986409215,0.557871950150472,0.62654033525020214,0.6394234093758725,-0.557871950150472,
        -0.62654033525020214,-0.6394234093758725,0.0,0.0,0.0,0.0,0.0,0.0,0.0,1.0,0.0,0.0,-0.0,-0.0,-0.0,-0.0,-0.0,
        -0.0,-1.0,-0.047984758880296068,0.38139322558672084,0.70313339581753054,-0.0,-0.041515729018567704,
        -0.62654033525020214,0.70313108620605158,0.0,0.0,0.0,0.0,0.0,0.0,0.0,0.0,-0.0,-0.0,-0.0,-0.0,-0.0,-0.0,
        -0.045941301434432633,-0.040021361425923357,0.55787198584888142,0.0528794069864092,-0.63942378652894072,0.0,
        0.0,0.0,0.0,0.0,0.0,0.0,0.0,-0.0,-0.0,-0.0,-0.0,-0.0,-0.0,-1.0,-0.047934264404490841,0.587326232489261,-0.0,
        -0.041479097778282452,-0.6394234093758725,0.0,0.0,0.0,0.0,0.0,0.0,0.0,1.0,0.0,-0.0,-0.0,-0.0,-0.0,-0.0,-0.0,
        -0.047942655141777091,0.557872509055183,-0.0,-0.041486488318378048,0.027677161979573293,
        -0.70294159791647837,0.0,0.0,0.0,0.0,0.0,0.0,1.0,0.0,-0.0,-0.0,-0.0,-0.0,-0.0,-0.0,-0.0,
        -0.047984758880296068,0.62654217515979649,0.044660621016635559,-0.38139322558672084,-0.70313339581753065,
        0.0,0.0,0.0,0.0,0.0,0.0,-0.0,-0.0,-0.0,-0.0,-0.0,-0.0,-0.0,-0.047934264404490841,0.63942545184526778,
        0.0446006835917423,0.040327604063683457,-0.45973364369000819,-0.587326232489261,0.0,0.0,0.0,0.0,0.0,0.0,0.0,
        -0.0,-0.0,-0.0,-0.0,-0.0,-0.0,-0.0,-1.0,-0.55787171658183987,-0.049198241144151271,-0.38141432182325924,
        0.041543427917705961,0.027753531302003462,0.0,0.0,0.0,0.0,0.0,0.0,1.0,0.0,-0.0,-0.0,-0.0,-0.0,-0.0,-0.0,
        -0.381386025829566,-0.702875228655225,0.048014979218259819,0.049198241144151264,0.047663646280299156,
        0.70314122138856006,-0.048014979218259819,-0.049198241144151271,-0.047663646280299156,0.0,0.0,0.0,0.0,0.0,
        0.0,0.0,0.0,-0.0,-0.0,-0.0,-0.0,-0.0,-0.0,-0.55787142569916048,-0.04758231784929319,0.046165728248822986,
        0.052734339992385214,0.70286396678410767,0.0,0.0,0.0,0.0,0.0,0.0,0.0,0.0,-0.0,-0.0,-0.0,-0.0,-0.0,-0.0,-1.0,
        -0.45972838564453744,-0.70295568967385458,0.04765651814247162,-0.048008393947647693,-0.049191105586226781,
        -0.047656518142471613,0.0,0.0,0.0,0.0,0.0,0.0,0.0,1.0,0.0,0.0,-0.0,-0.0,-0.0,-0.0,-0.0,-0.0,-0.0,
        -0.557872509055183,0.0479426551417771,0.70286297549379462,-0.044607913288061025,-0.040334527208629151,0.0,
        0.0,0.0,0.0,0.0,0.0,0.0,0.0,-0.0,-0.0,-0.0,-0.0,-0.0,-0.0,-1.0,-0.0,-0.55787171658183987,
        0.049117799127055085,0.70286143698134129,-0.041486488318378041,-0.027661054311066195,0.0,0.0,0.0,0.0,0.0,
        0.0,0.0,-0.0,-0.0,-0.0,-0.0,-0.0,-0.0,-1.0,-0.55787142569916048,0.04758231784929319,0.70286396678410767,
        0.70294533564091966,-0.046165728248822986,-0.052734339992385255,0.0,0.0,0.0,0.0,0.0,0.0,0.0,-0.0,-0.0,-0.0,
        -0.0,-0.0,-0.0,-0.0,-1.0,-0.049164972356125373,-0.62654101707515264,-0.052779600708881172,
        -0.58732523320298258,0.041521734602731605,0.38141436310945664,0.0,0.0,0.0,0.0,0.0,0.0,0.0,1.0,-0.0,-0.0,
        -0.0,-0.0,-0.0,-0.0,-0.049109391571511091,-0.63942424475811355,-0.052725613098002319,0.041479097778282452,
        0.58732507052489791,0.0,0.0,0.0,0.0,0.0,0.0,0.0,1.0,-0.0,-0.0,-0.0,-0.0,-0.0,-0.0,-0.049117799127055078,
        -0.70294302173702006,-0.052734339992385228,0.557871608027596,0.041486711482857687,-0.70286111061272671,0.0,
        0.0,0.0,0.0,0.0,0.0,0.0,1.0,-0.0,-0.0,-0.0,-0.0,-0.0,-0.0,-0.0,-0.052779600708881172,0.62654080641868259,
        0.041515729018567711,-0.381393060579516,-0.70313207851881332,0.0,0.0,0.0,0.0,0.0,-0.0,-0.0,-0.0,-0.0,-0.0,
        -0.62654193427993921,-0.047630065906767147,-0.58732556690019289,0.38141260703668056,0.052788975072809517,
        0.0,0.0,0.0,0.0,0.0,0.0,0.0,1.0,-0.0,-0.0,-0.0,-0.0,-0.0,-0.0,-0.62654217515979649,-0.040386220026432475,
        -0.587326232489261,0.047993536136706476,0.38141452789755637,-0.044671688889686353,0.0,0.0,0.0,0.0,0.0,0.0,
        0.0,1.0,-0.0,-0.0,-0.0,-0.0,-0.0,-0.0,-0.0,-0.62654101707515253,-0.58732523320298247,0.049174830154444668,
        0.38141432182325907,-0.041521509739207062,-0.027720209169872088,0.0,0.0,0.0,0.0,0.0,-0.0,-0.0,-0.0,-0.0,
        -0.0,-0.62654193427993921,-0.04620090230449761,-0.0527796007088812,-0.58732556690019289,0.0476400757415157,
        0.38141260703668056,0.0,0.0,0.0,0.0,0.0,0.0,1.0,-0.0,-0.0,-0.0,-0.0,-0.0,-0.0,-0.0,-0.047574057845813457,
        -0.639425363845251,0.052725613098002347,0.58732556690019289,0.0,0.0,0.0,0.0,0.0,0.0,0.0,1.0,-0.0,-0.0,-0.0,
        -0.0,-0.0,-0.0,-0.04758231784929319,0.55787142569916037,0.052734339992385269,-0.70286396678410767,
        -0.70294533564091966,0.0,0.0,0.0,0.0,0.0,0.0,0.0,1.0,-0.0,-0.0,-0.0,-0.0,-0.0,-0.0,-0.0,
        -0.04763006590676714,0.62654193427993921,0.052779600708881193,-0.38139130491870232,-0.703133933677141,0.0,
        0.0,0.0,0.0,0.0,-0.0,-0.0,-0.0,-0.0,-0.0,-0.047574057845813457,0.639425363845251,0.04615757913241255,
        0.052725613098002347,-0.45973190050489804,-0.58732556690019289,0.0,0.0,0.0,0.0,0.0,0.0,0.0,-0.0,-0.0,-0.0,
        -0.0,-0.0,-0.0,-1.0,-0.63942545184526778,0.047934264404490834,0.587326232489261,-0.044600683591742338,
        -0.04032760406368343,0.0,0.0,0.0,0.0,0.0,0.0,0.0,1.0,-0.0,-0.0,-0.0,-0.0,-0.0,-0.0,-0.0,
        -0.63942424475811355,0.0491093915715111,0.58732523320298258,-0.041478874690674995,-0.027655051949837254,0.0,
        0.0,0.0,0.0,0.0,-0.0,-0.0,-0.0,-0.0,-0.0,-0.639425363845251,0.047574057845813443,0.58732556690019289,
        -0.04615757913241255,-0.052725613098002382,0.0,0.0,0.0,0.0,0.0,0.0,1.0,-0.0,-0.0,-0.0,-0.0,-0.0,-0.0,-0.0,
        0.047942655141777091,0.557872509055183,-0.044607913288061012,-0.70286297549379462,-0.040334527208629144,
        -0.70294446596883164,0.0,0.0,0.0,0.0,0.0,0.0,0.0,1.0,-0.0,-0.0,-0.0,-0.0,-0.0,-0.0,-0.0,-0.0,
        0.041297934356687133,0.0442889011251372,0.55787205898156167,-0.027381569976781938,-0.63942363589545237,0.0,
        0.0,0.0,0.0,0.0,0.0,0.0,-0.0,-0.0,-0.0,-0.0,-0.0,-0.0,-1.0,-0.0,0.047984758880296068,0.62654217515979649,
        -0.38139322558672084,-0.044660621016635579,-0.040386220026432489,-0.70313339581753065,0.0,0.0,0.0,0.0,0.0,
        -0.0,-0.0,-0.0,-0.0,-0.0,-0.0,0.045941301434432633,0.04002136142592335,0.041298149353625628,
        0.027381569976781941,0.557871950150472,0.62654033525020214,0.6394234093758725,-0.557871950150472,
        -0.6394234093758725,0.0,0.0,0.0,0.0,0.0,0.0,1.0,0.0,-0.0,-0.0,-0.0,-0.0,-0.0,-0.0,-0.0,-1.0,-0.0,
        0.047934264404490841,0.63942545184526778,-0.45973364369000819,-0.044600683591742324,-0.587326232489261,
        -0.040327604063683443,0.0,0.0,0.0,0.0,0.0,0.0,0.0,-0.0,-0.0,-0.0,-0.0,-0.0,-0.0,-1.0,-0.0,
        0.55787171658183987,0.049117799127055085,-0.041486488318378041,-0.70286143698134129,-0.027661054311066195,
        -0.70294302173702006,0.0,0.0,0.0,0.0,0.0,-0.0,-0.0,-0.0,-0.0,-0.0,-0.0,0.381386025829566,
        0.70287522865522511,0.048014979218259819,0.049198241144151264,0.047663646280299156,-0.048014979218259819,
        -0.049198241144151271,-0.047663646280299156,-0.70314122138856006,0.0,0.0,0.0,0.0,0.0,0.0,-0.0,-0.0,-0.0,
        -0.0,-0.0,-0.0,-0.0,-0.0,0.55787142569916048,0.04758231784929319,-0.046165728248822986,
        -0.052734339992385255,-0.70286396678410767,-0.70294533564091966,0.0,0.0,0.0,0.0,0.0,0.0,1.0,-0.0,-0.0,-0.0,
        -0.0,-0.0,-0.0,-0.0,-0.0,0.45972838564453744,0.70295568967385458,0.04765651814247162,-0.048008393947647693,
        -0.70268597089371387,0.0,0.0,0.0,0.0,0.0,0.0,0.0,-0.0,-0.0,-0.0,-0.0,-0.0,-0.0,-0.0,0.049164972356125373,
        0.62654101707515264,-0.041515504461835731,-0.38139301933175634,-0.027709698583410016,-0.70313230364575241,
        0.0,0.0,0.0,0.0,-0.0,-0.0,-0.0,-0.0,0.049109391571511105,0.052725613098002361,0.63942401877909172,
        -0.041479097778282459,-0.45973321032477427,-0.58732507052489791,0.0,0.0,0.0,0.0,0.0,0.0,-0.0,-0.0,-0.0,-0.0,
        -0.0,-0.0,-0.0,-1.0,0.62654193427993921,0.047630065906767147,-0.04620090230449761,-0.38139130491870232,
        -0.052779600708881227,-0.703133933677141,0.0,0.0,0.0,0.0,0.0,0.0,-0.0,-0.0,-0.0,-0.0,-0.0,-0.0,-0.0,
        0.047574057845813457,0.639425363845251,-0.046157579132412557,-0.45973190050489804,-0.052725613098002388,
        -0.58732556690019289,0.0,0.0,0.0,0.0,0.0,0.0,-0.0,-0.0,-0.0,-0.0,-0.0,-0.0,-0.0,-1.0,-0.044696511233766632,
        -0.041537644408465073,-0.38139435220779871,-0.0046455551781967915,0.70313098732427648,0.0,0.0,0.0,0.0,0.0,
        0.0,0.0,0.0,0.0,-0.0,-0.0,-0.0,-0.0,-0.0,-0.0,-0.048014979218259812,-0.38139322558672073,
        -0.70286297549379451,0.04469651123376666,0.70313329820348291,0.0,0.0,0.0,0.0,0.0,0.0,-0.0,-0.0,-0.0,-0.0,
        -0.0,-0.0,-0.046165728248822986,-0.040334527208629165,-0.041486711482857673,-0.55787195015047186,
        0.70285954634074388,0.0,0.0,0.0,0.0,0.0,0.0,0.0,0.0,0.0,-0.0,-0.0,-0.0,-0.0,-0.0,-0.0,-1.0,
        -0.047993536136706476,0.38141452789755642,-0.0,-0.70313131216765046,-0.0415217346027316,
        -0.0053499825507371153,-0.0015656878741349531,0.0,0.0,0.0,0.0,0.0,0.0,0.0,1.0,0.0,-0.0,-0.0,-0.0,-0.0,-0.0,
        -0.0,-0.04615757913241255,-0.040327604063683457,-0.041479097778282452,-0.027671157031094271,
        0.6394234093758725,-0.45973424542066693,-0.58732499879699229,0.0,0.0,0.0,0.0,0.0,0.0,0.0,0.0,-0.0,-0.0,-0.0,
        -0.0,-0.0,-0.0,-1.0,-0.048014979218259812,0.38139322558672073,0.70286297549379451,0.04469651123376666,
        -0.70313329820348291,0.0,0.0,0.0,0.0,0.0,0.0,-0.0,-0.0,-0.0,-0.0,-0.0,-0.0,-0.0,-0.0,-0.047993536136706476,
        0.587326232489261,0.044671688889686333,0.040397149349959804,-0.38141452789755642,0.0,0.0,0.0,0.0,0.0,0.0,
        0.0,-0.0,-0.0,-0.0,-0.0,-0.0,-0.0,-0.0,-1.0,-0.557871608027596,-0.052734339992385235,-0.027661054311066337,
        0.041486711482857694,0.70286111061272671,0.0,0.0,0.0,0.0,0.0,0.0,0.0,0.0,-0.0,-0.0,-0.0,-0.0,-0.0,-0.0,-1.0,
        -0.70286396678410779,-0.047663646280299149,-0.38141260703668067,0.052821149416567043,0.0,0.0,0.0,0.0,0.0,
        0.0,0.0,1.0,0.0,-0.0,-0.0,-0.0,-0.0,-0.0,-0.0,-0.38140732638781988,-0.0015661221639725058,
        0.048023761687426413,0.049208104725552843,0.047673661972528605,-0.048023761687426413,-0.049208104725552849,
        -0.0476736619725286,0.0,0.0,0.0,0.0,0.0,0.0,0.0,1.0,0.0,0.0,-0.0,-0.0,-0.0,-0.0,-0.0,-0.0,-0.0,
        -0.70286297549379451,-0.04042146861842183,-0.38141452789755653,0.048023761687426413,-0.044707585477670696,
        0.0,0.0,0.0,0.0,0.0,0.0,0.0,1.0,0.0,-0.0,-0.0,-0.0,-0.0,-0.0,-0.0,-0.0,-0.70286143698134129,
        -0.38141432182325918,0.049208104725552843,-0.041543427917705954,-0.027753531302003361,0.0,0.0,0.0,0.0,0.0,
        0.0,-0.0,-0.0,-0.0,-0.0,-0.0,-0.38139130491870249,-0.70286396678410779,0.047663646280299149,
        0.70313383642924188,-0.046226776721425993,-0.052811769511494744,0.0,0.0,0.0,0.0,0.0,0.0,0.0,-0.0,-0.0,-0.0,
        -0.0,-0.0,-0.0,-0.38141260703668073,-0.0015661807001885121,0.0003808990881292652,-0.046234063364270737,
        -0.052821149416567105,0.0,0.0,0.0,0.0,0.0,0.0,1.0,0.0,-0.0,-0.0,-0.0,-0.0,-0.0,-0.0,-0.0,
        -0.55787205898156167,0.041486488318378034,0.044607913288061032,-0.02767716197957313,0.0,0.0,0.0,0.0,0.0,0.0,
        0.0,-0.0,-0.0,-0.0,-0.0,-0.0,-0.0,-1.0,-0.0,-0.55787198584888142,-0.38139402411953655,0.046226776721426013,
        0.04042146861842183,0.70313145912642394,-0.053301939043787668,0.0,0.0,0.0,0.0,0.0,0.0,-0.0,-0.0,-0.0,-0.0,
        -0.0,-0.0,-0.0,-0.557871608027596,0.052734339992385269,0.70286111061272671,0.70294271779415229,
        -0.041486711482857687,0.0,0.0,0.0,0.0,0.0,0.0,0.0,-0.0,-0.0,-0.0,-0.0,-0.0,-0.0,-0.0,-1.0,
        -0.052725613098002319,-0.027655051949837452,0.63942401877909172,0.041479097778282452,-0.45973321032477427,
        -0.58732507052489791,0.0,0.0,0.0,0.0,0.0,0.0,0.0,-0.0,-0.0,-0.0,-0.0,-0.0,-0.0,-1.0,-0.052811769511494709,
        0.381393060579516,0.70286111061272671,0.041537644408465066,-0.70313198021515855,0.0,0.0,0.0,0.0,0.0,-0.0,
        -0.0,-0.0,-0.0,-0.0,-0.0,-0.049174830154444661,-0.052788975072809545,0.58732507052489813,
        0.041521734602731612,-0.38141436310945631,0.0,0.0,0.0,0.0,0.0,0.0,0.0,-0.0,-0.0,-0.0,-0.0,-0.0,-0.0,-1.0,
        -0.6265406645097189,0.046200902304497617,0.040386220026432475,0.38139402411953627,0.70313155774868141,
        -0.053264773578912634,0.0,0.0,0.0,0.0,0.0,-0.0,-0.0,-0.0,-0.0,-0.0,-0.0,-0.0,-0.62654080641868248,
        -0.58732507052489791,0.052788975072809559,0.38141436310945637,-0.0415217346027316,0.0,0.0,0.0,0.0,0.0,0.0,
        1.0,-0.0,-0.0,-0.0,-0.0,-0.0,-0.0,-0.0,-0.047663646280299156,0.38139130491870238,0.70286396678410779,
        0.052811769511494681,-0.70313383642924188,0.0,0.0,0.0,0.0,0.0,-0.0,-0.0,-0.0,-0.0,-0.0,-0.0,
        0.45973190050489809,0.70294533564091954,0.052804674695198853,-0.00038089908812926509,0.38141260703668056,
        0.046234063364270724,0.0,0.0,0.0,0.0,0.0,0.0,0.0,-0.0,-0.0,-0.0,-0.0,-0.0,-0.0,-1.0,-0.0,
        -0.047640075741515714,0.58732556690019289,0.046208184541143907,0.0527889750728095,-0.38141260703668045,0.0,
        0.0,0.0,0.0,0.0,0.0,0.0,-0.0,-0.0,-0.0,-0.0,-0.0,-0.0,-1.0,-0.63942378652894072,0.046157579132412543,
        0.040327604063683443,0.587325187651558,-0.053202204406742878,0.0,0.0,0.0,0.0,0.0,0.0,1.0,-0.0,-0.0,-0.0,
        -0.0,-0.0,-0.0,-0.0,-0.63942401877909172,0.052725613098002388,0.5873250705248978,-0.041479097778282417,0.0,
        0.0,0.0,0.0,0.0,0.0,1.0,-0.0,-0.0,-0.0,-0.0,-0.0,-0.0,-0.0,0.046165728248822993,0.55787198584888142,
        0.040334527208629144,0.041486711482857666,-0.70285954634074388,-0.70294129315678422,0.0,0.0,0.0,0.0,0.0,0.0,
        1.0,-0.0,-0.0,-0.0,-0.0,-0.0,-0.0,-0.0,-0.0,-0.0,0.048008393947647693,0.45973364369000813,
        0.70294446596883153,-0.04468906953870326,-0.7026717750678485,-0.040414301735567953,0.0,0.0,0.0,0.0,0.0,0.0,
        -0.0,-0.0,-0.0,-0.0,-0.0,-0.0,-0.0,-0.0,0.044600683591742331,0.041479097778282431,0.053202204406742781,
        0.6394234093758725,-0.58732499879699229,0.0,0.0,0.0,0.0,0.0,0.0,-0.0,-0.0,-0.0,-0.0,-0.0,-0.0,-0.0,-1.0,
        -0.0,0.04620090230449761,0.62654066450971879,0.040386220026432489,-0.38139402411953638,
        -0.053264773578912634,-0.70313155774868152,0.0,0.0,0.0,0.0,-0.0,-0.0,-0.0,-0.0,-0.0,-0.0,
        0.047993536136706476,0.587326232489261,-0.38141452789755642,-0.044671688889686353,-0.040397149349959791,0.0,
        0.0,0.0,0.0,0.0,0.0,0.0,-0.0,-0.0,-0.0,-0.0,-0.0,-0.0,-1.0,-0.0,0.046157579132412557,0.040327604063683437,
        0.63942378652894072,-0.4597340245185435,-0.0532022044067428,-0.58732518765155828,0.0,0.0,0.0,0.0,0.0,-0.0,
        -0.0,-0.0,-0.0,-0.0,-0.0,-0.0,0.557871608027596,0.052734339992385269,-0.041486711482857687,
        -0.70286111061272671,-0.70294271779415229,0.0,0.0,0.0,0.0,0.0,0.0,1.0,-0.0,-0.0,-0.0,-0.0,-0.0,-0.0,-0.0,
        -0.0,0.45973321958975349,0.049191105586226788,0.70294302173702006,-0.041532433509010709,
        -0.70267008402296527,-0.027736669979992645,0.0,0.0,0.0,0.0,-0.0,-0.0,-0.0,-0.0,-0.0,-0.0,
        0.38140732638781988,0.0030799473449444718,0.048023761687426413,0.049208104725552843,0.047673661972528605,
        -0.048023761687426413,-0.049208104725552849,-0.0476736619725286,0.0,0.0,0.0,0.0,0.0,0.0,0.0,0.0,-0.0,-0.0,
        -0.0,-0.0,-0.0,-0.0,-0.0,-1.0,-0.0,0.052779600708881207,0.62654080641868259,-0.0415157290185677,
        -0.38139306057951583,-0.70313207851881332,0.0,0.0,0.0,0.0,0.0,0.0,-0.0,-0.0,-0.0,-0.0,-0.0,-0.0,-0.0,
        0.049174830154444675,0.58732523320298258,-0.041521509739207041,-0.381414321823259,-0.027720209169872008,0.0,
        0.0,0.0,0.0,0.0,0.0,-0.0,-0.0,-0.0,-0.0,-0.0,-0.0,-1.0,0.58732556690019289,0.047640075741515707,
        -0.046208184541143907,-0.38141260703668056,-0.052788975072809566,0.0,0.0,0.0,0.0,0.0,0.0,-0.0,-0.0,-0.0,
        -0.0,-0.0,-0.0,-0.0,-1.0,-0.048023761687426413,-0.38141452789755642,-0.70313329820348291,
        0.044707585477670654,0.0,0.0,0.0,0.0,0.0,0.0,1.0,0.0,0.0,-0.0,-0.0,-0.0,-0.0,-0.0,-0.0,-0.0,
        -0.0414867114828577,-6.14559350203706E-5,0.55787195015047186,-0.70285954634074388,-0.70294129315678422,0.0,
        0.0,0.0,0.0,0.0,0.0,0.0,1.0,0.0,-0.0,-0.0,-0.0,-0.0,-0.0,-0.0,-0.0,-0.041515729018567704,
        -0.027725808084743217,0.62654033525020214,-0.38139435220779894,-0.70313108620605158,0.0,0.0,0.0,0.0,0.0,0.0,
        -0.0,-0.0,-0.0,-0.0,-0.0,-0.044696511233766639,0.70285987351907608,-0.04153764440846508,0.3813943522077986,
        0.0046455551781967924,-0.70313098732427659,0.0,0.0,0.0,0.0,0.0,-0.0,-0.0,-0.0,-0.0,-0.0,-0.0,
        -0.046208184541143921,-0.040397149349959804,0.58732518765155828,-0.041521734602731619,0.0053499825507371188,
        -0.38141565496819624,0.0,0.0,0.0,0.0,0.0,0.0,0.0,0.0,-0.0,-0.0,-0.0,-0.0,-0.0,-0.0,-1.0,
        -0.048023761687426413,0.38141452789755642,0.7026717750678485,0.044707585477670654,0.040432404230908,0.0,0.0,
        0.0,0.0,0.0,0.0,0.0,-0.0,-0.0,-0.0,-0.0,-0.0,-0.0,-0.0,-1.0,-0.0,-0.041521509739207062,
        -0.044671688889686333,0.58732516183395489,0.027736318903840668,-0.3814156136550157,0.0,0.0,0.0,0.0,0.0,0.0,
        0.0,-0.0,-0.0,-0.0,-0.0,-0.0,-0.0,-0.052811769511494695,-0.70286111061272671,-0.027743014678389594,
        -0.38141436310945653,-6.1605929268691053E-5,0.04154365368638769,0.0,0.0,0.0,0.0,0.0,0.0,0.0,1.0,0.0,-0.0,
        -0.0,-0.0,-0.0,-0.0,-0.0,-0.38139306057951616,-0.70286111061272671,0.052811769511494744,0.70313198021515855,
        -0.04153764440846508,0.0,0.0,0.0,0.0,0.0,0.0,0.0,-0.0,-0.0,-0.0,-0.0,-0.0,-0.0,-0.0015662095088587794,1.0,
        -0.0,-0.38139435220779888,0.041537644408465059,0.00023256610403676135,0.0,0.0,0.0,0.0,0.0,0.0,0.0,-0.0,-0.0,
        -0.0,-0.0,-0.0,-0.0,-0.0,-0.38141436310945653,-0.0015661981899676553,0.0004794577441265344,
        -0.041543653686387648,0.0,0.0,0.0,0.0,0.0,0.0,1.0,0.0,-0.0,-0.0,-0.0,-0.0,-0.0,-0.0,-0.0,
        -0.55787195015047186,0.041486711482857659,0.00023216176133703439,0.70285954634074388,0.70294129315678422,
        0.0,0.0,0.0,0.0,0.0,0.0,0.0,-0.0,-0.0,-0.0,-0.0,-0.0,-0.0,-0.0,-1.0,-0.0,0.45973321032477421,
        0.70294271779415229,0.041532658817056131,-0.0004794577441265338,0.38141436310945637,0.0,0.0,0.0,0.0,0.0,0.0,
        0.0,-0.0,-0.0,-0.0,-0.0,-0.0,-0.0,-1.0,-0.0,-0.70313155774868141,0.046208184541143935,0.040397149349959777,
        0.38141532678103607,-0.0053499825507371248,-0.0015656878741349477,0.041521734602731612,0.0,0.0,0.0,0.0,0.0,
        0.0,1.0,-0.0,-0.0,-0.0,-0.0,-0.0,-0.0,-0.0,-0.0,-0.62654033525020214,0.041515729018567704,
        0.053264773578912579,0.38139435220779877,0.70313108620605158,0.0,0.0,0.0,0.0,0.0,0.0,-0.0,-0.0,-0.0,-0.0,
        -0.0,-0.0,-0.0,-0.0,-0.63942340937587239,0.041479097778282424,0.053202204406742795,0.58732499879699218,0.0,
        0.0,0.0,0.0,0.0,0.0,1.0,-0.0,-0.0,-0.0,-0.0,-0.0,-0.0,-0.0,-0.0,0.046220967236855211,0.45973402451854339,
        0.04041430173556794,0.7029419471796341,-0.05329394831239747,-0.70266869475347082,0.0,0.0,0.0,0.0,-0.0,-0.0,
        -0.0,-0.0,-0.0,-0.0,-0.0,-0.0,0.048023761687426413,0.38141452789755642,0.7026717750678485,
        -0.044707585477670675,-0.040432404230907985,0.0,0.0,0.0,0.0,0.0,0.0,0.0,-0.0,-0.0,-0.0,-0.0,-0.0,-0.0,-1.0,
        -0.0,-0.0,0.62654033525020214,-0.0,0.041521509739207055,0.04467168888968636,0.58732516183395489,
        -0.3814156136550157,0.0,0.0,0.0,0.0,0.0,0.0,-0.0,-0.0,-0.0,-0.0,-0.0,-0.0,-1.0,-0.0,0.046208184541143914,
        0.58732518765155806,0.040397149349959791,-0.38141532678103618,-0.053276115903559441,0.0,0.0,0.0,0.0,0.0,
        -0.0,-0.0,-0.0,-0.0,-0.0,-0.0,-0.0,0.049208104725552843,0.38141436310945653,0.00047945774412653418,
        0.0015661981899676573,-0.041543653686387676,0.0,0.0,0.0,0.0,0.0,0.0,-0.0,-0.0,-0.0,-0.0,-0.0,-0.0,-0.0,-1.0,
        -0.0,0.38141260703668067,0.0030800493725469838,0.00038089908812926525,-0.046234063364270724,
        -0.052821149416567063,0.0,0.0,0.0,0.0,0.0,0.0,-0.0,-0.0,-0.0,-0.0,-0.0,-0.0,-0.0,-1.0,-0.0,
        0.052788975072809573,0.5873250705248978,0.027720209169872036,0.70313207851881321,-0.041521734602731585,
        -0.38141436310945664,0.0,0.0,0.0,0.0,0.0,0.0,-0.0,-0.0,-0.0,-0.0,-0.0,-0.0,-0.0,-1.0,-0.041543427917705968,
        -0.38141561365501536,-0.00029424831666778297,-0.0015662085872463908,0.027769643467705708,0.0,0.0,0.0,0.0,
        0.0,0.0,1.0,0.0,0.0,-0.0,-0.0,-0.0,-0.0,-0.0,-0.0,-0.041532658817056138,0.0031055287133001592,
        -0.70266788285587956,0.0,0.0,0.0,0.0,0.0,0.0,1.0,0.0,0.0,-0.0,-0.0,-0.0,-0.0,-0.0,-0.0,-0.0,
        -0.041543427917705961,0.0030801002245625041,-0.00023261598934981646,0.381415654968196,0.0030801017285724173,
        0.0,0.0,0.0,0.0,0.0,0.0,0.0,0.0,-0.0,-0.0,-0.0,-0.0,-0.0,-0.0,-1.0,-0.0,-0.046234063364270724,
        -0.00017791507742684638,0.38141532678103585,0.053313287899267439,0.0,0.0,0.0,0.0,0.0,0.0,0.0,-0.0,-0.0,-0.0,
        -0.0,-0.0,-0.0,-1.0,-0.0,0.04623406336427073,0.38141532678103612,0.003080095298344224,
        0.00017791507742684627,-0.053313287899267488,0.0,0.0,0.0,0.0,0.0,-0.0,-0.0,-0.0,-0.0,-0.0,-0.0,-0.0,-0.0,
        0.041543427917705961,0.00029424831666778313,0.38141565496819613,0.0015662095088587807,0.0,0.0,0.0,0.0,0.0,
        0.0,-0.0,-0.0,-0.0,-0.0,-0.0,-0.0,-0.0,-1.0,-0.0,-0.0,-0.041543653686387669,-0.38141565496819613,
        -6.1661881147355389E-5,-0.0015662095088587807,0.0,0.0,0.0,0.0,0.0,0.0,0.0,1.0,0.0,0.0,-0.0,-0.0,-0.0,-0.0,
        -0.0,-0.0,0.60965291149047529,-0.00028893057593309761,0.45432670979185558,-0.00033174749061995039,
        0.41630255411925293,-0.00034245830389696241,-0.60965291149047529,0.00028893057593309761,
        -0.45432670979185558,0.00033174749061995045,-0.41630255411925293,0.00034245830389696241,0.0,0.0,0.0,0.0,0.0,
        0.0,0.0,0.0,1.0,0.0,-0.0,-0.0,-0.0,-0.0,-0.0,-0.0,-0.0,-0.0,-0.60965291149047518,0.0,
        -1.6889645757588247E-16,9.8644403672779264E-20,-1.2631111769540146E-16,4.5223656320158784E-20,0.0,
        -4.9322201836389632E-20,-4.5223656320158784E-20,0.0,0.0,0.0,0.0,0.0,0.0,0.0,1.0,0.0,-0.0,-0.0,-0.0,-0.0,
        -0.0,-0.0,-0.0,-0.0,0.00028893057593309761,0.60962843737462846,0.45430524726196975,-0.00038816816420182134,
        0.41628290531231787,-0.00039473384869379718,-0.60962843737462846,-0.45430524726196975,-0.41628290531231782,
        0.0,0.0,0.0,0.0,0.0,0.0,0.0,1.0,0.0,-0.0,-0.0,-0.0,-0.0,-0.0,-0.0,-0.0,-0.0,-0.45432670979185558,
        7.4814395651655677E-5,8.7898076503418541E-5,-0.55043530483183312,0.84085614120956309,-7.48192953866797E-5,
        -8.5505485825256925E-5,-8.790393854946284E-5,8.5505485825256979E-5,0.0,0.0,0.0,0.0,0.0,0.0,0.0,0.0,0.0,-0.0,
        -0.0,-0.0,-0.0,-0.0,-0.0,-0.0,0.00033174749061995039,-0.609625471048958,-0.416280549869921,
        0.00030075035944006475,0.60962481916553923,-0.00018417146899711554,0.45430208183095055,0.41628002822785948,
        0.0,0.0,0.0,0.0,0.0,0.0,0.0,0.0,1.0,-0.0,-0.0,-0.0,-0.0,-0.0,-0.0,-0.0,-0.41630255411925293,
        0.75758587834764834,-0.0001318993713365724,0.55043530483183345,-0.00015110237018723787,
        -0.00015561198793193225,0.0001318993713365724,0.00015110237018723792,0.00015561198793193225,0.0,0.0,0.0,0.0,
        0.0,0.0,0.0,0.0,0.0,-0.0,-0.0,-0.0,-0.0,-0.0,-0.0,-0.0,0.00034245830389696241,0.60963041253671413,
        -0.00022788856259313032,0.45430697881955218,-0.00030075035944006486,0.41628450770674136,
        -0.60963041253671413,-0.45430697881955218,-0.41628450770674136,0.0,0.0,0.0,0.0,0.0,0.0,0.0,0.0,1.0,-0.0,
        -0.0,-0.0,-0.0,-0.0,-0.0,-0.0,0.60965291149047518,0.0,9.8644403672779264E-20,4.5223656320158784E-20,0.0,
        1.6889645757588247E-16,-4.9322201836389632E-20,1.2631111769540143E-16,-4.5223656320158784E-20,0.0,0.0,0.0,
        0.0,0.0,0.0,0.0,0.0,0.0,-0.0,-0.0,-0.0,-0.0,-0.0,-0.0,-0.0,-1.0,-0.00028893057593309761,0.60962843737462846,
        0.45430524726196975,0.41628290531231787,-0.60962843737462846,-0.45430524726196975,0.00038816816420182151,
        -0.41628290531231782,0.00039473384869379718,0.0,0.0,0.0,0.0,0.0,0.0,0.0,0.0,1.0,-0.0,-0.0,-0.0,-0.0,-0.0,
        -0.0,-0.0,-0.0,0.45432670979185558,0.55043530483183334,-7.48192953866797E-5,-8.5505485825256925E-5,
        -8.790393854946284E-5,-0.84085614120956309,7.48192953866797E-5,8.790393854946284E-5,0.0,0.0,0.0,0.0,0.0,0.0,
        0.0,0.0,-0.0,-0.0,-0.0,-0.0,-0.0,-0.0,-0.0,-0.0,-0.00033174749061995045,0.609625471048958,
        0.41628054986992108,-0.00030075035944006497,0.45430208183095055,-0.60962481916553923,0.00018417146899711535,
        -0.45430208183095055,-0.41628002822785942,0.0,0.0,0.0,0.0,0.0,0.0,0.0,1.0,-0.0,-0.0,-0.0,-0.0,-0.0,-0.0,
        -0.0,-0.0,0.41630255411925293,-0.0001318993713365724,-0.00015110237018723787,-0.00015561198793193225,
        -0.75758587834764834,0.0001318993713365724,-0.55043530483183345,0.00015110237018723792,
        0.00015561198793193225,0.0,0.0,0.0,0.0,0.0,0.0,0.0,0.0,-0.0,-0.0,-0.0,-0.0,-0.0,-0.0,-0.0,-0.0,
        -0.00034245830389696241,0.60963041253671413,0.45430697881955218,0.41628450770674136,-0.60963041253671413,
        0.00022788856259313032,-0.45430697881955218,0.000300750359440065,-0.41628450770674136,0.0,0.0,0.0,0.0,0.0,
        0.0,0.0,1.0,-0.0,-0.0,-0.0,-0.0,-0.0,-0.0,-0.0,-0.0,-0.60962843737462846,6.6103931646927414E-20,
        1.6888786255250324E-16,3.2847016711299215E-19,1.2630515651810637E-16,1.2285470046927208E-19,0.0,0.0,0.0,0.0,
        0.0,0.0,1.0,0.0,-0.0,-0.0,-0.0,-0.0,-0.0,-0.0,-0.0,-0.0,-1.6889645757588244E-16,-0.840856141209563,
        -5.0906254663616592E-16,-6.6103349467276677E-20,4.9321661480447027E-20,0.0,6.6103349467276677E-20,0.0,0.0,
        0.0,0.0,0.0,0.0,0.0,0.0,0.0,0.0,1.0,0.0,-0.0,-0.0,-0.0,-0.0,-0.0,-0.0,-0.0,-0.609625471048958,
        -1.8210324712466985E-19,-4.8702744413524358E-19,-0.0,-0.84083456430118952,-1.2392259909544564E-20,0.0,0.0,
        0.0,0.0,0.0,0.0,0.0,0.0,1.0,-0.0,-0.0,-0.0,-0.0,-0.0,-0.0,-0.75758587834764846,0.0,-3.3051742928782641E-20,
        5.0906254663616612E-16,0.0,0.0,0.0,0.0,0.0,0.0,0.0,1.0,0.0,-0.0,-0.0,-0.0,-0.0,-0.0,-0.0,-0.0,
        -0.60963041253671413,3.5734093577646393E-19,-0.0,-0.84083847313020632,3.2392852856704325E-20,0.0,0.0,0.0,
        0.0,0.0,0.0,0.0,0.0,1.0,-0.0,-0.0,-0.0,-0.0,-0.0,-0.0,-0.60962843737462846,-6.6103931646927414E-20,-0.0,
        -0.84085610383552944,0.0,0.0,0.0,0.0,0.0,0.0,0.0,0.0,0.0,1.0,-0.0,-0.0,-0.0,-0.0,-0.0,-0.0,-0.0,
        -0.609625471048958,0.0,1.6888683968347326E-16,9.1051623562334923E-20,0.0,0.0,0.0,0.0,0.0,0.0,1.0,-0.0,-0.0,
        -0.0,-0.0,-0.0,-0.0,-0.0,-0.60963041253671413,-4.522365632015879E-20,1.6888856812294667E-16,
        1.2630566289979805E-16,0.0,-1.7867046788823196E-19,0.0,0.0,0.0,0.0,0.0,0.0,1.0,-0.0,-0.0,-0.0,-0.0,-0.0,
        -0.0,-0.0,-0.0,7.481439565165569E-5,-0.45429994164840926,4.8427929846470528E-5,0.84085082053685611,
        -0.00051016981098213191,0.0,0.0,0.0,0.0,0.0,0.0,0.0,0.0,-0.0,-0.0,-0.0,-0.0,-0.0,-0.0,
        0.00018415797916782135,0.00038816816420182129,0.60962237832884059,0.4542999416484092,0.41627806175091842,
        -0.0004141582836222081,-0.60962237832884059,-0.4542999416484092,-0.41627806175091842,0.0,0.0,0.0,0.0,0.0,
        0.0,0.0,0.0,-0.0,-0.0,-0.0,-0.0,-0.0,-0.0,0.00013189937133657251,-0.41628290531231782,0.757562300931841,
        0.55040967557980414,-0.00017606010923842055,0.0,0.0,0.0,0.0,0.0,0.0,0.0,0.0,-0.0,-0.0,-0.0,-0.0,-0.0,-0.0,
        -0.0,0.00022788856259313035,0.00039473384869379729,0.41627862603096338,-0.6096230881794128,
        -0.45430056003742264,-0.41627862603096327,0.0,0.0,0.0,0.0,0.0,0.0,0.0,0.0,1.0,0.0,-0.0,-0.0,-0.0,-0.0,-0.0,
        -0.0,-0.0,8.5975056991699629E-20,0.60962843737462846,1.642350835564962E-19,-3.3777572510500658E-16,
        -2.5261031303621274E-16,0.0,0.0,0.0,0.0,0.0,0.0,0.0,0.0,-0.0,-0.0,-0.0,-0.0,-0.0,-0.0,-0.0,-1.0,
        7.481439565165569E-5,0.45430524726196975,-9.9174781569828316E-5,-0.84085610383552944,0.00051016158613891569,
        0.0,0.0,0.0,0.0,0.0,0.0,0.0,-0.0,-0.0,-0.0,-0.0,-0.0,-0.0,-0.0,0.00013189937133657251,0.41628290531231782,
        -0.00017606010923842055,-0.0001782357389326195,-0.757562300931841,-0.55040967557980436,0.0,0.0,0.0,0.0,0.0,
        0.0,0.0,-0.0,-0.0,-0.0,-0.0,-0.0,-0.0,-0.0,-0.0,-0.45430265350071453,8.5499847267427823E-5,
        -0.55040651377225314,7.846411462241605E-5,0.8408340548111205,-4.8431021786366918E-5,0.0,0.0,0.0,0.0,0.0,0.0,
        0.0,0.0,-0.0,-0.0,-0.0,-0.0,-0.0,-0.0,-0.45430697881955229,8.7898076503418581E-5,-0.55041168721633849,
        0.8408384731302061,-7.8469117928435135E-5,0.0,0.0,0.0,0.0,0.0,0.0,0.0,0.0,-0.0,-0.0,-0.0,-0.0,-0.0,-0.0,
        -0.45430524726196975,0.00010010180270488143,-0.550409675579804,-7.4819295386679732E-5,0.84083690387628529,
        9.9181420037518247E-5,0.0,0.0,0.0,0.0,0.0,0.0,0.0,0.0,-0.0,-0.0,-0.0,-0.0,-0.0,-0.0,-0.0,
        -0.55040651377225314,-8.5505485825257047E-5,0.8408345643011893,4.8427734256521668E-5,0.0001028531289785517,
        0.0,0.0,0.0,0.0,0.0,-0.0,-0.0,-0.0,-0.0,-0.0,0.00015110237018723782,-0.41628054986992113,
        0.00013795452656197144,-8.4707990552849259E-5,0.55040582594762266,0.0,0.0,0.0,0.0,0.0,0.0,0.0,0.0,-0.0,-0.0,
        -0.0,-0.0,-0.0,-0.0,-3.1149970082996928E-20,-1.2630446370897993E-16,-2.3845293855353908E-19,
        0.60962481916553923,-1.8209900679330059E-19,1.6888661273616133E-16,0.0,0.0,0.0,0.0,0.0,0.0,0.0,0.0,-0.0,
        -0.0,-0.0,-0.0,-0.0,-0.0,-1.0,8.54998472674278E-5,7.8464114622416064E-5,0.4543020818309505,
        -4.842792984647046E-5,-0.84085325521465437,0.0005101680221438746,0.0,0.0,0.0,0.0,0.0,-0.0,-0.0,-0.0,-0.0,
        -0.0,0.00015110237018723782,-0.757559413479883,-0.550406513772253,0.00013795452656197138,
        0.41628002822785937,-8.4707990552849354E-5,0.0,0.0,0.0,0.0,0.0,0.0,0.0,-0.0,-0.0,-0.0,-0.0,-0.0,-0.0,-0.0,
        -0.41628450770674136,0.00015561198793193225,0.55041168721633849,-0.0001379545265619716,0.0,0.0,0.0,0.0,0.0,
        0.0,0.0,0.0,-0.0,-0.0,-0.0,-0.0,-0.0,-0.0,-0.41628290531231787,-0.00013189937133657249,0.55040967557980436,
        0.00017606010923842063,0.00017823573893261942,0.0,0.0,0.0,0.0,0.0,0.0,0.0,0.0,-0.0,-0.0,-0.0,-0.0,-0.0,-0.0,
        -0.0,-0.41628054986992108,-0.00015110237018723798,0.55040651377225314,8.4702035317903214E-5,
        0.00018467833523565694,0.0,0.0,0.0,0.0,0.0,-0.0,-0.0,-0.0,-0.0,-0.0,-0.41628450770674136,
        -0.00015561198793193225,0.75756418984348128,0.55041168721633849,0.00010468726281301101,
        0.00013795452656197179,0.0,0.0,0.0,0.0,0.0,0.0,0.0,-0.0,-0.0,-0.0,-0.0,-0.0,-0.0,-0.0,
        -8.803423606264926E-20,0.60963041253671413,3.5734093577646412E-19,3.3777713624589364E-16,
        3.7891698869939418E-16,0.0,0.0,0.0,0.0,0.0,0.0,0.0,0.0,-0.0,-0.0,-0.0,-0.0,-0.0,-0.0,-1.0,
        8.7898076503418486E-5,0.45430697881955218,-7.8464114622416145E-5,-0.84085767302744141,
        0.00051016354941838882,0.0,0.0,0.0,0.0,0.0,-0.0,-0.0,-0.0,-0.0,-0.0,0.00015561198793193222,
        0.41628450770674136,-0.00013795452656197141,-0.75756418984348128,-0.5504116872163386,0.0,0.0,0.0,0.0,0.0,
        0.0,0.0,-0.0,-0.0,-0.0,-0.0,-0.0,-0.0,-0.0,0.60962843737462846,-6.6103931646927414E-20,
        -1.6888786255250324E-16,-1.6423508355649608E-19,-1.2630515651810632E-16,-1.228547004692721E-19,0.0,0.0,0.0,
        0.0,0.0,0.0,0.0,0.0,-0.0,-0.0,-0.0,-0.0,-0.0,-0.0,-1.0,-0.0,0.84087533887700028,1.6889645757588244E-16,
        -6.6103393866630849E-20,0.0,4.5223181965109357E-20,0.0,0.0,0.0,0.0,0.0,0.0,0.0,-0.0,-0.0,-0.0,-0.0,-0.0,
        -0.0,-0.0,-1.0,0.609625471048958,0.0,9.1051623562334923E-20,-1.6888683968347326E-16,-1.2630446370897993E-16,
        0.0,0.0,0.0,0.0,0.0,0.0,-0.0,-0.0,-0.0,-0.0,-0.0,-1.0,0.75758587834764846,0.0,0.84085614120956309,
        -4.9989848646664218E-16,-6.6103349467276677E-20,4.9321661480447027E-20,0.0,6.6103349467276677E-20,0.0,0.0,
        0.0,0.0,0.0,0.0,0.0,0.0,0.0,-0.0,-0.0,-0.0,-0.0,-0.0,-0.0,-0.0,-0.0,-1.0,0.60963041253671413,
        -4.522365632015879E-20,0.0,-1.6888856812294667E-16,-1.7867046788823196E-19,-1.26305662899798E-16,0.0,0.0,
        0.0,0.0,0.0,0.0,0.0,-0.0,-0.0,-0.0,-0.0,-0.0,-0.0,-0.0,-1.0,-7.481439565165569E-5,0.45430524726196975,
        -0.84085610383552944,9.9174781569828492E-5,0.00051016158613891569,0.0001001018027048814,0.0,0.0,0.0,0.0,0.0,
        -0.0,-0.0,-0.0,-0.0,-0.0,-0.0,-0.00018415797916782124,-0.00038816816420182151,0.60962237832884059,
        0.4542999416484092,0.41627806175091842,-0.60962237832884059,-0.4542999416484092,-0.41627806175091842,
        0.00041415828362220767,0.0,0.0,0.0,0.0,0.0,1.0,-0.0,-0.0,-0.0,-0.0,-0.0,-0.0,-0.0,-0.0,
        -0.00013189937133657251,0.41628290531231782,-0.757562300931841,-0.55040967557980436,0.00017606010923842071,
        0.0001782357389326195,0.0,0.0,0.0,0.0,0.0,0.0,0.0,-0.0,-0.0,-0.0,-0.0,-0.0,-0.0,-0.0,-0.0,
        -0.00022788856259313035,-0.00039473384869379729,0.41627862603096338,-0.6096230881794128,
        0.00037493747421003197,0.0,0.0,0.0,0.0,0.0,0.0,0.0,-0.0,-0.0,-0.0,-0.0,-0.0,-0.0,-0.0,0.45430265350071453,
        -8.5499847267427864E-5,-0.84085376462535322,4.8424642574532886E-5,0.00051016694671599048,
        0.00010284562563608354,0.0,0.0,0.0,0.0,-0.0,-0.0,-0.0,-0.0,0.45430697881955229,0.55041168721633871,
        -8.790393854946284E-5,-0.84083847313020632,5.9714664557388114E-5,7.8469117928435325E-5,0.0,0.0,0.0,0.0,0.0,
        0.0,-0.0,-0.0,-0.0,-0.0,-0.0,-0.0,-0.0,-0.0,-0.00015110237018723787,0.41628054986992113,-0.757559413479883,
        8.4702035317903214E-5,-0.55040651377225336,0.00018467833523565724,0.0,0.0,0.0,0.0,0.0,0.0,-0.0,-0.0,-0.0,
        -0.0,-0.0,-0.0,-0.0,0.41628450770674136,-0.00015561198793193225,-0.75756418984348139,0.00010468726281301101,
        -0.55041168721633871,0.00013795452656197179,0.0,0.0,0.0,0.0,0.0,0.0,-0.0,-0.0,-0.0,-0.0,-0.0,-0.0,-0.0,-0.0,
        -1.6888573396344759E-16,-0.84083212995208934,1.753764380417449E-19,-1.1802018608337481E-21,0.0,0.0,0.0,0.0,
        0.0,0.0,0.0,0.0,1.0,0.0,-0.0,-0.0,-0.0,-0.0,-0.0,-0.0,-0.60962237832884059,1.8210324712466982E-19,
        -1.6392577615272447E-19,1.6888575123732502E-16,0.0,0.0,0.0,0.0,0.0,0.0,0.0,-0.0,-0.0,-0.0,-0.0,-0.0,-0.0,
        -0.75756230093184107,3.7331729402847582E-23,-0.84083690387628518,5.53660320073937E-20,
        3.2846577158052279E-19,0.0,0.0,0.0,0.0,0.0,0.0,0.0,1.0,0.0,-0.0,-0.0,-0.0,-0.0,-0.0,-0.0,-0.0,
        -0.60962481916553923,-9.104950339665027E-20,-0.0,4.6369306445630311E-19,-0.84083405481112061,
        -1.1852459228007919E-21,1.0491070505542491E-21,0.0,0.0,0.0,0.0,0.0,0.0,0.0,0.0,1.0,-0.0,-0.0,-0.0,-0.0,-0.0,
        -0.0,-0.75756418984348139,2.1781387555242696E-23,-0.84083847313020632,4.9988181455745605E-16,
        -3.2392852856704325E-20,1.2302723083271699E-19,0.0,0.0,0.0,0.0,0.0,0.0,0.0,0.0,1.0,-0.0,-0.0,-0.0,-0.0,-0.0,
        -0.0,-0.0,-0.60962237832884059,-9.1145916457961507E-20,-3.0930740377156518E-22,1.6888575123732502E-16,
        -4.8686518566049995E-19,0.0,0.0,0.0,0.0,0.0,1.0,-0.0,-0.0,-0.0,-0.0,-0.0,-0.0,-0.0,-0.0,
        -0.60962481916553923,-5.9686710504540159E-20,1.6888661273616133E-16,1.263043082212299E-16,0.0,0.0,0.0,0.0,
        0.0,0.0,0.0,1.0,-0.0,-0.0,-0.0,-0.0,-0.0,-0.0,-0.0,-0.0,7.4819295386679732E-5,-0.55040967557980436,
        0.000510161586138917,0.84083690387628518,-9.9181420037517732E-5,0.0,0.0,0.0,0.0,0.0,0.0,0.0,0.0,-0.0,-0.0,
        -0.0,-0.0,-0.0,-0.0,-0.0,0.00017606010923842057,-0.41627806175091836,8.4707990552849435E-5,
        0.55040260512924977,0.0,0.0,0.0,0.0,0.0,0.0,0.0,0.0,0.0,-0.0,-0.0,-0.0,-0.0,-0.0,-0.0,
        0.00018417146899711557,9.2246400529989555E-7,0.60962172564668826,0.45429936926246767,0.41627753944540197,
        -0.60962172564668826,-0.45429936926246767,-0.41627753944540186,0.0,0.0,0.0,0.0,0.0,0.0,0.0,0.0,1.0,0.0,-0.0,
        -0.0,-0.0,-0.0,-0.0,-0.0,-0.0,-3.3840557120343592E-19,1.2630370373302073E-16,2.7260181487290321E-19,
        0.60962172564668826,-1.6888552398678938E-16,0.0,0.0,0.0,0.0,0.0,0.0,0.0,0.0,0.0,-0.0,-0.0,-0.0,-0.0,-0.0,
        -0.0,-1.0,9.9174781569828235E-5,4.842792984647044E-5,0.45429936926246772,-0.84085082053685589,
        0.00051016981098363212,0.0,0.0,0.0,0.0,0.0,0.0,-0.0,-0.0,-0.0,-0.0,-0.0,8.470203531790335E-5,
        0.00017606010923842057,0.41627806175091836,-0.00018466881149421227,-0.75755643964663877,
        -0.55040329378266917,0.0,0.0,0.0,0.0,0.0,0.0,0.0,-0.0,-0.0,-0.0,-0.0,-0.0,-0.0,8.4707990552849408E-5,
        4.1133666665477103E-7,0.0033259399136323126,-0.75755581033457731,-0.5504026051292501,0.0,0.0,0.0,0.0,0.0,
        0.0,0.0,0.0,-0.0,-0.0,-0.0,-0.0,-0.0,-0.0,-0.0,6.5147957832588729E-20,0.84085610383552933,
        5.0666358765750976E-16,1.0002394461110747E-15,0.0,0.0,0.0,0.0,0.0,0.0,0.0,-0.0,-0.0,-0.0,-0.0,-0.0,-0.0,
        -0.0,-1.0,9.752374880021247E-20,2.69219864857825E-19,0.75755643964663866,-1.2630370373302068E-16,
        -4.8686050246126125E-19,0.0,0.0,0.0,0.0,0.0,0.0,0.0,-0.0,-0.0,-0.0,-0.0,-0.0,-0.0,-1.0,
        7.4819295386679732E-5,0.55040967557980447,-9.9181420037517732E-5,-0.0001001086588859579,
        -0.84083690387628518,0.0,0.0,0.0,0.0,0.0,0.0,0.0,-0.0,-0.0,-0.0,-0.0,-0.0,-0.0,-0.0,-0.0,
        -0.55041168721633849,0.00051016354941819909,-8.790393854946284E-5,0.8408384731302061,5.9714664557388114E-5,
        7.8469117928435325E-5,0.0,0.0,0.0,0.0,0.0,0.0,0.0,-0.0,-0.0,-0.0,-0.0,-0.0,-0.0,-0.0,-0.55040329378266928,
        -4.8427734256521736E-5,-9.9181420037518044E-5,0.84083212995208922,0.00010284859467966867,0.0,0.0,0.0,0.0,
        0.0,-0.0,-0.0,-0.0,-0.0,-0.0,-0.0,-0.45430208183095055,-0.55040582594762288,-7.8469117928435352E-5,
        0.84083405481112039,4.843102178636683E-5,0.0,0.0,0.0,0.0,0.0,0.0,0.0,-0.0,-0.0,-0.0,-0.0,-0.0,-0.0,-0.0,
        -3.1149707480090415E-20,0.75755941347988309,0.0,-1.8210264972536316E-19,-4.8702276280530372E-19,
        -5.090289676538971E-16,0.0,0.0,0.0,0.0,0.0,-0.0,-0.0,-0.0,-0.0,-0.0,-0.0,-1.0,8.5505485825256939E-5,
        7.8469117928435148E-5,0.55040582594762255,-4.843102178636702E-5,-0.84083405481112061,0.0,0.0,0.0,0.0,0.0,
        0.0,0.0,-0.0,-0.0,-0.0,-0.0,-0.0,-0.0,-0.0,-0.4162780617509183,-8.4702035317903322E-5,
        -0.00017606010923842068,0.55040329378266928,0.00018466881149421203,0.0,0.0,0.0,0.0,0.0,-0.0,-0.0,-0.0,-0.0,
        -0.0,-0.0,-0.00010468726281301108,-0.00017823573893261944,0.55040403961997142,-0.0033259399136323117,
        -8.4707990552849354E-5,0.75755581033457708,0.0,0.0,0.0,0.0,0.0,0.0,0.0,-0.0,-0.0,-0.0,-0.0,-0.0,-0.0,-0.0,
        -0.0,-0.41628002822785942,-0.0001379545265619716,0.757558784908481,0.55040582594762277,
        8.4707990552849286E-5,0.0,0.0,0.0,0.0,0.0,0.0,0.0,-0.0,-0.0,-0.0,-0.0,-0.0,-0.0,-0.0,
        -3.9166243175019444E-20,0.75756418984348139,-1.2630566289979805E-16,3.5733825445920967E-19,
        5.0903497598883843E-16,0.0,0.0,0.0,0.0,0.0,0.0,0.0,-0.0,-0.0,-0.0,-0.0,-0.0,-0.0,-1.0,8.7903938549462773E-5,
        0.5504116872163386,-7.8469117928435311E-5,-0.84083847313020632,0.0,0.0,0.0,0.0,0.0,0.0,0.0,-0.0,-0.0,-0.0,
        -0.0,-0.0,-0.0,-0.0,0.75756230093184118,-6.61034858575653E-20,-3.7331729402847559E-23,0.84083690387628518,
        -1.642328857902614E-19,-1.2285307508338753E-19,0.0,0.0,0.0,0.0,0.0,0.0,0.0,-0.0,-0.0,-0.0,-0.0,-0.0,-0.0,
        -0.0,-1.0,-0.0,0.6096230881794128,-8.2110521488695769E-20,-3.1878054029127235E-22,-1.6888599687103994E-16,
        -4.948054548592409E-19,-1.2630387361850009E-16,0.0,0.0,0.0,0.0,0.0,0.0,-0.0,-0.0,-0.0,-0.0,-0.0,-0.0,-1.0,
        -0.0,1.68888545925672E-16,0.84083847313020632,5.090349529564296E-16,-3.2392852856704325E-20,0.0,0.0,0.0,0.0,
        0.0,0.0,0.0,-0.0,-0.0,-0.0,-0.0,-0.0,-0.0,-0.0,-0.0,-1.0,0.75755941347988309,-4.9321788734096E-20,
        -2.8888103944906731E-23,0.0,-5.090289676538971E-16,-4.8702276280530247E-19,0.0,0.0,0.0,0.0,-0.0,-0.0,-0.0,
        -0.0,-0.0,-1.0,0.60962481916553923,-5.9686710504540159E-20,0.0,-1.6888661273616133E-16,
        -1.2630430822122988E-16,0.0,0.0,0.0,0.0,0.0,0.0,0.0,-0.0,-0.0,-0.0,-0.0,-0.0,-0.0,-0.0,-1.0,
        0.75756418984348139,-2.1781387555242688E-23,-4.5223264325215918E-20,0.0,-5.0903497598883764E-16,
        -1.786691272296046E-19,0.0,0.0,0.0,0.0,0.0,-0.0,-0.0,-0.0,-0.0,-0.0,-0.0,-1.0,-7.4819295386679732E-5,
        0.55040967557980447,-0.84083690387628518,9.91814200375179E-5,0.0001001086588859579,0.0,0.0,0.0,0.0,0.0,0.0,
        0.0,-0.0,-0.0,-0.0,-0.0,-0.0,-0.0,-0.0,-0.0,-5.9710851674489663E-5,0.4543005600374227,
        -0.00010010180270488141,-0.84085190118769138,9.7305019763635448E-5,0.0005101684703272578,0.0,0.0,0.0,0.0,
        -0.0,-0.0,-0.0,-0.0,-0.0,-0.0,-0.00018417146899711554,-1.6433908261248681E-6,0.60962172564668826,
        0.45429936926246767,0.41627753944540197,-0.60962172564668826,-0.45429936926246767,-0.41627753944540186,0.0,
        0.0,0.0,0.0,0.0,0.0,0.0,1.0,-0.0,-0.0,-0.0,-0.0,-0.0,-0.0,-0.0,-0.0,-0.0,0.55040651377225325,
        -8.5505485825257E-5,-0.8408345643011893,4.8427734256521695E-5,0.00010285312897855262,0.0,0.0,0.0,0.0,0.0,
        0.0,-0.0,-0.0,-0.0,-0.0,-0.0,-0.0,-0.0,0.45430208183095055,-7.846411462241624E-5,-0.840853255214654,
        4.8427929846470358E-5,0.00051016802214387308,0.0,0.0,0.0,0.0,0.0,0.0,-0.0,-0.0,-0.0,-0.0,-0.0,-0.0,-0.0,
        -0.00013795452656197157,0.41628002822785942,-0.75755878490848116,8.4707990552849259E-5,-0.550405825947623,
        0.0,0.0,0.0,0.0,0.0,0.0,-0.0,-0.0,-0.0,-0.0,-0.0,-0.0,-0.0,-0.0,-0.60962172564668826,1.8211991325743819E-19,
        4.869769891576791E-19,1.6888552398678938E-16,0.0,0.0,0.0,0.0,0.0,0.0,0.0,1.0,0.0,-0.0,-0.0,-0.0,-0.0,-0.0,
        -0.0,-0.0,-0.84083690387628529,1.1099619416141393E-18,-5.5366032007393707E-20,-1.642328857902614E-19,
        -1.2285307508338753E-19,0.0,0.0,0.0,0.0,0.0,0.0,0.0,0.0,1.0,-0.0,-0.0,-0.0,-0.0,-0.0,-0.0,-0.0,
        -0.84083456430118952,4.998780955584154E-16,-3.6929401570902465E-20,9.1051235165092008E-20,
        -4.8702128521147154E-19,0.0,0.0,0.0,0.0,0.0,1.0,-0.0,-0.0,-0.0,-0.0,-0.0,-1.6888571313082695E-16,
        2.0933278467107486E-20,-0.84083212995208934,-8.4419497240682937E-20,9.4703432327985161E-23,
        -4.8685902445272773E-19,0.0,0.0,0.0,0.0,0.0,-0.0,-0.0,-0.0,-0.0,-0.0,-0.0,-0.75755878490848128,
        2.8892611608762185E-23,-5.9686264459664926E-20,-0.84083405481112061,-4.4225931473166894E-22,
        9.10491149162437E-20,0.0,0.0,0.0,0.0,0.0,0.0,0.0,1.0,-0.0,-0.0,-0.0,-0.0,-0.0,-0.0,-0.0,
        -0.60962172564668826,-9.1143806586707121E-20,-2.9022766546388333E-22,1.6888552398678938E-16,
        1.2630354803031406E-16,0.0,0.0,0.0,0.0,0.0,0.0,1.0,-0.0,-0.0,-0.0,-0.0,-0.0,-0.0,-0.0,-0.0,-0.0,
        -0.84085325521465415,-1.6888658327079123E-16,-4.3588336687542244E-20,0.0,9.1049145421375812E-20,0.0,0.0,0.0,
        0.0,0.0,0.0,1.0,-0.0,-0.0,-0.0,-0.0,-0.0,-0.0,-0.550403293782669,9.91814200375178E-5,0.00051016873546545674,
        4.8431021786367026E-5,1.1324499555899527E-6,0.84083161987084709,0.0,0.0,0.0,0.0,0.0,0.0,0.0,0.0,0.0,-0.0,
        -0.0,-0.0,-0.0,-0.0,-0.0,4.8427734256521838E-5,9.91814200375178E-5,0.55040329378266961,
        -0.00010284859467966931,-0.840832129952089,0.0,0.0,0.0,0.0,0.0,0.0,0.0,-0.0,-0.0,-0.0,-0.0,-0.0,-0.0,
        4.932282965723688E-22,0.0,-0.0,2.3390148868998579E-19,0.84083212995208911,-2.0997770285150725E-18,0.0,0.0,
        0.0,0.0,0.0,0.0,0.0,-0.0,-0.0,-0.0,-0.0,-0.0,-0.0,-1.0,4.8431021786366952E-5,2.2909110573910174E-7,
        0.0049960062272682909,-0.840831619870847,0.0,0.0,0.0,0.0,0.0,0.0,0.0,0.0,-0.0,-0.0,-0.0,-0.0,-0.0,-0.0,-0.0,
        9.752354635032987E-20,0.84083690387628507,1.1110082532230706E-18,3.2846577158052289E-19,
        1.2285307508338753E-19,0.0,0.0,0.0,0.0,0.0,0.0,0.0,-0.0,-0.0,-0.0,-0.0,-0.0,-0.0,-0.0,-0.0,-1.0,
        -5.9714664557388216E-5,-0.000100108658885958,0.84083270065149018,-0.0049960062272682874,
        -4.8431021786366918E-5,0.0,0.0,0.0,0.0,0.0,0.0,0.0,-0.0,-0.0,-0.0,-0.0,-0.0,-0.0,-0.0,-0.0,
        6.12256505583179E-19,0.75755878490848116,-1.2630430822122988E-16,-1.8209840926457502E-19,
        -2.0076641711829734E-21,1.184453526596045E-21,0.84083405481112039,0.0,0.0,0.0,0.0,0.0,0.0,0.0,-0.0,-0.0,
        -0.0,-0.0,-0.0,-0.0,-0.0,-1.0,-6.0614409112096141E-20,0.84083456430118952,5.090289676538969E-16,
        -2.7315370549527618E-19,-4.8702128521147357E-19,0.0,0.0,0.0,0.0,0.0,0.0,-0.0,-0.0,-0.0,-0.0,-0.0,-0.0,-0.0,
        -1.0,9.7009564648539721E-21,0.84083847313020621,-7.6367237767394E-16,1.7866871575948447E-19,0.0,0.0,0.0,0.0,
        0.0,0.0,0.0,-0.0,-0.0,-0.0,-0.0,-0.0,-0.0,-0.0,-1.0,0.75755713294087956,-8.2110137308287566E-20,
        -3.7367713213901915E-23,-3.1878155269934057E-22,-5.0902608880363241E-16,-4.9480031627697222E-19,0.0,0.0,0.0,
        0.0,-0.0,-0.0,-0.0,-0.0,-0.0,-0.0,-1.0,-0.0,0.60962172564668826,-9.1143806586707121E-20,
        -2.9022766546388333E-22,-1.6888552398678938E-16,-1.2630354803031404E-16,0.0,0.0,0.0,0.0,0.0,0.0,0.0,-0.0,
        -0.0,-0.0,-0.0,-0.0,-0.0,-0.0,-1.0,-0.0,-3.6929401570902471E-20,-0.0,0.84085325521465415,
        1.6888658327079123E-16,-4.3588336687542244E-20,9.1049145421375812E-20,0.0,0.0,0.0,0.0,0.0,0.0,-0.0,-0.0,
        -0.0,-0.0,-0.0,-0.0,-0.0,-1.0,0.75755878490848128,-5.9686264459664962E-20,-2.8892611608762185E-23,0.0,
        -5.0902816324565257E-16,0.0,0.0,0.0,0.0,0.0,-0.0,-0.0,-0.0,-0.0,-0.0,-0.0,-1.0,0.45429936926246767,
        -4.8431021786366857E-5,0.0049960062272682891,-2.2909110573910145E-7,-0.84083161987084709,0.0,0.0,0.0,0.0,
        0.0,0.0,-0.0,-0.0,-0.0,-0.0,-0.0,-0.0,-0.0,-0.0,-0.0,-8.4707990552849313E-5,-7.5250479866203283E-7,
        0.003325939913632313,-0.75755581033457731,-0.55040260512924977,0.0,0.0,0.0,0.0,0.0,0.0,-0.0,-0.0,-0.0,-0.0,
        -0.0,-0.0,-0.0,-0.0,-0.0,0.55040582594762288,-7.8469117928435392E-5,-0.00051016802214399538,
        -0.0001028531289785522,-0.84083405481112039,4.8431021786366823E-5,0.0,0.0,0.0,0.0,0.0,0.0,-0.0,-0.0,-0.0,
        -0.0,-0.0,-0.0,-0.0,-0.0,-0.840850820536856,1.7234498339055512E-19,-1.1115400945908851E-18,
        1.0327571811693951E-21,0.0,0.0,0.0,0.0,0.0,0.0,0.0,0.0,1.0,0.0,-0.0,-0.0,-0.0,-0.0,-0.0,-0.0,
        -0.84083270065149041,6.4644696919149857E-23,-4.9479871196138011E-19,0.0,0.0,0.0,0.0,0.0,0.0,0.0,1.0,0.0,
        -0.0,-0.0,-0.0,-0.0,-0.0,-0.0,-0.0,-0.84085082053685589,8.7195661360134582E-23,-2.220969953600735E-18,
        -8.4416862202560415E-20,6.0122310366782144E-23,0.0,0.0,0.0,0.0,0.0,0.0,0.0,1.0,-0.0,-0.0,-0.0,-0.0,-0.0,
        -0.0,-0.0,-0.0,-0.75755581033457731,1.6446215595724026E-25,-9.1143508979403014E-20,5.0902442300953653E-16,
        0.0,0.0,0.0,0.0,0.0,0.0,1.0,-0.0,-0.0,-0.0,-0.0,-0.0,-0.0,-0.0,-0.0,0.75755581033457731,
        -9.1143508979403E-20,-1.2721949911164169E-24,-1.6446215595724021E-25,-5.0902442300953574E-16,0.0,0.0,0.0,
        0.0,0.0,-0.0,-0.0,-0.0,-0.0,-0.0,-0.0,-1.0,-0.0,0.840850820536856,1.1115400081964914E-18,
        -8.4416862202560415E-20,3.4597823432971686E-23,0.0,0.0,0.0,0.0,0.0,0.0,-0.0,-0.0,-0.0,-0.0,-0.0,-0.0,-0.0,
        -0.0,-1.0,-0.0,-0.84083161987084709,1.753925793255534E-19,1.1099619109243672E-18,1.0493469223541793E-21,0.0,
        0.0,0.0,0.0,0.0,0.0,0.0,0.0,1.0,0.0,-0.0,-0.0,-0.0,-0.0,-0.0,-0.0,-0.00028983042660450772,
        0.60774185316849594,-0.00032104499842707462,0.45260561554757484,-0.00032423089662980361,0.41470020324647255,
        0.00028983042660450772,-0.60774185316849594,0.00032104499842707462,-0.45260561554757484,
        0.00032423089662980361,-0.41470020324647255,0.0,0.0,0.0,0.0,0.0,0.0,0.0,0.0,0.0,1.0,-0.0,-0.0,-0.0,-0.0,
        -0.0,-0.0,-0.0,-0.0,0.00028983042660450767,0.60771760732198055,-0.00034998845489279349,0.45258306322192471,
        -0.00034322043275703971,0.41467880541713448,-0.60771760732198055,-0.45258306322192471,-0.41467880541713448,
        0.0,0.0,0.0,0.0,0.0,0.0,0.0,0.0,1.0,-0.0,-0.0,-0.0,-0.0,-0.0,-0.0,-0.0,-0.0,-0.60774185316849594,0.0,
        4.9507562444117341E-20,-1.6818696161191519E-16,9.0792333081773271E-20,-1.2581077755555868E-16,0.0,
        -4.9507562444117341E-20,-9.0792333081773247E-20,0.0,0.0,0.0,0.0,0.0,0.0,0.0,0.0,1.0,-0.0,-0.0,-0.0,-0.0,
        -0.0,-0.0,-0.0,-0.0,0.00032104499842707462,-0.60771627901050718,-0.41467763318781908,0.00030990522922148058,
        -0.00020644223064780165,0.60771586837025782,0.45258145885114326,0.414677276341478,-0.45258145885114326,0.0,
        0.0,0.0,0.0,0.0,0.0,0.0,0.0,1.0,-0.0,-0.0,-0.0,-0.0,-0.0,-0.0,-0.0,-0.45260561554757484,
        6.705637981480354E-5,7.4542022764773985E-5,-0.54849096138382369,-6.70627819526479E-5,0.83950908011157221,
        -7.3882932570663252E-5,-7.4549313422904716E-5,0.0,0.0,0.0,0.0,0.0,0.0,0.0,0.0,0.0,-0.0,-0.0,-0.0,-0.0,-0.0,
        -0.0,-0.0,0.00032423089662980361,-0.00024604276486503597,0.607721627098605,-0.00030990522922148096,
        0.45258682574740111,0.41468237096544258,-0.607721627098605,-0.45258682574740111,-0.41468237096544258,0.0,
        0.0,0.0,0.0,0.0,0.0,0.0,0.0,1.0,-0.0,-0.0,-0.0,-0.0,-0.0,-0.0,-0.0,-0.41470020324647261,
        -0.00012282470380310523,0.75586897491059513,-0.00013548671280111892,0.54849096138382369,
        -0.0001366776091554688,0.00012282470380310523,0.00013548671280111892,0.0001366776091554688,0.0,0.0,0.0,0.0,
        0.0,0.0,0.0,0.0,0.0,-0.0,-0.0,-0.0,-0.0,-0.0,-0.0,-0.0,-0.00028983042660450767,0.60771760732198055,
        0.45258306322192471,0.41467880541713448,-0.60771760732198055,0.00034998845489279349,-0.45258306322192471,
        0.00034322043275703966,-0.41467880541713448,0.0,0.0,0.0,0.0,0.0,0.0,0.0,0.0,1.0,-0.0,-0.0,-0.0,-0.0,-0.0,
        -0.0,-0.0,-0.0,0.60774185316849594,0.0,4.9507562444117341E-20,9.0792333081773271E-20,0.0,
        -4.9507562444117341E-20,1.6818696161191519E-16,-9.0792333081773247E-20,1.2581077755555868E-16,0.0,0.0,0.0,
        0.0,0.0,0.0,0.0,0.0,0.0,-0.0,-0.0,-0.0,-0.0,-0.0,-0.0,-0.0,-1.0,-0.00032104499842707462,
        -0.00030990522922148069,0.60771586837025782,0.45258145885114326,0.414677276341478,0.00020644223064780165,
        -0.60771586837025782,-0.414677276341478,0.0,0.0,0.0,0.0,0.0,0.0,0.0,1.0,-0.0,-0.0,-0.0,-0.0,-0.0,-0.0,-0.0,
        -0.0,0.45260561554757484,-6.705637981480354E-5,-7.4542022764774E-5,0.54849096138382369,
        -7.3882932570663252E-5,6.70627819526479E-5,-0.83950908011157221,7.3882932570663252E-5,7.45493134229047E-5,
        0.0,0.0,0.0,0.0,0.0,0.0,0.0,0.0,-0.0,-0.0,-0.0,-0.0,-0.0,-0.0,-0.0,-0.0,-0.00032423089662980361,
        0.607721627098605,0.45258682574740111,0.41468237096544258,0.00024604276486503597,-0.607721627098605,
        0.00030990522922148096,-0.45258682574740111,-0.41468237096544258,0.0,0.0,0.0,0.0,0.0,0.0,0.0,1.0,-0.0,-0.0,
        -0.0,-0.0,-0.0,-0.0,-0.0,-0.0,0.41470020324647261,-0.00012282470380310523,-0.00013548671280111892,
        -0.0001366776091554688,0.00012282470380310523,-0.75586897491059513,0.00013548671280111892,
        -0.54849096138382369,0.0001366776091554688,0.0,0.0,0.0,0.0,0.0,0.0,0.0,0.0,-0.0,-0.0,-0.0,-0.0,-0.0,-0.0,
        -0.0,-0.0,2.9755061164947574E-20,-0.60771760732198044,0.0,1.6817672556185198E-16,1.2334487941221325E-19,
        1.2580321328053461E-16,0.0,0.0,0.0,0.0,0.0,0.0,0.0,1.0,-0.0,-0.0,-0.0,-0.0,-0.0,-0.0,-0.0,-0.0,
        0.00034998845489279343,0.00020644223064780157,0.00036358068816811083,0.60771221968588129,
        0.45257806398899236,0.41467405969907745,-0.60771221968588129,-0.45257806398899236,-0.41467405969907745,0.0,
        0.0,0.0,0.0,0.0,0.0,0.0,0.0,0.0,1.0,-0.0,-0.0,-0.0,-0.0,-0.0,-0.0,-0.0,6.7056379814803486E-5,
        0.83951256820538323,-0.00051559608946867748,-0.0,4.8503929239195573E-5,-0.45257806398899236,
        -0.000515601666520195,0.0,0.0,0.0,0.0,0.0,0.0,0.0,0.0,-0.0,-0.0,-0.0,-0.0,-0.0,-0.0,0.00024604276486503592,
        0.00034322043275703961,0.60771348124036872,-0.00036358068816811078,-0.41467517776491791,0.0,0.0,0.0,0.0,0.0,
        0.0,0.0,1.0,-0.0,-0.0,-0.0,-0.0,-0.0,-0.0,-0.0,0.00012282470380310523,0.54846656219268941,-0.0,
        8.8527830239323147E-5,-0.4146740596990775,0.0,0.0,0.0,0.0,0.0,0.0,0.0,0.0,0.0,-0.0,-0.0,-0.0,-0.0,-0.0,-0.0,
        2.9755061164947574E-20,0.60771760732198044,-0.0,2.0638347693417836E-20,4.8839816704642384E-19,
        2.5160334196432531E-16,0.0,0.0,0.0,0.0,0.0,0.0,0.0,0.0,-0.0,-0.0,-0.0,-0.0,-0.0,-0.0,-1.0,
        6.7056379814803486E-5,0.45258306322192476,-7.9634662796535162E-5,-0.83951256820538323,
        0.00051559608946867759,0.0,0.0,0.0,0.0,0.0,0.0,-0.0,-0.0,-0.0,-0.0,-0.0,-0.0,-0.0,0.00012282470380310523,
        0.41467880541713448,-0.00014643395598641436,-0.00014348094203993502,-0.75584811392108253,
        -0.54846656219268941,0.0,0.0,0.0,0.0,0.0,0.0,0.0,-0.0,-0.0,-0.0,-0.0,-0.0,-0.0,-0.0,-0.0,
        -0.60771627901050718,-4.9506989144368247E-20,-0.83949211543668667,-1.8239303391070821E-19,
        4.8855338534453015E-19,0.0,0.0,0.0,0.0,0.0,0.0,0.0,1.0,-0.0,-0.0,-0.0,-0.0,-0.0,-0.0,-0.83952864747628941,
        3.3637392322383048E-16,0.0,4.9506989144368241E-20,9.0791286551000237E-20,0.0,0.0,-4.9506989144368241E-20,
        -9.0791286551000237E-20,0.0,0.0,0.0,0.0,0.0,0.0,0.0,1.0,-0.0,-0.0,-0.0,-0.0,-0.0,-0.0,-0.607721627098605,
        -1.3618849962265987E-19,-1.2330609381155307E-19,-1.7930100380701504E-19,-1.681784660206933E-16,0.0,0.0,0.0,
        0.0,0.0,0.0,0.0,1.0,-0.0,-0.0,-0.0,-0.0,-0.0,-0.0,-0.0,-0.75586897491059513,1.2581077755555871E-16,
        4.53957044533439E-20,3.3154606304565777E-20,0.0,-4.5395704453343891E-20,0.0,0.0,0.0,0.0,0.0,0.0,0.0,0.0,0.0,
        1.0,-0.0,-0.0,-0.0,-0.0,-0.0,-0.0,-0.0,-0.60771760732198032,3.315489520239038E-20,-1.681767255618521E-16,
        -1.64929553273929E-19,-2.466897588244265E-19,0.0,0.0,0.0,0.0,0.0,0.0,0.0,1.0,-0.0,-0.0,-0.0,-0.0,-0.0,-0.0,
        -0.0,-0.0,-0.60771627901050718,9.9015124888234682E-20,-1.6817618571481423E-16,1.8239417817919302E-19,0.0,
        0.0,0.0,0.0,0.0,0.0,0.0,1.0,-0.0,-0.0,-0.0,-0.0,-0.0,-0.0,-0.0,-0.607721627098605,1.3618849962265987E-19,
        -1.681784660206933E-16,-1.2580449590377112E-16,1.2330609381155307E-19,1.7930100380701509E-19,0.0,0.0,0.0,
        0.0,0.0,0.0,1.0,-0.0,-0.0,-0.0,-0.0,-0.0,-0.0,-0.0,-0.0,7.38757514247254E-5,-0.45258183585658091,
        7.14882463612096E-5,-0.54846526788387562,-4.8508322153241939E-5,0.83949183414948236,0.0,0.0,0.0,0.0,0.0,0.0,
        0.0,0.0,-0.0,-0.0,-0.0,-0.0,-0.0,-0.0,0.00013548671280111887,-0.41467763318781908,0.00013118967602768769,
        -8.85278302393231E-5,0.54846485840188586,0.0,0.0,0.0,0.0,0.0,0.0,0.0,0.0,-0.0,-0.0,-0.0,-0.0,-0.0,-0.0,
        -6.370397382786412E-20,2.5160561935436607E-16,1.7976260569382681E-19,0.60771586837025771,0.0,
        1.6817602023351553E-16,0.0,0.0,0.0,0.0,0.0,0.0,0.0,0.0,-0.0,-0.0,-0.0,-0.0,-0.0,-0.0,-1.0,
        7.1488246361209635E-5,0.45258145885114326,-4.8503929239195519E-5,-0.839511404940604,0.00051560018494341568,
        0.0,0.0,0.0,0.0,0.0,-0.0,-0.0,-0.0,-0.0,-0.0,-0.452586825747401,7.4542022764773945E-5,-0.54847065730144762,
        0.83949563162130481,-7.1495079606071117E-5,0.0,0.0,0.0,0.0,0.0,0.0,0.0,0.0,-0.0,-0.0,-0.0,-0.0,-0.0,-0.0,
        -0.45258306322192471,7.8123623135183722E-5,-0.54846656219268941,-6.7062781952647926E-5,0.83949299775843811,
        7.9642715680471464E-5,0.0,0.0,0.0,0.0,0.0,0.0,0.0,0.0,-0.0,-0.0,-0.0,-0.0,-0.0,-0.0,-0.0,
        -0.45258183585658085,-0.54846526788387551,-7.3882932570663293E-5,0.83949211543668689,4.8506315421467726E-5,
        7.3636376402749123E-5,0.0,0.0,0.0,0.0,0.0,-0.0,-0.0,-0.0,-0.0,-0.0,-0.452586825747401,5.7353204127738534E-5,
        7.1488246361209526E-5,-0.54847065730144762,-7.4549313422904716E-5,0.83949563162130481,0.0,0.0,0.0,0.0,0.0,
        0.0,0.0,-0.0,-0.0,-0.0,-0.0,-0.0,-0.0,-0.0,0.0001366776091554688,-0.41468237096544247,
        -0.00013118967602768778,0.54847065730144773,0.0,0.0,0.0,0.0,0.0,0.0,0.0,0.0,-0.0,-0.0,-0.0,-0.0,-0.0,-0.0,
        -7.9990129001169258E-20,0.607721627098605,0.0,1.6817846602069321E-16,1.2580449590377107E-16,0.0,0.0,0.0,0.0,
        0.0,0.0,0.0,0.0,-0.0,-0.0,-0.0,-0.0,-0.0,-0.0,-1.0,7.4542022764773972E-5,0.45258682574740106,
        -7.1488246361209486E-5,-0.83951520168604254,0.000515596671407826,0.0,0.0,0.0,0.0,0.0,-0.0,-0.0,-0.0,-0.0,
        -0.0,0.0001366776091554688,0.41468237096544247,-0.00010492369622770082,-0.00013118967602768778,
        -0.75585156501645778,-0.54847065730144773,0.0,0.0,0.0,0.0,0.0,0.0,0.0,-0.0,-0.0,-0.0,-0.0,-0.0,-0.0,-0.0,
        -0.41467880541713448,-0.00012282470380310526,0.54846656219268952,0.00014643395598641431,
        0.0001434809420399348,0.0,0.0,0.0,0.0,0.0,0.0,0.0,0.0,-0.0,-0.0,-0.0,-0.0,-0.0,-0.0,-0.0,-0.414677633187819,
        -0.00013548671280111889,0.54846526788387573,8.8524154773604152E-5,0.00013469943293139259,0.0,0.0,0.0,0.0,
        0.0,-0.0,-0.0,-0.0,-0.0,-0.0,-0.41468237096544253,-0.00013667760915546878,0.54847065730144762,
        0.0001049236962277008,0.00013118967602768775,0.0,0.0,0.0,0.0,0.0,0.0,0.0,-0.0,-0.0,-0.0,-0.0,-0.0,-0.0,-0.0,
        -2.9755061164947574E-20,0.60771760732198044,0.0,-1.6817672556185198E-16,-1.233448794122132E-19,
        -1.2580321328053463E-16,0.0,0.0,0.0,0.0,0.0,0.0,0.0,0.0,-0.0,-0.0,-0.0,-0.0,-0.0,-0.0,-0.0,-1.0,
        -0.00020643328051976208,-0.00034998845489279343,0.60771263100274964,0.00032311337431655543,
        -0.41467441716242903,0.0,0.0,0.0,0.0,0.0,0.0,1.0,-0.0,-0.0,-0.0,-0.0,-0.0,-0.0,-0.0,-0.0,
        -6.7056379814803486E-5,0.45258306322192476,-0.83951256820538323,7.9634662796535162E-5,7.8123623135183722E-5,
        0.00051559608946867759,0.0,0.0,0.0,0.0,0.0,-0.0,-0.0,-0.0,-0.0,-0.0,-0.0,-0.00024604276486503592,
        -0.00034322043275703955,-0.0002064422306478016,-0.00032311337431655576,0.60771221968588129,
        0.45257806398899236,0.41467405969907745,-0.60771221968588129,-0.41467405969907745,0.0,0.0,0.0,0.0,0.0,0.0,
        0.0,1.0,-0.0,-0.0,-0.0,-0.0,-0.0,-0.0,-0.0,-0.0,-0.0,-0.00012282470380310523,0.41467880541713448,
        -0.75584811392108253,0.00014643395598641436,-0.54846656219268941,0.00014348094203993497,0.0,0.0,0.0,0.0,0.0,
        0.0,0.0,-0.0,-0.0,-0.0,-0.0,-0.0,-0.0,-0.0,-0.0,0.60771627901050718,9.9015124888234682E-20,
        1.8239417817919302E-19,1.6817618571481423E-16,0.0,1.2580280967718299E-16,0.0,0.0,0.0,0.0,0.0,-0.0,-0.0,-0.0,
        -0.0,-0.0,-1.0,0.83952864747628941,-3.3637392322383053E-16,0.0,4.9506989144368241E-20,
        9.0791286551000237E-20,0.0,-4.9506989144368241E-20,-9.0791286551000237E-20,0.0,0.0,0.0,0.0,0.0,0.0,0.0,-0.0,
        -0.0,-0.0,-0.0,-0.0,-0.0,-0.0,-1.0,0.607721627098605,1.3618849962265987E-19,1.2330609381155307E-19,
        1.7930100380701509E-19,1.681784660206933E-16,1.2580449590377112E-16,0.0,0.0,0.0,0.0,0.0,0.0,0.0,-0.0,-0.0,
        -0.0,-0.0,-0.0,-0.0,-0.0,-1.0,0.75586897491059513,-1.2581077755555871E-16,4.53957044533439E-20,
        3.3154606304565777E-20,0.0,0.0,0.0,0.0,0.0,0.0,0.0,0.0,-0.0,-0.0,-0.0,-0.0,-0.0,-0.0,-1.0,
        -7.38757514247254E-5,0.45258183585658091,4.850192273613149E-5,-0.83951168616294036,7.3628717755583559E-5,
        0.00051559955622434669,0.0,0.0,0.0,0.0,-0.0,-0.0,-0.0,-0.0,-0.00013548671280111887,-0.00013118967602768775,
        0.414677276341478,8.852783023932312E-5,-0.75584662495331045,-0.54846485840188586,0.0,0.0,0.0,0.0,0.0,0.0,
        -0.0,-0.0,-0.0,-0.0,-0.0,-0.0,-0.0,-0.0,0.452586825747401,-7.4542022764773945E-5,5.7353204127738534E-5,
        -0.83951520168604254,7.1488246361209567E-5,0.00051559667140782691,0.0,0.0,0.0,0.0,0.0,0.0,-0.0,-0.0,-0.0,
        -0.0,-0.0,-0.0,-0.0,-0.0001366776091554688,0.41468237096544247,0.00010492369622770083,-0.75585156501645778,
        0.00013118967602768764,-0.54847065730144773,0.0,0.0,0.0,0.0,0.0,0.0,-0.0,-0.0,-0.0,-0.0,-0.0,-0.0,-0.0,-0.0,
        -8.246374572135012E-20,9.8108818261083368E-20,-0.83950898205466618,-8.9882277746204806E-26,
        4.985436410395924E-16,0.0,0.0,0.0,0.0,0.0,0.0,0.0,0.0,1.0,-0.0,-0.0,-0.0,-0.0,-0.0,-0.0,
        2.9754765431896156E-20,-0.83951256820538334,0.0,0.0,4.9854995011635195E-16,0.0,0.0,0.0,0.0,0.0,0.0,-0.0,
        -0.0,-0.0,-0.0,-0.0,-0.0,8.8392842585362538E-20,-1.8501731911831992E-19,9.8109375285541218E-20,
        -0.60771221968588129,1.6817447504922767E-16,0.0,0.0,0.0,0.0,0.0,0.0,0.0,0.0,1.0,-0.0,-0.0,-0.0,-0.0,-0.0,
        -0.0,-0.0,6.7062781952647967E-5,0.839492997758438,-0.0,0.00051560103798285685,4.8508322153242075E-5,
        -0.0049959693296679321,1.1481092117693212E-6,0.0,0.0,0.0,0.0,0.0,0.0,0.0,0.0,0.0,-0.0,-0.0,-0.0,-0.0,-0.0,
        -0.0,0.00010492369622770083,0.0001434809420399351,8.8527830239323147E-5,0.00013470903175427876,
        0.4146740596990775,-0.75584347736259117,-0.54846116837011871,0.0,0.0,0.0,0.0,0.0,0.0,0.0,0.0,-0.0,-0.0,-0.0,
        -0.0,-0.0,-0.0,-0.0,2.9754765431896156E-20,0.83951256820538334,0.0,0.0,-4.9854995011635195E-16,0.0,0.0,0.0,
        0.0,0.0,0.0,-0.0,-0.0,-0.0,-0.0,-0.0,-0.0,-0.0,-1.0,6.7062781952647967E-5,0.54846656219268952,
        -7.9642715680471464E-5,-7.8131577710013753E-5,-0.839492997758438,0.0,0.0,0.0,0.0,0.0,0.0,0.0,-0.0,-0.0,-0.0,
        -0.0,-0.0,-0.0,-0.0,-0.0,-0.60771586837025771,5.9508718159756055E-20,-4.8884752457005644E-19,
        -9.1195009050586689E-20,-1.6817602023351548E-16,0.0,0.0,0.0,0.0,0.0,0.0,0.0,1.0,-0.0,-0.0,-0.0,-0.0,-0.0,
        -0.0,-0.0,-4.625701589801718E-23,-9.0791286551000225E-20,-0.83949563162130469,0.0,0.0,0.0,0.0,0.0,0.0,0.0,
        0.0,0.0,1.0,-0.0,-0.0,-0.0,-0.0,-0.0,-0.0,-0.8395090801115721,1.1104954790887438E-18,
        -3.3154532651703232E-20,4.950692740610004E-20,9.0791173929120774E-20,3.3154532651703232E-20,
        -4.950692740610004E-20,-9.0791173929120762E-20,0.0,0.0,0.0,0.0,0.0,0.0,0.0,0.0,0.0,1.0,-0.0,-0.0,-0.0,-0.0,
        -0.0,-0.0,-0.0,0.0,-2.4668692135355611E-19,-0.83949299775843789,-6.2635751390691967E-21,
        -1.64927269518349E-19,0.0,0.0,0.0,0.0,0.0,0.0,0.0,0.0,1.0,-0.0,-0.0,-0.0,-0.0,-0.0,-0.0,-0.0,
        -3.1490119814551088E-23,-0.83949211543668667,4.2469420815797451E-20,1.8239303391070821E-19,
        -4.8855338534452948E-19,0.0,0.0,0.0,0.0,0.0,1.0,-0.0,-0.0,-0.0,-0.0,-0.0,-0.83951520168604232,
        -4.625701589801718E-23,9.0791286551000225E-20,-4.9855482999028193E-16,6.1652571145841663E-20,0.0,0.0,0.0,
        0.0,0.0,0.0,0.0,1.0,-0.0,-0.0,-0.0,-0.0,-0.0,-0.0,-0.83949563162130458,1.1104953763821025E-18,
        6.683190108752474E-22,1.2330504017361608E-19,0.0,0.0,0.0,0.0,0.0,0.0,0.0,0.0,1.0,-0.0,-0.0,-0.0,-0.0,-0.0,
        -0.0,-0.0,-0.60771263100274964,-9.1103604592422571E-20,1.6492955327392894E-19,-4.8839816704642317E-19,0.0,
        0.0,0.0,0.0,0.0,0.0,1.0,-0.0,-0.0,-0.0,-0.0,-0.0,-0.0,-0.0,-0.0,-0.60771348124036884,-0.83950981017513349,
        -8.20210993821808E-20,2.46686921353556E-19,-4.9854515452033152E-16,0.0,0.0,0.0,0.0,0.0,0.0,1.0,-0.0,-0.0,
        -0.0,-0.0,-0.0,-0.0,-0.0,-0.60771586837025771,-5.9508718159756067E-20,-1.6817602023351548E-16,
        -1.2580268781145876E-16,9.1195009050586689E-20,0.0,0.0,0.0,0.0,0.0,0.0,1.0,-0.0,-0.0,-0.0,-0.0,-0.0,-0.0,
        -0.0,-0.0,0.00013118967602768769,0.00013469943293139243,0.414677276341478,-8.85278302393231E-5,
        -0.75584662495331045,-0.54846485840188586,0.0,0.0,0.0,0.0,0.0,0.0,0.0,-0.0,-0.0,-0.0,-0.0,-0.0,-0.0,-0.0,
        1.8151062270724029E-19,0.83951140494060406,-1.6817602023351545E-16,0.0,0.0,0.0,0.0,0.0,0.0,0.0,-0.0,-0.0,
        -0.0,-0.0,-0.0,-1.0,7.3882932570663347E-5,7.1495079606071347E-5,0.54846485840188541,-4.8508322153242115E-5,
        -0.83949183414948259,0.0,0.0,0.0,0.0,0.0,0.0,0.0,-0.0,-0.0,-0.0,-0.0,-0.0,-0.0,-0.0,-0.45257924052569581,
        -5.73532041277385E-5,-7.8123623135183614E-5,0.83950981017513371,-0.00051560065177808285,
        8.2669047804172151E-5,0.0,0.0,0.0,0.0,0.0,-0.0,-0.0,-0.0,-0.0,-0.0,-0.0,-0.0,-0.45258145885114337,
        -0.54846485840188586,-7.1495079606071212E-5,0.83949183414948259,4.8508322153242129E-5,0.0,0.0,0.0,0.0,0.0,
        0.0,0.0,-0.0,-0.0,-0.0,-0.0,-0.0,-0.0,-0.0,-8.7176738319430579E-20,0.83951520168604243,
        -1.6817846602069328E-16,0.0,0.0,0.0,0.0,0.0,0.0,0.0,-0.0,-0.0,-0.0,-0.0,-0.0,-1.0,0.75585156501645778,
        -1.2580449590377104E-16,-1.7929917369533893E-19,-6.96516636356949E-22,0.83949563162130481,
        -6.1652520086808E-20,0.0,0.0,0.0,0.0,0.0,0.0,0.0,-0.0,-0.0,-0.0,-0.0,-0.0,-0.0,-0.0,-1.0,
        7.454931342290477E-5,0.54847065730144728,-5.7358524655122212E-5,-7.1495079606071239E-5,-0.83949563162130492,
        0.0,0.0,0.0,0.0,0.0,0.0,0.0,-0.0,-0.0,-0.0,-0.0,-0.0,-0.0,-0.0,-0.41467517776491786,-0.00010492369622770092,
        -0.00014348094203993486,0.54846243479694534,0.00015236510263377253,0.0,0.0,0.0,0.0,0.0,0.0,0.0,-0.0,-0.0,
        -0.0,-0.0,-0.0,-0.0,-0.0,-0.41467727634147794,-0.0001311896760276878,0.548464858401886,8.85278302393231E-5,
        0.0,0.0,0.0,0.0,0.0,0.0,0.0,-0.0,-0.0,-0.0,-0.0,-0.0,-0.0,-0.0,-8.839284258536255E-20,0.60771348124036884,
        1.8501731911831983E-19,-9.8109375285541218E-20,-1.6817447504922767E-16,-1.2580154888538883E-16,0.0,0.0,0.0,
        0.0,0.0,0.0,0.0,-0.0,-0.0,-0.0,-0.0,-0.0,-0.0,-0.0,-0.0,-1.0,-2.975480007865129E-20,0.75584811392108275,0.0,
        0.0,-5.0668078577586268E-16,-1.2334362658056649E-19,0.0,0.0,0.0,0.0,0.0,0.0,-0.0,-0.0,-0.0,-0.0,-0.0,-0.0,
        -0.0,-1.0,-0.00014643395598641445,-8.8527830239323147E-5,-0.00015236510263377253,0.4146740596990775,
        -0.54846116837011871,0.0,0.0,0.0,0.0,0.0,0.0,-0.0,-0.0,-0.0,-0.0,-0.0,-0.0,-0.0,-0.0,-0.0,
        -5.7353204127738527E-5,0.45257924052569587,-7.8123623135183655E-5,-0.8395098101751336,8.2669047804172151E-5,
        0.00051560065177708408,0.0,0.0,0.0,0.0,-0.0,-0.0,-0.0,-0.0,-0.0,-0.0,-6.7062781952647967E-5,
        0.54846656219268952,-0.839492997758438,7.9642715680471464E-5,7.81315777100136E-5,0.0,0.0,0.0,0.0,0.0,0.0,
        0.0,-0.0,-0.0,-0.0,-0.0,-0.0,-0.0,-0.0,-0.0,-0.00010492369622770084,-0.00014348094203993505,
        0.41467517776491797,-0.75584455578182586,0.0001523651026337728,-0.54846243479694468,0.0,0.0,0.0,0.0,0.0,
        -0.0,-0.0,-0.0,-0.0,-0.0,-0.0,-0.0,0.60771586837025771,-5.9508718159756067E-20,9.1195009050586689E-20,
        1.6817602023351548E-16,1.2580268781145876E-16,0.0,0.0,0.0,0.0,0.0,0.0,0.0,-0.0,-0.0,-0.0,-0.0,-0.0,-0.0,
        -0.0,-1.0,0.75584698353565438,3.6297211588305579E-20,-1.258027775726083E-16,1.8239326798807447E-19,0.0,0.0,
        0.0,0.0,0.0,0.0,-0.0,-0.0,-0.0,-0.0,-0.0,-1.0,0.8395090801115721,1.1099594411114691E-18,
        -3.3154532651703232E-20,4.950692740610004E-20,9.0791173929120774E-20,3.3154532651703232E-20,
        -4.950692740610004E-20,-9.0791173929120762E-20,0.0,0.0,0.0,0.0,0.0,0.0,0.0,0.0,-0.0,-0.0,-0.0,-0.0,-0.0,
        -0.0,-0.0,-0.0,-1.0,-7.1488246361209608E-5,0.4525814588511432,4.8503929239195519E-5,-0.83951140494060417,
        0.00051560018494391658,0.0,0.0,0.0,0.0,0.0,0.0,-0.0,-0.0,-0.0,-0.0,-0.0,-0.0,-0.0,-7.3882932570663347E-5,
        0.54846526788387562,4.8506315421467529E-5,-0.83949211543668678,7.36363764027489E-5,0.0,0.0,0.0,0.0,0.0,0.0,
        -0.0,-0.0,-0.0,-0.0,-0.0,-0.0,-0.0,0.54847065730144762,-7.454931342290473E-5,5.7358524655122233E-5,
        -0.83949563162130481,7.1495079606071144E-5,0.0,0.0,0.0,0.0,0.0,0.0,-0.0,-0.0,-0.0,-0.0,-0.0,-0.0,-0.0,-0.0,
        2.9754733575446928E-20,-0.839492997758438,-4.9854995011635155E-16,0.0,0.0,0.0,0.0,0.0,0.0,0.0,0.0,0.0,1.0,
        -0.0,-0.0,-0.0,-0.0,-0.0,-0.0,-0.0,5.6433356177770327E-20,-7.00966397529624E-22,0.60771221968588141,
        1.6817447504922767E-16,1.2580154888538883E-16,0.0,0.0,0.0,0.0,0.0,0.0,0.0,0.0,0.0,-0.0,-0.0,-0.0,-0.0,-0.0,
        -0.0,-1.0,4.8503929239195573E-5,7.3634033153687213E-5,0.45257806398899231,-0.83950898205466606,
        0.000515601666520195,0.0,0.0,0.0,0.0,0.0,0.0,-0.0,-0.0,-0.0,-0.0,-0.0,-1.6262870258933998E-19,
        -1.6817464083486873E-16,4.9240506899104478E-20,0.8395089820546664,-1.1115503907899016E-18,0.0,0.0,0.0,0.0,
        0.0,0.0,-0.0,-0.0,-0.0,-0.0,-0.0,-1.0,5.7358524655122206E-5,7.8131577710013631E-5,0.54846243479694479,
        4.8508322153242088E-5,0.004995969329667933,-0.83948941084011008,0.0,0.0,0.0,0.0,0.0,0.0,0.0,0.0,-0.0,-0.0,
        -0.0,-0.0,-0.0,-0.0,-0.0,2.9754733575446928E-20,0.839492997758438,-2.5322003579499064E-16,0.0,
        1.2334330862335358E-19,0.0,0.0,0.0,0.0,0.0,0.0,0.0,-0.0,-0.0,-0.0,-0.0,-0.0,-0.0,-0.0,-0.0,-1.0,
        4.850631542146761E-5,7.9642715680471531E-5,0.54846157851902466,-7.3641691938526E-5,-0.839489692551959,0.0,
        0.0,0.0,0.0,0.0,0.0,0.0,-0.0,-0.0,-0.0,-0.0,-0.0,-0.0,5.9508025155671187E-20,-3.7944716262115873E-23,
        -4.88843264703953E-19,-0.83949183414948236,-1.0685174091063236E-21,-1.8238887367955244E-19,0.0,0.0,0.0,0.0,
        0.0,0.0,0.0,0.0,1.0,-0.0,-0.0,-0.0,-0.0,-0.0,-0.0,-0.83951140494060383,-3.7944716262115873E-23,
        -5.9508025155671235E-20,-4.9854794748204026E-16,9.119449206614489E-20,0.0,0.0,0.0,0.0,0.0,0.0,1.0,-0.0,-0.0,
        -0.0,-0.0,-0.0,-0.0,1.1104954242848737E-18,0.0,-0.0,-0.83950898205466606,-9.1080341125208536E-20,
        1.0218805379139446E-24,0.0,0.0,0.0,0.0,0.0,0.0,1.0,-0.0,-0.0,-0.0,-0.0,-0.0,-0.0,-0.0,-0.83949183414948236,
        1.110495398303592E-18,-6.0094685994419228E-22,1.8238887367955241E-19,0.0,0.0,0.0,0.0,0.0,0.0,0.0,1.0,-0.0,
        -0.0,-0.0,-0.0,-0.0,-0.0,-0.0,-0.60771221968588141,-9.1080860224906571E-20,1.0218648896758904E-24,
        -1.6817447504922772E-16,-1.2580154888538883E-16,0.0,0.0,0.0,0.0,0.0,0.0,1.0,-0.0,-0.0,-0.0,-0.0,-0.0,-0.0,
        -0.0,-0.0,-0.0,0.75584662495331045,-3.7740806343437641E-16,-9.1194553892523224E-20,1.6475704522131309E-21,
        0.83949183414948247,0.0,0.0,0.0,0.0,0.0,0.0,0.0,-0.0,-0.0,-0.0,-0.0,-0.0,-0.0,-0.0,-1.0,
        0.00051560065177795838,-5.7358524655122192E-5,-7.81315777100136E-5,0.83949023913090359,
        -0.0049959693296679373,1.1481092117723822E-6,-4.8508322153242E-5,0.0,0.0,0.0,0.0,0.0,0.0,0.0,-0.0,-0.0,-0.0,
        -0.0,-0.0,-0.0,-0.0,-0.0,-0.45257806398899231,-4.8503929239195492E-5,-8.2669047804172476E-5,
        0.83950898205466629,-0.00051560166652169328,0.0,0.0,0.0,0.0,0.0,0.0,-0.0,-0.0,-0.0,-0.0,-0.0,-0.0,-0.0,-0.0,
        -0.41467405969907745,-8.852783023932331E-5,-0.00015236510263377218,0.54846116837011893,0.0,0.0,0.0,0.0,0.0,
        0.0,0.0,-0.0,-0.0,-0.0,-0.0,-0.0,-0.0,-0.0,-0.0,-3.6975241712266472E-20,0.755844555781826,
        1.3769388015871068E-19,1.2580195959048207E-16,0.0,0.0,0.0,0.0,0.0,0.0,-0.0,-0.0,-0.0,-0.0,-0.0,-0.0,-0.0,
        -1.0,-2.9754733575446928E-20,0.839492997758438,-2.5322003579499064E-16,0.0,-1.2334330862335355E-19,0.0,0.0,
        0.0,0.0,0.0,0.0,0.0,-0.0,-0.0,-0.0,-0.0,-0.0,-0.0,-0.0,-0.0,-1.0,0.45257806398899236,-0.0,
        -4.850631542146761E-5,-7.9642715680471531E-5,0.54846157851902466,-0.839489692551959,0.0,0.0,0.0,0.0,0.0,0.0,
        -0.0,-0.0,-0.0,-0.0,-0.0,-0.0,-0.0,-0.0,-5.7358524655122206E-5,0.548462434796945,-7.8131577710013631E-5,
        -0.83949023913090348,8.2677296121898793E-5,0.0,0.0,0.0,0.0,0.0,-0.0,-0.0,-0.0,-0.0,-0.0,-0.0,-0.0,
        4.2469420815797463E-20,0.83949183414948236,-6.0094685994419191E-22,-1.110495398303592E-18,
        1.8238887367955244E-19,0.0,0.0,0.0,0.0,0.0,0.0,-0.0,-0.0,-0.0,-0.0,-0.0,-0.0,-0.0,-0.0,-1.0,
        0.83949563162130469,1.1099596201273517E-18,6.683190108752475E-22,1.2330504017361606E-19,0.0,0.0,0.0,0.0,0.0,
        0.0,0.0,-0.0,-0.0,-0.0,-0.0,-0.0,-0.0,-0.0,-0.0,-1.0,-7.149507960607132E-5,0.54846485840188608,
        -7.3636376402749177E-5,-0.00051560018494413527,4.8508322153241933E-5,-0.83949183414948236,0.0,0.0,0.0,0.0,
        0.0,0.0,-0.0,-0.0,-0.0,-0.0,-0.0,-0.0,-0.0,-0.0,9.811099909019153E-20,-0.83948969255195927,
        -5.9470437978074124E-22,-1.1104954909955548E-18,4.8839345513964346E-19,0.0,0.0,0.0,0.0,0.0,0.0,0.0,0.0,1.0,
        -0.0,-0.0,-0.0,-0.0,-0.0,-0.0,8.5051560381848912E-20,-5.5577944565858811E-19,0.0,0.0,0.0,0.0,0.0,0.0,0.0,
        0.0,0.0,1.0,-0.0,-0.0,-0.0,-0.0,-0.0,-0.0,-1.0,7.7873197452969825E-20,2.803986063763796E-19,
        6.4296063569359765E-22,0.83948941084011031,3.330933417383221E-18,0.0,0.0,0.0,0.0,0.0,0.0,0.0,0.0,-0.0,-0.0,
        -0.0,-0.0,-0.0,-0.0,-0.0,-1.0,3.3215168474146733E-20,-1.0697498708079556E-21,0.83949023913090381,0.0,0.0,
        0.0,0.0,0.0,0.0,0.0,0.0,-0.0,-0.0,-0.0,-0.0,-0.0,-0.0,-0.0,-1.0,-8.8392085258418591E-20,0.83949023913090348,
        -1.109959330793548E-18,5.7702323571187137E-22,0.0,0.0,0.0,0.0,0.0,0.0,-0.0,-0.0,-0.0,-0.0,-0.0,-0.0,-0.0,
        -1.0,-9.811099909019153E-20,5.9470437978074124E-22,0.83948941084011031,1.1104955074523147E-18,0.0,0.0,0.0,
        0.0,0.0,0.0,-0.0,-0.0,-0.0,-0.0,-0.0,-0.0,-0.0,-0.0,-0.0,-1.0,4.1039746089312351E-20,-0.83948941084011031,
        -1.1010645961606569E-21,-1.1104955074523147E-18,0.0,0.0,0.0,0.0,0.0,0.0,0.0,0.0,0.0,1.0,-0.0,-0.0,-0.0,-0.0,
        -0.0,-0.0;
    Explicit_b_G: ARRAY [0..249] OF LREAL := 0.0,0.0,140.328,-0.066712260924210731,-0.06481259658265906,136.328,
        70.09208224196523,-0.049529802998884785,-0.04991060377936854,68.093414975642048,46.672260105606064,
        -0.036349978139805554,-0.037442373571299752,45.340877278654531,-10.0,0.0047540234966799736,
        0.0066558326400829385,-14.0,-4.9948750243689952,0.0035295737841973653,0.005125494783985384,
        -6.9927513765256482,-3.3259406608521505,0.0025903581708429926,0.0038450885364576352,-4.6562135577516246,
        140.32799999999997,136.32800000000003,140.328,-0.0667725858975615,140.328,68.077973963187517,
        140.32799999999997,-0.066766750479010858,140.328,45.312597285515771,140.328,-13.999999999999998,
        140.32799999999997,-7.0081863352279727,140.32799999999997,-4.684485232538492,70.07529315333116,136.328,
        -0.064878459045791162,136.32800000000003,46.642663706148113,136.32800000000003,-0.064874276850442433,
        136.32800000000003,-9.9999999999999982,136.32800000000003,-5.0116575809989987,136.32800000000006,
        -3.355528608733493,136.328,70.0792111192775,68.082011032644715,70.08246539490186,45.319965612648112,
        70.09379964864479,-14.000000000000004,70.093396079164137,-7.0041486765756957,46.64951683334678,
        68.085052658968351,-10.0,68.09450944594461,-5.0077384299939975,68.094221185452341,-3.34867392142978,
        68.094005674607914,46.655237788220333,45.3255467924812,46.675290764014974,-14.0,46.674585386490143,
        -7.0011083270071328,46.6739994865459,-4.6715366480995613,-10.000000000000004,45.342884475415772,
        -5.0044853711592667,45.342358586139262,-3.3429545257648674,45.341962568857838,-9.9999999999999964,
        -13.999999999999998,-9.9999999999999964,0.0047583223517445906,-9.9999999999999982,-6.9916508524709053,
        -9.9999999999999982,0.0047579065103907177,-10.0,-4.6541980426384946,-4.9931510856853736,-14.000000000000004,
        0.0066625962871976127,-14.0,-3.3229015508666389,-14.0,0.0066621668029032488,-14.000000000000004,
        -4.9935534701073809,-6.991938523768094,-4.9938876273720858,-4.65472309775716,-3.3236053682864015,
        -6.9921553113675454,-3.3241928274392922,-4.6551208717229278,140.32799999999997,136.328,140.32799999999997,
        136.32800000000003,140.32799999999997,136.32800000000003,140.32799999999995,68.077963122328043,
        140.32799999999997,-4.68450785771074,140.32799999999997,-13.999999999999998,140.328,-7.0081868651731956,
        70.075282628673619,136.32800000000003,46.642631530347757,136.32800000000003,-0.06488741702733633,136.328,
        -10.000000000000004,136.32800000000006,-5.011674285092937,136.32800000000006,-3.3555583211233451,136.328,
        -3.3555622946665142,136.32800000000006,-9.9999999999999964,136.32800000000003,-10.0,136.328,
        -5.0116580206210077,136.32800000000003,70.093053791180637,-4.6771185392883865,70.093799613272623,
        -14.000000000000002,70.093396046853826,-7.0041488385579989,-10.0,68.094509232290008,-5.0077386181549555,
        68.094221158296435,46.675291532571208,-14.0,46.675291501195034,-14.000000000000004,46.674585433917038,
        -7.0011081945976974,-10.000000000000002,45.342884578934964,-5.0044853494808894,45.342358591863047,
        -9.9999999999999982,-13.999999999999998,-9.9999999999999964,-14.000000000000002,-9.9999999999999982,
        -4.6541960622305716,-9.9999999999999964,-6.9916498557988653,-9.9999999999999964,-6.99164978602478,
        -9.9999999999999947,-4.6541962631244216,-4.9931503007764517,-14.000000000000002,-4.9931493636029334,
        -13.999999999999998,0.0066635162137103814,-14.000000000000002,-4.9935527110051181,-6.9919384142123366,
        -4.9935532626124521,-6.9919374835265442,-3.3236050032142765,-6.9921542921360684,140.32799999999997,136.328,
        140.32799999999997,-13.999999999999998,140.328,-7.0082015385777172,140.32799999999997,-14.000000000000004,
        140.328,-7.0081991580918,140.32799999999997,-13.999999999999998,140.32799999999997,-7.0082004632995671,
        70.0752640337138,136.32800000000006,-5.01167472585953,136.32800000000003,-10.0,136.32800000000003,
        -5.0116769347395431,136.32800000000003,-10.000000000000002,136.328,70.093790333120168,-14.000000000000002,
        -10.000000000000004,68.094499987629192,-9.9999999999999982,68.094509139194315,-10.0,45.342884545523674,
        -9.9999999999999982,-13.999999999999996,-9.9999999999999947,-14.0,-9.9999999999999947,-6.99164961499385,
        -9.9999999999999982,-6.99164878923034,-4.9931489872730346,-13.999999999999996,-3.3228978875299795,-14.0,
        -4.9935525034925687,-6.9919373739570769,140.32799999999997,136.328,140.32799999999997,-13.999999999999998,
        140.328,-14.000000000000002,140.32799999999997,-14.0,-9.9999999999999947,-14.0,-9.9999999999999982,
        -14.000000000000002,140.32799999999997,136.328;
    Explicit_b_F: ARRAY [0..2499] OF LREAL := -0.12667340248608433,-0.006063437668709459,-8.3619092552944529E-18,
        -0.0061236585018917839,-0.12667628514510906,-5.4210108624275222E-20,-0.031816478047680653,
        -0.0061304672764802117,-0.12667642439759061,-0.0019406208995937544,-0.056510051660952777,
        -0.0061180833246716549,-0.12667579011109506,-0.0031721409299244907,-8.3619092552944529E-18,
        -0.0061236585018917839,-0.12667628514510906,-5.4210108624275222E-20,-0.031816478047680653,
        -0.0061304672764802117,-0.12667642439759061,-0.0019406208995937544,-0.056510051660952777,
        -0.0061180833246716549,-0.12667579011109506,-0.0031721409299244907,-2.9402207665091273E-17,
        -1.7279472123987727E-19,-3.8997820408061615E-17,-0.0061382781607270242,-2.781635022959441E-17,
        -0.001954554803000661,-4.4508616762898093E-17,-0.0061364362134341171,-3.6496532114819666E-17,
        -0.0031976628134779668,-2.9402207665091273E-17,-1.7279472123987727E-19,-2.781635022959441E-17,
        -0.001954554803000661,-3.6496532114819666E-17,-0.0031976628134779668,-0.031817232753816052,
        1.1705995331054431E-18,-0.12667685008982194,-5.6920614055488983E-19,-0.05651137952441581,
        6.1325185381211345E-19,-0.12667674648668509,2.7105054312137611E-19,-7.7886797082401052E-18,
        1.1655173354219173E-18,-0.031817232753816052,1.1705995331054431E-18,-0.05651137952441581,
        6.1325185381211345E-19,-0.031817266661648996,-0.0019560462806767378,-0.03181709911953777,
        -0.0032004303747762012,-0.031817232753816052,-1.8126505071242027E-19,-0.031817266661648996,
        -0.0019560462806767378,-0.056511442169811681,-0.0019531851178935223,-6.2021869980328007E-18,
        -0.001954554803000661,-0.031817266661648996,-0.0019560462806767387,-0.056511442169811681,
        -0.0019531851178935223,-0.056511148498327293,-0.0031951779041220494,-0.056511379524415789,
        -7.555533889508359E-19,-0.056511442169811694,-0.0019531851178935223,-0.056511148498327293,
        -0.0031951779041220494,2.834532230515472E-17,-0.0031976628134779664,-0.031817099119537742,
        -0.0032004303747762012,-0.056511148498327286,-0.0031951779041220485,-2.9402207665091273E-17,
        -1.7279472123987727E-19,-3.8997820408061615E-17,-0.0061382781607270242,-2.781635022959441E-17,
        -0.001954554803000661,-4.4508616762898093E-17,-0.0061364362134341171,-3.6496532114819666E-17,
        -0.0031976628134779668,-0.031817232753816052,1.1705995331054431E-18,-0.12667685008982194,
        -5.6920614055488983E-19,-0.05651137952441581,6.1325185381211345E-19,-0.12667674648668509,
        2.7105054312137611E-19,-0.031817266661648996,-0.0019560462806767378,-0.03181709911953777,
        -0.0032004303747762012,-0.056511442169811681,-0.0019531851178935223,-0.056511148498327293,
        -0.0031951779041220494,-3.1637633492013779E-17,-2.1218175328720223E-19,-2.9586609384686495E-17,
        -1.2874900798265365E-18,-3.629303244924182E-17,-1.3844753522871539E-18,-3.5260975742571659E-17,
        -0.0019546071360561261,-3.7007716498487636E-17,-0.0032030047769573962,-2.9586609384686495E-17,
        -1.2874900798265365E-18,-3.5260975742571659E-17,-0.0019546071360561261,-0.031819629222642885,
        -5.5904174518783822E-20,-0.056511639234444355,6.7762635780344027E-19,-0.12667689109875555,
        4.87890977618477E-19,1.3640969307162975E-17,4.0657581468206416E-20,-0.031817379490146271,
        2.6427427954334171E-19,-0.056511639234444355,6.7762635780344027E-19,-0.0565116579667842,
        -1.2197274440461925E-19,-9.9828126789839634E-18,-2.1747570920754161E-19,-1.4679504492390652E-17,
        -4.4045713257223618E-20,-0.031819629222642885,-5.5904174518783822E-20,-0.031819495581118705,
        -0.0032010631169945782,-0.031817379490146284,2.6935647722686751E-19,-0.031817277135142374,
        -0.0019560987878057871,-9.8746042199722266E-18,-0.0019574634784031352,-0.031819663167738495,
        -0.0019563921511248318,-0.056511639234444369,-6.6068569885835426E-19,-0.056511591038165096,
        -3.3203691532368573E-19,-0.056511460878431695,-0.0019532373498035932,6.2570323813675166E-18,
        -0.0032030047769573944,-0.031819495581118684,-0.003201063116994579,-3.629303244924182E-17,
        -1.3844753522871539E-18,-5.39196557327058E-17,-1.3755815063409838E-18,-2.2981062650193236E-17,
        -0.0032037800282279736,-3.1515396049813143E-17,-0.0019574634784031361,-3.5260975742571659E-17,
        -0.0019546071360561261,-3.7007716498487636E-17,-0.0032030047769573962,-0.031819629222642885,
        -5.5904174518783822E-20,-0.031817351949048972,2.2700482986415249E-19,-0.12667689109875555,
        4.87890977618477E-19,-0.031819663167738495,-0.0019563921511248322,-0.031817277135142374,
        -0.0019560987878057871,-0.056511460878431688,-0.0019532373498035924,-4.5264312426914288E-17,
        -6.4374503991326826E-20,-1.8829860054818317E-17,-1.4162771898161559E-18,-9.05149995347786E-18,
        -0.0019582276830549272,-4.01097761444595E-17,-1.7999450129153882E-20,-3.2785416075102559E-17,
        -0.0019575161121738087,-4.5264312426914288E-17,-6.4374503991326826E-20,-8.1940908526196947E-18,
        -0.0019579342315898221,-0.031819776023428871,-6.9287295085401768E-19,-0.031819776023428878,
        -6.8609668727598327E-19,-2.6619971612698751E-17,3.5575383784680614E-19,-0.031819786518259209,
        8.7752613335545515E-19,-1.8776920495614923E-17,-1.4095957935146237E-18,-0.031819748476883458,
        -1.1892342579450377E-18,-1.1073949933725112E-17,-0.0019575161121738074,1.2611473551669278E-17,
        -0.0019582276830549259,7.93648695753598E-18,-0.0032044132383236136,-3.4094373146186072E-17,
        -1.3349239248727773E-18,-4.5264312426914288E-17,-6.4374503991326826E-20,-9.0567409698389962E-18,
        -0.001958227683054928,-5.43860797190673E-17,-0.0019575161121738087,-0.031817389976958411,
        -1.5280474368467578E-18,-0.0565116579667842,-1.2197274440461925E-19,-0.031819673649245137,
        -0.0019564446946577791,-4.0445883408782404E-17,-2.0629487430378485E-18,-1.4750814078637623E-17,
        -8.2818133307315491E-19,-4.0447185391066563E-17,6.3866284222974246E-19,-4.8277910069457279E-17,
        -9.9229909770841285E-19,-2.6619429395807223E-17,-9.9568722949743E-19,-4.0445883408782404E-17,
        -2.0629487430378485E-18,-4.3236735011029394E-17,-1.334067109051033E-18,-0.010939895258464375,
        -0.12940337663776541,1.8973538018496328E-19,-0.12940857748967641,-0.011001415774033131,
        -1.1907589172500954E-17,-0.0034622111951241163,-0.12940866066139117,-0.011010925708052186,
        -0.032495995972325727,-0.005684687311205988,-0.12940746957634541,-0.010999089451642668,-0.0577221130716327,
        1.8973538018496328E-19,-0.12940857748967641,-0.011001415774033131,-1.1907589172500954E-17,
        -0.0034622111951241163,-0.12940866066139117,-0.011010925708052186,-0.032495995972325727,
        -0.0056846873112059888,-0.12940746957634541,-0.010999089451642668,-0.057722113071632712,
        -1.8499199568033919E-18,-3.1316290367649179E-17,-2.5207700510287978E-18,-0.12940951062758926,
        -3.3627208005995723E-18,-0.032497207130407976,-2.3445871979999033E-18,-0.12940931580424303,
        -1.5958100726271018E-18,-0.057724329102651205,-1.8499199568033919E-18,-3.1316290367649179E-17,
        -3.3627208005995723E-18,-0.032497207130407976,-1.5856456772600502E-18,-0.057724329102651212,
        -0.0034781423641150754,-1.4472616695023789E-17,-0.011018053990055782,-1.9238659330986924E-17,
        -0.0057127737954156535,4.3457025358881879E-18,-0.011016492215632667,-1.3649088912055796E-17,
        -5.1838416371963181E-19,1.1910130271342717E-17,-0.0034781423641150754,-1.4472616695023789E-17,
        -0.0057127737954156543,4.3465495688354422E-18,-0.0034805192947300781,-0.032497220518183073,
        -0.0034774059198201877,-0.057724356242492864,-0.0034781423641150754,7.140911261827379E-18,
        -0.0034805192947300781,-0.032497220518183073,-0.00571704223028016,-0.032496943931058939,
        -6.7593229190893167E-19,-0.032497207130407955,-0.0034805192947300781,-0.032497220518183059,
        -0.0057170422302801607,-0.032496943931058939,-0.0057115870095412712,-0.057723849103550343,
        -0.0057127737954156535,4.3457025358881879E-18,-0.0057170422302801616,-0.032496943931058932,
        -0.0057115870095412712,-0.05772384910355035,3.7980957354882827E-18,-0.057724329102651191,
        -0.0034774059198201864,-0.057724356242492864,-0.00571158700954127,-0.057723849103550329,
        -1.8499199568033919E-18,-3.1316290367649179E-17,-2.5207700510287978E-18,-0.12940951062758926,
        -3.3627208005995723E-18,-0.032497207130407976,-2.3445871979999033E-18,-0.12940931580424303,
        -1.5856456772600502E-18,-0.057724329102651212,-0.0034781423641150754,-1.4472616695023789E-17,
        -0.011018053990055782,-1.9238659330986924E-17,-0.0057127737954156543,4.3465495688354422E-18,
        -0.011016492215632667,7.9917558573443237E-18,-0.0034805192947300781,-0.032497220518183073,
        -0.0034774059198201877,-0.057724356242492864,-0.0057170422302801607,-0.032496943931058939,
        -0.005711587009541272,-0.05772384910355035,-1.1180834903756764E-18,-2.8703842234969904E-17,
        -2.2514135738019303E-18,-1.6261338521388058E-17,-2.1785687403380605E-18,-3.0005983337805979E-17,
        -2.4496192834594366E-18,-0.032499690181368147,-2.4530074152484538E-18,-0.057724640166312291,
        -2.2514135738019303E-18,-1.6261338521388058E-17,-2.447925217564928E-18,-0.032499690181368147,
        -0.0034782384082034431,-2.9130521847259457E-18,-0.0057203209764982678,-1.5056010637445189E-17,
        -0.011020049672395411,1.9245435594564958E-17,1.7885100681274552E-18,5.3299548205976849E-18,
        -0.0034823937966747143,-4.7944182396961535E-18,-0.0057203209764982686,-1.5054740088024307E-17,
        -0.0057212109064913585,-3.6574882662440689E-17,2.1345230270808369E-19,1.4522843101818009E-17,
        -8.3348042009823153E-19,-8.3925083205140145E-18,-0.0034782384082034418,-2.9136874594363864E-18,
        -0.0034775019361867527,-0.057724381593873116,-0.0034823937966747156,1.6840391419954779E-17,
        -0.003481014589598143,-0.032499703597191981,3.1001405869507392E-19,-0.03249737675610765,
        -0.0034806155086637754,-0.032497234404046518,-0.0057203209764982695,-1.499333019934837E-17,
        -0.0057195819017150417,7.3615633445871242E-18,-0.0057179316027686257,-0.032499426937493366,
        2.9341221292888964E-18,-0.057724640166312263,-0.0034775019361867514,-0.057724381593873109,
        -2.1751806085490433E-18,-3.0005401002654742E-17,-2.1590869825512116E-18,-1.8180291663392675E-17,
        -2.6393546636444E-18,-0.057724722338242183,-1.0333801956502464E-18,-0.032497376756107664,
        -2.447925217564928E-18,-0.032499690181368147,-2.4496192834594366E-18,-0.057724640166312291,
        -0.0034782384082034418,-2.9136874594363864E-18,-0.0034819660630087974,-1.42590585131973E-17,
        -0.011020049672395411,-2.3488223627361748E-18,-0.0034806155086637754,-0.032497234404046539,
        -0.003481014589598143,-0.032499703597191981,-0.0057179316027686248,-0.032499426937493379,
        -2.4321715627988556E-19,-2.4769572718320691E-17,-3.2932640989247197E-18,-4.3098028973033865E-17,
        -3.0493186101154812E-20,-0.032497435184955785,-1.1608586542120186E-18,-7.0482140936622365E-18,
        -1.7508171019746388E-18,-0.032499859870392257,-2.3045448321122832E-19,-4.6363830675621824E-17,
        -1.2468324983583301E-18,-0.032499904406537286,-0.0034824901317153855,-1.3784825941853297E-17,
        -0.0034824901317153868,-3.5417518019136094E-17,2.2535452699392677E-19,-1.0840645296315756E-17,
        -0.0034829857776749878,-6.0625324408542479E-18,-5.8614679949997583E-19,-4.309872711347086E-17,
        -0.0034820623747332268,-5.69567188348657E-17,9.4867690092481638E-19,-0.032499859870392236,
        2.6495190590114515E-18,-0.032497435184955743,2.8426425709854319E-18,-0.05772474772329142,
        -1.74022919013396E-18,-3.8454607591075591E-17,-2.3045448321122832E-19,-4.6363830675621824E-17,
        -4.072534410398676E-18,-0.0324974351849558,-3.0823528950583989E-18,-0.032499859870392278,
        -0.0034828894057362539,-1.4940390640144977E-17,-0.0057212109064913577,-1.4962837013247215E-17,
        -0.0034811108404072628,-0.032499717489793044,-4.6570117914014579E-19,-5.4131969834891012E-17,
        -7.75458663211312E-19,-5.4659205244755268E-17,-4.7875783090603467E-19,-1.0848096539273634E-17,
        -1.1109398035093036E-18,-5.4060977885999261E-17,-2.4568260686969107E-18,-5.4074900990069754E-17,
        8.7612459859210622E-19,-3.2500058616106466E-17,-2.7055760048624738E-18,-2.1687985305904772E-17,
        -0.021835439137868347,-0.0011520122606157824,8.3760970571609625E-19,-0.0011623928796879576,
        -0.021835986823640203,2.9815559743351372E-19,-0.0046660193730712375,-0.0011641448432321742,
        -0.021836028047420925,-0.00034855849507587592,-0.0088399634659200779,-0.0011621335886920921,
        -0.021835908054478017,-0.00058417725377516751,8.3760970571609625E-19,-0.0011623928796879576,
        -0.021835986823640203,2.9815559743351372E-19,-0.0046660193730712375,-0.0011641448432321742,
        -0.021836028047420925,-0.00034855849507587592,-0.0088399634659200761,-0.0011621335886920921,
        -0.021835908054478017,-0.00058417725377516751,-1.1794933790516132E-19,3.5151867311053464E-19,
        -1.6721489169983957E-18,-0.0011652903420256554,-2.9172079401234121E-18,-0.00035096037140803615,
        -2.1520989607363636E-18,-0.0011650045622868016,-2.9730327053033908E-18,-0.00058857662244823472,
        -1.1794933790516132E-19,3.5151867311053464E-19,-2.9172079401234121E-18,-0.00035096037140803615,
        -2.9730327053033908E-18,-0.00058857662244823472,-0.0046661626879632477,3.7269449679189215E-19,
        -0.021836104506786864,2.2869889575866109E-19,-0.0088402156943794986,4.7137383514701814E-19,
        -0.021836084179334414,3.1340219048409113E-19,-2.8197197418503624E-18,3.5278922253141609E-19,
        -0.0046661626879632477,3.7269449679189215E-19,-0.0088402156943794968,4.6925625277888239E-19,
        -0.0046661729227340945,-0.00035135054557220417,-0.00466614122182821,-0.00058929774581286808,
        -0.0046661626879632477,3.7269449679189215E-19,-0.0046661729227340945,-0.00035135054557220417,
        -0.0088402343122757146,-0.00035088561017350455,-2.1543753617821095E-19,-0.00035096037140803615,
        -0.0046661729227340919,-0.000351350545572204,-0.0088402343122757129,-0.00035088561017350455,
        -0.0088401787462571157,-0.00058844410776131336,-0.0088402156943794986,3.0239076216978522E-19,
        -0.00884023431227572,-0.00035088561017350455,-0.0088401787462571157,-0.00058844410776131336,
        2.430455163027808E-18,-0.00058857662244823472,-0.0046661412218282064,-0.00058929774581286819,
        -0.00884017874625711,-0.00058844410776131336,-1.1794933790516132E-19,3.5151867311053464E-19,
        -1.6721489169983957E-18,-0.0011652903420256554,-2.9172079401234121E-18,-0.00035096037140803615,
        5.4284224007159973E-19,-0.0011650045622868016,-2.9730327053033908E-18,-0.00058857662244823472,
        -0.0046661626879632477,3.7269449679189215E-19,-0.021836104506786864,2.2869889575866109E-19,
        -0.0088402156943794968,4.6925625277888239E-19,-0.021836084179334414,3.1340219048409113E-19,
        -0.0046661729227340945,-0.00035135054557220417,-0.00466614122182821,-0.00058929774581286808,
        -0.0088402343122757129,-0.00035088561017350455,-0.0088401787462571123,-0.00058844410776131336,
        -1.3346592270767604E-18,2.82326669231699E-19,-1.99168547890518E-19,2.2658131339052534E-19,
        -1.578684125224804E-18,2.3727510434961088E-19,-8.3673620298924025E-19,-0.00035097205163314076,
        3.0059081715686983E-19,-0.00058966848483959448,-1.99168547890518E-19,2.2658131339052534E-19,
        -8.3673620298924025E-19,-0.00035097205163314076,-0.004666697129121284,4.8174998875088332E-19,
        -0.008840269714523688,4.3410438546782892E-19,-0.021836113712710516,2.0837010502455788E-19,
        7.9059491036817479E-18,3.9048218868423246E-19,-0.0046661931893067525,4.5655075857006788E-19,
        -0.0088402697145236846,4.3198680309969317E-19,-0.0088402739021540347,5.6158284402960112E-19,
        1.3670317675296357E-18,4.4993331366964366E-19,-1.5821516663526262E-18,4.0562290261640307E-19,
        -0.0046666971291212866,4.8302053817176477E-19,-0.0046666756618988928,-0.00058943885502096274,
        -0.0046661931893067577,2.9116757561866574E-19,-0.0046661752611696682,-0.00035136226893268138,
        -1.4712035851521137E-18,-0.0003515548854198116,-0.004666707372365379,-0.00035142767883477574,
        -0.008840269714523688,9.6561755986990239E-20,-0.0088402602471837673,2.9730856448625942E-19,
        -0.0088402384954132315,-0.00035089728892171812,3.0045846825886135E-19,-0.00058966848483959437,
        -0.0046666756618988928,-0.00058943885502096285,-1.5888485205918556E-18,2.3611043404713622E-19,
        -6.3560558268574647E-19,3.1890790464124408E-19,-1.3013867141174274E-18,-0.00058978898971890226,
        -1.4744726029329233E-18,-0.00035155488541981176,-8.3673620298924025E-19,-0.00035097205163314076,
        2.9381455357883543E-19,-0.00058966848483959448,-0.0046666971291212866,4.8302053817176477E-19,
        -0.004666187775523677,4.7222086809427244E-19,-0.021836113712710516,2.0837010502455788E-19,
        -0.0046667073723653842,-0.00035142767883477574,-0.0046661752611696682,-0.00035136226893268138,
        -0.0088402384954132263,-0.00035089728892171796,-1.8489761437244689E-18,1.232432938255007E-19,
        -1.4251329337553603E-19,1.5386230185264307E-19,-2.7136156303169605E-18,-0.00035169687999964154,
        -4.9415935230040384E-19,4.258458142320995E-19,5.2317519382753894E-19,-0.00035156662712727745,
        -1.8489761437244689E-18,1.232432938255007E-19,-2.4459399840948007E-19,-0.00035163144666093126,
        -0.0046667276446882341,4.1102273765514924E-19,-0.0046667276446882315,4.0890515528701349E-19,
        -9.5356553834500477E-19,4.2679872629776058E-19,-0.00466672998743669,5.14784273693801E-19,
        -1.4592789494415493E-19,3.2237967214500863E-19,-0.0046667222297373193,1.0630263488041469E-19,
        5.2647068138795021E-19,-0.00035156662712727729,2.6900972311408528E-18,-0.00035169687999964138,
        -5.7968817327716179E-20,-0.00058993018680938666,1.5512217288880434E-18,2.3791037906005161E-19,
        -1.8489761437244689E-18,1.232432938255007E-19,-1.6953893834886855E-20,-0.00035169687999964171,
        -4.890516774540114E-18,-0.00035156662712727745,-0.0046661955302668917,3.2441361879839703E-19,
        -0.0088402739021540312,5.5946526166146537E-19,-0.00466670971258821,-0.00035143941031378837,
        -2.460318683737051E-18,2.4156320864508578E-19,-1.9600474748362518E-18,2.4520144624712663E-19,
        -2.4653401353443424E-18,2.413514504082722E-19,-9.535282635186516E-19,2.5770977420212088E-19,
        -9.47597120032705E-19,2.5845092803096839E-19,-2.460318683737051E-18,2.4156320864508578E-19,
        -2.7015815614391379E-18,1.7057475020245581E-19,-0.0034982247754591846,-0.037913871321265488,
        3.2864878353466853E-19,-0.03791553438554341,-0.003516249659905755,6.0562855728682474E-20,
        -0.0010483412940467669,-0.037915602504622059,-0.00352001142228519,-0.0081901839499625134,
        -0.0017637665131279233,-0.037915222177636647,-0.003516769828667967,-0.015456721801501918,
        3.2864878353466853E-19,-0.03791553438554341,-0.003516249659905755,6.0562855728682474E-20,
        -0.0010483412940467669,-0.037915602504622059,-0.00352001142228519,-0.0081901839499625134,
        -0.0017637665131279229,-0.037915222177636647,-0.003516769828667967,-0.015456721801501924,
        -2.0159384144652348E-19,-1.1845226371759356E-18,-4.7433845046240819E-20,-0.037915859870396064,
        -9.1564261598189867E-19,-0.0081905711372341986,-4.8111471404044259E-19,-0.037915794999810175,
        -3.7438856268640075E-19,-0.015457430339336756,-2.0159384144652348E-19,-1.1845226371759356E-18,
        -9.1564261598189867E-19,-0.0081905711372341986,-3.6930636500287495E-19,-0.015457430339336761,
        -0.0010530089868256581,5.6347808024908262E-18,-0.0035218080110374283,-2.732951804316E-18,
        -0.0017719955998451308,3.356897449087199E-18,-0.0035214299089605374,8.1734444245303711E-18,
        -2.0413494028828638E-19,4.2188593520368564E-18,-0.0010530089868256581,5.6347808024908262E-18,
        -0.0017719955998451308,3.356897449087199E-18,-0.0010539568187064221,-0.0081905849637701356,
        -0.0010531016854318472,-0.015457456534433,-0.0010530089868256581,5.6347808024908262E-18,
        -0.0010539568187064221,-0.0081905849637701356,-0.0017736905237788257,-0.0081904966580441437,
        4.3113977015243887E-19,-0.0081905711372341934,-0.0010539568187064217,-0.00819058496377013,
        -0.0017736905237788255,-0.0081904966580441437,-0.0017721939819592,-0.015457294593549919,
        -0.0017719955998451308,-2.0464316005663896E-18,-0.0017736905237788266,-0.0081904966580441437,
        -0.0017721939819592,-0.015457294593549924,9.7493492228969969E-19,-0.015457430339336754,
        -0.0010531016854318466,-0.015457456534433001,-0.0017721939819591993,-0.015457294593549914,
        -2.0159384144652348E-19,-1.1845226371759356E-18,-4.7433845046240819E-20,-0.037915859870396064,
        -9.1564261598189867E-19,-0.0081905711372341986,-4.8450284582945979E-19,-0.037915794999810175,
        -3.6930636500287495E-19,-0.015457430339336761,-0.0010530089868256581,5.6347808024908262E-18,
        -0.0035218080110374283,-2.732951804316E-18,-0.0017719955998451308,3.356897449087199E-18,
        -0.0035214299089605374,8.18699695168644E-18,-0.0010539568187064221,-0.0081905849637701356,
        -0.0010531016854318472,-0.015457456534433004,-0.0017736905237788255,-0.0081904966580441437,
        -0.0017721939819591997,-0.015457294593549924,-4.7010328572613669E-19,-1.3141914699997482E-19,
        -8.4385657370209671E-20,-1.1857402470376137E-18,-8.6736173798840355E-19,-3.407203265220224E-18,
        -5.8720559068404371E-19,-0.0081914952946237352,-2.388632911257127E-19,-0.015457540044886605,
        -8.4385657370209671E-20,-1.1857402470376137E-18,-5.9038196423624734E-19,-0.0081914952946237282,
        -0.001053044746302335,1.5328649367342666E-18,-0.0017745168956370212,2.7445985073407467E-18,
        -0.0035225506987666363,7.3653749928497686E-18,1.262820245237755E-18,9.6305528520445813E-18,
        -0.0010544292673404124,7.4725246606774376E-18,-0.001774516895637021,2.7442808699855263E-18,
        -0.0017748480792266457,-1.0456621733854338E-18,-4.70950318673391E-19,5.2720720300536742E-18,
        -1.9566461081574338E-19,1.9956890330699367E-18,-0.0010530447463023354,1.5330766949710802E-18,
        -0.0010531374576252502,-0.015457465979431909,-0.0010544292673404132,2.0594017925712211E-18,
        -0.001054141160788231,-0.0081915091323479083,3.2314306937751558E-19,-0.00819063094036294,
        -0.0010539926448452485,-0.0081905901342984883,-0.0017745168956370219,-8.0768826685433809E-18,
        -0.001774334854501361,-4.3972656665522934E-18,-0.001774021536753176,-0.0081914208010279415,
        4.2775163836342167E-19,-0.015457540044886595,-0.0010531374576252493,-0.015457465979431904,
        -8.6820877093565785E-19,-3.4073620838978341E-18,-3.4050724479622874E-19,-2.993361496037494E-18,
        -2.447925217564928E-19,-0.015457567403298908,-3.4813054132151744E-19,-0.0081906309403629463,
        -5.9038196423624734E-19,-0.0081914952946237282,-2.405573570202213E-19,-0.015457540044886605,
        -0.0010530447463023354,1.5330766949710802E-18,-0.0010543228028200187,5.2656332561655615E-18,
        -0.0035225506987666363,7.3810451023739732E-18,-0.0010539926448452492,-0.0081905901342984935,
        -0.001054141160788231,-0.0081915091323479083,-0.0017740215367531753,-0.0081914208010279415,
        -4.6609629359195911E-19,-4.648622693650007E-19,-2.7782680669941051E-19,3.4962161709370553E-18,
        -1.7575933655526732E-19,-0.00819065093434982,-3.6348301349050163E-19,1.1533177448757402E-17,
        8.9573734172142261E-20,-0.00819155512097787,-4.6485265339037978E-19,-4.55227269589983E-19,
        -6.9393174203808555E-19,-0.0081915699426062215,-0.0010544651240993646,-2.1534753892756518E-18,
        -0.0010544651240993646,-2.1535812683940586E-18,-1.4930700529461648E-20,-2.1646721060471696E-18,
        -0.0010546495763118805,4.4861511864547916E-18,4.0064658405128406E-19,-1.907404046292152E-18,
        -0.0010543586543143618,-2.3973149989664835E-18,8.1950437646853558E-20,-0.00819155512097786,
        4.921261423547485E-19,-0.0081906509343498083,3.5998900258307764E-19,-0.015457576859199004,
        -4.6120943977996653E-19,1.749573022333359E-18,-4.6485265339037978E-19,-4.55227269589983E-19,
        -8.4745646372792749E-19,-0.0081906509343498256,8.8726701224887961E-20,-0.00819155512097787,
        -0.001054613705821476,-5.1583777092194857E-18,-0.0017748480792266462,-1.0256510200065509E-18,
        -0.0010541770006516429,-0.0081915143053841559,4.1312398320618707E-20,-3.1012490089715603E-18,
        -1.0894961284058438E-18,5.3833863454703946E-18,4.23171206500766E-20,7.7514036411160156E-18,
        -1.3193265813930833E-20,-2.1547194689169316E-18,-1.1759897521695683E-20,-7.5663467944756522E-18,
        4.5249235199094131E-20,-8.4940530125110242E-18,5.4294849001241571E-22,-5.4233692790932017E-18,
        -0.90852126123084109,-0.043908146081154252,1.1237416704633352E-16,-0.044340059223466725,
        -0.90854213589311628,5.4210108624275222E-18,-0.22499743169378195,-0.044391150716473024,-0.90854320277576739,
        -0.013973130057841329,-0.40175302414947389,-0.044302834795567785,-0.90853861186181406,-0.02289738328452481,
        1.1237416704633352E-16,-0.044340059223466725,-0.90854213589311628,5.4210108624275222E-18,
        -0.22499743169378195,-0.044391150716473024,-0.90854320277576739,-0.013973130057841329,-0.40175302414947389,
        -0.044302834795567785,-0.90853861186181406,-0.02289738328452481,-2.0211137857729586E-16,
        -3.3610267347050637E-18,1.4233541645661263E-17,-0.044446387153773116,-1.2255042087464668E-16,
        -0.014073066200566241,-1.7068052700353054E-16,-0.044433312973263257,-1.4178653910679184E-16,
        -0.02308043023166,-2.0211137857729586E-16,-3.3610267347050637E-18,-1.2254660922638404E-16,
        -0.014073066200566246,-1.4178653910679184E-16,-0.02308043023166,-0.22500289657472694,1.6127507315721878E-18,
        -0.90854626790451765,5.4210108624275222E-19,-0.4017626395980568,1.0543866127421531E-17,-0.90854551524313676,
        7.48099499014998E-18,-2.9203154922486513E-17,7.37257477290143E-18,-0.22500289657472694,
        1.6127507315721878E-18,-0.40176263959805669,1.0489656018797255E-17,-0.2250031571391346,
        -0.014084282907403574,-0.22500194445913865,-0.023101232532859166,-0.22500289657472694,
        1.7821573210230479E-17,-0.2250031571391346,-0.014084282907403586,-0.40176311984350016,-0.014063877541696803,
        -1.2255465603938295E-16,-0.014073066200566236,-0.2250031571391346,-0.014084282907403574,
        -0.40176311984350005,-0.014063877541696803,-0.4017609942320583,-0.023063772260979193,-0.40176263959805669,
        5.0957502106818708E-18,-0.40176311984350022,-0.014063877541696813,-0.4017609942320583,-0.023063772260979193,
        2.0403837853229939E-16,-0.02308043023166,-0.22500194445913849,-0.023101232532859169,-0.401760994232058,
        -0.023063772260979186,-2.0211137857729586E-16,-3.3610267347050637E-18,1.4233541645661263E-17,
        -0.044446387153773116,-1.2254660922638404E-16,-0.014073066200566246,1.9888333601530972E-18,
        -0.044433312973263257,-1.4178653910679184E-16,-0.02308043023166,-0.22500289657472694,1.6127507315721878E-18,
        -0.90854626790451765,5.9631119486702744E-18,-0.40176263959805669,1.0489656018797255E-17,
        -0.90854551524313676,7.48099499014998E-18,-0.2250031571391346,-0.014084282907403586,-0.22500194445913865,
        -0.023101232532859166,-0.40176311984350005,-0.014063877541696808,-0.40176099423205819,-0.023063772260979193,
        -1.1948500863853337E-16,-7.8316666303132609E-18,-1.0077230382823216E-16,-2.5478751053409354E-18,
        -4.0905762121751926E-17,1.6703489719854803E-18,-8.65074749030817E-18,-0.014073452133259199,
        -5.3407121390278145E-17,-0.023119416718676764,-1.0077092739969287E-16,-2.5343225781848666E-18,
        -8.643971226730135E-18,-0.014073452133259209,-0.22502056771591866,8.2263839837337649E-18,
        -0.40176453880416918,6.5323180892251642E-18,-0.90854657053851451,5.5294310796760726E-18,
        2.45051555019675E-16,2.6834003769016235E-18,-0.22500396954755839,9.4867690092481638E-19,
        -0.40176453880416907,6.478107980600889E-18,-0.40176467697335466,-2.439454888092385E-19,
        5.3732382042023796E-17,8.3331101350878067E-18,-4.1341984089587891E-17,7.0235971986326584E-18,
        -0.22502056771591855,8.1518450843753865E-18,-0.22501961554900995,-0.023105898263657981,-0.22500396954755847,
        1.1858461261560205E-17,-0.225003234379625,-0.014084670139843564,-5.3978445113201171E-17,
        -0.014094294168846267,-0.22502082855573682,-0.014086833295573026,-0.40176453880416929,
        6.6407383064737147E-18,-0.40176418862008356,6.3967928176644762E-18,-0.40176325784096573,
        -0.014064262811759857,1.1939607017907167E-16,-0.023119416718676764,-0.22501961554900987,
        -0.023105898263657981,-4.1339442990746128E-17,1.6195269951502222E-18,-4.3272795692854069E-18,
        2.1819568721270777E-18,-8.3520836731063031E-17,-0.023124920378727248,-5.4079242033924432E-17,
        -0.014094294168846278,-8.643971226730135E-18,-0.014073452133259209,-2.2653726767726812E-16,
        -0.023119416718676764,-0.22502056771591855,8.1518450843753865E-18,-0.22500376942411082,
        4.2283884726934673E-18,-0.90854657053851451,1.0950441942103595E-17,-0.225020828555737,-0.014086833295573026,
        -0.225003234379625,-0.014084670139843564,-0.4017632578409655,-0.014064262811759858,-6.8140584528386856E-17,
        -4.7298319774680131E-18,-1.5717712775840248E-16,-4.8427867988345792E-18,-1.8241786255363338E-16,
        -0.014099813725742058,-9.7153620258884181E-18,1.44774871344705E-17,-1.9124479289697044E-16,
        -0.014094682296279696,-6.8139128690508763E-17,-4.7162794503119443E-18,-6.6146920433456449E-17,
        -0.014097649905087963,-0.22502164116342194,6.8711312681268844E-18,-0.2250216411634221,
        1.5517643593698782E-18,-1.0201159574812646E-16,2.2158381900172497E-18,-0.22502171855946634,
        2.1480755542369057E-18,1.5798011499239956E-17,4.91865166871488E-19,-0.22502144099999252,
        2.6766241133235891E-18,-1.8120999357084874E-17,-0.014094682296279686,-9.6193296654934618E-18,
        -0.014099813725742047,1.9217822320484468E-16,-0.023129589494450122,-1.5185585502551415E-16,
        -3.1611269591530489E-18,-6.8139128690508763E-17,-4.7162794503119443E-18,-9.698950762535366E-18,
        -0.014099813725742063,-1.9135406014716624E-16,-0.014094682296279696,-0.22500404688447739,
        8.40256683676266E-18,-0.40176467697335472,1.0625181290357943E-17,-0.22502090585531667,-0.0140872207964491,
        -2.8013481348918148E-16,5.2482161411876449E-18,-1.0580415599095554E-16,-2.786738913454531E-18,
        -1.0705883760614638E-16,1.0608240631412857E-17,-1.0176638301861879E-16,2.2463313761184045E-18,
        -1.0165657313794115E-16,-3.1509625637859973E-18,-2.8013342961601668E-16,5.2583805365546965E-18,
        -5.7474348667278365E-20,-2.9607205860406696E-20,-0.077953938048960669,-0.91495630205656719,
        1.5395670849294163E-17,-0.91499336154188149,-0.078388923478923359,-1.2000762796698927E-17,
        -0.024548090137893282,-0.91499404071464974,-0.0784581439271197,-0.22706440144138565,-0.040393877243513461,
        -0.91498555513722191,-0.07837495020825766,-0.405131234178429,1.5395670849294163E-17,-0.91499336154188149,
        -0.078388923478923359,-1.2000762796698927E-17,-0.024548090137893282,-0.91499404071464974,
        -0.0784581439271197,-0.22706440144138565,-0.040393877243513461,-0.91498555513722191,-0.07837495020825766,
        -0.405131234178429,-1.2197274440461925E-18,-6.8118389618190833E-17,-4.9873299934333204E-18,
        -0.91500006722362592,-4.8382521947165635E-18,-0.22707303152550876,-3.2526065174565133E-18,
        -0.91499867394199985,-9.7849246066816775E-18,-0.4051470246964986,-1.2197274440461925E-18,
        -6.8118389618190833E-17,-4.8382521947165635E-18,-0.22707303152550876,-9.7849246066816775E-18,
        -0.4051470246964986,-0.024660732712307117,1.417594340524797E-17,-0.078507952497007219,
        1.9447876468958736E-17,-0.040592464909515784,1.8488357546309064E-16,-0.078497094095205028,
        7.5948362182609586E-17,-1.3823577699190182E-18,2.7769805769142786E-16,-0.024660732712307103,
        1.4168320108722682E-17,-0.040592464909515784,1.8488357546309064E-16,-0.024678049245177087,
        -0.22707314681162666,-0.02465616095779212,-0.405147254584257,-0.024660732712307117,1.8708416706005732E-16,
        -0.024678049245177087,-0.22707314681162666,-0.0406235469714099,-0.22707117636130061,5.9089018400459992E-18,
        -0.22707303152550867,-0.024678049245177074,-0.22707314681162657,-0.0406235469714099,-0.22707117636130061,
        -0.040585198407018679,-0.405143641589301,-0.040592464909515784,1.1975351808281298E-17,-0.040623546971409907,
        -0.2270711763613007,-0.040585198407018679,-0.405143641589301,1.1763593571467723E-17,-0.40514702469649849,
        -0.0246561609577921,-0.405147254584257,-0.040585198407018672,-0.405143641589301,-1.2197274440461925E-18,
        -6.8118389618190833E-17,-4.9873299934333204E-18,-0.91500006722362592,-4.8382521947165635E-18,
        -0.22707303152550876,-3.2526065174565133E-18,-0.91499867394199985,-9.7849246066816775E-18,
        -0.4051470246964986,-0.024660732712307103,1.4168320108722682E-17,-0.078507952497007219,
        1.9447876468958736E-17,-0.040592464909515784,1.8488357546309064E-16,-0.078497094095205028,
        7.5948362182609586E-17,-0.024678049245177087,-0.22707314681162666,-0.024656160957792109,-0.405147254584257,
        -0.0406235469714099,-0.22707117636130061,-0.040585198407018679,-0.405143641589301,-1.4094628242311558E-18,
        6.5815518792843204E-18,-1.4894227344519617E-17,-4.6953577365147631E-17,7.3183646642771549E-19,
        -1.4633468251707381E-16,5.2922618544448685E-18,-0.22709100233229687,-9.5680841721845766E-18,
        -0.40514926269585039,-1.4894227344519617E-17,-4.6953577365147631E-17,5.2922618544448685E-18,
        -0.22709100233229687,-0.02466142784965503,1.1036924006018259E-16,-0.040646457087583146,
        1.5888644024596166E-17,-0.0785223958657716,8.3937576941112146E-17,2.8192644616412132E-17,
        2.9900517147960978E-16,-0.02469114725936063,9.6381337969225073E-17,-0.040646457087583146,
        1.5888644024596166E-17,-0.040652897782438434,1.9426361832098477E-16,-1.5178830414797062E-18,
        1.7948585800671261E-16,6.5052130349130266E-19,2.657311762126191E-17,-0.02466142784965503,
        1.1037008709312984E-16,-0.024656855942051376,-0.40514743808224646,-0.024691147259360651,
        9.639658456227565E-17,-0.024681633887332338,-0.22709111782296573,7.15573433840433E-18,-0.22707425188322058,
        -0.024678745617735788,-0.22707324731405812,-0.040646457087583153,1.5893726222279692E-17,
        -0.040641311777483369,4.953956895311501E-17,-0.04062998370810441,-0.22708914685042259,
        1.0299920638612292E-18,-0.40514926269585017,-0.024656855942051355,-0.40514743808224646,
        7.3183646642771549E-19,-1.4633468251707381E-16,-2.0464316005663896E-18,-2.880081427254072E-17,
        6.2341624917916505E-18,-0.40514985034555978,7.26415455565288E-18,-0.22707425188322075,
        5.2922618544448685E-18,-0.22709100233229687,-9.5680841721845766E-18,-0.40514926269585039,
        -0.02466142784965503,1.1037008709312984E-16,-0.02468816702271235,1.2348385118252092E-16,-0.0785223958657716,
        8.3937576941112146E-17,-0.0246787456177358,-0.22707324731405804,-0.024681633887332327,-0.22709111782296573,
        -0.040629983708104396,-0.22708914685042267,-5.7716990462030536E-18,-4.7925971188595567E-17,
        5.9360068943581368E-18,-6.1272563459363171E-17,5.0279875749015268E-18,-0.2270746709188694,
        -1.1826274009564541E-17,8.3068944653702861E-17,-3.8692465030576439E-18,-0.22709222314756114,
        -5.7716990462030536E-18,-4.7925971188595567E-17,-9.1547320939244781E-18,-0.22709254163278178,
        -0.024691844478350409,7.8430168718064686E-17,-0.024691844478350409,2.5117660907994846E-16,
        -4.7238965429826388E-18,1.0376068900570454E-16,-0.024695431618763558,2.0548256970736797E-16,
        -1.5720931501039814E-17,-6.1264569585923459E-17,-0.024688864080425831,-8.9425503406372758E-17,
        1.7767363101606204E-17,-0.22709222314756114,1.5666721392415539E-17,-0.22707467091886915,
        1.0164395367051604E-17,-0.40515003408376971,-7.1692868655603981E-18,-2.8378144831860824E-17,
        -5.7716990462030536E-18,-4.7925971188595567E-17,5.082197683525802E-18,-0.22707467091886949,
        -1.463672932855431E-17,-0.22709222314756122,-0.024694734132731256,1.6721192708452418E-16,
        -0.040652897782438434,2.1352006534386403E-17,-0.024682330526772954,-0.22709121837416038,
        1.1786722988960778E-18,-1.8853815205357853E-16,-1.7381116077658243E-18,-2.3392575078771017E-17,
        1.10285525039494E-18,1.5792918713644589E-16,-4.7470079692973704E-18,-6.9875982983743506E-17,
        -4.645797251472679E-18,-6.9338328820473839E-17,1.148179112794923E-18,-1.8854191076228197E-16,
        -1.0777346329819693E-17,8.4682682732228818E-20,0.90852126123084109,0.043908146081154252,
        -1.1237416704633352E-16,0.044340059223466725,0.90854213589311628,-5.4210108624275222E-18,
        0.22499743169378195,0.044391150716473024,0.90854320277576739,0.013973130057841329,0.40175302414947389,
        0.044302834795567785,0.90853861186181406,0.02289738328452481,-1.1237416704633352E-16,0.044340059223466725,
        0.90854213589311628,-5.4210108624275222E-18,0.22499743169378195,0.044391150716473024,0.90854320277576739,
        0.013973130057841329,0.40175302414947389,0.044302834795567785,0.90853861186181406,0.02289738328452481,
        2.0211137857729586E-16,3.3610267347050637E-18,-1.4233541645661263E-17,0.044446387153773116,
        1.2255042087464668E-16,0.014073066200566241,1.7068052700353054E-16,0.044433312973263257,
        1.4178653910679184E-16,0.02308043023166,2.0211137857729586E-16,3.3610267347050637E-18,
        1.2254660922638404E-16,0.014073066200566246,1.4178653910679184E-16,0.02308043023166,0.22500289657472694,
        -1.6127507315721878E-18,0.90854626790451765,-5.4210108624275222E-19,0.4017626395980568,
        -1.0543866127421531E-17,0.90854551524313676,-7.48099499014998E-18,2.9203154922486513E-17,
        -7.37257477290143E-18,0.22500289657472694,-1.6127507315721878E-18,0.40176263959805669,
        -1.0489656018797255E-17,0.2250031571391346,0.014084282907403574,0.22500194445913865,0.023101232532859166,
        0.22500289657472694,-1.7821573210230479E-17,0.2250031571391346,0.014084282907403586,0.40176311984350016,
        0.014063877541696803,1.2255465603938295E-16,0.014073066200566236,0.2250031571391346,0.014084282907403574,
        0.40176311984350005,0.014063877541696803,0.4017609942320583,0.023063772260979193,0.40176263959805669,
        -5.0957502106818708E-18,0.40176311984350022,0.014063877541696813,0.4017609942320583,0.023063772260979193,
        -2.0403837853229939E-16,0.02308043023166,0.22500194445913849,0.023101232532859169,0.401760994232058,
        0.023063772260979186,2.0211137857729586E-16,3.3610267347050637E-18,-1.4233541645661263E-17,
        0.044446387153773116,1.2254660922638404E-16,0.014073066200566246,-1.9888333601530972E-18,
        0.044433312973263257,1.4178653910679184E-16,0.02308043023166,0.22500289657472694,-1.6127507315721878E-18,
        0.90854626790451765,-5.9631119486702744E-18,0.40176263959805669,-1.0489656018797255E-17,0.90854551524313676,
        -7.48099499014998E-18,0.2250031571391346,0.014084282907403586,0.22500194445913865,0.023101232532859166,
        0.40176311984350005,0.014063877541696808,0.40176099423205819,0.023063772260979193,1.1948500863853337E-16,
        7.8316666303132609E-18,1.0077230382823216E-16,2.5478751053409354E-18,4.0905762121751926E-17,
        -1.6703489719854803E-18,8.65074749030817E-18,0.014073452133259199,5.3407121390278145E-17,
        0.023119416718676764,1.0077092739969287E-16,2.5343225781848666E-18,8.643971226730135E-18,
        0.014073452133259209,0.22502056771591866,-8.2263839837337649E-18,0.40176453880416918,
        -6.5323180892251642E-18,0.90854657053851451,-5.5294310796760726E-18,-2.45051555019675E-16,
        -2.6834003769016235E-18,0.22500396954755839,-9.4867690092481638E-19,0.40176453880416907,
        -6.478107980600889E-18,0.40176467697335466,2.439454888092385E-19,-5.3732382042023796E-17,
        -8.3331101350878067E-18,4.1341984089587891E-17,-7.0235971986326584E-18,0.22502056771591855,
        -8.1518450843753865E-18,0.22501961554900995,0.023105898263657981,0.22500396954755847,
        -1.1858461261560205E-17,0.225003234379625,0.014084670139843564,5.3978445113201171E-17,0.014094294168846267,
        0.22502082855573682,0.014086833295573026,0.40176453880416929,-6.6407383064737147E-18,0.40176418862008356,
        -6.3967928176644762E-18,0.40176325784096573,0.014064262811759857,-1.1939607017907167E-16,
        0.023119416718676764,0.22501961554900987,0.023105898263657981,4.1339442990746128E-17,
        -1.6195269951502222E-18,4.3272795692854069E-18,-2.1819568721270777E-18,8.3520836731063031E-17,
        0.023124920378727248,5.4079242033924432E-17,0.014094294168846278,8.643971226730135E-18,0.014073452133259209,
        2.2653726767726812E-16,0.023119416718676764,0.22502056771591855,-8.1518450843753865E-18,0.22500376942411082,
        -4.2283884726934673E-18,0.90854657053851451,-1.0950441942103595E-17,0.225020828555737,0.014086833295573026,
        0.225003234379625,0.014084670139843564,0.4017632578409655,0.014064262811759858,6.8140584528386856E-17,
        4.7298319774680131E-18,1.5717712775840248E-16,4.8427867988345792E-18,1.8241786255363338E-16,
        0.014099813725742058,9.7153620258884181E-18,-1.44774871344705E-17,1.9124479289697044E-16,
        0.014094682296279696,6.8139128690508763E-17,4.7162794503119443E-18,6.6146920433456449E-17,
        0.014097649905087963,0.22502164116342194,-6.8711312681268844E-18,0.2250216411634221,-1.5517643593698782E-18,
        1.0201159574812646E-16,-2.2158381900172497E-18,0.22502171855946634,-2.1480755542369057E-18,
        -1.5798011499239956E-17,-4.91865166871488E-19,0.22502144099999252,-2.6766241133235891E-18,
        1.8120999357084874E-17,0.014094682296279686,9.6193296654934618E-18,0.014099813725742047,
        -1.9217822320484468E-16,0.023129589494450122,1.5185585502551415E-16,3.1611269591530489E-18,
        6.8139128690508763E-17,4.7162794503119443E-18,9.698950762535366E-18,0.014099813725742063,
        1.9135406014716624E-16,0.014094682296279696,0.22500404688447739,-8.40256683676266E-18,0.40176467697335472,
        -1.0625181290357943E-17,0.22502090585531667,0.0140872207964491,2.8013481348918148E-16,
        -5.2482161411876449E-18,1.0580415599095554E-16,2.786738913454531E-18,1.0705883760614638E-16,
        -1.0608240631412857E-17,1.0176638301861879E-16,-2.2463313761184045E-18,1.0165657313794115E-16,
        3.1509625637859973E-18,2.8013342961601668E-16,-5.2583805365546965E-18,5.7474348667278365E-20,
        2.9607205860406696E-20,0.077953938048960669,0.91495630205656719,-1.5395670849294163E-17,0.91499336154188149,
        0.078388923478923359,1.2000762796698927E-17,0.024548090137893282,0.91499404071464974,0.0784581439271197,
        0.22706440144138565,0.040393877243513461,0.91498555513722191,0.07837495020825766,0.405131234178429,
        -1.5395670849294163E-17,0.91499336154188149,0.078388923478923359,1.2000762796698927E-17,
        0.024548090137893282,0.91499404071464974,0.0784581439271197,0.22706440144138565,0.040393877243513461,
        0.91498555513722191,0.07837495020825766,0.405131234178429,1.2197274440461925E-18,6.8118389618190833E-17,
        4.9873299934333204E-18,0.91500006722362592,4.8382521947165635E-18,0.22707303152550876,
        3.2526065174565133E-18,0.91499867394199985,9.7849246066816775E-18,0.4051470246964986,1.2197274440461925E-18,
        6.8118389618190833E-17,4.8382521947165635E-18,0.22707303152550876,9.7849246066816775E-18,0.4051470246964986,
        0.024660732712307117,-1.417594340524797E-17,0.078507952497007219,-1.9447876468958736E-17,
        0.040592464909515784,-1.8488357546309064E-16,0.078497094095205028,-7.5948362182609586E-17,
        1.3823577699190182E-18,-2.7769805769142786E-16,0.024660732712307103,-1.4168320108722682E-17,
        0.040592464909515784,-1.8488357546309064E-16,0.024678049245177087,0.22707314681162666,0.02465616095779212,
        0.405147254584257,0.024660732712307117,-1.8708416706005732E-16,0.024678049245177087,0.22707314681162666,
        0.0406235469714099,0.22707117636130061,-5.9089018400459992E-18,0.22707303152550867,0.024678049245177074,
        0.22707314681162657,0.0406235469714099,0.22707117636130061,0.040585198407018679,0.405143641589301,
        0.040592464909515784,-1.1975351808281298E-17,0.040623546971409907,0.2270711763613007,0.040585198407018679,
        0.405143641589301,-1.1763593571467723E-17,0.40514702469649849,0.0246561609577921,0.405147254584257,
        0.040585198407018672,0.405143641589301,1.2197274440461925E-18,6.8118389618190833E-17,4.9873299934333204E-18,
        0.91500006722362592,4.8382521947165635E-18,0.22707303152550876,3.2526065174565133E-18,0.91499867394199985,
        9.7849246066816775E-18,0.4051470246964986,0.024660732712307103,-1.4168320108722682E-17,0.078507952497007219,
        -1.9447876468958736E-17,0.040592464909515784,-1.8488357546309064E-16,0.078497094095205028,
        -7.5948362182609586E-17,0.024678049245177087,0.22707314681162666,0.024656160957792109,0.405147254584257,
        0.0406235469714099,0.22707117636130061,0.040585198407018679,0.405143641589301,1.4094628242311558E-18,
        -6.5815518792843204E-18,1.4894227344519617E-17,4.6953577365147631E-17,-7.3183646642771549E-19,
        1.4633468251707381E-16,-5.2922618544448685E-18,0.22709100233229687,9.5680841721845766E-18,
        0.40514926269585039,1.4894227344519617E-17,4.6953577365147631E-17,-5.2922618544448685E-18,
        0.22709100233229687,0.02466142784965503,-1.1036924006018259E-16,0.040646457087583146,
        -1.5888644024596166E-17,0.0785223958657716,-8.3937576941112146E-17,-2.8192644616412132E-17,
        -2.9900517147960978E-16,0.02469114725936063,-9.6381337969225073E-17,0.040646457087583146,
        -1.5888644024596166E-17,0.040652897782438434,-1.9426361832098477E-16,1.5178830414797062E-18,
        -1.7948585800671261E-16,-6.5052130349130266E-19,-2.657311762126191E-17,0.02466142784965503,
        -1.1037008709312984E-16,0.024656855942051376,0.40514743808224646,0.024691147259360651,
        -9.639658456227565E-17,0.024681633887332338,0.22709111782296573,-7.15573433840433E-18,0.22707425188322058,
        0.024678745617735788,0.22707324731405812,0.040646457087583153,-1.5893726222279692E-17,0.040641311777483369,
        -4.953956895311501E-17,0.04062998370810441,0.22708914685042259,-1.0299920638612292E-18,0.40514926269585017,
        0.024656855942051355,0.40514743808224646,-7.3183646642771549E-19,1.4633468251707381E-16,
        2.0464316005663896E-18,2.880081427254072E-17,-6.2341624917916505E-18,0.40514985034555978,
        -7.26415455565288E-18,0.22707425188322075,-5.2922618544448685E-18,0.22709100233229687,
        9.5680841721845766E-18,0.40514926269585039,0.02466142784965503,-1.1037008709312984E-16,0.02468816702271235,
        -1.2348385118252092E-16,0.0785223958657716,-8.3937576941112146E-17,0.0246787456177358,0.22707324731405804,
        0.024681633887332327,0.22709111782296573,0.040629983708104396,0.22708914685042267,5.7716990462030536E-18,
        4.7925971188595567E-17,-5.9360068943581368E-18,6.1272563459363171E-17,-5.0279875749015268E-18,
        0.2270746709188694,1.1826274009564541E-17,-8.3068944653702861E-17,3.8692465030576439E-18,
        0.22709222314756114,5.7716990462030536E-18,4.7925971188595567E-17,9.1547320939244781E-18,
        0.22709254163278178,0.024691844478350409,-7.8430168718064686E-17,0.024691844478350409,
        -2.5117660907994846E-16,4.7238965429826388E-18,-1.0376068900570454E-16,0.024695431618763558,
        -2.0548256970736797E-16,1.5720931501039814E-17,6.1264569585923459E-17,0.024688864080425831,
        8.9425503406372758E-17,-1.7767363101606204E-17,0.22709222314756114,-1.5666721392415539E-17,
        0.22707467091886915,-1.0164395367051604E-17,0.40515003408376971,7.1692868655603981E-18,
        2.8378144831860824E-17,5.7716990462030536E-18,4.7925971188595567E-17,-5.082197683525802E-18,
        0.22707467091886949,1.463672932855431E-17,0.22709222314756122,0.024694734132731256,-1.6721192708452418E-16,
        0.040652897782438434,-2.1352006534386403E-17,0.024682330526772954,0.22709121837416038,
        -1.1786722988960778E-18,1.8853815205357853E-16,1.7381116077658243E-18,2.3392575078771017E-17,
        -1.10285525039494E-18,-1.5792918713644589E-16,4.7470079692973704E-18,6.9875982983743506E-17,
        4.645797251472679E-18,6.9338328820473839E-17,-1.148179112794923E-18,1.8854191076228197E-16,
        1.0777346329819693E-17,-8.4682682732228818E-20,-0.0032231717786674243,-0.00047387004623103532,-1.0,
        1.0842021724855044E-19,-0.0032233970643617714,1.5670109524204556E-20,-0.50017152346648186,
        -0.00012270693090584496,-0.003223438748220626,-0.0001096414616121335,-0.33389281505076362,
        -0.00021633303651176036,-0.0032233972588470859,-0.00020082461188265349,-1.0,1.0842021724855044E-19,
        -0.0032233970643617714,1.5670109524204556E-20,-0.50017152346648186,-0.00012270693090584496,
        -0.003223438748220626,-0.00010964146161213346,-0.33389281505076362,-0.00021633303651176036,
        -0.0032233972588470859,-0.00020082461188265349,-1.0,5.4210108624275222E-20,-1.0,0.0,-1.0,
        -1.0842021724855044E-19,-1.0,0.0,-1.0,0.0,-1.0,5.4210108624275222E-20,-1.0,0.0,-1.0,0.0,-0.500171538572618,
        0.0,-0.0032234627990377889,3.7692966152816365E-20,-0.33389286200349694,5.4210108624275222E-20,
        -0.0032234578058911562,6.5645053412208276E-20,-0.99999999999999978,5.4210108624275222E-20,
        -0.500171538572618,0.0,-0.33389286200349694,5.4210108624275222E-20,-0.50017154120112894,
        -2.8830983828423548E-5,-0.50017153832237338,-5.2621143293484158E-5,-0.500171538572618,0.0,
        -0.50017154120112894,-2.8830983828423494E-5,-0.33389287043993776,-5.0429547165299263E-5,-1.0,0.0,
        -0.50017154120112894,-2.8830983828423548E-5,-0.33389287043993776,-5.0429547165299263E-5,-0.3338928616111102,
        -9.2256767123402269E-5,-0.333892862003497,2.7105054312137611E-20,-0.33389287043993771,
        -5.0429547165299263E-5,-0.3338928616111102,-9.2256767123402269E-5,-1.0000000000000002,
        5.4210108624275222E-20,-0.50017153832237338,-5.2621143293484266E-5,-0.33389286161111031,
        -9.225676712340216E-5,-1.0,5.4210108624275222E-20,-1.0,0.0,-1.0,0.0,-1.0,0.0,-1.0,0.0,-0.500171538572618,
        0.0,-0.0032234627990377889,3.7269449679189215E-20,-0.33389286200349694,5.4210108624275222E-20,
        -0.0032234578058911562,6.5645053412208276E-20,-0.50017154120112894,-2.8830983828423494E-5,
        -0.50017153832237338,-5.2621143293484158E-5,-0.33389287043993776,-5.0429547165299263E-5,-0.3338928616111102,
        -9.2256767123402269E-5,-1.0,5.4210108624275222E-20,-1.0,5.4210108624275222E-20,-1.0,5.4210108624275222E-20,
        -1.0,0.0,-1.0,0.0,-1.0,5.4210108624275222E-20,-1.0,5.4210108624275222E-20,-0.50017155139325642,
        5.4210108624275222E-20,-0.33389287552797581,0.0,-0.0032234713063484617,3.7269449679189215E-20,-1.0,
        1.6263032587282567E-19,-0.50017154286415544,0.0,-0.33389287552797581,0.0,-0.3338928772195392,
        5.4210108624275222E-20,-1.0,1.0842021724855044E-19,-0.99999999999999978,1.0842021724855044E-19,
        -0.50017155139325642,5.4210108624275222E-20,-0.50017155114301959,-5.2624528352597055E-5,
        -0.50017154286415533,-5.4210108624275222E-20,-0.50017154172544676,-2.8833612408983415E-5,-1.0,0.0,
        -0.50017155402213676,-2.8832834192057944E-5,-0.3338928755279757,-2.7105054312137611E-20,
        -0.33389287438889476,8.1315162936412833E-20,-0.33389287213054836,-5.0434267119571795E-5,-1.0000000000000002,
        1.6263032587282567E-19,-0.50017155114301959,-5.2624528352597164E-5,-1.0,5.4210108624275222E-20,-1.0,
        5.4210108624275222E-20,-1.0,0.0,-1.0,5.4210108624275222E-20,-1.0,5.4210108624275222E-20,-1.0,0.0,
        -0.50017155139325642,5.4210108624275222E-20,-0.5001715424793699,-5.4210108624275222E-20,
        -0.0032234713063484617,3.7269449679189215E-20,-0.50017155402213676,-2.8832834192057835E-5,
        -0.50017154172544676,-2.8833612408983415E-5,-0.33389287213054852,-5.0434267119571713E-5,-1.0,
        5.4210108624275222E-20,-0.99999999999999978,0.0,-0.99999999999999978,-5.4210108624275222E-20,-1.0,
        5.4210108624275222E-20,-1.0,5.4210108624275222E-20,-1.0,5.4210108624275222E-20,-1.0,0.0,
        -0.50017155568537663,5.4210108624275222E-20,-0.50017155568537675,0.0,-1.0,5.4210108624275222E-20,
        -0.50017155621007536,0.0,-1.0,1.6263032587282567E-19,-0.50017155530055091,0.0,-1.0,-5.4210108624275222E-20,
        -0.99999999999999978,-1.6263032587282567E-19,-1.0,5.4210108624275222E-20,-1.0,5.4210108624275222E-20,-1.0,
        5.4210108624275222E-20,-0.99999999999999978,-5.4210108624275222E-20,-1.0,5.4210108624275222E-20,
        -0.50017154338877634,0.0,-0.3338928772195392,2.7105054312137611E-20,-0.500171554546532,
        -2.883546297236672E-5,-1.0,5.4210108624275222E-20,-0.99999999999999978,0.0,-1.0,5.4210108624275222E-20,-1.0,
        5.4210108624275222E-20,-1.0,5.4210108624275222E-20,-1.0,5.4210108624275222E-20,-0.99999999999999978,0.0,
        -0.00047387004623103553,-0.0032530855295321241,-4.1504614415460717E-20,-0.00325331080846554,
        -5.4210108624275222E-20,-0.99999999999999989,-0.00012270693090584504,-0.003253333675105293,
        -0.0001096414616121335,-0.50017290377260126,-0.00021633303651176052,-0.0032532861083053037,
        -0.00020082461188265359,-0.33389770950648251,-4.1504614415460717E-20,-0.00325331080846554,
        -5.4210108624275222E-20,-0.99999999999999989,-0.00012270693090584504,-0.003253333675105293,
        -0.0001096414616121335,-0.50017290377260126,-0.00021633303651176052,-0.0032532861083053037,
        -0.00020082461188265359,-0.33389770950648251,0.0,-0.99999999999999989,-1.300195574035351E-19,
        -0.0032533637994211317,-5.4210108624275222E-20,-0.50017291583272638,-1.0418505251227894E-19,
        -0.0032533563672422191,-5.4210108624275222E-20,-0.33389774996742894,0.0,-0.99999999999999989,
        -5.4210108624275222E-20,-0.50017291583272638,-5.4210108624275222E-20,-0.33389774996742894,
        -1.0842021724855044E-19,-0.99999999999999989,0.0,-1.0,-1.0842021724855044E-19,-0.99999999999999989,
        -5.4210108624275222E-20,-0.99999999999999989,-1.0842021724855044E-19,-0.99999999999999989,
        -1.0842021724855044E-19,-0.99999999999999989,-1.0842021724855044E-19,-0.99999999999999989,
        -2.8830983828423494E-5,-0.500172916913477,-5.2621143293484266E-5,-0.3338977537047928,0.0,-1.0,
        -2.8830983828423494E-5,-0.500172916913477,-5.0429547165299344E-5,-0.50017291437548894,
        -5.4210108624275222E-20,-0.50017291583272638,-2.8830983828423385E-5,-0.50017291691347721,
        -5.0429547165299344E-5,-0.50017291437548894,-9.2256767123402269E-5,-0.33389774515228049,
        -1.0842021724855044E-19,-0.99999999999999989,-5.0429547165299344E-5,-0.50017291437548894,
        -9.2256767123402269E-5,-0.33389774515228049,1.0842021724855044E-19,-0.333897749967429,
        -5.2621143293484212E-5,-0.3338977537047928,-9.2256767123402215E-5,-0.33389774515228055,0.0,
        -0.99999999999999989,-1.300195574035351E-19,-0.0032533637994211317,-5.4210108624275222E-20,
        -0.50017291583272638,-1.0418505251227894E-19,-0.0032533563672422191,-5.4210108624275222E-20,
        -0.33389774996742894,-1.0842021724855044E-19,-0.99999999999999989,0.0,-1.0,-1.0842021724855044E-19,
        -0.99999999999999989,-5.4210108624275222E-20,-0.99999999999999989,-2.8830983828423494E-5,-0.500172916913477,
        -5.2621143293484266E-5,-0.3338977537047928,-5.0429547165299344E-5,-0.50017291437548894,
        -9.2256767123402269E-5,-0.33389774515228049,0.0,-0.99999999999999989,0.0,-0.99999999999999989,
        -1.0842021724855044E-19,-0.99999999999999989,-5.4210108624275222E-20,-0.50017292901042176,
        -1.0842021724855044E-19,-0.33389775792997123,0.0,-0.99999999999999989,-5.4210108624275222E-20,
        -0.50017292901042176,-1.0842021724855044E-19,-0.99999999999999989,-1.0842021724855044E-19,
        -0.99999999999999989,-5.4210108624275222E-20,-0.99999999999999989,-5.4210108624275222E-20,
        -0.99999999999999989,-1.0842021724855044E-19,-0.99999999999999989,-1.0842021724855044E-19,
        -0.99999999999999989,-1.0842021724855044E-19,-0.99999999999999989,-5.4210108624275222E-20,
        -0.99999999999999989,-5.4210108624275222E-20,-0.99999999999999989,-1.0842021724855044E-19,
        -0.99999999999999989,-5.2624528352597055E-5,-0.33389775459855631,0.0,-1.0,-2.8833612408983415E-5,
        -0.50017293009143149,-5.4210108624275222E-20,-0.50017291819340215,-2.8832834192057727E-5,
        -0.50017291718052692,-1.0842021724855044E-19,-0.99999999999999989,-5.4210108624275222E-20,
        -0.99999999999999989,-5.0434267119571822E-5,-0.50017292755295606,5.4210108624275222E-20,
        -0.33389775792997128,-5.2624528352597055E-5,-0.33389775459855625,-1.0842021724855044E-19,
        -0.99999999999999989,0.0,-0.99999999999999989,-5.4210108624275222E-20,-0.33389775924466275,0.0,
        -0.500172918193402,-5.4210108624275222E-20,-0.50017292901042176,-1.0842021724855044E-19,
        -0.33389775792997123,-1.0842021724855044E-19,-0.99999999999999989,-5.4210108624275222E-20,
        -0.99999999999999989,-5.4210108624275222E-20,-0.99999999999999989,-2.8832834192057781E-5,
        -0.5001729171805267,-2.8833612408983415E-5,-0.50017293009143149,-5.0434267119571822E-5,-0.50017292755295606,
        0.0,-0.99999999999999989,-5.4210108624275222E-20,-0.99999999999999989,5.4210108624275222E-20,
        -0.50017291884376192,-1.0842021724855044E-19,-0.99999999999999989,0.0,-0.50017293137158414,0.0,
        -0.99999999999999989,-5.4210108624275222E-20,-0.50017293175475663,-1.0842021724855044E-19,
        -0.99999999999999989,-1.0842021724855044E-19,-0.99999999999999989,-5.4210108624275222E-20,
        -0.99999999999999989,-1.0842021724855044E-19,-0.99999999999999989,-5.4210108624275222E-20,
        -0.99999999999999989,-1.0842021724855044E-19,-0.99999999999999989,-1.6263032587282567E-19,
        -0.500172931371584,0.0,-0.50017291884376214,5.4210108624275222E-20,-0.33389776013913919,
        -1.0842021724855044E-19,-0.99999999999999989,0.0,-0.99999999999999989,5.4210108624275222E-20,
        -0.50017291884376192,0.0,-0.50017293137158414,-1.0842021724855044E-19,-0.99999999999999989,
        -1.0842021724855044E-19,-0.99999999999999989,-2.8835462972366666E-5,-0.50017293035853716,0.0,
        -0.99999999999999989,-5.4210108624275222E-20,-0.99999999999999989,-1.0842021724855044E-19,
        -0.99999999999999989,-1.6263032587282567E-19,-0.99999999999999989,0.0,-0.99999999999999989,0.0,
        -0.99999999999999989,0.0,-0.99999999999999989;
END_VAR
VAR_TEMP
    new_x: ARRAY [0..5] OF LREAL;
    y_innov: ARRAY [0..1] OF LREAL;
    th: ARRAY [0..9] OF LREAL;
    b_k: DINT;
    du: ARRAY [0..1] OF LREAL;
    found: BOOL;
    regionmin: DINT;
    betamin: LREAL;
    beta: LREAL;
    betah: LREAL;
    b_h: DINT;
    rtb_xest: ARRAY [0..5] OF LREAL;
    i: DINT;
END_VAR
CASE ssMethodType OF
    SS_INITIALIZE:
        (* SystemInitialize for Atomic SubSystem: '<Root>/Explicit Controller' *)
        (* InitializeConditions for Memory: '<S3>/last_x' *)
        FOR i := 0 TO 5 DO
            last_x_PreviousInput[i] := 0.0;
        END_FOR;
        (* End of InitializeConditions for Memory: '<S3>/last_x' *)
